(* CODESYS project PVCleaningRobot.project

Project tree, tasks and I/O mapping:
  Device : AC801-0221-U0R0, Shenzhen Inovance Technology Co., Ltd., version 3.5.11.50
      settings: PersistentStartAdddr = 0; PersistentStartEndAddr = 5242879; Mode = 0
    application Application
      libraries: Standard, * (System); CmpHCCom, 1.1.0.1 (Inovance); HC_CommBus, 1.3.12.0 (Inovance); CallCFunction, 1.7.2 (Inovance); CmpHCCom, 1.1.0.1 (Inovance); CmpEventMgr, 3.5.8.0 (System); ISysTypes2, 3.5.0.0 (System); CmpApp, 3.5.11.0 (System); IOBlockHandle, 1.3.0.0 (Inovance); HC_OmronUtils, 1.5.4.0 (Inovance); VisuDialogs, * (System); CmpHCTCPIP, 1.0.0.5 (Inovance); Util, 3.5.11.0 (System)
      task ETHERCAT_C (cyclic, interval 4000 µs, priority 0) calls ETHERCAT_C.EtherCAT_Task, 机械臂控制, 运动控制
      task 电池数据通讯 (cyclic, interval t#20ms, priority 16) calls 电池数据通讯
      task 业务逻辑 (cyclic, interval t#4ms, priority 1) calls DCH遥控控制, SLAM指令通讯, SLAM业务通讯
      task 伺服控制 (cyclic, interval t#5ms, priority 1) calls 底盘算法处理
      task 逻辑处理 (cyclic, interval t#20ms, priority 16) calls 报警处理
      program 机械臂控制 [ST]
      DifferentialMonitor
      Symbols
      trace Trace (task ETHERCAT_C): 机械臂控制.sMotionOutputs.dCmdPos[0], 机械臂控制.sMotionOutputs.dCmdPos[1], 机械臂控制.sMotionOutputs.dCmdPos[2], 机械臂控制.sMotionInputs.dFbPos[0], 机械臂控制.sMotionInputs.dFbPos[1], 机械臂控制.sMotionInputs.dFbPos[2], 机械臂控制.sMotionOutputs.dCmdSpace[0], 机械臂控制.sMotionOutputs.dCmdSpace[1], 机械臂控制.sMotionOutputs.dCmdSpace[2], 机械臂控制.sMotionInputs.dFbSpace[0], 机械臂控制.sMotionInputs.dFbPos[0], 机械臂控制.sMotionInputs.dFbPos[1], 机械臂控制.sMotionInputs.dFbPos[2], 机械臂控制.sMotionInputs.dFbPos[3], 机械臂控制.aiCcmdac[0], 机械臂控制.aiCcmdac[1], 机械臂控制.aiCcmdac[2]
      program 末端控制 [ST]: 上下卷扬控制, 传感器检测, 对中机构控制, 回零控制, 报警检测, 滚刷控制, ACT_test
      program 底盘算法处理 [ST]
      数据结构/
        data type 伺服参数结构体
        data type 底盘运行参数结构体
        data type 陀螺仪
        data type 机械臂参数结构体
        data type 系统状态
        data type 功能块状态
        data type PID控制参数
      函数/
        function block EventCallbackFunBLock [ST]: EventCallback, FB_Exit, FB_Init
        SLAM通讯/
          function block 上传信息处理 [ST]
          function block 校验功能块 [ST]
          function block 上传信息处理_1 [ST]
        运动控制/
          function block 伺服控制 [ST]
          function block 底盘平衡算法 [ST]
          function block 底盘控制运动 [ST]
          function block 清扫作业流程 [ST]
          function block 底盘控制运动_1 [ST]
          function block 低通滤波模块 [ST]
          function block 底盘控制运动_2 [ST]
          function block 超声波实时检测调整 [ST]
      全局变量/
        global variables 全局电池数据
        global variables 全局机械臂参数
        global variables 全局伺服参数
        global variables SLAM指令控制
        global variables 全局底盘参数
        global variables 业务流程
        global variables IO刷新数据
        global variables 末端控制参数
        global variables SLAM业务控制
        global variables 报警参数
      program 电池数据通讯 [ST]
      program SLAM指令通讯 [ST]: 系统状态上传, BMS数据上传, 温湿度数据上传, 单体电池电压数据上传, 单体电池温度数据上传, 行走电机状态上传, 悬挂电机状态上传, 轮速计数据上传, UPS数据上传, 超声波数据上传
      program 底盘控制 [ST]: 点动
      trace Trace_2 (task ETHERCAT_C): 末端控制.上卷扬滤波力矩, 末端控制.下卷扬滤波力矩, 末端控制.adFbForce[2]
      program 运动控制 [ST]
      trace Trace_1 (task ETHERCAT_C): 上卷扬运行位置保存, 下卷扬运行位置保存, DCH读遥控数据[0], test3
      program SLAM业务通讯 [ST]: 上装数据上传
      program DCH遥控控制 [ST]: DCH末端控制, DCH遥控数值刷新, DCH底盘控制, DCH机械臂控制
      trace Trace_3 (task ETHERCAT_C): 上侧滤波距离, 下侧滤波距离, 上侧距离, 下侧距离, 末端控制.PID_1.Y, 末端控制.PID_2.Y
      trace Trace_4 (task ETHERCAT_C): 右上轮.fActTorque, 右下轮.fActTorque, 左上轮.fActTorque, 左下轮.fActTorque, 左上轮.fActVelocity, 右上轮.fActVelocity, 左下轮.fActVelocity, 右下轮.fActVelocity, 右上轮.fSetTorque, 右下轮.fSetTorque, 左上轮.fSetTorque, 左下轮.fSetTorque, 左下轮.fSetVelocity, 右下轮.fSetVelocity, 左上轮.fSetVelocity, 右上轮.fSetVelocity, 左上轮.nAxisState, 右上轮.nAxisState, 右下轮.nAxisState, 左下轮.nAxisState, 左上轮.diActVelocity, 左上轮最大轮廓速度, 上卷扬伺服参数.运行位置, 下卷扬伺服参数.运行位置, 上下卷扬自动流程
      program 报警处理 [ST]
      trace Trace_5 (task ETHERCAT_C): 上卷扬运行位置保存, 上侧实际位置值暂存, 上卷扬伺服参数.运行位置, 上卷扬.fActPosition, 上侧距离, 左1滤波距离, 左2滤波距离, 下卷扬运行位置保存, 下侧实际位置值暂存, 下卷扬伺服参数.运行位置, 下卷扬.fActPosition, 下侧距离, 右1滤波距离, 右2滤波距离
    Network Configuration
      EtherCAT Config
    Resources List
    ConfigStorage
    HardWare Configuration
    Device Diagnosis
    SoftMotion General Axis Pool
    MODBUS_TCP : ModbusTCP本地从站, inovance, version 00.00.00.10
    HwConfiguratioinDevice : SystemConfig, Inovance, version 00.00.00.10
        settings: NetworkConfigArray.NetworkConfigArray.BusType = 10; NetworkConfigArray.NetworkConfigArray.RackSum = 1; NetworkConfigArray.NetworkConfigArray.HardwareConfigArray.HardwareConfigArray.RackNo = 1; EnableFun = 12
    ETHERCAT_C : EtherCAT Master SoftMotion, 3S - Smart Software Solutions GmbH, version 3.5.11.10
        settings:  = 0; Autoconfig = 0; NetworkName = 'enp3s0'; SelectNetworkByName = TRUE; DisableTaskGeneration = True
      InoSV630N_机械臂3轴 : SV630_1Axis_03715, Inovance, order no. InoSV630N, version Revision=16#00010000
          settings: Number of Outputs = 6; Number of Inputs = 10; Number of Infos about Outputs = 6; Number of Infos about Inputs = 10; Physical Address of the Slave = 1008; AutoIncr Address of the Slave = 4294967289; StationAlias = 0; Sync.Length = 18; Sync.Length = 32; FMMU.Global Start Address = 16#02000070; FMMU.Length = 18; FMMU.Physical Start Address = 16#1800; FMMU.Access = 16#02; FMMU.Global Start Address = 16#010000DE; FMMU.Length = 32; FMMU.Physical Start Address = 16#1C00; FMMU.Access = 16#01; FMMU.Global Start Address = 16#00080000; FMMU.StartBit = 6; FMMU.EndBit = 6; FMMU.Physical Start Address = 16#080D; FMMU.Access = 16#01; AutoUpdate = False; DC sync0 cycletime = 4000; DC sync1 cycletime = 4000; Number of SDO = 10; Homing method.Index = 16#6098; Homing method.Subindex = 16#00; Homing method.Value = 1; Homing method.Size = 8; Homing method.AbortIfError = FALSE; Homing method.JumpToLine = FALSE; Homing method.Line = 0; Homing method.CompleteAccess = FALSE; Actual Position Calculation Method.Index = 16#60E6; Actual Position Calculation Method.Subindex = 16#00; Actual Position Calculation Method.Value = 0; Actual Position Calculation Method.Size = 8; Actual Position Calculation Method.AbortIfError = FALSE; Actual Position Calculation Method.JumpToLine = FALSE;
            Actual Position Calculation Method.Line = 0; Actual Position Calculation Method.CompleteAccess = FALSE; Speed during search for switch.Index = 16#6099; Speed during search for switch.Subindex = 16#01; Speed during search for switch.Value = 436907; Speed during search for switch.Size = 32; Speed during search for switch.AbortIfError = FALSE; Speed during search for switch.JumpToLine = FALSE; Speed during search for switch.Line = 0; Speed during search for switch.CompleteAccess = FALSE; Homing acceleration.Index = 16#609A; Homing acceleration.Subindex = 16#00; Homing acceleration.Value = 43690666; Homing acceleration.Size = 32; Homing acceleration.AbortIfError = FALSE; Homing acceleration.JumpToLine = FALSE; Homing acceleration.Line = 0; Homing acceleration.CompleteAccess = FALSE; Speed during search for zero.Index = 16#6099; Speed during search for zero.Subindex = 16#02; Speed during search for zero.Value = 43691; Speed during search for zero.Size = 32; Speed during search for zero.AbortIfError = FALSE; Speed during search for zero.JumpToLine = FALSE; Speed during search for zero.Line = 0; Speed during search for zero.CompleteAccess = FALSE; Time of home searching.Index = 16#2005; Time of home searching.Subindex = 16#24; Time of home searching.Value = 50000; Time of home searching.Size = 16; Time of home searching.AbortIfError = FALSE; Time of home searching.JumpToLine = FALSE; Time of home searching.Line = 0; Time of home searching.CompleteAccess = FALSE; Positive torque limit value.Index = 16#60E0; Positive torque limit value.Subindex = 16#00; Positive torque limit value.Value = 3500; Positive torque limit value.Size = 16; Positive torque limit value.AbortIfError = FALSE; Positive torque limit value.JumpToLine = FALSE;
            Positive torque limit value.Line = 0; Positive torque limit value.CompleteAccess = FALSE; Negative torque limit value.Index = 16#60E1; Negative torque limit value.Subindex = 16#00; Negative torque limit value.Value = 3500; Negative torque limit value.Size = 16; Negative torque limit value.AbortIfError = FALSE; Negative torque limit value.JumpToLine = FALSE; Negative torque limit value.Line = 0; Negative torque limit value.CompleteAccess = FALSE; Max profile velocity.Index = 16#607F; Max profile velocity.Subindex = 16#00; Max profile velocity.Value = 26214400; Max profile velocity.Size = 32; Max profile velocity.AbortIfError = FALSE; Max profile velocity.JumpToLine = FALSE; Max profile velocity.Line = 0; Max profile velocity.CompleteAccess = FALSE; RxTxPdo.NumberofEntries = 6; RxTxPdo.Sm = 2; Controlword.Index = 16#6040; Controlword.SubIndex = 0; Controlword.Size = 16; Controlword.DependOnSlot = false; Controlword.DependOnSlotGroup = false; Target position.Index = 16#607A; Target position.SubIndex = 0; Target position.Size = 32; Target position.DependOnSlot = false; Target position.DependOnSlotGroup = false; Touch probe function.Index = 16#60B8; Touch probe function.SubIndex = 0; Touch probe function.Size = 16; Touch probe function.DependOnSlot = false; Touch probe function.DependOnSlotGroup = false; Physical outputs.Index = 16#60FE; Physical outputs.SubIndex = 1; Physical outputs.Size = 32; Physical outputs.DependOnSlot = false; Physical outputs.DependOnSlotGroup = false;
            Target velocity.Index = 16#60FF; Target velocity.SubIndex = 0; Target velocity.Size = 32; Target velocity.DependOnSlot = false; Target velocity.DependOnSlotGroup = false; Target torque.Index = 16#6071; Target torque.SubIndex = 0; Target torque.Size = 16; Target torque.DependOnSlot = false; Target torque.DependOnSlotGroup = false; RxTxPdo.Sm = -1; RxTxPdo.NumberofEntries = 10; RxTxPdo.Sm = 3; Error code.Index = 16#603F; Error code.SubIndex = 0; Error code.Size = 16; Error code.DependOnSlot = false; Error code.DependOnSlotGroup = false; Statusword.Index = 16#6041; Statusword.SubIndex = 0; Statusword.Size = 16; Statusword.DependOnSlot = false; Statusword.DependOnSlotGroup = false; Position actual value.Index = 16#6064; Position actual value.SubIndex = 0; Position actual value.Size = 32; Position actual value.DependOnSlot = false; Position actual value.DependOnSlotGroup = false; Torque actual value.Index = 16#6077; Torque actual value.SubIndex = 0; Torque actual value.Size = 16; Torque actual value.DependOnSlot = false; Torque actual value.DependOnSlotGroup = false; Following error actual value.Index = 16#60F4; Following error actual value.SubIndex = 0; Following error actual value.Size = 32; Following error actual value.DependOnSlot = false; Following error actual value.DependOnSlotGroup = false; Touch probe status.Index = 16#60B9; Touch probe status.SubIndex = 0;
            Touch probe status.Size = 16; Touch probe status.DependOnSlot = false; Touch probe status.DependOnSlotGroup = false; Touch probe pos1 pos value.Index = 16#60BA; Touch probe pos1 pos value.SubIndex = 0; Touch probe pos1 pos value.Size = 32; Touch probe pos1 pos value.DependOnSlot = false; Touch probe pos1 pos value.DependOnSlotGroup = false; Touch probe pos2 pos value.Index = 16#60BC; Touch probe pos2 pos value.SubIndex = 0; Touch probe pos2 pos value.Size = 32; Touch probe pos2 pos value.DependOnSlot = false; Touch probe pos2 pos value.DependOnSlotGroup = false; Digital inputs.Index = 16#60FD; Digital inputs.SubIndex = 0; Digital inputs.Size = 32; Digital inputs.DependOnSlot = false; Digital inputs.DependOnSlotGroup = false; Velocity actual value.Index = 16#606C; Velocity actual value.SubIndex = 0; Velocity actual value.Size = 32; Velocity actual value.DependOnSlot = false; Velocity actual value.DependOnSlotGroup = false; RxTxPdo.Sm = -1; Controlword.Name = 'Controlword'; Controlword.DataType = 'UINT'; Target position.Name = 'Target position'; Target position.DataType = 'DINT'; Touch probe function.Name = 'Touch probe function'; Touch probe function.DataType = 'UINT'; Physical outputs.Name = 'Physical outputs'; Physical outputs.DataType = 'UDINT'; Target velocity.Name = 'Target velocity'; Target velocity.DataType = 'DINT'; Target torque.Name = 'Target torque'; Target torque.DataType = 'INT'; Error code.Name = 'Error code'; Error code.DataType = 'UINT'; Statusword.Name = 'Statusword'; Statusword.DataType = 'UINT';
            Position actual value.Name = 'Position actual value'; Position actual value.DataType = 'DINT'; Torque actual value.Name = 'Torque actual value'; Torque actual value.DataType = 'INT'; Following error actual value.Name = 'Following error actual value'; Following error actual value.DataType = 'DINT'; Touch probe status.Name = 'Touch probe status'; Touch probe status.DataType = 'UINT'; Touch probe pos1 pos value.Name = 'Touch probe pos1 pos value'; Touch probe pos1 pos value.DataType = 'DINT'; Touch probe pos2 pos value.Name = 'Touch probe pos2 pos value'; Touch probe pos2 pos value.DataType = 'DINT'; Digital inputs.Name = 'Digital inputs'; Digital inputs.DataType = 'UDINT'; Velocity actual value.Name = 'Velocity actual value'; Velocity actual value.DataType = 'DINT'
          input  Application.机械臂控制.伺服错误码[2] : UINT  // Error code
          unmapped channels: Controlword, Target position, Touch probe function, Physical outputs, Target velocity, Target torque, Statusword, Position actual value, Torque actual value, Following error actual value, Touch probe status, Touch probe pos1 pos value, Touch probe pos2 pos value, Digital inputs, Velocity actual value
        机械臂3轴 : Axis, Inovance, order no. 0, version 1.0.0.0
            settings: wDriveID = 22; dwRatioTechUnitsDenom = 262144; fSWMaxVelocity = 1000; fSWMaxAcceleration = 10000; fSWMaxDeceleration = 10000; fSWMaxJerk = 100000; iEncoderType = 1; iAbsEncoderOption = 1; HomingMode = 10; ZeroSignal = 0; StartDirction = 1; EndDirection = 1; PosLimitMode = 0; NegLimitMode = 0; HomingVelocity = 10; HomingApproachVelocity = 2; HomingAcceleration = 100; HomingDeceleration = 100; HomingJerk = 0; HomeMaskDistance = 0; HomePositionOffset = 0; HomePushTime = 0; HomeCompensation = 0; HomeTimeout = 0; HomeCompensationVelocity = 1000; 4000 = 0; 4001 = 0; 4003 = true; 4004 = 3; 4005 = 0; 4006 = 1.666667; 4007 = 166.666666; 4008 = 0.166667; 4009 = 50000; 4010 = 3500; 4011 = 3500; 4012 = 100.000000; ScalingIncs = 16#40000; 6005 = 1; AdrOffset_8010 = 148;
              BitOffset_8010 = 0; BitLength_8010 = 16; Address_8010 = '%QW74'; Type_8010 = 'UINT'; AddressPointer_8010 = ADR(%QW74); AdrOffset_8020 = 152; BitOffset_8020 = 0; BitLength_8020 = 32; Address_8020 = '%QD38'; Type_8020 = 'DINT'; AddressPointer_8020 = ADR(%QD38); AdrOffset_8030 = 164; BitOffset_8030 = 0; BitLength_8030 = 32; Address_8030 = '%QD41'; Type_8030 = 'DINT'; AddressPointer_8030 = ADR(%QD41); AdrOffset_8040 = 168; BitOffset_8040 = 0; BitLength_8040 = 16; Address_8040 = '%QW84'; Type_8040 = 'INT'; AddressPointer_8040 = ADR(%QW84); AdrOffset_8050 = 4294967295; BitOffset_8050 = 0; BitLength_8050 = 0; Address_8050 = ''; Type_8050 = ''; AddressPointer_8050 = 0; AdrOffset_8060 = 156; BitOffset_8060 = 0; BitLength_8060 = 16; Address_8060 = '%QW78'; Type_8060 = 'UINT'; AddressPointer_8060 = ADR(%QW78); AdrOffset_8070 = 4294967295; BitOffset_8070 = 0; BitLength_8070 = 0; Address_8070 = ''; Type_8070 = '';
              AddressPointer_8070 = 0; AdrOffset_8080 = 4294967295; BitOffset_8080 = 0; BitLength_8080 = 0; Address_8080 = ''; Type_8080 = ''; AddressPointer_8080 = 0; AdrOffset_8090 = 160; BitOffset_8090 = 0; BitLength_8090 = 32; Address_8090 = '%QD40'; Type_8090 = 'UDINT'; AddressPointer_8090 = ADR(%QD40); AdrOffset_8100 = 4294967295; BitOffset_8100 = 0; BitLength_8100 = 0; Address_8100 = ''; Type_8100 = ''; AddressPointer_8100 = 0; AdrOffset_8510 = 250; BitOffset_8510 = 0; BitLength_8510 = 16; Address_8510 = '%IW125'; Type_8510 = 'UINT'; AddressPointer_8510 = ADR(%IW125); AdrOffset_8520 = 252; BitOffset_8520 = 0; BitLength_8520 = 32; Address_8520 = '%ID63'; Type_8520 = 'DINT'; AddressPointer_8520 = ADR(%ID63); AdrOffset_8530 = 280; BitOffset_8530 = 0; BitLength_8530 = 32; Address_8530 = '%ID70'; Type_8530 = 'DINT'; AddressPointer_8530 = ADR(%ID70); AdrOffset_8540 = 256; BitOffset_8540 = 0; BitLength_8540 = 16;
              Address_8540 = '%IW128'; Type_8540 = 'INT'; AddressPointer_8540 = ADR(%IW128); AdrOffset_8550 = 4294967295; BitOffset_8550 = 0; BitLength_8550 = 0; Address_8550 = ''; Type_8550 = ''; AddressPointer_8550 = 0; AdrOffset_8560 = 276; BitOffset_8560 = 0; BitLength_8560 = 32; Address_8560 = '%ID69'; Type_8560 = 'UDINT'; AddressPointer_8560 = ADR(%ID69); AdrOffset_8570 = 264; BitOffset_8570 = 0; BitLength_8570 = 16; Address_8570 = '%IW132'; Type_8570 = 'UINT'; AddressPointer_8570 = ADR(%IW132); AdrOffset_8580 = 268; BitOffset_8580 = 0; BitLength_8580 = 32; Address_8580 = '%ID67'; Type_8580 = 'DINT'; AddressPointer_8580 = ADR(%ID67); AdrOffset_8590 = 4294967295; BitOffset_8590 = 0; BitLength_8590 = 0; Address_8590 = ''; Type_8590 = ''; AddressPointer_8590 = 0; AdrOffset_8600 = 272; BitOffset_8600 = 0; BitLength_8600 = 32; Address_8600 = '%ID68'; Type_8600 = 'DINT'; AddressPointer_8600 = ADR(%ID68); AdrOffset_8600 = 4294967295;
              BitOffset_8600 = 0; BitLength_8600 = 0; Address_8610 = ''; Type_8610 = ''; AddressPointer_8610 = 0; AdrOffset_8620 = 0; BitOffset_8620 = 0; BitLength_8620 = 16; Address_8620 = '机械臂控制.伺服错误码[2]'; Type_8620 = 'UINT'; AddressPointer_8620 = ADR(机械臂控制.伺服错误码[2]); IsValid = True; IsHostHoming = False; PulseSelectIndex = 2
      InoSV630N_机械臂4轴 : SV630_1Axis_03715, Inovance, order no. InoSV630N, version Revision=16#00010000
          settings: Number of Outputs = 6; Number of Inputs = 10; Number of Infos about Outputs = 6; Number of Infos about Inputs = 10; Physical Address of the Slave = 1009; AutoIncr Address of the Slave = 4294967288; StationAlias = 0; Sync.Length = 18; Sync.Length = 32; FMMU.Global Start Address = 16#02000082; FMMU.Length = 18; FMMU.Physical Start Address = 16#1800; FMMU.Access = 16#02; FMMU.Global Start Address = 16#010000FE; FMMU.Length = 32; FMMU.Physical Start Address = 16#1C00; FMMU.Access = 16#01; FMMU.Global Start Address = 16#00080000; FMMU.StartBit = 7; FMMU.EndBit = 7; FMMU.Physical Start Address = 16#080D; FMMU.Access = 16#01; AutoUpdate = False; DC sync0 cycletime = 4000; DC sync1 cycletime = 4000; Number of SDO = 10; Homing method.Index = 16#6098; Homing method.Subindex = 16#00; Homing method.Value = 1; Homing method.Size = 8; Homing method.AbortIfError = FALSE; Homing method.JumpToLine = FALSE; Homing method.Line = 0; Homing method.CompleteAccess = FALSE; Actual Position Calculation Method.Index = 16#60E6; Actual Position Calculation Method.Subindex = 16#00; Actual Position Calculation Method.Value = 0; Actual Position Calculation Method.Size = 8; Actual Position Calculation Method.AbortIfError = FALSE; Actual Position Calculation Method.JumpToLine = FALSE;
            Actual Position Calculation Method.Line = 0; Actual Position Calculation Method.CompleteAccess = FALSE; Speed during search for switch.Index = 16#6099; Speed during search for switch.Subindex = 16#01; Speed during search for switch.Value = 436907; Speed during search for switch.Size = 32; Speed during search for switch.AbortIfError = FALSE; Speed during search for switch.JumpToLine = FALSE; Speed during search for switch.Line = 0; Speed during search for switch.CompleteAccess = FALSE; Homing acceleration.Index = 16#609A; Homing acceleration.Subindex = 16#00; Homing acceleration.Value = 43690666; Homing acceleration.Size = 32; Homing acceleration.AbortIfError = FALSE; Homing acceleration.JumpToLine = FALSE; Homing acceleration.Line = 0; Homing acceleration.CompleteAccess = FALSE; Speed during search for zero.Index = 16#6099; Speed during search for zero.Subindex = 16#02; Speed during search for zero.Value = 43691; Speed during search for zero.Size = 32; Speed during search for zero.AbortIfError = FALSE; Speed during search for zero.JumpToLine = FALSE; Speed during search for zero.Line = 0; Speed during search for zero.CompleteAccess = FALSE; Time of home searching.Index = 16#2005; Time of home searching.Subindex = 16#24; Time of home searching.Value = 50000; Time of home searching.Size = 16; Time of home searching.AbortIfError = FALSE; Time of home searching.JumpToLine = FALSE; Time of home searching.Line = 0; Time of home searching.CompleteAccess = FALSE; Positive torque limit value.Index = 16#60E0; Positive torque limit value.Subindex = 16#00; Positive torque limit value.Value = 3500; Positive torque limit value.Size = 16; Positive torque limit value.AbortIfError = FALSE; Positive torque limit value.JumpToLine = FALSE;
            Positive torque limit value.Line = 0; Positive torque limit value.CompleteAccess = FALSE; Negative torque limit value.Index = 16#60E1; Negative torque limit value.Subindex = 16#00; Negative torque limit value.Value = 3500; Negative torque limit value.Size = 16; Negative torque limit value.AbortIfError = FALSE; Negative torque limit value.JumpToLine = FALSE; Negative torque limit value.Line = 0; Negative torque limit value.CompleteAccess = FALSE; Max profile velocity.Index = 16#607F; Max profile velocity.Subindex = 16#00; Max profile velocity.Value = 26214400; Max profile velocity.Size = 32; Max profile velocity.AbortIfError = FALSE; Max profile velocity.JumpToLine = FALSE; Max profile velocity.Line = 0; Max profile velocity.CompleteAccess = FALSE; RxTxPdo.NumberofEntries = 6; RxTxPdo.Sm = 2; Controlword.Index = 16#6040; Controlword.SubIndex = 0; Controlword.Size = 16; Controlword.DependOnSlot = false; Controlword.DependOnSlotGroup = false; Target position.Index = 16#607A; Target position.SubIndex = 0; Target position.Size = 32; Target position.DependOnSlot = false; Target position.DependOnSlotGroup = false; Touch probe function.Index = 16#60B8; Touch probe function.SubIndex = 0; Touch probe function.Size = 16; Touch probe function.DependOnSlot = false; Touch probe function.DependOnSlotGroup = false; Physical outputs.Index = 16#60FE; Physical outputs.SubIndex = 1; Physical outputs.Size = 32; Physical outputs.DependOnSlot = false; Physical outputs.DependOnSlotGroup = false;
            Target velocity.Index = 16#60FF; Target velocity.SubIndex = 0; Target velocity.Size = 32; Target velocity.DependOnSlot = false; Target velocity.DependOnSlotGroup = false; Target torque.Index = 16#6071; Target torque.SubIndex = 0; Target torque.Size = 16; Target torque.DependOnSlot = false; Target torque.DependOnSlotGroup = false; RxTxPdo.Sm = -1; RxTxPdo.NumberofEntries = 10; RxTxPdo.Sm = 3; Error code.Index = 16#603F; Error code.SubIndex = 0; Error code.Size = 16; Error code.DependOnSlot = false; Error code.DependOnSlotGroup = false; Statusword.Index = 16#6041; Statusword.SubIndex = 0; Statusword.Size = 16; Statusword.DependOnSlot = false; Statusword.DependOnSlotGroup = false; Position actual value.Index = 16#6064; Position actual value.SubIndex = 0; Position actual value.Size = 32; Position actual value.DependOnSlot = false; Position actual value.DependOnSlotGroup = false; Torque actual value.Index = 16#6077; Torque actual value.SubIndex = 0; Torque actual value.Size = 16; Torque actual value.DependOnSlot = false; Torque actual value.DependOnSlotGroup = false; Following error actual value.Index = 16#60F4; Following error actual value.SubIndex = 0; Following error actual value.Size = 32; Following error actual value.DependOnSlot = false; Following error actual value.DependOnSlotGroup = false; Touch probe status.Index = 16#60B9; Touch probe status.SubIndex = 0;
            Touch probe status.Size = 16; Touch probe status.DependOnSlot = false; Touch probe status.DependOnSlotGroup = false; Touch probe pos1 pos value.Index = 16#60BA; Touch probe pos1 pos value.SubIndex = 0; Touch probe pos1 pos value.Size = 32; Touch probe pos1 pos value.DependOnSlot = false; Touch probe pos1 pos value.DependOnSlotGroup = false; Touch probe pos2 pos value.Index = 16#60BC; Touch probe pos2 pos value.SubIndex = 0; Touch probe pos2 pos value.Size = 32; Touch probe pos2 pos value.DependOnSlot = false; Touch probe pos2 pos value.DependOnSlotGroup = false; Digital inputs.Index = 16#60FD; Digital inputs.SubIndex = 0; Digital inputs.Size = 32; Digital inputs.DependOnSlot = false; Digital inputs.DependOnSlotGroup = false; Velocity actual value.Index = 16#606C; Velocity actual value.SubIndex = 0; Velocity actual value.Size = 32; Velocity actual value.DependOnSlot = false; Velocity actual value.DependOnSlotGroup = false; RxTxPdo.Sm = -1; Controlword.Name = 'Controlword'; Controlword.DataType = 'UINT'; Target position.Name = 'Target position'; Target position.DataType = 'DINT'; Touch probe function.Name = 'Touch probe function'; Touch probe function.DataType = 'UINT'; Physical outputs.Name = 'Physical outputs'; Physical outputs.DataType = 'UDINT'; Target velocity.Name = 'Target velocity'; Target velocity.DataType = 'DINT'; Target torque.Name = 'Target torque'; Target torque.DataType = 'INT'; Error code.Name = 'Error code'; Error code.DataType = 'UINT'; Statusword.Name = 'Statusword'; Statusword.DataType = 'UINT';
            Position actual value.Name = 'Position actual value'; Position actual value.DataType = 'DINT'; Torque actual value.Name = 'Torque actual value'; Torque actual value.DataType = 'INT'; Following error actual value.Name = 'Following error actual value'; Following error actual value.DataType = 'DINT'; Touch probe status.Name = 'Touch probe status'; Touch probe status.DataType = 'UINT'; Touch probe pos1 pos value.Name = 'Touch probe pos1 pos value'; Touch probe pos1 pos value.DataType = 'DINT'; Touch probe pos2 pos value.Name = 'Touch probe pos2 pos value'; Touch probe pos2 pos value.DataType = 'DINT'; Digital inputs.Name = 'Digital inputs'; Digital inputs.DataType = 'UDINT'; Velocity actual value.Name = 'Velocity actual value'; Velocity actual value.DataType = 'DINT'
          input  Application.机械臂控制.伺服错误码[3] : UINT  // Error code
          unmapped channels: Controlword, Target position, Touch probe function, Physical outputs, Target velocity, Target torque, Statusword, Position actual value, Torque actual value, Following error actual value, Touch probe status, Touch probe pos1 pos value, Touch probe pos2 pos value, Digital inputs, Velocity actual value
        机械臂4轴 : Axis, Inovance, order no. 0, version 1.0.0.0
            settings: wDriveID = 23; dwRatioTechUnitsDenom = 262144; fSWMaxVelocity = 1000; fSWMaxAcceleration = 10000; fSWMaxDeceleration = 10000; fSWMaxJerk = 100000; iEncoderType = 1; iAbsEncoderOption = 1; HomingMode = 10; ZeroSignal = 0; StartDirction = 1; EndDirection = 1; PosLimitMode = 0; NegLimitMode = 0; HomingVelocity = 10; HomingApproachVelocity = 2; HomingAcceleration = 100; HomingDeceleration = 100; HomingJerk = 0; HomeMaskDistance = 0; HomePositionOffset = 0; HomePushTime = 0; HomeCompensation = 0; HomeTimeout = 0; HomeCompensationVelocity = 1000; 4000 = 0; 4001 = 0; 4003 = true; 4004 = 3; 4005 = 0; 4006 = 1.666667; 4007 = 166.666666; 4008 = 0.166667; 4009 = 50000; 4010 = 3500; 4011 = 3500; 4012 = 100.000000; ScalingIncs = 16#40000; 6005 = 1; AdrOffset_8010 = 172;
              BitOffset_8010 = 0; BitLength_8010 = 16; Address_8010 = '%QW86'; Type_8010 = 'UINT'; AddressPointer_8010 = ADR(%QW86); AdrOffset_8020 = 176; BitOffset_8020 = 0; BitLength_8020 = 32; Address_8020 = '%QD44'; Type_8020 = 'DINT'; AddressPointer_8020 = ADR(%QD44); AdrOffset_8030 = 188; BitOffset_8030 = 0; BitLength_8030 = 32; Address_8030 = '%QD47'; Type_8030 = 'DINT'; AddressPointer_8030 = ADR(%QD47); AdrOffset_8040 = 192; BitOffset_8040 = 0; BitLength_8040 = 16; Address_8040 = '%QW96'; Type_8040 = 'INT'; AddressPointer_8040 = ADR(%QW96); AdrOffset_8050 = 4294967295; BitOffset_8050 = 0; BitLength_8050 = 0; Address_8050 = ''; Type_8050 = ''; AddressPointer_8050 = 0; AdrOffset_8060 = 180; BitOffset_8060 = 0; BitLength_8060 = 16; Address_8060 = '%QW90'; Type_8060 = 'UINT'; AddressPointer_8060 = ADR(%QW90); AdrOffset_8070 = 4294967295; BitOffset_8070 = 0; BitLength_8070 = 0; Address_8070 = ''; Type_8070 = '';
              AddressPointer_8070 = 0; AdrOffset_8080 = 4294967295; BitOffset_8080 = 0; BitLength_8080 = 0; Address_8080 = ''; Type_8080 = ''; AddressPointer_8080 = 0; AdrOffset_8090 = 184; BitOffset_8090 = 0; BitLength_8090 = 32; Address_8090 = '%QD46'; Type_8090 = 'UDINT'; AddressPointer_8090 = ADR(%QD46); AdrOffset_8100 = 4294967295; BitOffset_8100 = 0; BitLength_8100 = 0; Address_8100 = ''; Type_8100 = ''; AddressPointer_8100 = 0; AdrOffset_8510 = 286; BitOffset_8510 = 0; BitLength_8510 = 16; Address_8510 = '%IW143'; Type_8510 = 'UINT'; AddressPointer_8510 = ADR(%IW143); AdrOffset_8520 = 288; BitOffset_8520 = 0; BitLength_8520 = 32; Address_8520 = '%ID72'; Type_8520 = 'DINT'; AddressPointer_8520 = ADR(%ID72); AdrOffset_8530 = 316; BitOffset_8530 = 0; BitLength_8530 = 32; Address_8530 = '%ID79'; Type_8530 = 'DINT'; AddressPointer_8530 = ADR(%ID79); AdrOffset_8540 = 292; BitOffset_8540 = 0; BitLength_8540 = 16;
              Address_8540 = '%IW146'; Type_8540 = 'INT'; AddressPointer_8540 = ADR(%IW146); AdrOffset_8550 = 4294967295; BitOffset_8550 = 0; BitLength_8550 = 0; Address_8550 = ''; Type_8550 = ''; AddressPointer_8550 = 0; AdrOffset_8560 = 312; BitOffset_8560 = 0; BitLength_8560 = 32; Address_8560 = '%ID78'; Type_8560 = 'UDINT'; AddressPointer_8560 = ADR(%ID78); AdrOffset_8570 = 300; BitOffset_8570 = 0; BitLength_8570 = 16; Address_8570 = '%IW150'; Type_8570 = 'UINT'; AddressPointer_8570 = ADR(%IW150); AdrOffset_8580 = 304; BitOffset_8580 = 0; BitLength_8580 = 32; Address_8580 = '%ID76'; Type_8580 = 'DINT'; AddressPointer_8580 = ADR(%ID76); AdrOffset_8590 = 4294967295; BitOffset_8590 = 0; BitLength_8590 = 0; Address_8590 = ''; Type_8590 = ''; AddressPointer_8590 = 0; AdrOffset_8600 = 308; BitOffset_8600 = 0; BitLength_8600 = 32; Address_8600 = '%ID77'; Type_8600 = 'DINT'; AddressPointer_8600 = ADR(%ID77); AdrOffset_8600 = 4294967295;
              BitOffset_8600 = 0; BitLength_8600 = 0; Address_8610 = ''; Type_8610 = ''; AddressPointer_8610 = 0; AdrOffset_8620 = 0; BitOffset_8620 = 0; BitLength_8620 = 16; Address_8620 = '机械臂控制.伺服错误码[3]'; Type_8620 = 'UINT'; AddressPointer_8620 = ADR(机械臂控制.伺服错误码[3]); IsValid = True; IsHostHoming = False; PulseSelectIndex = 2
      InoSV630N_机械臂1轴 : SV630_1Axis_03715, Inovance, order no. InoSV630N, version Revision=16#00010000
          settings: Number of Outputs = 7; Number of Inputs = 10; Number of Infos about Outputs = 7; Number of Infos about Inputs = 10; EnableExpertSettings = True; Physical Address of the Slave = 1006; AutoIncr Address of the Slave = 4294967291; StationAlias = 0; Sync.Length = 19; Sync.Length = 32; FMMU.Global Start Address = 16#0200004B; FMMU.Length = 19; FMMU.Physical Start Address = 16#1800; FMMU.Access = 16#02; FMMU.Global Start Address = 16#0100009E; FMMU.Length = 32; FMMU.Physical Start Address = 16#1C00; FMMU.Access = 16#01; FMMU.Global Start Address = 16#00080000; FMMU.StartBit = 4; FMMU.EndBit = 4; FMMU.Physical Start Address = 16#080D; FMMU.Access = 16#01; AutoUpdate = False; DC sync0 cycletime = 4000; DC sync0 cycletime = 4000000; DC sync1 cycletime = 4000; DC sync1 cycletime = 4000000; Number of SDO = 10; Homing method.Index = 16#6098; Homing method.Subindex = 16#00; Homing method.Value = 1; Homing method.Size = 8; Homing method.AbortIfError = FALSE; Homing method.JumpToLine = FALSE; Homing method.Line = 0; Homing method.CompleteAccess = False; Actual Position Calculation Method.Index = 16#60E6; Actual Position Calculation Method.Subindex = 16#00; Actual Position Calculation Method.Value = 0;
            Actual Position Calculation Method.Size = 8; Actual Position Calculation Method.AbortIfError = FALSE; Actual Position Calculation Method.JumpToLine = FALSE; Actual Position Calculation Method.Line = 0; Actual Position Calculation Method.CompleteAccess = False; Speed during search for switch.Index = 16#6099; Speed during search for switch.Subindex = 16#01; Speed during search for switch.Value = 436907; Speed during search for switch.Size = 32; Speed during search for switch.AbortIfError = FALSE; Speed during search for switch.JumpToLine = FALSE; Speed during search for switch.Line = 0; Speed during search for switch.CompleteAccess = False; Homing acceleration.Index = 16#609A; Homing acceleration.Subindex = 16#00; Homing acceleration.Value = 43690666; Homing acceleration.Size = 32; Homing acceleration.AbortIfError = FALSE; Homing acceleration.JumpToLine = FALSE; Homing acceleration.Line = 0; Homing acceleration.CompleteAccess = False; Speed during search for zero.Index = 16#6099; Speed during search for zero.Subindex = 16#02; Speed during search for zero.Value = 43691; Speed during search for zero.Size = 32; Speed during search for zero.AbortIfError = FALSE; Speed during search for zero.JumpToLine = FALSE; Speed during search for zero.Line = 0; Speed during search for zero.CompleteAccess = False; Time of home searching.Index = 16#2005; Time of home searching.Subindex = 16#24; Time of home searching.Value = 50000; Time of home searching.Size = 16; Time of home searching.AbortIfError = FALSE; Time of home searching.JumpToLine = FALSE; Time of home searching.Line = 0; Time of home searching.CompleteAccess = False; Positive torque limit value.Index = 16#60E0; Positive torque limit value.Subindex = 16#00; Positive torque limit value.Value = 3500;
            Positive torque limit value.Size = 16; Positive torque limit value.AbortIfError = FALSE; Positive torque limit value.JumpToLine = FALSE; Positive torque limit value.Line = 0; Positive torque limit value.CompleteAccess = False; Negative torque limit value.Index = 16#60E1; Negative torque limit value.Subindex = 16#00; Negative torque limit value.Value = 3500; Negative torque limit value.Size = 16; Negative torque limit value.AbortIfError = FALSE; Negative torque limit value.JumpToLine = FALSE; Negative torque limit value.Line = 0; Negative torque limit value.CompleteAccess = False; Max profile velocity.Index = 16#607F; Max profile velocity.Subindex = 16#00; Max profile velocity.Value = 26214400; Max profile velocity.Size = 32; Max profile velocity.AbortIfError = FALSE; Max profile velocity.JumpToLine = FALSE; Max profile velocity.Line = 0; Max profile velocity.CompleteAccess = False; RxTxPdo.NumberofEntries = 7; RxTxPdo.Sm = 2; RxTxPdo.DependOnSlot = False; RxTxPdo.DependOnSlotGroup = False; RxTxPdo.OverwrittenByModule = False; Exclude = [16#1701,16#1702,16#1703,16#1704,16#1705]; Controlword.Index = 16#6040; Controlword.SubIndex = 0; Controlword.Size = 16; Controlword.Offset = 0; Controlword.DependOnSlot = False; Controlword.DependOnSlotGroup = False; Target position.Index = 16#607A; Target position.SubIndex = 0; Target position.Size = 32; Target position.Offset = 0; Target position.DependOnSlot = False; Target position.DependOnSlotGroup = False; Touch probe function.Index = 16#60B8;
            Touch probe function.SubIndex = 0; Touch probe function.Size = 16; Touch probe function.Offset = 0; Touch probe function.DependOnSlot = False; Touch probe function.DependOnSlotGroup = False; Physical outputs.Index = 16#60FE; Physical outputs.SubIndex = 1; Physical outputs.Size = 32; Physical outputs.Offset = 0; Physical outputs.DependOnSlot = False; Physical outputs.DependOnSlotGroup = False; Target velocity.Index = 16#60FF; Target velocity.SubIndex = 0; Target velocity.Size = 32; Target velocity.Offset = 0; Target velocity.DependOnSlot = False; Target velocity.DependOnSlotGroup = False; Modes of operation.Index = 16#6060; Modes of operation.SubIndex = 0; Modes of operation.Size = 8; Modes of operation.Offset = 0; Modes of operation.DependOnSlot = False; Modes of operation.DependOnSlotGroup = False; Target torque.Index = 16#6071; Target torque.SubIndex = 0; Target torque.Size = 16; Target torque.Offset = 0; Target torque.DependOnSlot = False; Target torque.DependOnSlotGroup = False; RxTxPdo.Sm = -1; RxTxPdo.NumberofEntries = 10; RxTxPdo.Sm = 3; Error code.Index = 16#603F; Error code.SubIndex = 0; Error code.Size = 16; Error code.DependOnSlot = false; Error code.DependOnSlotGroup = false; Statusword.Index = 16#6041; Statusword.SubIndex = 0; Statusword.Size = 16;
            Statusword.DependOnSlot = false; Statusword.DependOnSlotGroup = false; Position actual value.Index = 16#6064; Position actual value.SubIndex = 0; Position actual value.Size = 32; Position actual value.DependOnSlot = false; Position actual value.DependOnSlotGroup = false; Torque actual value.Index = 16#6077; Torque actual value.SubIndex = 0; Torque actual value.Size = 16; Torque actual value.DependOnSlot = false; Torque actual value.DependOnSlotGroup = false; Following error actual value.Index = 16#60F4; Following error actual value.SubIndex = 0; Following error actual value.Size = 32; Following error actual value.DependOnSlot = false; Following error actual value.DependOnSlotGroup = false; Touch probe status.Index = 16#60B9; Touch probe status.SubIndex = 0; Touch probe status.Size = 16; Touch probe status.DependOnSlot = false; Touch probe status.DependOnSlotGroup = false; Touch probe pos1 pos value.Index = 16#60BA; Touch probe pos1 pos value.SubIndex = 0; Touch probe pos1 pos value.Size = 32; Touch probe pos1 pos value.DependOnSlot = false; Touch probe pos1 pos value.DependOnSlotGroup = false; Touch probe pos2 pos value.Index = 16#60BC; Touch probe pos2 pos value.SubIndex = 0; Touch probe pos2 pos value.Size = 32; Touch probe pos2 pos value.DependOnSlot = false; Touch probe pos2 pos value.DependOnSlotGroup = false; Digital inputs.Index = 16#60FD; Digital inputs.SubIndex = 0; Digital inputs.Size = 32; Digital inputs.DependOnSlot = false; Digital inputs.DependOnSlotGroup = false; Velocity actual value.Index = 16#606C; Velocity actual value.SubIndex = 0; Velocity actual value.Size = 32;
            Velocity actual value.DependOnSlot = false; Velocity actual value.DependOnSlotGroup = false; RxTxPdo.Sm = -1; Controlword.Name = 'Controlword'; Controlword.DataType = 'UINT'; Controlword.Default = ''; Controlword.Comment = ''; Target position.Name = 'Target position'; Target position.DataType = 'DINT'; Target position.Default = ''; Target position.Comment = ''; Touch probe function.Name = 'Touch probe function'; Touch probe function.DataType = 'UINT'; Touch probe function.Default = ''; Touch probe function.Comment = ''; Physical outputs.Name = 'Physical outputs'; Physical outputs.DataType = 'UDINT'; Physical outputs.Default = ''; Physical outputs.Comment = ''; Target velocity.Name = 'Target velocity'; Target velocity.DataType = 'DINT'; Target velocity.Default = ''; Target velocity.Comment = ''; Modes of operation.Name = 'Modes of operation'; Modes of operation.DataType = 'SINT'; Modes of operation.Default = ''; Modes of operation.Comment = ''; Target torque.Name = 'Target torque'; Target torque.DataType = 'INT'; Target torque.Default = ''; Target torque.Comment = ''; Error code.Name = 'Error code'; Error code.DataType = 'UINT'; Statusword.Name = 'Statusword'; Statusword.DataType = 'UINT'; Position actual value.Name = 'Position actual value'; Position actual value.DataType = 'DINT'; Torque actual value.Name = 'Torque actual value'; Torque actual value.DataType = 'INT'; Following error actual value.Name = 'Following error actual value';
            Following error actual value.DataType = 'DINT'; Touch probe status.Name = 'Touch probe status'; Touch probe status.DataType = 'UINT'; Touch probe pos1 pos value.Name = 'Touch probe pos1 pos value'; Touch probe pos1 pos value.DataType = 'DINT'; Touch probe pos2 pos value.Name = 'Touch probe pos2 pos value'; Touch probe pos2 pos value.DataType = 'DINT'; Digital inputs.Name = 'Digital inputs'; Digital inputs.DataType = 'UDINT'; Velocity actual value.Name = 'Velocity actual value'; Velocity actual value.DataType = 'DINT'
          input  Application.机械臂控制.伺服错误码[0] : UINT  // Error code
          unmapped channels: Controlword, Target position, Touch probe function, Physical outputs, Target velocity, Modes of operation, Target torque, Statusword, Position actual value, Torque actual value, Following error actual value, Touch probe status, Touch probe pos1 pos value, Touch probe pos2 pos value, Digital inputs, Velocity actual value
        机械臂1轴 : Axis, Inovance, order no. 0, version 1.0.0.0
            settings: wDriveID = 20; dwRatioTechUnitsDenom = 262144; fSWMaxVelocity = 1000; fSWMaxAcceleration = 10000; fSWMaxDeceleration = 10000; fSWMaxJerk = 100000; iEncoderType = 1; iAbsEncoderOption = 1; HomingMode = 10; ZeroSignal = 0; StartDirction = 1; EndDirection = 1; PosLimitMode = 0; NegLimitMode = 0; HomingVelocity = 10; HomingApproachVelocity = 2; HomingAcceleration = 100; HomingDeceleration = 100; HomingJerk = 0; HomeMaskDistance = 0; HomePositionOffset = 0; HomePushTime = 0; HomeCompensation = 0; HomeTimeout = 0; HomeCompensationVelocity = 1000; 4000 = 0; 4001 = 0; 4003 = true; 4004 = 3; 4005 = 0; 4006 = 1.666667; 4007 = 166.666666; 4008 = 0.166667; 4009 = 50000; 4010 = 3500; 4011 = 3500; 4012 = 100.000000; ScalingIncs = 16#40000; 6005 = 1; AdrOffset_8010 = 100;
              BitOffset_8010 = 0; BitLength_8010 = 16; Address_8010 = '%QW50'; Type_8010 = 'UINT'; AddressPointer_8010 = ADR(%QW50); AdrOffset_8020 = 104; BitOffset_8020 = 0; BitLength_8020 = 32; Address_8020 = '%QD26'; Type_8020 = 'DINT'; AddressPointer_8020 = ADR(%QD26); AdrOffset_8030 = 116; BitOffset_8030 = 0; BitLength_8030 = 32; Address_8030 = '%QD29'; Type_8030 = 'DINT'; AddressPointer_8030 = ADR(%QD29); AdrOffset_8040 = 122; BitOffset_8040 = 0; BitLength_8040 = 16; Address_8040 = '%QW61'; Type_8040 = 'INT'; AddressPointer_8040 = ADR(%QW61); AdrOffset_8050 = 120; BitOffset_8050 = 0; BitLength_8050 = 8; Address_8050 = '%QB120'; Type_8050 = 'SINT'; AddressPointer_8050 = ADR(%QB120); AdrOffset_8060 = 108; BitOffset_8060 = 0; BitLength_8060 = 16; Address_8060 = '%QW54'; Type_8060 = 'UINT'; AddressPointer_8060 = ADR(%QW54); AdrOffset_8070 = 4294967295; BitOffset_8070 = 0; BitLength_8070 = 0; Address_8070 = ''; Type_8070 = '';
              AddressPointer_8070 = 0; AdrOffset_8080 = 4294967295; BitOffset_8080 = 0; BitLength_8080 = 0; Address_8080 = ''; Type_8080 = ''; AddressPointer_8080 = 0; AdrOffset_8090 = 112; BitOffset_8090 = 0; BitLength_8090 = 32; Address_8090 = '%QD28'; Type_8090 = 'UDINT'; AddressPointer_8090 = ADR(%QD28); AdrOffset_8100 = 4294967295; BitOffset_8100 = 0; BitLength_8100 = 0; Address_8100 = ''; Type_8100 = ''; AddressPointer_8100 = 0; AdrOffset_8510 = 178; BitOffset_8510 = 0; BitLength_8510 = 16; Address_8510 = '%IW89'; Type_8510 = 'UINT'; AddressPointer_8510 = ADR(%IW89); AdrOffset_8520 = 180; BitOffset_8520 = 0; BitLength_8520 = 32; Address_8520 = '%ID45'; Type_8520 = 'DINT'; AddressPointer_8520 = ADR(%ID45); AdrOffset_8530 = 208; BitOffset_8530 = 0; BitLength_8530 = 32; Address_8530 = '%ID52'; Type_8530 = 'DINT'; AddressPointer_8530 = ADR(%ID52); AdrOffset_8540 = 184; BitOffset_8540 = 0; BitLength_8540 = 16;
              Address_8540 = '%IW92'; Type_8540 = 'INT'; AddressPointer_8540 = ADR(%IW92); AdrOffset_8550 = 4294967295; BitOffset_8550 = 0; BitLength_8550 = 0; Address_8550 = ''; Type_8550 = ''; AddressPointer_8550 = 0; AdrOffset_8560 = 204; BitOffset_8560 = 0; BitLength_8560 = 32; Address_8560 = '%ID51'; Type_8560 = 'UDINT'; AddressPointer_8560 = ADR(%ID51); AdrOffset_8570 = 192; BitOffset_8570 = 0; BitLength_8570 = 16; Address_8570 = '%IW96'; Type_8570 = 'UINT'; AddressPointer_8570 = ADR(%IW96); AdrOffset_8580 = 196; BitOffset_8580 = 0; BitLength_8580 = 32; Address_8580 = '%ID49'; Type_8580 = 'DINT'; AddressPointer_8580 = ADR(%ID49); AdrOffset_8590 = 4294967295; BitOffset_8590 = 0; BitLength_8590 = 0; Address_8590 = ''; Type_8590 = ''; AddressPointer_8590 = 0; AdrOffset_8600 = 200; BitOffset_8600 = 0; BitLength_8600 = 32; Address_8600 = '%ID50'; Type_8600 = 'DINT'; AddressPointer_8600 = ADR(%ID50); AdrOffset_8600 = 4294967295;
              BitOffset_8600 = 0; BitLength_8600 = 0; Address_8610 = ''; Type_8610 = ''; AddressPointer_8610 = 0; AdrOffset_8620 = 0; BitOffset_8620 = 0; BitLength_8620 = 16; Address_8620 = '机械臂控制.伺服错误码[0]'; Type_8620 = 'UINT'; AddressPointer_8620 = ADR(机械臂控制.伺服错误码[0]); Automatic Mapping = True; IsValid = True; IsHostHoming = False; PulseSelectIndex = 2
      InoSV630N_机械臂2轴 : SV630_1Axis_03715, Inovance, order no. InoSV630N, version Revision=16#00010000
          settings: Number of Outputs = 6; Number of Inputs = 10; Number of Infos about Outputs = 6; Number of Infos about Inputs = 10; EnableExpertSettings = True; Physical Address of the Slave = 1007; AutoIncr Address of the Slave = 4294967290; StationAlias = 0; Sync.Length = 18; Sync.Length = 32; FMMU.Global Start Address = 16#0200005E; FMMU.Length = 18; FMMU.Physical Start Address = 16#1800; FMMU.Access = 16#02; FMMU.Global Start Address = 16#010000BE; FMMU.Length = 32; FMMU.Physical Start Address = 16#1C00; FMMU.Access = 16#01; FMMU.Global Start Address = 16#00080000; FMMU.StartBit = 5; FMMU.EndBit = 5; FMMU.Physical Start Address = 16#080D; FMMU.Access = 16#01; AutoUpdate = False; DC sync0 cycletime = 4000; DC sync0 cycletime = 4000000; DC sync1 cycletime = 4000; DC sync1 cycletime = 4000000; Number of SDO = 10; Homing method.Index = 16#6098; Homing method.Subindex = 16#00; Homing method.Value = 1; Homing method.Size = 8; Homing method.AbortIfError = FALSE; Homing method.JumpToLine = FALSE; Homing method.Line = 0; Homing method.CompleteAccess = FALSE; Actual Position Calculation Method.Index = 16#60E6; Actual Position Calculation Method.Subindex = 16#00; Actual Position Calculation Method.Value = 0;
            Actual Position Calculation Method.Size = 8; Actual Position Calculation Method.AbortIfError = FALSE; Actual Position Calculation Method.JumpToLine = FALSE; Actual Position Calculation Method.Line = 0; Actual Position Calculation Method.CompleteAccess = FALSE; Speed during search for switch.Index = 16#6099; Speed during search for switch.Subindex = 16#01; Speed during search for switch.Value = 436907; Speed during search for switch.Size = 32; Speed during search for switch.AbortIfError = FALSE; Speed during search for switch.JumpToLine = FALSE; Speed during search for switch.Line = 0; Speed during search for switch.CompleteAccess = FALSE; Homing acceleration.Index = 16#609A; Homing acceleration.Subindex = 16#00; Homing acceleration.Value = 43690666; Homing acceleration.Size = 32; Homing acceleration.AbortIfError = FALSE; Homing acceleration.JumpToLine = FALSE; Homing acceleration.Line = 0; Homing acceleration.CompleteAccess = FALSE; Speed during search for zero.Index = 16#6099; Speed during search for zero.Subindex = 16#02; Speed during search for zero.Value = 43691; Speed during search for zero.Size = 32; Speed during search for zero.AbortIfError = FALSE; Speed during search for zero.JumpToLine = FALSE; Speed during search for zero.Line = 0; Speed during search for zero.CompleteAccess = FALSE; Time of home searching.Index = 16#2005; Time of home searching.Subindex = 16#24; Time of home searching.Value = 50000; Time of home searching.Size = 16; Time of home searching.AbortIfError = FALSE; Time of home searching.JumpToLine = FALSE; Time of home searching.Line = 0; Time of home searching.CompleteAccess = FALSE; Positive torque limit value.Index = 16#60E0; Positive torque limit value.Subindex = 16#00; Positive torque limit value.Value = 3500;
            Positive torque limit value.Size = 16; Positive torque limit value.AbortIfError = FALSE; Positive torque limit value.JumpToLine = FALSE; Positive torque limit value.Line = 0; Positive torque limit value.CompleteAccess = FALSE; Negative torque limit value.Index = 16#60E1; Negative torque limit value.Subindex = 16#00; Negative torque limit value.Value = 3500; Negative torque limit value.Size = 16; Negative torque limit value.AbortIfError = FALSE; Negative torque limit value.JumpToLine = FALSE; Negative torque limit value.Line = 0; Negative torque limit value.CompleteAccess = FALSE; Max profile velocity.Index = 16#607F; Max profile velocity.Subindex = 16#00; Max profile velocity.Value = 26214400; Max profile velocity.Size = 32; Max profile velocity.AbortIfError = FALSE; Max profile velocity.JumpToLine = FALSE; Max profile velocity.Line = 0; Max profile velocity.CompleteAccess = FALSE; RxTxPdo.NumberofEntries = 6; RxTxPdo.Sm = 2; Controlword.Index = 16#6040; Controlword.SubIndex = 0; Controlword.Size = 16; Controlword.DependOnSlot = false; Controlword.DependOnSlotGroup = false; Target position.Index = 16#607A; Target position.SubIndex = 0; Target position.Size = 32; Target position.DependOnSlot = false; Target position.DependOnSlotGroup = false; Touch probe function.Index = 16#60B8; Touch probe function.SubIndex = 0; Touch probe function.Size = 16; Touch probe function.DependOnSlot = false; Touch probe function.DependOnSlotGroup = false; Physical outputs.Index = 16#60FE; Physical outputs.SubIndex = 1;
            Physical outputs.Size = 32; Physical outputs.DependOnSlot = false; Physical outputs.DependOnSlotGroup = false; Target velocity.Index = 16#60FF; Target velocity.SubIndex = 0; Target velocity.Size = 32; Target velocity.DependOnSlot = false; Target velocity.DependOnSlotGroup = false; Target torque.Index = 16#6071; Target torque.SubIndex = 0; Target torque.Size = 16; Target torque.DependOnSlot = false; Target torque.DependOnSlotGroup = false; RxTxPdo.Sm = -1; RxTxPdo.NumberofEntries = 10; RxTxPdo.Sm = 3; Error code.Index = 16#603F; Error code.SubIndex = 0; Error code.Size = 16; Error code.DependOnSlot = false; Error code.DependOnSlotGroup = false; Statusword.Index = 16#6041; Statusword.SubIndex = 0; Statusword.Size = 16; Statusword.DependOnSlot = false; Statusword.DependOnSlotGroup = false; Position actual value.Index = 16#6064; Position actual value.SubIndex = 0; Position actual value.Size = 32; Position actual value.DependOnSlot = false; Position actual value.DependOnSlotGroup = false; Torque actual value.Index = 16#6077; Torque actual value.SubIndex = 0; Torque actual value.Size = 16; Torque actual value.DependOnSlot = false; Torque actual value.DependOnSlotGroup = false; Following error actual value.Index = 16#60F4; Following error actual value.SubIndex = 0; Following error actual value.Size = 32; Following error actual value.DependOnSlot = false;
            Following error actual value.DependOnSlotGroup = false; Touch probe status.Index = 16#60B9; Touch probe status.SubIndex = 0; Touch probe status.Size = 16; Touch probe status.DependOnSlot = false; Touch probe status.DependOnSlotGroup = false; Touch probe pos1 pos value.Index = 16#60BA; Touch probe pos1 pos value.SubIndex = 0; Touch probe pos1 pos value.Size = 32; Touch probe pos1 pos value.DependOnSlot = false; Touch probe pos1 pos value.DependOnSlotGroup = false; Touch probe pos2 pos value.Index = 16#60BC; Touch probe pos2 pos value.SubIndex = 0; Touch probe pos2 pos value.Size = 32; Touch probe pos2 pos value.DependOnSlot = false; Touch probe pos2 pos value.DependOnSlotGroup = false; Digital inputs.Index = 16#60FD; Digital inputs.SubIndex = 0; Digital inputs.Size = 32; Digital inputs.DependOnSlot = false; Digital inputs.DependOnSlotGroup = false; Velocity actual value.Index = 16#606C; Velocity actual value.SubIndex = 0; Velocity actual value.Size = 32; Velocity actual value.DependOnSlot = false; Velocity actual value.DependOnSlotGroup = false; RxTxPdo.Sm = -1; Controlword.Name = 'Controlword'; Controlword.DataType = 'UINT'; Target position.Name = 'Target position'; Target position.DataType = 'DINT'; Touch probe function.Name = 'Touch probe function'; Touch probe function.DataType = 'UINT'; Physical outputs.Name = 'Physical outputs'; Physical outputs.DataType = 'UDINT'; Target velocity.Name = 'Target velocity'; Target velocity.DataType = 'DINT'; Target torque.Name = 'Target torque'; Target torque.DataType = 'INT'; Error code.Name = 'Error code';
            Error code.DataType = 'UINT'; Statusword.Name = 'Statusword'; Statusword.DataType = 'UINT'; Position actual value.Name = 'Position actual value'; Position actual value.DataType = 'DINT'; Torque actual value.Name = 'Torque actual value'; Torque actual value.DataType = 'INT'; Following error actual value.Name = 'Following error actual value'; Following error actual value.DataType = 'DINT'; Touch probe status.Name = 'Touch probe status'; Touch probe status.DataType = 'UINT'; Touch probe pos1 pos value.Name = 'Touch probe pos1 pos value'; Touch probe pos1 pos value.DataType = 'DINT'; Touch probe pos2 pos value.Name = 'Touch probe pos2 pos value'; Touch probe pos2 pos value.DataType = 'DINT'; Digital inputs.Name = 'Digital inputs'; Digital inputs.DataType = 'UDINT'; Velocity actual value.Name = 'Velocity actual value'; Velocity actual value.DataType = 'DINT'
          input  Application.机械臂控制.伺服错误码[1] : UINT  // Error code
          unmapped channels: Controlword, Target position, Touch probe function, Physical outputs, Target velocity, Target torque, Statusword, Position actual value, Torque actual value, Following error actual value, Touch probe status, Touch probe pos1 pos value, Touch probe pos2 pos value, Digital inputs, Velocity actual value
        机械臂2轴 : Axis, Inovance, order no. 0, version 1.0.0.0
            settings: wDriveID = 21; dwRatioTechUnitsDenom = 262144; fSWMaxVelocity = 1000; fSWMaxAcceleration = 10000; fSWMaxDeceleration = 10000; fSWMaxJerk = 100000; iEncoderType = 1; iAbsEncoderOption = 1; HomingMode = 10; ZeroSignal = 0; StartDirction = 1; EndDirection = 1; PosLimitMode = 0; NegLimitMode = 0; HomingVelocity = 10; HomingApproachVelocity = 2; HomingAcceleration = 100; HomingDeceleration = 100; HomingJerk = 0; HomeMaskDistance = 0; HomePositionOffset = 0; HomePushTime = 0; HomeCompensation = 0; HomeTimeout = 0; HomeCompensationVelocity = 1000; 4000 = 0; 4001 = 0; 4003 = true; 4004 = 3; 4005 = 0; 4006 = 1.666667; 4007 = 166.666666; 4008 = 0.166667; 4009 = 50000; 4010 = 3500; 4011 = 3500; 4012 = 100.000000; ScalingIncs = 16#40000; 6005 = 1; AdrOffset_8010 = 124;
              BitOffset_8010 = 0; BitLength_8010 = 16; Address_8010 = '%QW62'; Type_8010 = 'UINT'; AddressPointer_8010 = ADR(%QW62); AdrOffset_8020 = 128; BitOffset_8020 = 0; BitLength_8020 = 32; Address_8020 = '%QD32'; Type_8020 = 'DINT'; AddressPointer_8020 = ADR(%QD32); AdrOffset_8030 = 140; BitOffset_8030 = 0; BitLength_8030 = 32; Address_8030 = '%QD35'; Type_8030 = 'DINT'; AddressPointer_8030 = ADR(%QD35); AdrOffset_8040 = 144; BitOffset_8040 = 0; BitLength_8040 = 16; Address_8040 = '%QW72'; Type_8040 = 'INT'; AddressPointer_8040 = ADR(%QW72); AdrOffset_8050 = 4294967295; BitOffset_8050 = 0; BitLength_8050 = 0; Address_8050 = ''; Type_8050 = ''; AddressPointer_8050 = 0; AdrOffset_8060 = 132; BitOffset_8060 = 0; BitLength_8060 = 16; Address_8060 = '%QW66'; Type_8060 = 'UINT'; AddressPointer_8060 = ADR(%QW66); AdrOffset_8070 = 4294967295; BitOffset_8070 = 0; BitLength_8070 = 0; Address_8070 = ''; Type_8070 = '';
              AddressPointer_8070 = 0; AdrOffset_8080 = 4294967295; BitOffset_8080 = 0; BitLength_8080 = 0; Address_8080 = ''; Type_8080 = ''; AddressPointer_8080 = 0; AdrOffset_8090 = 136; BitOffset_8090 = 0; BitLength_8090 = 32; Address_8090 = '%QD34'; Type_8090 = 'UDINT'; AddressPointer_8090 = ADR(%QD34); AdrOffset_8100 = 4294967295; BitOffset_8100 = 0; BitLength_8100 = 0; Address_8100 = ''; Type_8100 = ''; AddressPointer_8100 = 0; AdrOffset_8510 = 214; BitOffset_8510 = 0; BitLength_8510 = 16; Address_8510 = '%IW107'; Type_8510 = 'UINT'; AddressPointer_8510 = ADR(%IW107); AdrOffset_8520 = 216; BitOffset_8520 = 0; BitLength_8520 = 32; Address_8520 = '%ID54'; Type_8520 = 'DINT'; AddressPointer_8520 = ADR(%ID54); AdrOffset_8530 = 244; BitOffset_8530 = 0; BitLength_8530 = 32; Address_8530 = '%ID61'; Type_8530 = 'DINT'; AddressPointer_8530 = ADR(%ID61); AdrOffset_8540 = 220; BitOffset_8540 = 0; BitLength_8540 = 16;
              Address_8540 = '%IW110'; Type_8540 = 'INT'; AddressPointer_8540 = ADR(%IW110); AdrOffset_8550 = 4294967295; BitOffset_8550 = 0; BitLength_8550 = 0; Address_8550 = ''; Type_8550 = ''; AddressPointer_8550 = 0; AdrOffset_8560 = 240; BitOffset_8560 = 0; BitLength_8560 = 32; Address_8560 = '%ID60'; Type_8560 = 'UDINT'; AddressPointer_8560 = ADR(%ID60); AdrOffset_8570 = 228; BitOffset_8570 = 0; BitLength_8570 = 16; Address_8570 = '%IW114'; Type_8570 = 'UINT'; AddressPointer_8570 = ADR(%IW114); AdrOffset_8580 = 232; BitOffset_8580 = 0; BitLength_8580 = 32; Address_8580 = '%ID58'; Type_8580 = 'DINT'; AddressPointer_8580 = ADR(%ID58); AdrOffset_8590 = 4294967295; BitOffset_8590 = 0; BitLength_8590 = 0; Address_8590 = ''; Type_8590 = ''; AddressPointer_8590 = 0; AdrOffset_8600 = 236; BitOffset_8600 = 0; BitLength_8600 = 32; Address_8600 = '%ID59'; Type_8600 = 'DINT'; AddressPointer_8600 = ADR(%ID59); AdrOffset_8600 = 4294967295;
              BitOffset_8600 = 0; BitLength_8600 = 0; Address_8610 = ''; Type_8610 = ''; AddressPointer_8610 = 0; AdrOffset_8620 = 0; BitOffset_8620 = 0; BitLength_8620 = 16; Address_8620 = '机械臂控制.伺服错误码[1]'; Type_8620 = 'UINT'; AddressPointer_8620 = ADR(机械臂控制.伺服错误码[1]); IsValid = True; IsHostHoming = False; PulseSelectIndex = 2
      InoSV630N_伸缩轴 : SV630_1Axis_03715, Inovance, order no. InoSV630N, version Revision=16#00010000
          settings: Number of Outputs = 6; Number of Inputs = 10; Number of Infos about Outputs = 6; Number of Infos about Inputs = 10; Physical Address of the Slave = 1001; StationAlias = 0; Sync.Length = 18; Sync.Length = 32; FMMU.Global Start Address = 16#02000000; FMMU.Length = 18; FMMU.Physical Start Address = 16#1800; FMMU.Access = 16#02; FMMU.Global Start Address = 16#01000000; FMMU.Length = 32; FMMU.Physical Start Address = 16#1C00; FMMU.Access = 16#01; FMMU.Global Start Address = 16#00080000; FMMU.Physical Start Address = 16#080D; FMMU.Access = 16#01; AutoUpdate = False; DC sync0 cycletime = 4000; DC sync1 cycletime = 4000; Number of SDO = 10; Homing method.Index = 16#6098; Homing method.Subindex = 16#00; Homing method.Value = 1; Homing method.Size = 8; Homing method.AbortIfError = FALSE; Homing method.JumpToLine = FALSE; Homing method.Line = 0; Homing method.CompleteAccess = FALSE; Actual Position Calculation Method.Index = 16#60E6; Actual Position Calculation Method.Subindex = 16#00; Actual Position Calculation Method.Value = 0; Actual Position Calculation Method.Size = 8; Actual Position Calculation Method.AbortIfError = FALSE; Actual Position Calculation Method.JumpToLine = FALSE; Actual Position Calculation Method.Line = 0; Actual Position Calculation Method.CompleteAccess = FALSE; Speed during search for switch.Index = 16#6099;
            Speed during search for switch.Subindex = 16#01; Speed during search for switch.Value = 87381; Speed during search for switch.Size = 32; Speed during search for switch.AbortIfError = FALSE; Speed during search for switch.JumpToLine = FALSE; Speed during search for switch.Line = 0; Speed during search for switch.CompleteAccess = FALSE; Homing acceleration.Index = 16#609A; Homing acceleration.Subindex = 16#00; Homing acceleration.Value = 8738133; Homing acceleration.Size = 32; Homing acceleration.AbortIfError = FALSE; Homing acceleration.JumpToLine = FALSE; Homing acceleration.Line = 0; Homing acceleration.CompleteAccess = FALSE; Speed during search for zero.Index = 16#6099; Speed during search for zero.Subindex = 16#02; Speed during search for zero.Value = 8738; Speed during search for zero.Size = 32; Speed during search for zero.AbortIfError = FALSE; Speed during search for zero.JumpToLine = FALSE; Speed during search for zero.Line = 0; Speed during search for zero.CompleteAccess = FALSE; Time of home searching.Index = 16#2005; Time of home searching.Subindex = 16#24; Time of home searching.Value = 50000; Time of home searching.Size = 16; Time of home searching.AbortIfError = FALSE; Time of home searching.JumpToLine = FALSE; Time of home searching.Line = 0; Time of home searching.CompleteAccess = FALSE; Positive torque limit value.Index = 16#60E0; Positive torque limit value.Subindex = 16#00; Positive torque limit value.Value = 3500; Positive torque limit value.Size = 16; Positive torque limit value.AbortIfError = FALSE; Positive torque limit value.JumpToLine = FALSE; Positive torque limit value.Line = 0; Positive torque limit value.CompleteAccess = FALSE; Negative torque limit value.Index = 16#60E1;
            Negative torque limit value.Subindex = 16#00; Negative torque limit value.Value = 3500; Negative torque limit value.Size = 16; Negative torque limit value.AbortIfError = FALSE; Negative torque limit value.JumpToLine = FALSE; Negative torque limit value.Line = 0; Negative torque limit value.CompleteAccess = FALSE; Max profile velocity.Index = 16#607F; Max profile velocity.Subindex = 16#00; Max profile velocity.Value = 5242880; Max profile velocity.Size = 32; Max profile velocity.AbortIfError = FALSE; Max profile velocity.JumpToLine = FALSE; Max profile velocity.Line = 0; Max profile velocity.CompleteAccess = FALSE; RxTxPdo.NumberofEntries = 6; RxTxPdo.Sm = 2; Controlword.Index = 16#6040; Controlword.SubIndex = 0; Controlword.Size = 16; Controlword.DependOnSlot = false; Controlword.DependOnSlotGroup = false; Target position.Index = 16#607A; Target position.SubIndex = 0; Target position.Size = 32; Target position.DependOnSlot = false; Target position.DependOnSlotGroup = false; Touch probe function.Index = 16#60B8; Touch probe function.SubIndex = 0; Touch probe function.Size = 16; Touch probe function.DependOnSlot = false; Touch probe function.DependOnSlotGroup = false; Physical outputs.Index = 16#60FE; Physical outputs.SubIndex = 1; Physical outputs.Size = 32; Physical outputs.DependOnSlot = false; Physical outputs.DependOnSlotGroup = false; Target velocity.Index = 16#60FF; Target velocity.SubIndex = 0; Target velocity.Size = 32;
            Target velocity.DependOnSlot = false; Target velocity.DependOnSlotGroup = false; Target torque.Index = 16#6071; Target torque.SubIndex = 0; Target torque.Size = 16; Target torque.DependOnSlot = false; Target torque.DependOnSlotGroup = false; RxTxPdo.Sm = -1; RxTxPdo.NumberofEntries = 10; RxTxPdo.Sm = 3; Error code.Index = 16#603F; Error code.SubIndex = 0; Error code.Size = 16; Error code.DependOnSlot = false; Error code.DependOnSlotGroup = false; Statusword.Index = 16#6041; Statusword.SubIndex = 0; Statusword.Size = 16; Statusword.DependOnSlot = false; Statusword.DependOnSlotGroup = false; Position actual value.Index = 16#6064; Position actual value.SubIndex = 0; Position actual value.Size = 32; Position actual value.DependOnSlot = false; Position actual value.DependOnSlotGroup = false; Torque actual value.Index = 16#6077; Torque actual value.SubIndex = 0; Torque actual value.Size = 16; Torque actual value.DependOnSlot = false; Torque actual value.DependOnSlotGroup = false; Following error actual value.Index = 16#60F4; Following error actual value.SubIndex = 0; Following error actual value.Size = 32; Following error actual value.DependOnSlot = false; Following error actual value.DependOnSlotGroup = false; Touch probe status.Index = 16#60B9; Touch probe status.SubIndex = 0; Touch probe status.Size = 16; Touch probe status.DependOnSlot = false; Touch probe status.DependOnSlotGroup = false;
            Touch probe pos1 pos value.Index = 16#60BA; Touch probe pos1 pos value.SubIndex = 0; Touch probe pos1 pos value.Size = 32; Touch probe pos1 pos value.DependOnSlot = false; Touch probe pos1 pos value.DependOnSlotGroup = false; Touch probe pos2 pos value.Index = 16#60BC; Touch probe pos2 pos value.SubIndex = 0; Touch probe pos2 pos value.Size = 32; Touch probe pos2 pos value.DependOnSlot = false; Touch probe pos2 pos value.DependOnSlotGroup = false; Digital inputs.Index = 16#60FD; Digital inputs.SubIndex = 0; Digital inputs.Size = 32; Digital inputs.DependOnSlot = false; Digital inputs.DependOnSlotGroup = false; Velocity actual value.Index = 16#606C; Velocity actual value.SubIndex = 0; Velocity actual value.Size = 32; Velocity actual value.DependOnSlot = false; Velocity actual value.DependOnSlotGroup = false; RxTxPdo.Sm = -1; Controlword.Name = 'Controlword'; Controlword.DataType = 'UINT'; Target position.Name = 'Target position'; Target position.DataType = 'DINT'; Touch probe function.Name = 'Touch probe function'; Touch probe function.DataType = 'UINT'; Physical outputs.Name = 'Physical outputs'; Physical outputs.DataType = 'UDINT'; Target velocity.Name = 'Target velocity'; Target velocity.DataType = 'DINT'; Target torque.Name = 'Target torque'; Target torque.DataType = 'INT'; Error code.Name = 'Error code'; Error code.DataType = 'UINT'; Statusword.Name = 'Statusword'; Statusword.DataType = 'UINT'; Position actual value.Name = 'Position actual value'; Position actual value.DataType = 'DINT'; Torque actual value.Name = 'Torque actual value';
            Torque actual value.DataType = 'INT'; Following error actual value.Name = 'Following error actual value'; Following error actual value.DataType = 'DINT'; Touch probe status.Name = 'Touch probe status'; Touch probe status.DataType = 'UINT'; Touch probe pos1 pos value.Name = 'Touch probe pos1 pos value'; Touch probe pos1 pos value.DataType = 'DINT'; Touch probe pos2 pos value.Name = 'Touch probe pos2 pos value'; Touch probe pos2 pos value.DataType = 'DINT'; Digital inputs.Name = 'Digital inputs'; Digital inputs.DataType = 'UDINT'; Velocity actual value.Name = 'Velocity actual value'; Velocity actual value.DataType = 'DINT'
          input  Application.末端控制.adFbForce[0] : INT  // Torque actual value
          unmapped channels: Controlword, Target position, Touch probe function, Physical outputs, Target velocity, Target torque, Error code, Statusword, Position actual value, Following error actual value, Touch probe status, Touch probe pos1 pos value, Touch probe pos2 pos value, Digital inputs, Velocity actual value
        伸缩轴 : Axis, Inovance, order no. 0, version 1.0.0.0
            settings: wDriveID = 16; dwRatioTechUnitsDenom = 262144; iRatioTechUnitsNum = 5; fSWMaxVelocity = 1000; fSWMaxAcceleration = 10000; fSWMaxDeceleration = 10000; fSWMaxJerk = 100000; iEncoderType = 1; iAbsEncoderOption = 1; HomingMode = 10; ZeroSignal = 0; StartDirction = 1; EndDirection = 1; PosLimitMode = 0; NegLimitMode = 0; HomingVelocity = 10; HomingApproachVelocity = 2; HomingAcceleration = 100; HomingDeceleration = 100; HomingJerk = 0; HomeMaskDistance = 0; HomePositionOffset = 0; HomePushTime = 0; HomeCompensation = 0; HomeTimeout = 0; HomeCompensationVelocity = 1000; 4000 = 0; 4001 = 0; 4003 = true; 4004 = 3; 4005 = 0; 4006 = 1.666667; 4007 = 166.666666; 4008 = 0.166667; 4009 = 50000; 4010 = 3500; 4011 = 3500; 4012 = 100.000000; ScalingIncs = 16#40000; 6005 = 5;
              AdrOffset_8010 = 0; BitOffset_8010 = 0; BitLength_8010 = 16; Address_8010 = '%QW0'; Type_8010 = 'UINT'; AddressPointer_8010 = ADR(%QW0); AdrOffset_8020 = 4; BitOffset_8020 = 0; BitLength_8020 = 32; Address_8020 = '%QD1'; Type_8020 = 'DINT'; AddressPointer_8020 = ADR(%QD1); AdrOffset_8030 = 16; BitOffset_8030 = 0; BitLength_8030 = 32; Address_8030 = '%QD4'; Type_8030 = 'DINT'; AddressPointer_8030 = ADR(%QD4); AdrOffset_8040 = 20; BitOffset_8040 = 0; BitLength_8040 = 16; Address_8040 = '%QW10'; Type_8040 = 'INT'; AddressPointer_8040 = ADR(%QW10); AdrOffset_8050 = 4294967295; BitOffset_8050 = 0; BitLength_8050 = 0; Address_8050 = ''; Type_8050 = ''; AddressPointer_8050 = 0; AdrOffset_8060 = 8; BitOffset_8060 = 0; BitLength_8060 = 16; Address_8060 = '%QW4'; Type_8060 = 'UINT'; AddressPointer_8060 = ADR(%QW4); AdrOffset_8070 = 4294967295; BitOffset_8070 = 0; BitLength_8070 = 0; Address_8070 = '';
              Type_8070 = ''; AddressPointer_8070 = 0; AdrOffset_8080 = 4294967295; BitOffset_8080 = 0; BitLength_8080 = 0; Address_8080 = ''; Type_8080 = ''; AddressPointer_8080 = 0; AdrOffset_8090 = 12; BitOffset_8090 = 0; BitLength_8090 = 32; Address_8090 = '%QD3'; Type_8090 = 'UDINT'; AddressPointer_8090 = ADR(%QD3); AdrOffset_8100 = 4294967295; BitOffset_8100 = 0; BitLength_8100 = 0; Address_8100 = ''; Type_8100 = ''; AddressPointer_8100 = 0; AdrOffset_8510 = 2; BitOffset_8510 = 0; BitLength_8510 = 16; Address_8510 = '%IW1'; Type_8510 = 'UINT'; AddressPointer_8510 = ADR(%IW1); AdrOffset_8520 = 4; BitOffset_8520 = 0; BitLength_8520 = 32; Address_8520 = '%ID1'; Type_8520 = 'DINT'; AddressPointer_8520 = ADR(%ID1); AdrOffset_8530 = 32; BitOffset_8530 = 0; BitLength_8530 = 32; Address_8530 = '%ID8'; Type_8530 = 'DINT'; AddressPointer_8530 = ADR(%ID8); AdrOffset_8540 = 0; BitOffset_8540 = 0;
              BitLength_8540 = 16; Address_8540 = '末端控制.adFbForce[0]'; Type_8540 = 'INT'; AddressPointer_8540 = ADR(末端控制.adFbForce[0]); AdrOffset_8550 = 4294967295; BitOffset_8550 = 0; BitLength_8550 = 0; Address_8550 = ''; Type_8550 = ''; AddressPointer_8550 = 0; AdrOffset_8560 = 28; BitOffset_8560 = 0; BitLength_8560 = 32; Address_8560 = '%ID7'; Type_8560 = 'UDINT'; AddressPointer_8560 = ADR(%ID7); AdrOffset_8570 = 16; BitOffset_8570 = 0; BitLength_8570 = 16; Address_8570 = '%IW8'; Type_8570 = 'UINT'; AddressPointer_8570 = ADR(%IW8); AdrOffset_8580 = 20; BitOffset_8580 = 0; BitLength_8580 = 32; Address_8580 = '%ID5'; Type_8580 = 'DINT'; AddressPointer_8580 = ADR(%ID5); AdrOffset_8590 = 4294967295; BitOffset_8590 = 0; BitLength_8590 = 0; Address_8590 = ''; Type_8590 = ''; AddressPointer_8590 = 0; AdrOffset_8600 = 24; BitOffset_8600 = 0; BitLength_8600 = 32; Address_8600 = '%ID6'; Type_8600 = 'DINT'; AddressPointer_8600 = ADR(%ID6);
              AdrOffset_8600 = 4294967295; BitOffset_8600 = 0; BitLength_8600 = 0; Address_8610 = ''; Type_8610 = ''; AddressPointer_8610 = 0; AdrOffset_8620 = 0; BitOffset_8620 = 0; BitLength_8620 = 16; Address_8620 = '%IW0'; Type_8620 = 'UINT'; AddressPointer_8620 = ADR(%IW0); IsValid = True; IsHostHoming = False; PulseSelectIndex = 2
      InoSV630N_上卷扬 : SV630_1Axis_03715, Inovance, order no. InoSV630N, version Revision=16#00010000
          settings: Number of Outputs = 6; Number of Inputs = 10; Number of Infos about Outputs = 6; Number of Infos about Inputs = 10; Physical Address of the Slave = 1002; AutoIncr Address of the Slave = 4294967295; StationAlias = 0; Sync.Length = 18; Sync.Length = 32; FMMU.Global Start Address = 16#02000012; FMMU.Length = 18; FMMU.Physical Start Address = 16#1800; FMMU.Access = 16#02; FMMU.Global Start Address = 16#01000020; FMMU.Length = 32; FMMU.Physical Start Address = 16#1C00; FMMU.Access = 16#01; FMMU.Global Start Address = 16#00080000; FMMU.StartBit = 1; FMMU.EndBit = 1; FMMU.Physical Start Address = 16#080D; FMMU.Access = 16#01; AutoUpdate = False; DC sync0 cycletime = 4000; DC sync1 cycletime = 4000; Number of SDO = 10; Homing method.Index = 16#6098; Homing method.Subindex = 16#00; Homing method.Value = 1; Homing method.Size = 8; Homing method.AbortIfError = FALSE; Homing method.JumpToLine = FALSE; Homing method.Line = 0; Homing method.CompleteAccess = FALSE; Actual Position Calculation Method.Index = 16#60E6; Actual Position Calculation Method.Subindex = 16#00; Actual Position Calculation Method.Value = 0; Actual Position Calculation Method.Size = 8; Actual Position Calculation Method.AbortIfError = FALSE; Actual Position Calculation Method.JumpToLine = FALSE;
            Actual Position Calculation Method.Line = 0; Actual Position Calculation Method.CompleteAccess = FALSE; Speed during search for switch.Index = 16#6099; Speed during search for switch.Subindex = 16#01; Speed during search for switch.Value = 43460; Speed during search for switch.Size = 32; Speed during search for switch.AbortIfError = FALSE; Speed during search for switch.JumpToLine = FALSE; Speed during search for switch.Line = 0; Speed during search for switch.CompleteAccess = FALSE; Homing acceleration.Index = 16#609A; Homing acceleration.Subindex = 16#00; Homing acceleration.Value = 4345995; Homing acceleration.Size = 32; Homing acceleration.AbortIfError = FALSE; Homing acceleration.JumpToLine = FALSE; Homing acceleration.Line = 0; Homing acceleration.CompleteAccess = FALSE; Speed during search for zero.Index = 16#6099; Speed during search for zero.Subindex = 16#02; Speed during search for zero.Value = 4346; Speed during search for zero.Size = 32; Speed during search for zero.AbortIfError = FALSE; Speed during search for zero.JumpToLine = FALSE; Speed during search for zero.Line = 0; Speed during search for zero.CompleteAccess = FALSE; Time of home searching.Index = 16#2005; Time of home searching.Subindex = 16#24; Time of home searching.Value = 50000; Time of home searching.Size = 16; Time of home searching.AbortIfError = FALSE; Time of home searching.JumpToLine = FALSE; Time of home searching.Line = 0; Time of home searching.CompleteAccess = FALSE; Positive torque limit value.Index = 16#60E0; Positive torque limit value.Subindex = 16#00; Positive torque limit value.Value = 3500; Positive torque limit value.Size = 16; Positive torque limit value.AbortIfError = FALSE; Positive torque limit value.JumpToLine = FALSE;
            Positive torque limit value.Line = 0; Positive torque limit value.CompleteAccess = FALSE; Negative torque limit value.Index = 16#60E1; Negative torque limit value.Subindex = 16#00; Negative torque limit value.Value = 3500; Negative torque limit value.Size = 16; Negative torque limit value.AbortIfError = FALSE; Negative torque limit value.JumpToLine = FALSE; Negative torque limit value.Line = 0; Negative torque limit value.CompleteAccess = FALSE; Max profile velocity.Index = 16#607F; Max profile velocity.Subindex = 16#00; Max profile velocity.Value = 2607597; Max profile velocity.Size = 32; Max profile velocity.AbortIfError = FALSE; Max profile velocity.JumpToLine = FALSE; Max profile velocity.Line = 0; Max profile velocity.CompleteAccess = FALSE; RxTxPdo.NumberofEntries = 6; RxTxPdo.Sm = 2; Controlword.Index = 16#6040; Controlword.SubIndex = 0; Controlword.Size = 16; Controlword.DependOnSlot = false; Controlword.DependOnSlotGroup = false; Target position.Index = 16#607A; Target position.SubIndex = 0; Target position.Size = 32; Target position.DependOnSlot = false; Target position.DependOnSlotGroup = false; Touch probe function.Index = 16#60B8; Touch probe function.SubIndex = 0; Touch probe function.Size = 16; Touch probe function.DependOnSlot = false; Touch probe function.DependOnSlotGroup = false; Physical outputs.Index = 16#60FE; Physical outputs.SubIndex = 1; Physical outputs.Size = 32; Physical outputs.DependOnSlot = false; Physical outputs.DependOnSlotGroup = false;
            Target velocity.Index = 16#60FF; Target velocity.SubIndex = 0; Target velocity.Size = 32; Target velocity.DependOnSlot = false; Target velocity.DependOnSlotGroup = false; Target torque.Index = 16#6071; Target torque.SubIndex = 0; Target torque.Size = 16; Target torque.DependOnSlot = false; Target torque.DependOnSlotGroup = false; RxTxPdo.Sm = -1; RxTxPdo.NumberofEntries = 10; RxTxPdo.Sm = 3; Error code.Index = 16#603F; Error code.SubIndex = 0; Error code.Size = 16; Error code.DependOnSlot = false; Error code.DependOnSlotGroup = false; Statusword.Index = 16#6041; Statusword.SubIndex = 0; Statusword.Size = 16; Statusword.DependOnSlot = false; Statusword.DependOnSlotGroup = false; Position actual value.Index = 16#6064; Position actual value.SubIndex = 0; Position actual value.Size = 32; Position actual value.DependOnSlot = false; Position actual value.DependOnSlotGroup = false; Torque actual value.Index = 16#6077; Torque actual value.SubIndex = 0; Torque actual value.Size = 16; Torque actual value.DependOnSlot = false; Torque actual value.DependOnSlotGroup = false; Following error actual value.Index = 16#60F4; Following error actual value.SubIndex = 0; Following error actual value.Size = 32; Following error actual value.DependOnSlot = false; Following error actual value.DependOnSlotGroup = false; Touch probe status.Index = 16#60B9; Touch probe status.SubIndex = 0;
            Touch probe status.Size = 16; Touch probe status.DependOnSlot = false; Touch probe status.DependOnSlotGroup = false; Touch probe pos1 pos value.Index = 16#60BA; Touch probe pos1 pos value.SubIndex = 0; Touch probe pos1 pos value.Size = 32; Touch probe pos1 pos value.DependOnSlot = false; Touch probe pos1 pos value.DependOnSlotGroup = false; Touch probe pos2 pos value.Index = 16#60BC; Touch probe pos2 pos value.SubIndex = 0; Touch probe pos2 pos value.Size = 32; Touch probe pos2 pos value.DependOnSlot = false; Touch probe pos2 pos value.DependOnSlotGroup = false; Digital inputs.Index = 16#60FD; Digital inputs.SubIndex = 0; Digital inputs.Size = 32; Digital inputs.DependOnSlot = false; Digital inputs.DependOnSlotGroup = false; Velocity actual value.Index = 16#606C; Velocity actual value.SubIndex = 0; Velocity actual value.Size = 32; Velocity actual value.DependOnSlot = false; Velocity actual value.DependOnSlotGroup = false; RxTxPdo.Sm = -1; Controlword.Name = 'Controlword'; Controlword.DataType = 'UINT'; Target position.Name = 'Target position'; Target position.DataType = 'DINT'; Touch probe function.Name = 'Touch probe function'; Touch probe function.DataType = 'UINT'; Physical outputs.Name = 'Physical outputs'; Physical outputs.DataType = 'UDINT'; Target velocity.Name = 'Target velocity'; Target velocity.DataType = 'DINT'; Target torque.Name = 'Target torque'; Target torque.DataType = 'INT'; Error code.Name = 'Error code'; Error code.DataType = 'UINT'; Statusword.Name = 'Statusword'; Statusword.DataType = 'UINT';
            Position actual value.Name = 'Position actual value'; Position actual value.DataType = 'DINT'; Torque actual value.Name = 'Torque actual value'; Torque actual value.DataType = 'INT'; Following error actual value.Name = 'Following error actual value'; Following error actual value.DataType = 'DINT'; Touch probe status.Name = 'Touch probe status'; Touch probe status.DataType = 'UINT'; Touch probe pos1 pos value.Name = 'Touch probe pos1 pos value'; Touch probe pos1 pos value.DataType = 'DINT'; Touch probe pos2 pos value.Name = 'Touch probe pos2 pos value'; Touch probe pos2 pos value.DataType = 'DINT'; Digital inputs.Name = 'Digital inputs'; Digital inputs.DataType = 'UDINT'; Velocity actual value.Name = 'Velocity actual value'; Velocity actual value.DataType = 'DINT'
          input  Application.末端控制.adFbForce[1] : INT  // Torque actual value
          unmapped channels: Controlword, Target position, Touch probe function, Physical outputs, Target velocity, Target torque, Error code, Statusword, Position actual value, Following error actual value, Touch probe status, Touch probe pos1 pos value, Touch probe pos2 pos value, Digital inputs, Velocity actual value
        上卷扬 : Axis, Inovance, order no. 0, version 1.0.0.0
            settings: wDriveID = 17; dwRatioTechUnitsDenom = 260759679; iRatioTechUnitsNum = 10000; fSWMaxVelocity = 1000; fSWMaxAcceleration = 10000; fSWMaxDeceleration = 10000; fSWMaxJerk = 100000; iEncoderType = 1; iAbsEncoderOption = 1; HomingMode = 10; ZeroSignal = 0; StartDirction = 1; EndDirection = 1; PosLimitMode = 0; NegLimitMode = 0; HomingVelocity = 10; HomingApproachVelocity = 2; HomingAcceleration = 100; HomingDeceleration = 100; HomingJerk = 0; HomeMaskDistance = 0; HomePositionOffset = 0; HomePushTime = 0; HomeCompensation = 0; HomeTimeout = 0; HomeCompensationVelocity = 1000; 4000 = 1; 4001 = 1; 4003 = true; 4004 = 3; 4005 = 0; 4006 = 1.666667; 4007 = 166.666666; 4008 = 0.166667; 4009 = 50000; 4010 = 3500; 4011 = 3500; 4012 = 100.000000; ScalingIncs = 16#40000; ScalingMotorTurns2 = 50;
              6005 = 502.6544; AdrOffset_8010 = 24; BitOffset_8010 = 0; BitLength_8010 = 16; Address_8010 = '%QW12'; Type_8010 = 'UINT'; AddressPointer_8010 = ADR(%QW12); AdrOffset_8020 = 28; BitOffset_8020 = 0; BitLength_8020 = 32; Address_8020 = '%QD7'; Type_8020 = 'DINT'; AddressPointer_8020 = ADR(%QD7); AdrOffset_8030 = 40; BitOffset_8030 = 0; BitLength_8030 = 32; Address_8030 = '%QD10'; Type_8030 = 'DINT'; AddressPointer_8030 = ADR(%QD10); AdrOffset_8040 = 44; BitOffset_8040 = 0; BitLength_8040 = 16; Address_8040 = '%QW22'; Type_8040 = 'INT'; AddressPointer_8040 = ADR(%QW22); AdrOffset_8050 = 4294967295; BitOffset_8050 = 0; BitLength_8050 = 0; Address_8050 = ''; Type_8050 = ''; AddressPointer_8050 = 0; AdrOffset_8060 = 32; BitOffset_8060 = 0; BitLength_8060 = 16; Address_8060 = '%QW16'; Type_8060 = 'UINT'; AddressPointer_8060 = ADR(%QW16); AdrOffset_8070 = 4294967295; BitOffset_8070 = 0; BitLength_8070 = 0;
              Address_8070 = ''; Type_8070 = ''; AddressPointer_8070 = 0; AdrOffset_8080 = 4294967295; BitOffset_8080 = 0; BitLength_8080 = 0; Address_8080 = ''; Type_8080 = ''; AddressPointer_8080 = 0; AdrOffset_8090 = 36; BitOffset_8090 = 0; BitLength_8090 = 32; Address_8090 = '%QD9'; Type_8090 = 'UDINT'; AddressPointer_8090 = ADR(%QD9); AdrOffset_8100 = 4294967295; BitOffset_8100 = 0; BitLength_8100 = 0; Address_8100 = ''; Type_8100 = ''; AddressPointer_8100 = 0; AdrOffset_8510 = 38; BitOffset_8510 = 0; BitLength_8510 = 16; Address_8510 = '%IW19'; Type_8510 = 'UINT'; AddressPointer_8510 = ADR(%IW19); AdrOffset_8520 = 40; BitOffset_8520 = 0; BitLength_8520 = 32; Address_8520 = '%ID10'; Type_8520 = 'DINT'; AddressPointer_8520 = ADR(%ID10); AdrOffset_8530 = 68; BitOffset_8530 = 0; BitLength_8530 = 32; Address_8530 = '%ID17'; Type_8530 = 'DINT'; AddressPointer_8530 = ADR(%ID17); AdrOffset_8540 = 0;
              BitOffset_8540 = 0; BitLength_8540 = 16; Address_8540 = '末端控制.adFbForce[1]'; Type_8540 = 'INT'; AddressPointer_8540 = ADR(末端控制.adFbForce[1]); AdrOffset_8550 = 4294967295; BitOffset_8550 = 0; BitLength_8550 = 0; Address_8550 = ''; Type_8550 = ''; AddressPointer_8550 = 0; AdrOffset_8560 = 64; BitOffset_8560 = 0; BitLength_8560 = 32; Address_8560 = '%ID16'; Type_8560 = 'UDINT'; AddressPointer_8560 = ADR(%ID16); AdrOffset_8570 = 52; BitOffset_8570 = 0; BitLength_8570 = 16; Address_8570 = '%IW26'; Type_8570 = 'UINT'; AddressPointer_8570 = ADR(%IW26); AdrOffset_8580 = 56; BitOffset_8580 = 0; BitLength_8580 = 32; Address_8580 = '%ID14'; Type_8580 = 'DINT'; AddressPointer_8580 = ADR(%ID14); AdrOffset_8590 = 4294967295; BitOffset_8590 = 0; BitLength_8590 = 0; Address_8590 = ''; Type_8590 = ''; AddressPointer_8590 = 0; AdrOffset_8600 = 60; BitOffset_8600 = 0; BitLength_8600 = 32; Address_8600 = '%ID15'; Type_8600 = 'DINT';
              AddressPointer_8600 = ADR(%ID15); AdrOffset_8600 = 4294967295; BitOffset_8600 = 0; BitLength_8600 = 0; Address_8610 = ''; Type_8610 = ''; AddressPointer_8610 = 0; AdrOffset_8620 = 36; BitOffset_8620 = 0; BitLength_8620 = 16; Address_8620 = '%IW18'; Type_8620 = 'UINT'; AddressPointer_8620 = ADR(%IW18); IsValid = True; IsHostHoming = False; PulseSelectIndex = 2
      InoSV630N_下卷扬 : SV630_1Axis_03715, Inovance, order no. InoSV630N, version Revision=16#00010000
          settings: Number of Outputs = 6; Number of Inputs = 10; Number of Infos about Outputs = 6; Number of Infos about Inputs = 10; Physical Address of the Slave = 1003; AutoIncr Address of the Slave = 4294967294; StationAlias = 0; Sync.Length = 18; Sync.Length = 32; FMMU.Global Start Address = 16#02000024; FMMU.Length = 18; FMMU.Physical Start Address = 16#1800; FMMU.Access = 16#02; FMMU.Global Start Address = 16#01000040; FMMU.Length = 32; FMMU.Physical Start Address = 16#1C00; FMMU.Access = 16#01; FMMU.Global Start Address = 16#00080000; FMMU.StartBit = 2; FMMU.EndBit = 2; FMMU.Physical Start Address = 16#080D; FMMU.Access = 16#01; AutoUpdate = False; DC sync0 cycletime = 4000; DC sync1 cycletime = 4000; Number of SDO = 10; Homing method.Index = 16#6098; Homing method.Subindex = 16#00; Homing method.Value = 1; Homing method.Size = 8; Homing method.AbortIfError = FALSE; Homing method.JumpToLine = FALSE; Homing method.Line = 0; Homing method.CompleteAccess = FALSE; Actual Position Calculation Method.Index = 16#60E6; Actual Position Calculation Method.Subindex = 16#00; Actual Position Calculation Method.Value = 0; Actual Position Calculation Method.Size = 8; Actual Position Calculation Method.AbortIfError = FALSE; Actual Position Calculation Method.JumpToLine = FALSE;
            Actual Position Calculation Method.Line = 0; Actual Position Calculation Method.CompleteAccess = FALSE; Speed during search for switch.Index = 16#6099; Speed during search for switch.Subindex = 16#01; Speed during search for switch.Value = 43460; Speed during search for switch.Size = 32; Speed during search for switch.AbortIfError = FALSE; Speed during search for switch.JumpToLine = FALSE; Speed during search for switch.Line = 0; Speed during search for switch.CompleteAccess = FALSE; Homing acceleration.Index = 16#609A; Homing acceleration.Subindex = 16#00; Homing acceleration.Value = 4345995; Homing acceleration.Size = 32; Homing acceleration.AbortIfError = FALSE; Homing acceleration.JumpToLine = FALSE; Homing acceleration.Line = 0; Homing acceleration.CompleteAccess = FALSE; Speed during search for zero.Index = 16#6099; Speed during search for zero.Subindex = 16#02; Speed during search for zero.Value = 4346; Speed during search for zero.Size = 32; Speed during search for zero.AbortIfError = FALSE; Speed during search for zero.JumpToLine = FALSE; Speed during search for zero.Line = 0; Speed during search for zero.CompleteAccess = FALSE; Time of home searching.Index = 16#2005; Time of home searching.Subindex = 16#24; Time of home searching.Value = 50000; Time of home searching.Size = 16; Time of home searching.AbortIfError = FALSE; Time of home searching.JumpToLine = FALSE; Time of home searching.Line = 0; Time of home searching.CompleteAccess = FALSE; Positive torque limit value.Index = 16#60E0; Positive torque limit value.Subindex = 16#00; Positive torque limit value.Value = 3500; Positive torque limit value.Size = 16; Positive torque limit value.AbortIfError = FALSE; Positive torque limit value.JumpToLine = FALSE;
            Positive torque limit value.Line = 0; Positive torque limit value.CompleteAccess = FALSE; Negative torque limit value.Index = 16#60E1; Negative torque limit value.Subindex = 16#00; Negative torque limit value.Value = 3500; Negative torque limit value.Size = 16; Negative torque limit value.AbortIfError = FALSE; Negative torque limit value.JumpToLine = FALSE; Negative torque limit value.Line = 0; Negative torque limit value.CompleteAccess = FALSE; Max profile velocity.Index = 16#607F; Max profile velocity.Subindex = 16#00; Max profile velocity.Value = 2607597; Max profile velocity.Size = 32; Max profile velocity.AbortIfError = FALSE; Max profile velocity.JumpToLine = FALSE; Max profile velocity.Line = 0; Max profile velocity.CompleteAccess = FALSE; RxTxPdo.NumberofEntries = 6; RxTxPdo.Sm = 2; Controlword.Index = 16#6040; Controlword.SubIndex = 0; Controlword.Size = 16; Controlword.DependOnSlot = false; Controlword.DependOnSlotGroup = false; Target position.Index = 16#607A; Target position.SubIndex = 0; Target position.Size = 32; Target position.DependOnSlot = false; Target position.DependOnSlotGroup = false; Touch probe function.Index = 16#60B8; Touch probe function.SubIndex = 0; Touch probe function.Size = 16; Touch probe function.DependOnSlot = false; Touch probe function.DependOnSlotGroup = false; Physical outputs.Index = 16#60FE; Physical outputs.SubIndex = 1; Physical outputs.Size = 32; Physical outputs.DependOnSlot = false; Physical outputs.DependOnSlotGroup = false;
            Target velocity.Index = 16#60FF; Target velocity.SubIndex = 0; Target velocity.Size = 32; Target velocity.DependOnSlot = false; Target velocity.DependOnSlotGroup = false; Target torque.Index = 16#6071; Target torque.SubIndex = 0; Target torque.Size = 16; Target torque.DependOnSlot = false; Target torque.DependOnSlotGroup = false; RxTxPdo.Sm = -1; RxTxPdo.NumberofEntries = 10; RxTxPdo.Sm = 3; Error code.Index = 16#603F; Error code.SubIndex = 0; Error code.Size = 16; Error code.DependOnSlot = false; Error code.DependOnSlotGroup = false; Statusword.Index = 16#6041; Statusword.SubIndex = 0; Statusword.Size = 16; Statusword.DependOnSlot = false; Statusword.DependOnSlotGroup = false; Position actual value.Index = 16#6064; Position actual value.SubIndex = 0; Position actual value.Size = 32; Position actual value.DependOnSlot = false; Position actual value.DependOnSlotGroup = false; Torque actual value.Index = 16#6077; Torque actual value.SubIndex = 0; Torque actual value.Size = 16; Torque actual value.DependOnSlot = false; Torque actual value.DependOnSlotGroup = false; Following error actual value.Index = 16#60F4; Following error actual value.SubIndex = 0; Following error actual value.Size = 32; Following error actual value.DependOnSlot = false; Following error actual value.DependOnSlotGroup = false; Touch probe status.Index = 16#60B9; Touch probe status.SubIndex = 0;
            Touch probe status.Size = 16; Touch probe status.DependOnSlot = false; Touch probe status.DependOnSlotGroup = false; Touch probe pos1 pos value.Index = 16#60BA; Touch probe pos1 pos value.SubIndex = 0; Touch probe pos1 pos value.Size = 32; Touch probe pos1 pos value.DependOnSlot = false; Touch probe pos1 pos value.DependOnSlotGroup = false; Touch probe pos2 pos value.Index = 16#60BC; Touch probe pos2 pos value.SubIndex = 0; Touch probe pos2 pos value.Size = 32; Touch probe pos2 pos value.DependOnSlot = false; Touch probe pos2 pos value.DependOnSlotGroup = false; Digital inputs.Index = 16#60FD; Digital inputs.SubIndex = 0; Digital inputs.Size = 32; Digital inputs.DependOnSlot = false; Digital inputs.DependOnSlotGroup = false; Velocity actual value.Index = 16#606C; Velocity actual value.SubIndex = 0; Velocity actual value.Size = 32; Velocity actual value.DependOnSlot = false; Velocity actual value.DependOnSlotGroup = false; RxTxPdo.Sm = -1; Controlword.Name = 'Controlword'; Controlword.DataType = 'UINT'; Target position.Name = 'Target position'; Target position.DataType = 'DINT'; Touch probe function.Name = 'Touch probe function'; Touch probe function.DataType = 'UINT'; Physical outputs.Name = 'Physical outputs'; Physical outputs.DataType = 'UDINT'; Target velocity.Name = 'Target velocity'; Target velocity.DataType = 'DINT'; Target torque.Name = 'Target torque'; Target torque.DataType = 'INT'; Error code.Name = 'Error code'; Error code.DataType = 'UINT'; Statusword.Name = 'Statusword'; Statusword.DataType = 'UINT';
            Position actual value.Name = 'Position actual value'; Position actual value.DataType = 'DINT'; Torque actual value.Name = 'Torque actual value'; Torque actual value.DataType = 'INT'; Following error actual value.Name = 'Following error actual value'; Following error actual value.DataType = 'DINT'; Touch probe status.Name = 'Touch probe status'; Touch probe status.DataType = 'UINT'; Touch probe pos1 pos value.Name = 'Touch probe pos1 pos value'; Touch probe pos1 pos value.DataType = 'DINT'; Touch probe pos2 pos value.Name = 'Touch probe pos2 pos value'; Touch probe pos2 pos value.DataType = 'DINT'; Digital inputs.Name = 'Digital inputs'; Digital inputs.DataType = 'UDINT'; Velocity actual value.Name = 'Velocity actual value'; Velocity actual value.DataType = 'DINT'
          input  Application.末端控制.adFbForce[2] : INT  // Torque actual value
          unmapped channels: Controlword, Target position, Touch probe function, Physical outputs, Target velocity, Target torque, Error code, Statusword, Position actual value, Following error actual value, Touch probe status, Touch probe pos1 pos value, Touch probe pos2 pos value, Digital inputs, Velocity actual value
        下卷扬 : Axis, Inovance, order no. 0, version 1.0.0.0
            settings: wDriveID = 18; dwRatioTechUnitsDenom = 260759679; iRatioTechUnitsNum = 10000; fSWMaxVelocity = 1000; fSWMaxAcceleration = 10000; fSWMaxDeceleration = 10000; fSWMaxJerk = 100000; iEncoderType = 1; iAbsEncoderOption = 1; HomingMode = 10; ZeroSignal = 0; StartDirction = 1; EndDirection = 1; PosLimitMode = 0; NegLimitMode = 0; HomingVelocity = 10; HomingApproachVelocity = 2; HomingAcceleration = 100; HomingDeceleration = 100; HomingJerk = 0; HomeMaskDistance = 0; HomePositionOffset = 0; HomePushTime = 0; HomeCompensation = 0; HomeTimeout = 0; HomeCompensationVelocity = 1000; 4000 = 1; 4001 = 1; 4003 = true; 4004 = 3; 4005 = 0; 4006 = 1.666667; 4007 = 166.666666; 4008 = 0.166667; 4009 = 50000; 4010 = 3500; 4011 = 3500; 4012 = 100.000000; ScalingIncs = 16#40000; ScalingMotorTurns2 = 50;
              6005 = 502.6544; AdrOffset_8010 = 48; BitOffset_8010 = 0; BitLength_8010 = 16; Address_8010 = '%QW24'; Type_8010 = 'UINT'; AddressPointer_8010 = ADR(%QW24); AdrOffset_8020 = 52; BitOffset_8020 = 0; BitLength_8020 = 32; Address_8020 = '%QD13'; Type_8020 = 'DINT'; AddressPointer_8020 = ADR(%QD13); AdrOffset_8030 = 64; BitOffset_8030 = 0; BitLength_8030 = 32; Address_8030 = '%QD16'; Type_8030 = 'DINT'; AddressPointer_8030 = ADR(%QD16); AdrOffset_8040 = 68; BitOffset_8040 = 0; BitLength_8040 = 16; Address_8040 = '%QW34'; Type_8040 = 'INT'; AddressPointer_8040 = ADR(%QW34); AdrOffset_8050 = 4294967295; BitOffset_8050 = 0; BitLength_8050 = 0; Address_8050 = ''; Type_8050 = ''; AddressPointer_8050 = 0; AdrOffset_8060 = 56; BitOffset_8060 = 0; BitLength_8060 = 16; Address_8060 = '%QW28'; Type_8060 = 'UINT'; AddressPointer_8060 = ADR(%QW28); AdrOffset_8070 = 4294967295; BitOffset_8070 = 0; BitLength_8070 = 0;
              Address_8070 = ''; Type_8070 = ''; AddressPointer_8070 = 0; AdrOffset_8080 = 4294967295; BitOffset_8080 = 0; BitLength_8080 = 0; Address_8080 = ''; Type_8080 = ''; AddressPointer_8080 = 0; AdrOffset_8090 = 60; BitOffset_8090 = 0; BitLength_8090 = 32; Address_8090 = '%QD15'; Type_8090 = 'UDINT'; AddressPointer_8090 = ADR(%QD15); AdrOffset_8100 = 4294967295; BitOffset_8100 = 0; BitLength_8100 = 0; Address_8100 = ''; Type_8100 = ''; AddressPointer_8100 = 0; AdrOffset_8510 = 74; BitOffset_8510 = 0; BitLength_8510 = 16; Address_8510 = '%IW37'; Type_8510 = 'UINT'; AddressPointer_8510 = ADR(%IW37); AdrOffset_8520 = 76; BitOffset_8520 = 0; BitLength_8520 = 32; Address_8520 = '%ID19'; Type_8520 = 'DINT'; AddressPointer_8520 = ADR(%ID19); AdrOffset_8530 = 104; BitOffset_8530 = 0; BitLength_8530 = 32; Address_8530 = '%ID26'; Type_8530 = 'DINT'; AddressPointer_8530 = ADR(%ID26); AdrOffset_8540 = 0;
              BitOffset_8540 = 0; BitLength_8540 = 16; Address_8540 = '末端控制.adFbForce[2]'; Type_8540 = 'INT'; AddressPointer_8540 = ADR(末端控制.adFbForce[2]); AdrOffset_8550 = 4294967295; BitOffset_8550 = 0; BitLength_8550 = 0; Address_8550 = ''; Type_8550 = ''; AddressPointer_8550 = 0; AdrOffset_8560 = 100; BitOffset_8560 = 0; BitLength_8560 = 32; Address_8560 = '%ID25'; Type_8560 = 'UDINT'; AddressPointer_8560 = ADR(%ID25); AdrOffset_8570 = 88; BitOffset_8570 = 0; BitLength_8570 = 16; Address_8570 = '%IW44'; Type_8570 = 'UINT'; AddressPointer_8570 = ADR(%IW44); AdrOffset_8580 = 92; BitOffset_8580 = 0; BitLength_8580 = 32; Address_8580 = '%ID23'; Type_8580 = 'DINT'; AddressPointer_8580 = ADR(%ID23); AdrOffset_8590 = 4294967295; BitOffset_8590 = 0; BitLength_8590 = 0; Address_8590 = ''; Type_8590 = ''; AddressPointer_8590 = 0; AdrOffset_8600 = 96; BitOffset_8600 = 0; BitLength_8600 = 32; Address_8600 = '%ID24'; Type_8600 = 'DINT';
              AddressPointer_8600 = ADR(%ID24); AdrOffset_8600 = 4294967295; BitOffset_8600 = 0; BitLength_8600 = 0; Address_8610 = ''; Type_8610 = ''; AddressPointer_8610 = 0; AdrOffset_8620 = 72; BitOffset_8620 = 0; BitLength_8620 = 16; Address_8620 = '%IW36'; Type_8620 = 'UINT'; AddressPointer_8620 = ADR(%IW36); IsValid = True; IsHostHoming = False; PulseSelectIndex = 2
      InoSV630N_滚刷 : SV630_1Axis_03715, Inovance, order no. InoSV630N, version Revision=16#00010000
          settings: Number of Outputs = 6; Number of Inputs = 10; Number of Infos about Outputs = 6; Number of Infos about Inputs = 10; Physical Address of the Slave = 1004; AutoIncr Address of the Slave = 4294967293; StationAlias = 0; Sync.Length = 18; Sync.Length = 32; FMMU.Global Start Address = 16#02000036; FMMU.Length = 18; FMMU.Physical Start Address = 16#1800; FMMU.Access = 16#02; FMMU.Global Start Address = 16#01000060; FMMU.Length = 32; FMMU.Physical Start Address = 16#1C00; FMMU.Access = 16#01; FMMU.Global Start Address = 16#00080000; FMMU.StartBit = 3; FMMU.EndBit = 3; FMMU.Physical Start Address = 16#080D; FMMU.Access = 16#01; AutoUpdate = False; DC sync0 cycletime = 4000; DC sync1 cycletime = 4000; Number of SDO = 10; Homing method.Index = 16#6098; Homing method.Subindex = 16#00; Homing method.Value = 1; Homing method.Size = 8; Homing method.AbortIfError = FALSE; Homing method.JumpToLine = FALSE; Homing method.Line = 0; Homing method.CompleteAccess = FALSE; Actual Position Calculation Method.Index = 16#60E6; Actual Position Calculation Method.Subindex = 16#00; Actual Position Calculation Method.Value = 0; Actual Position Calculation Method.Size = 8; Actual Position Calculation Method.AbortIfError = FALSE; Actual Position Calculation Method.JumpToLine = FALSE;
            Actual Position Calculation Method.Line = 0; Actual Position Calculation Method.CompleteAccess = FALSE; Speed during search for switch.Index = 16#6099; Speed during search for switch.Subindex = 16#01; Speed during search for switch.Value = 436907; Speed during search for switch.Size = 32; Speed during search for switch.AbortIfError = FALSE; Speed during search for switch.JumpToLine = FALSE; Speed during search for switch.Line = 0; Speed during search for switch.CompleteAccess = FALSE; Homing acceleration.Index = 16#609A; Homing acceleration.Subindex = 16#00; Homing acceleration.Value = 43690666; Homing acceleration.Size = 32; Homing acceleration.AbortIfError = FALSE; Homing acceleration.JumpToLine = FALSE; Homing acceleration.Line = 0; Homing acceleration.CompleteAccess = FALSE; Speed during search for zero.Index = 16#6099; Speed during search for zero.Subindex = 16#02; Speed during search for zero.Value = 43691; Speed during search for zero.Size = 32; Speed during search for zero.AbortIfError = FALSE; Speed during search for zero.JumpToLine = FALSE; Speed during search for zero.Line = 0; Speed during search for zero.CompleteAccess = FALSE; Time of home searching.Index = 16#2005; Time of home searching.Subindex = 16#24; Time of home searching.Value = 50000; Time of home searching.Size = 16; Time of home searching.AbortIfError = FALSE; Time of home searching.JumpToLine = FALSE; Time of home searching.Line = 0; Time of home searching.CompleteAccess = FALSE; Positive torque limit value.Index = 16#60E0; Positive torque limit value.Subindex = 16#00; Positive torque limit value.Value = 3500; Positive torque limit value.Size = 16; Positive torque limit value.AbortIfError = FALSE; Positive torque limit value.JumpToLine = FALSE;
            Positive torque limit value.Line = 0; Positive torque limit value.CompleteAccess = FALSE; Negative torque limit value.Index = 16#60E1; Negative torque limit value.Subindex = 16#00; Negative torque limit value.Value = 3500; Negative torque limit value.Size = 16; Negative torque limit value.AbortIfError = FALSE; Negative torque limit value.JumpToLine = FALSE; Negative torque limit value.Line = 0; Negative torque limit value.CompleteAccess = FALSE; Max profile velocity.Index = 16#607F; Max profile velocity.Subindex = 16#00; Max profile velocity.Value = 26214400; Max profile velocity.Size = 32; Max profile velocity.AbortIfError = FALSE; Max profile velocity.JumpToLine = FALSE; Max profile velocity.Line = 0; Max profile velocity.CompleteAccess = FALSE; RxTxPdo.NumberofEntries = 6; RxTxPdo.Sm = 2; Controlword.Index = 16#6040; Controlword.SubIndex = 0; Controlword.Size = 16; Controlword.DependOnSlot = false; Controlword.DependOnSlotGroup = false; Target position.Index = 16#607A; Target position.SubIndex = 0; Target position.Size = 32; Target position.DependOnSlot = false; Target position.DependOnSlotGroup = false; Touch probe function.Index = 16#60B8; Touch probe function.SubIndex = 0; Touch probe function.Size = 16; Touch probe function.DependOnSlot = false; Touch probe function.DependOnSlotGroup = false; Physical outputs.Index = 16#60FE; Physical outputs.SubIndex = 1; Physical outputs.Size = 32; Physical outputs.DependOnSlot = false; Physical outputs.DependOnSlotGroup = false;
            Target velocity.Index = 16#60FF; Target velocity.SubIndex = 0; Target velocity.Size = 32; Target velocity.DependOnSlot = false; Target velocity.DependOnSlotGroup = false; Target torque.Index = 16#6071; Target torque.SubIndex = 0; Target torque.Size = 16; Target torque.DependOnSlot = false; Target torque.DependOnSlotGroup = false; RxTxPdo.Sm = -1; RxTxPdo.NumberofEntries = 10; RxTxPdo.Sm = 3; Error code.Index = 16#603F; Error code.SubIndex = 0; Error code.Size = 16; Error code.DependOnSlot = false; Error code.DependOnSlotGroup = false; Statusword.Index = 16#6041; Statusword.SubIndex = 0; Statusword.Size = 16; Statusword.DependOnSlot = false; Statusword.DependOnSlotGroup = false; Position actual value.Index = 16#6064; Position actual value.SubIndex = 0; Position actual value.Size = 32; Position actual value.DependOnSlot = false; Position actual value.DependOnSlotGroup = false; Torque actual value.Index = 16#6077; Torque actual value.SubIndex = 0; Torque actual value.Size = 16; Torque actual value.DependOnSlot = false; Torque actual value.DependOnSlotGroup = false; Following error actual value.Index = 16#60F4; Following error actual value.SubIndex = 0; Following error actual value.Size = 32; Following error actual value.DependOnSlot = false; Following error actual value.DependOnSlotGroup = false; Touch probe status.Index = 16#60B9; Touch probe status.SubIndex = 0;
            Touch probe status.Size = 16; Touch probe status.DependOnSlot = false; Touch probe status.DependOnSlotGroup = false; Touch probe pos1 pos value.Index = 16#60BA; Touch probe pos1 pos value.SubIndex = 0; Touch probe pos1 pos value.Size = 32; Touch probe pos1 pos value.DependOnSlot = false; Touch probe pos1 pos value.DependOnSlotGroup = false; Touch probe pos2 pos value.Index = 16#60BC; Touch probe pos2 pos value.SubIndex = 0; Touch probe pos2 pos value.Size = 32; Touch probe pos2 pos value.DependOnSlot = false; Touch probe pos2 pos value.DependOnSlotGroup = false; Digital inputs.Index = 16#60FD; Digital inputs.SubIndex = 0; Digital inputs.Size = 32; Digital inputs.DependOnSlot = false; Digital inputs.DependOnSlotGroup = false; Velocity actual value.Index = 16#606C; Velocity actual value.SubIndex = 0; Velocity actual value.Size = 32; Velocity actual value.DependOnSlot = false; Velocity actual value.DependOnSlotGroup = false; RxTxPdo.Sm = -1; Controlword.Name = 'Controlword'; Controlword.DataType = 'UINT'; Target position.Name = 'Target position'; Target position.DataType = 'DINT'; Touch probe function.Name = 'Touch probe function'; Touch probe function.DataType = 'UINT'; Physical outputs.Name = 'Physical outputs'; Physical outputs.DataType = 'UDINT'; Target velocity.Name = 'Target velocity'; Target velocity.DataType = 'DINT'; Target torque.Name = 'Target torque'; Target torque.DataType = 'INT'; Error code.Name = 'Error code'; Error code.DataType = 'UINT'; Statusword.Name = 'Statusword'; Statusword.DataType = 'UINT';
            Position actual value.Name = 'Position actual value'; Position actual value.DataType = 'DINT'; Torque actual value.Name = 'Torque actual value'; Torque actual value.DataType = 'INT'; Following error actual value.Name = 'Following error actual value'; Following error actual value.DataType = 'DINT'; Touch probe status.Name = 'Touch probe status'; Touch probe status.DataType = 'UINT'; Touch probe pos1 pos value.Name = 'Touch probe pos1 pos value'; Touch probe pos1 pos value.DataType = 'DINT'; Touch probe pos2 pos value.Name = 'Touch probe pos2 pos value'; Touch probe pos2 pos value.DataType = 'DINT'; Digital inputs.Name = 'Digital inputs'; Digital inputs.DataType = 'UDINT'; Velocity actual value.Name = 'Velocity actual value'; Velocity actual value.DataType = 'DINT'
          input  Application.末端控制.adFbForce[3] : INT  // Torque actual value
          unmapped channels: Controlword, Target position, Touch probe function, Physical outputs, Target velocity, Target torque, Error code, Statusword, Position actual value, Following error actual value, Touch probe status, Touch probe pos1 pos value, Touch probe pos2 pos value, Digital inputs, Velocity actual value
        滚刷 : Axis, Inovance, order no. 0, version 1.0.0.0
            settings: wDriveID = 19; dwRatioTechUnitsDenom = 262144; fSWMaxVelocity = 1000; fSWMaxAcceleration = 10000; fSWMaxDeceleration = 10000; fSWMaxJerk = 100000; iEncoderType = 1; iAbsEncoderOption = 1; HomingMode = 10; ZeroSignal = 0; StartDirction = 1; EndDirection = 1; PosLimitMode = 0; NegLimitMode = 0; HomingVelocity = 10; HomingApproachVelocity = 2; HomingAcceleration = 100; HomingDeceleration = 100; HomingJerk = 0; HomeMaskDistance = 0; HomePositionOffset = 0; HomePushTime = 0; HomeCompensation = 0; HomeTimeout = 0; HomeCompensationVelocity = 1000; 4000 = 0; 4001 = 0; 4003 = true; 4004 = 3; 4005 = 0; 4006 = 1.666667; 4007 = 166.666666; 4008 = 0.166667; 4009 = 50000; 4010 = 3500; 4011 = 3500; 4012 = 100.000000; ScalingIncs = 16#40000; 6005 = 1; AdrOffset_8010 = 72;
              BitOffset_8010 = 0; BitLength_8010 = 16; Address_8010 = '%QW36'; Type_8010 = 'UINT'; AddressPointer_8010 = ADR(%QW36); AdrOffset_8020 = 76; BitOffset_8020 = 0; BitLength_8020 = 32; Address_8020 = '%QD19'; Type_8020 = 'DINT'; AddressPointer_8020 = ADR(%QD19); set velocity (diSetVelocity) = 1118; Object_8030 = 16#60FF:16#00; AdrOffset_8030 = 88; BitOffset_8030 = 0; BitLength_8030 = 32; Address_8030 = '%QD22'; Type_8030 = 'DINT'; AddressPointer_8030 = ADR(%QD22); set torque (wSetTorque) = 1168; Object_8040 = 16#6071:16#00; AdrOffset_8040 = 92; BitOffset_8040 = 0; BitLength_8040 = 16; Address_8040 = '%QW46'; Type_8040 = 'INT'; AddressPointer_8040 = ADR(%QW46); Modes of operation (OP) = 10096; Object_8050 = 16#6060:16#00; AdrOffset_8050 = 4294967295; BitOffset_8050 = 0; BitLength_8050 = 0; Address_8050 = ''; Type_8050 = ''; AddressPointer_8050 = 0; Touch Probe Function = 10184; Object_8060 = 16#60B8:16#00; AdrOffset_8060 = 80; BitOffset_8060 = 0; BitLength_8060 = 16;
              Address_8060 = '%QW40'; Type_8060 = 'UINT'; AddressPointer_8060 = ADR(%QW40); Add velocity value = 10177; Object_8070 = 16#60B1:16#00; AdrOffset_8070 = 4294967295; BitOffset_8070 = 0; BitLength_8070 = 0; Address_8070 = ''; Type_8070 = ''; AddressPointer_8070 = 0; Add torque value = 10178; Object_8080 = 16#60B2:16#00; AdrOffset_8080 = 4294967295; BitOffset_8080 = 0; BitLength_8080 = 0; Address_8080 = ''; Type_8080 = ''; AddressPointer_8080 = 0; Digital outputs (A637) = 10254; Object_8090 = 16#60FE:16#01; AdrOffset_8090 = 84; BitOffset_8090 = 0; BitLength_8090 = 32; Address_8090 = '%QD21'; Type_8090 = 'UDINT'; AddressPointer_8090 = ADR(%QD21); Max Profile Velocity = 2010; Object_8100 = 16#607F:16#00; AdrOffset_8100 = 4294967295; BitOffset_8100 = 0; BitLength_8100 = 0; Address_8100 = ''; Type_8100 = ''; AddressPointer_8100 = 0; AdrOffset_8510 = 110; BitOffset_8510 = 0; BitLength_8510 = 16; Address_8510 = '%IW55'; Type_8510 = 'UINT';
              AddressPointer_8510 = ADR(%IW55); AdrOffset_8520 = 112; BitOffset_8520 = 0; BitLength_8520 = 32; Address_8520 = '%ID28'; Type_8520 = 'DINT'; AddressPointer_8520 = ADR(%ID28); actual velocity (diActVelocity) = 1119; Object_8530 = 16#606C:16#00; AdrOffset_8530 = 140; BitOffset_8530 = 0; BitLength_8530 = 32; Address_8530 = '%ID35'; Type_8530 = 'DINT'; AddressPointer_8530 = ADR(%ID35); actual torque (wActTorque) = 1169; Object_8540 = 16#6077:16#00; AdrOffset_8540 = 0; BitOffset_8540 = 0; BitLength_8540 = 16; Address_8540 = '末端控制.adFbForce[3]'; Type_8540 = 'INT'; AddressPointer_8540 = ADR(末端控制.adFbForce[3]); Modes of operation display (OP) = 20097; Object_8550 = 16#6061:16#00; AdrOffset_8550 = 4294967295; BitOffset_8550 = 0; BitLength_8550 = 0; Address_8550 = ''; Type_8550 = ''; AddressPointer_8550 = 0; digital inputs (in.dwDigitalInputs) = 20253; Object_8560 = 16#60FD:16#00; AdrOffset_8560 = 136; BitOffset_8560 = 0; BitLength_8560 = 32; Address_8560 = '%ID34'; Type_8560 = 'UDINT'; AddressPointer_8560 = ADR(%ID34); Touch Probe Status = 20185;
              Object_8570 = 16#60B9:16#00; AdrOffset_8570 = 124; BitOffset_8570 = 0; BitLength_8570 = 16; Address_8570 = '%IW62'; Type_8570 = 'UINT'; AddressPointer_8570 = ADR(%IW62); Touch Probe 1 rising edge = 20186; Object_8580 = 16#60BA:16#00; AdrOffset_8580 = 128; BitOffset_8580 = 0; BitLength_8580 = 32; Address_8580 = '%ID32'; Type_8580 = 'DINT'; AddressPointer_8580 = ADR(%ID32); Touch Probe 1 falling edge = 20187; Object_8590 = 16#60BB:16#00; AdrOffset_8590 = 4294967295; BitOffset_8590 = 0; BitLength_8590 = 0; Address_8590 = ''; Type_8590 = ''; AddressPointer_8590 = 0; Touch Probe 2 rising edge = 20188; Object_8600 = 16#60BC:16#00; AdrOffset_8600 = 132; BitOffset_8600 = 0; BitLength_8600 = 32; Address_8600 = '%ID33'; Type_8600 = 'DINT'; AddressPointer_8600 = ADR(%ID33); Touch Probe 2 falling edge = 20189; Object_8600 = 16#60BD:16#00; AdrOffset_8600 = 4294967295; BitOffset_8600 = 0; BitLength_8600 = 0; Address_8610 = ''; Type_8610 = ''; AddressPointer_8610 = 0; Error Code(603F) = 2020;
              Object_8620 = 16#603F:16#00; AdrOffset_8620 = 108; BitOffset_8620 = 0; BitLength_8620 = 16; Address_8620 = '%IW54'; Type_8620 = 'UINT'; AddressPointer_8620 = ADR(%IW54); Automatic Mapping = True; IsValid = True; IsHostHoming = False; PulseSelectIndex = 2
      InoSV630N_左上轮 : SV630_1Axis_03715, Inovance, order no. InoSV630N, version Revision=16#00010000
          settings: Number of Outputs = 7; Number of Inputs = 10; Number of Infos about Outputs = 7; Number of Infos about Inputs = 10; EnableExpertSettings = True; Physical Address of the Slave = 1016; AutoIncr Address of the Slave = 4294967281; StationAlias = 0; Sync.Length = 19; Sync.Length = 32; FMMU.Global Start Address = 16#02000106; FMMU.Length = 19; FMMU.Physical Start Address = 16#1800; FMMU.Access = 16#02; FMMU.Global Start Address = 16#010001DE; FMMU.Length = 32; FMMU.Physical Start Address = 16#1C00; FMMU.Access = 16#01; FMMU.Global Start Address = 16#00080001; FMMU.StartBit = 6; FMMU.EndBit = 6; FMMU.Physical Start Address = 16#080D; FMMU.Access = 16#01; AutoUpdate = False; DC sync0 cycletime = 4000; DC sync0 cycletime = 4000000; DC sync1 cycletime = 4000; DC sync1 cycletime = 4000000; Number of SDO = 10; Homing method.Index = 16#6098; Homing method.Subindex = 16#00; Homing method.Value = 1; Homing method.Size = 8; Homing method.AbortIfError = FALSE; Homing method.JumpToLine = FALSE; Homing method.Line = 0; Homing method.CompleteAccess = FALSE; Actual Position Calculation Method.Index = 16#60E6; Actual Position Calculation Method.Subindex = 16#00; Actual Position Calculation Method.Value = 0;
            Actual Position Calculation Method.Size = 8; Actual Position Calculation Method.AbortIfError = FALSE; Actual Position Calculation Method.JumpToLine = FALSE; Actual Position Calculation Method.Line = 0; Actual Position Calculation Method.CompleteAccess = FALSE; Speed during search for switch.Index = 16#6099; Speed during search for switch.Subindex = 16#01; Speed during search for switch.Value = 11031; Speed during search for switch.Size = 32; Speed during search for switch.AbortIfError = FALSE; Speed during search for switch.JumpToLine = FALSE; Speed during search for switch.Line = 0; Speed during search for switch.CompleteAccess = FALSE; Homing acceleration.Index = 16#609A; Homing acceleration.Subindex = 16#00; Homing acceleration.Value = 1103102; Homing acceleration.Size = 32; Homing acceleration.AbortIfError = FALSE; Homing acceleration.JumpToLine = FALSE; Homing acceleration.Line = 0; Homing acceleration.CompleteAccess = FALSE; Speed during search for zero.Index = 16#6099; Speed during search for zero.Subindex = 16#02; Speed during search for zero.Value = 1103; Speed during search for zero.Size = 32; Speed during search for zero.AbortIfError = FALSE; Speed during search for zero.JumpToLine = FALSE; Speed during search for zero.Line = 0; Speed during search for zero.CompleteAccess = FALSE; Time of home searching.Index = 16#2005; Time of home searching.Subindex = 16#24; Time of home searching.Value = 50000; Time of home searching.Size = 16; Time of home searching.AbortIfError = FALSE; Time of home searching.JumpToLine = FALSE; Time of home searching.Line = 0; Time of home searching.CompleteAccess = FALSE; Positive torque limit value.Index = 16#60E0; Positive torque limit value.Subindex = 16#00; Positive torque limit value.Value = 3500;
            Positive torque limit value.Size = 16; Positive torque limit value.AbortIfError = FALSE; Positive torque limit value.JumpToLine = FALSE; Positive torque limit value.Line = 0; Positive torque limit value.CompleteAccess = FALSE; Negative torque limit value.Index = 16#60E1; Negative torque limit value.Subindex = 16#00; Negative torque limit value.Value = 3500; Negative torque limit value.Size = 16; Negative torque limit value.AbortIfError = FALSE; Negative torque limit value.JumpToLine = FALSE; Negative torque limit value.Line = 0; Negative torque limit value.CompleteAccess = FALSE; Max profile velocity.Index = 16#607F; Max profile velocity.Subindex = 16#00; Max profile velocity.Value = 661861; Max profile velocity.Size = 32; Max profile velocity.AbortIfError = FALSE; Max profile velocity.JumpToLine = FALSE; Max profile velocity.Line = 0; Max profile velocity.CompleteAccess = FALSE; RxTxPdo.NumberofEntries = 7; RxTxPdo.DependOnSlot = False; RxTxPdo.DependOnSlotGroup = False; RxTxPdo.OverwrittenByModule = False; Exclude = [16#1701,16#1702,16#1703,16#1704,16#1705]; Controlword.Index = 16#6040; Controlword.SubIndex = 0; Controlword.Size = 16; Controlword.Offset = 0; Controlword.DependOnSlot = False; Controlword.DependOnSlotGroup = False; Target position.Index = 16#607A; Target position.SubIndex = 0; Target position.Size = 32; Target position.Offset = 0; Target position.DependOnSlot = False; Target position.DependOnSlotGroup = False; Touch probe function.Index = 16#60B8; Touch probe function.SubIndex = 0;
            Touch probe function.Size = 16; Touch probe function.Offset = 0; Touch probe function.DependOnSlot = False; Touch probe function.DependOnSlotGroup = False; Physical outputs.Index = 16#60FE; Physical outputs.SubIndex = 1; Physical outputs.Size = 32; Physical outputs.Offset = 0; Physical outputs.DependOnSlot = False; Physical outputs.DependOnSlotGroup = False; Target velocity.Index = 16#60FF; Target velocity.SubIndex = 0; Target velocity.Size = 32; Target velocity.Offset = 0; Target velocity.DependOnSlot = False; Target velocity.DependOnSlotGroup = False; Modes of operation.Index = 16#6060; Modes of operation.SubIndex = 0; Modes of operation.Size = 8; Modes of operation.Offset = 0; Modes of operation.DependOnSlot = False; Modes of operation.DependOnSlotGroup = False; Target torque.Index = 16#6071; Target torque.SubIndex = 0; Target torque.Size = 16; Target torque.Offset = 0; Target torque.DependOnSlot = False; Target torque.DependOnSlotGroup = False; RxTxPdo.Sm = -1; RxTxPdo.Sm = 2; RxTxPdo.NumberofEntries = 10; RxTxPdo.Sm = 3; Error code.Index = 16#603F; Error code.SubIndex = 0; Error code.Size = 16; Error code.DependOnSlot = false; Error code.DependOnSlotGroup = false; Statusword.Index = 16#6041; Statusword.SubIndex = 0; Statusword.Size = 16;
            Statusword.DependOnSlot = false; Statusword.DependOnSlotGroup = false; Position actual value.Index = 16#6064; Position actual value.SubIndex = 0; Position actual value.Size = 32; Position actual value.DependOnSlot = false; Position actual value.DependOnSlotGroup = false; Torque actual value.Index = 16#6077; Torque actual value.SubIndex = 0; Torque actual value.Size = 16; Torque actual value.DependOnSlot = false; Torque actual value.DependOnSlotGroup = false; Following error actual value.Index = 16#60F4; Following error actual value.SubIndex = 0; Following error actual value.Size = 32; Following error actual value.DependOnSlot = false; Following error actual value.DependOnSlotGroup = false; Touch probe status.Index = 16#60B9; Touch probe status.SubIndex = 0; Touch probe status.Size = 16; Touch probe status.DependOnSlot = false; Touch probe status.DependOnSlotGroup = false; Touch probe pos1 pos value.Index = 16#60BA; Touch probe pos1 pos value.SubIndex = 0; Touch probe pos1 pos value.Size = 32; Touch probe pos1 pos value.DependOnSlot = false; Touch probe pos1 pos value.DependOnSlotGroup = false; Touch probe pos2 pos value.Index = 16#60BC; Touch probe pos2 pos value.SubIndex = 0; Touch probe pos2 pos value.Size = 32; Touch probe pos2 pos value.DependOnSlot = false; Touch probe pos2 pos value.DependOnSlotGroup = false; Digital inputs.Index = 16#60FD; Digital inputs.SubIndex = 0; Digital inputs.Size = 32; Digital inputs.DependOnSlot = false; Digital inputs.DependOnSlotGroup = false; Velocity actual value.Index = 16#606C; Velocity actual value.SubIndex = 0; Velocity actual value.Size = 32;
            Velocity actual value.DependOnSlot = false; Velocity actual value.DependOnSlotGroup = false; RxTxPdo.Sm = -1; Controlword.Name = 'Controlword'; Controlword.DataType = 'UINT'; Controlword.Default = ''; Controlword.Comment = ''; Target position.Name = 'Target position'; Target position.DataType = 'DINT'; Target position.Default = ''; Target position.Comment = ''; Touch probe function.Name = 'Touch probe function'; Touch probe function.DataType = 'UINT'; Touch probe function.Default = ''; Touch probe function.Comment = ''; Physical outputs.Name = 'Physical outputs'; Physical outputs.DataType = 'UDINT'; Physical outputs.Default = ''; Physical outputs.Comment = ''; Target velocity.Name = 'Target velocity'; Target velocity.DataType = 'DINT'; Target velocity.Default = ''; Target velocity.Comment = ''; Modes of operation.Name = 'Modes of operation'; Modes of operation.DataType = 'SINT'; Modes of operation.Default = ''; Modes of operation.Comment = ''; Target torque.Name = 'Target torque'; Target torque.DataType = 'INT'; Target torque.Default = ''; Target torque.Comment = ''; Error code.Name = 'Error code'; Error code.DataType = 'UINT'; Statusword.Name = 'Statusword'; Statusword.DataType = 'UINT'; Position actual value.Name = 'Position actual value'; Position actual value.DataType = 'DINT'; Torque actual value.Name = 'Torque actual value'; Torque actual value.DataType = 'INT'; Following error actual value.Name = 'Following error actual value';
            Following error actual value.DataType = 'DINT'; Touch probe status.Name = 'Touch probe status'; Touch probe status.DataType = 'UINT'; Touch probe pos1 pos value.Name = 'Touch probe pos1 pos value'; Touch probe pos1 pos value.DataType = 'DINT'; Touch probe pos2 pos value.Name = 'Touch probe pos2 pos value'; Touch probe pos2 pos value.DataType = 'DINT'; Digital inputs.Name = 'Digital inputs'; Digital inputs.DataType = 'UDINT'; Velocity actual value.Name = 'Velocity actual value'; Velocity actual value.DataType = 'DINT'
          output Application.左上轮最大轮廓速度 : UDINT  // Max profile velocity
          unmapped channels: Controlword, Target position, Target velocity, Target torque, Modes of operation, Touch probe function, Error code, Statusword, Position actual value, Torque actual value, Following error actual value, Touch probe status, Touch probe pos1 pos value, Touch probe pos2 pos value, Digital inputs, Velocity actual value
        左上轮 : Axis, Inovance, order no. 0, version 1.0.0.0
            settings: wDriveID = 8; dwRatioTechUnitsDenom = 2621440000; iRatioTechUnitsNum = 396071; fSWMaxVelocity = 1000; fSWMaxAcceleration = 10000; fSWMaxDeceleration = 10000; fSWMaxJerk = 100000; iEncoderType = 1; iAbsEncoderOption = 1; HomingMode = 10; ZeroSignal = 0; StartDirction = 1; EndDirection = 1; PosLimitMode = 0; NegLimitMode = 0; HomingVelocity = 10; HomingApproachVelocity = 2; HomingAcceleration = 100; HomingDeceleration = 100; HomingJerk = 0; HomeMaskDistance = 0; HomePositionOffset = 0; HomePushTime = 0; HomeCompensation = 0; HomeTimeout = 0; HomeCompensationVelocity = 1000; 4000 = 1; 4001 = 0; 4003 = true; 4004 = 3; 4005 = 0; 4006 = 1.666667; 4007 = 166.666666; 4008 = 0.166667; 4009 = 50000; 4010 = 3500; 4011 = 3500; 4012 = 100.000000; ScalingIncs = 16#40000; 6005 = 39.6071;
              AdrOffset_8010 = 340; BitOffset_8010 = 0; BitLength_8010 = 16; Address_8010 = '%QW170'; Type_8010 = 'UINT'; AddressPointer_8010 = ADR(%QW170); AdrOffset_8020 = 344; BitOffset_8020 = 0; BitLength_8020 = 32; Address_8020 = '%QD86'; Type_8020 = 'DINT'; AddressPointer_8020 = ADR(%QD86); AdrOffset_8030 = 348; BitOffset_8030 = 0; BitLength_8030 = 32; Address_8030 = '%QD87'; Type_8030 = 'DINT'; AddressPointer_8030 = ADR(%QD87); AdrOffset_8040 = 352; BitOffset_8040 = 0; BitLength_8040 = 16; Address_8040 = '%QW176'; Type_8040 = 'INT'; AddressPointer_8040 = ADR(%QW176); AdrOffset_8050 = 354; BitOffset_8050 = 0; BitLength_8050 = 8; Address_8050 = '%QB354'; Type_8050 = 'SINT'; AddressPointer_8050 = ADR(%QB354); AdrOffset_8060 = 356; BitOffset_8060 = 0; BitLength_8060 = 16; Address_8060 = '%QW178'; Type_8060 = 'UINT'; AddressPointer_8060 = ADR(%QW178); AdrOffset_8070 = 4294967295; BitOffset_8070 = 0; BitLength_8070 = 0; Address_8070 = '';
              Type_8070 = ''; AddressPointer_8070 = 0; AdrOffset_8080 = 4294967295; BitOffset_8080 = 0; BitLength_8080 = 0; Address_8080 = ''; Type_8080 = ''; AddressPointer_8080 = 0; AdrOffset_8090 = 4294967295; BitOffset_8090 = 0; BitLength_8090 = 0; Address_8090 = ''; Type_8090 = ''; AddressPointer_8090 = 0; AdrOffset_8100 = 0; BitOffset_8100 = 0; BitLength_8100 = 32; Address_8100 = '左上轮最大轮廓速度'; Type_8100 = 'UDINT'; AddressPointer_8100 = ADR(左上轮最大轮廓速度); AdrOffset_8510 = 538; BitOffset_8510 = 0; BitLength_8510 = 16; Address_8510 = '%IW269'; Type_8510 = 'UINT'; AddressPointer_8510 = ADR(%IW269); AdrOffset_8520 = 540; BitOffset_8520 = 0; BitLength_8520 = 32; Address_8520 = '%ID135'; Type_8520 = 'DINT'; AddressPointer_8520 = ADR(%ID135); AdrOffset_8530 = 568; BitOffset_8530 = 0; BitLength_8530 = 32; Address_8530 = '%ID142'; Type_8530 = 'DINT'; AddressPointer_8530 = ADR(%ID142); AdrOffset_8540 = 544; BitOffset_8540 = 0;
              BitLength_8540 = 16; Address_8540 = '%IW272'; Type_8540 = 'INT'; AddressPointer_8540 = ADR(%IW272); AdrOffset_8550 = 4294967295; BitOffset_8550 = 0; BitLength_8550 = 0; Address_8550 = ''; Type_8550 = ''; AddressPointer_8550 = 0; AdrOffset_8560 = 564; BitOffset_8560 = 0; BitLength_8560 = 32; Address_8560 = '%ID141'; Type_8560 = 'UDINT'; AddressPointer_8560 = ADR(%ID141); AdrOffset_8570 = 552; BitOffset_8570 = 0; BitLength_8570 = 16; Address_8570 = '%IW276'; Type_8570 = 'UINT'; AddressPointer_8570 = ADR(%IW276); AdrOffset_8580 = 556; BitOffset_8580 = 0; BitLength_8580 = 32; Address_8580 = '%ID139'; Type_8580 = 'DINT'; AddressPointer_8580 = ADR(%ID139); AdrOffset_8590 = 4294967295; BitOffset_8590 = 0; BitLength_8590 = 0; Address_8590 = ''; Type_8590 = ''; AddressPointer_8590 = 0; AdrOffset_8600 = 560; BitOffset_8600 = 0; BitLength_8600 = 32; Address_8600 = '%ID140'; Type_8600 = 'DINT'; AddressPointer_8600 = ADR(%ID140);
              AdrOffset_8600 = 4294967295; BitOffset_8600 = 0; BitLength_8600 = 0; Address_8610 = ''; Type_8610 = ''; AddressPointer_8610 = 0; AdrOffset_8620 = 536; BitOffset_8620 = 0; BitLength_8620 = 16; Address_8620 = '%IW268'; Type_8620 = 'UINT'; AddressPointer_8620 = ADR(%IW268); Automatic Mapping = True; IsValid = True; IsHostHoming = False; PulseSelectIndex = 2
      InoSV630N_左下轮 : SV630_1Axis_03715, Inovance, order no. InoSV630N, version Revision=16#00010000
          settings: Number of Outputs = 7; Number of Inputs = 10; Number of Infos about Outputs = 7; Number of Infos about Inputs = 10; EnableExpertSettings = True; Physical Address of the Slave = 1017; AutoIncr Address of the Slave = 4294967280; StationAlias = 0; Sync.Length = 19; Sync.Length = 32; FMMU.Global Start Address = 16#02000119; FMMU.Length = 19; FMMU.Physical Start Address = 16#1800; FMMU.Access = 16#02; FMMU.Global Start Address = 16#010001FE; FMMU.Length = 32; FMMU.Physical Start Address = 16#1C00; FMMU.Access = 16#01; FMMU.Global Start Address = 16#00080001; FMMU.StartBit = 7; FMMU.EndBit = 7; FMMU.Physical Start Address = 16#080D; FMMU.Access = 16#01; AutoUpdate = False; DC sync0 cycletime = 4000; DC sync0 cycletime = 4000000; DC sync1 cycletime = 4000; DC sync1 cycletime = 4000000; Number of SDO = 10; Homing method.Index = 16#6098; Homing method.Subindex = 16#00; Homing method.Value = 1; Homing method.Size = 8; Homing method.AbortIfError = FALSE; Homing method.JumpToLine = FALSE; Homing method.Line = 0; Homing method.CompleteAccess = FALSE; Actual Position Calculation Method.Index = 16#60E6; Actual Position Calculation Method.Subindex = 16#00; Actual Position Calculation Method.Value = 0;
            Actual Position Calculation Method.Size = 8; Actual Position Calculation Method.AbortIfError = FALSE; Actual Position Calculation Method.JumpToLine = FALSE; Actual Position Calculation Method.Line = 0; Actual Position Calculation Method.CompleteAccess = FALSE; Speed during search for switch.Index = 16#6099; Speed during search for switch.Subindex = 16#01; Speed during search for switch.Value = 11031; Speed during search for switch.Size = 32; Speed during search for switch.AbortIfError = FALSE; Speed during search for switch.JumpToLine = FALSE; Speed during search for switch.Line = 0; Speed during search for switch.CompleteAccess = FALSE; Homing acceleration.Index = 16#609A; Homing acceleration.Subindex = 16#00; Homing acceleration.Value = 1103102; Homing acceleration.Size = 32; Homing acceleration.AbortIfError = FALSE; Homing acceleration.JumpToLine = FALSE; Homing acceleration.Line = 0; Homing acceleration.CompleteAccess = FALSE; Speed during search for zero.Index = 16#6099; Speed during search for zero.Subindex = 16#02; Speed during search for zero.Value = 1103; Speed during search for zero.Size = 32; Speed during search for zero.AbortIfError = FALSE; Speed during search for zero.JumpToLine = FALSE; Speed during search for zero.Line = 0; Speed during search for zero.CompleteAccess = FALSE; Time of home searching.Index = 16#2005; Time of home searching.Subindex = 16#24; Time of home searching.Value = 50000; Time of home searching.Size = 16; Time of home searching.AbortIfError = FALSE; Time of home searching.JumpToLine = FALSE; Time of home searching.Line = 0; Time of home searching.CompleteAccess = FALSE; Positive torque limit value.Index = 16#60E0; Positive torque limit value.Subindex = 16#00; Positive torque limit value.Value = 3500;
            Positive torque limit value.Size = 16; Positive torque limit value.AbortIfError = FALSE; Positive torque limit value.JumpToLine = FALSE; Positive torque limit value.Line = 0; Positive torque limit value.CompleteAccess = FALSE; Negative torque limit value.Index = 16#60E1; Negative torque limit value.Subindex = 16#00; Negative torque limit value.Value = 3500; Negative torque limit value.Size = 16; Negative torque limit value.AbortIfError = FALSE; Negative torque limit value.JumpToLine = FALSE; Negative torque limit value.Line = 0; Negative torque limit value.CompleteAccess = FALSE; Max profile velocity.Index = 16#607F; Max profile velocity.Subindex = 16#00; Max profile velocity.Value = 661861; Max profile velocity.Size = 32; Max profile velocity.AbortIfError = FALSE; Max profile velocity.JumpToLine = FALSE; Max profile velocity.Line = 0; Max profile velocity.CompleteAccess = FALSE; RxTxPdo.NumberofEntries = 7; RxTxPdo.DependOnSlot = False; RxTxPdo.DependOnSlotGroup = False; RxTxPdo.OverwrittenByModule = False; Exclude = [16#1701,16#1702,16#1703,16#1704,16#1705]; Controlword.Index = 16#6040; Controlword.SubIndex = 0; Controlword.Size = 16; Controlword.Offset = 0; Controlword.DependOnSlot = False; Controlword.DependOnSlotGroup = False; Target position.Index = 16#607A; Target position.SubIndex = 0; Target position.Size = 32; Target position.Offset = 0; Target position.DependOnSlot = False; Target position.DependOnSlotGroup = False; Touch probe function.Index = 16#60B8; Touch probe function.SubIndex = 0;
            Touch probe function.Size = 16; Touch probe function.Offset = 0; Touch probe function.DependOnSlot = False; Touch probe function.DependOnSlotGroup = False; Physical outputs.Index = 16#60FE; Physical outputs.SubIndex = 1; Physical outputs.Size = 32; Physical outputs.Offset = 0; Physical outputs.DependOnSlot = False; Physical outputs.DependOnSlotGroup = False; Target velocity.Index = 16#60FF; Target velocity.SubIndex = 0; Target velocity.Size = 32; Target velocity.Offset = 0; Target velocity.DependOnSlot = False; Target velocity.DependOnSlotGroup = False; Modes of operation.Index = 16#6060; Modes of operation.SubIndex = 0; Modes of operation.Size = 8; Modes of operation.Offset = 0; Modes of operation.DependOnSlot = False; Modes of operation.DependOnSlotGroup = False; Target torque.Index = 16#6071; Target torque.SubIndex = 0; Target torque.Size = 16; Target torque.Offset = 0; Target torque.DependOnSlot = False; Target torque.DependOnSlotGroup = False; RxTxPdo.Sm = -1; RxTxPdo.Sm = 2; RxTxPdo.NumberofEntries = 10; RxTxPdo.Sm = 3; Error code.Index = 16#603F; Error code.SubIndex = 0; Error code.Size = 16; Error code.DependOnSlot = false; Error code.DependOnSlotGroup = false; Statusword.Index = 16#6041; Statusword.SubIndex = 0; Statusword.Size = 16;
            Statusword.DependOnSlot = false; Statusword.DependOnSlotGroup = false; Position actual value.Index = 16#6064; Position actual value.SubIndex = 0; Position actual value.Size = 32; Position actual value.DependOnSlot = false; Position actual value.DependOnSlotGroup = false; Torque actual value.Index = 16#6077; Torque actual value.SubIndex = 0; Torque actual value.Size = 16; Torque actual value.DependOnSlot = false; Torque actual value.DependOnSlotGroup = false; Following error actual value.Index = 16#60F4; Following error actual value.SubIndex = 0; Following error actual value.Size = 32; Following error actual value.DependOnSlot = false; Following error actual value.DependOnSlotGroup = false; Touch probe status.Index = 16#60B9; Touch probe status.SubIndex = 0; Touch probe status.Size = 16; Touch probe status.DependOnSlot = false; Touch probe status.DependOnSlotGroup = false; Touch probe pos1 pos value.Index = 16#60BA; Touch probe pos1 pos value.SubIndex = 0; Touch probe pos1 pos value.Size = 32; Touch probe pos1 pos value.DependOnSlot = false; Touch probe pos1 pos value.DependOnSlotGroup = false; Touch probe pos2 pos value.Index = 16#60BC; Touch probe pos2 pos value.SubIndex = 0; Touch probe pos2 pos value.Size = 32; Touch probe pos2 pos value.DependOnSlot = false; Touch probe pos2 pos value.DependOnSlotGroup = false; Digital inputs.Index = 16#60FD; Digital inputs.SubIndex = 0; Digital inputs.Size = 32; Digital inputs.DependOnSlot = false; Digital inputs.DependOnSlotGroup = false; Velocity actual value.Index = 16#606C; Velocity actual value.SubIndex = 0; Velocity actual value.Size = 32;
            Velocity actual value.DependOnSlot = false; Velocity actual value.DependOnSlotGroup = false; RxTxPdo.Sm = -1; Controlword.Name = 'Controlword'; Controlword.DataType = 'UINT'; Controlword.Default = ''; Controlword.Comment = ''; Target position.Name = 'Target position'; Target position.DataType = 'DINT'; Target position.Default = ''; Target position.Comment = ''; Touch probe function.Name = 'Touch probe function'; Touch probe function.DataType = 'UINT'; Touch probe function.Default = ''; Touch probe function.Comment = ''; Physical outputs.Name = 'Physical outputs'; Physical outputs.DataType = 'UDINT'; Physical outputs.Default = ''; Physical outputs.Comment = ''; Target velocity.Name = 'Target velocity'; Target velocity.DataType = 'DINT'; Target velocity.Default = ''; Target velocity.Comment = ''; Modes of operation.Name = 'Modes of operation'; Modes of operation.DataType = 'SINT'; Modes of operation.Default = ''; Modes of operation.Comment = ''; Target torque.Name = 'Target torque'; Target torque.DataType = 'INT'; Target torque.Default = ''; Target torque.Comment = ''; Error code.Name = 'Error code'; Error code.DataType = 'UINT'; Statusword.Name = 'Statusword'; Statusword.DataType = 'UINT'; Position actual value.Name = 'Position actual value'; Position actual value.DataType = 'DINT'; Torque actual value.Name = 'Torque actual value'; Torque actual value.DataType = 'INT'; Following error actual value.Name = 'Following error actual value';
            Following error actual value.DataType = 'DINT'; Touch probe status.Name = 'Touch probe status'; Touch probe status.DataType = 'UINT'; Touch probe pos1 pos value.Name = 'Touch probe pos1 pos value'; Touch probe pos1 pos value.DataType = 'DINT'; Touch probe pos2 pos value.Name = 'Touch probe pos2 pos value'; Touch probe pos2 pos value.DataType = 'DINT'; Digital inputs.Name = 'Digital inputs'; Digital inputs.DataType = 'UDINT'; Velocity actual value.Name = 'Velocity actual value'; Velocity actual value.DataType = 'DINT'
          unmapped channels: Controlword, Target position, Target velocity, Target torque, Modes of operation, Touch probe function, Max profile velocity, Error code, Statusword, Position actual value, Torque actual value, Following error actual value, Touch probe status, Touch probe pos1 pos value, Touch probe pos2 pos value, Digital inputs, Velocity actual value
        左下轮 : Axis, Inovance, order no. 0, version 1.0.0.0
            settings: wDriveID = 9; dwRatioTechUnitsDenom = 2621440000; iRatioTechUnitsNum = 396071; fSWMaxVelocity = 1000; fSWMaxAcceleration = 10000; fSWMaxDeceleration = 10000; fSWMaxJerk = 100000; iEncoderType = 1; iAbsEncoderOption = 1; HomingMode = 10; ZeroSignal = 0; StartDirction = 1; EndDirection = 1; PosLimitMode = 0; NegLimitMode = 0; HomingVelocity = 10; HomingApproachVelocity = 2; HomingAcceleration = 100; HomingDeceleration = 100; HomingJerk = 0; HomeMaskDistance = 0; HomePositionOffset = 0; HomePushTime = 0; HomeCompensation = 0; HomeTimeout = 0; HomeCompensationVelocity = 1000; 4000 = 1; 4001 = 0; 4003 = true; 4004 = 3; 4005 = 0; 4006 = 1.666667; 4007 = 166.666666; 4008 = 0.166667; 4009 = 50000; 4010 = 3500; 4011 = 3500; 4012 = 100.000000; ScalingIncs = 16#40000; 6005 = 39.6071;
              AdrOffset_8010 = 364; BitOffset_8010 = 0; BitLength_8010 = 16; Address_8010 = '%QW182'; Type_8010 = 'UINT'; AddressPointer_8010 = ADR(%QW182); AdrOffset_8020 = 368; BitOffset_8020 = 0; BitLength_8020 = 32; Address_8020 = '%QD92'; Type_8020 = 'DINT'; AddressPointer_8020 = ADR(%QD92); AdrOffset_8030 = 372; BitOffset_8030 = 0; BitLength_8030 = 32; Address_8030 = '%QD93'; Type_8030 = 'DINT'; AddressPointer_8030 = ADR(%QD93); AdrOffset_8040 = 376; BitOffset_8040 = 0; BitLength_8040 = 16; Address_8040 = '%QW188'; Type_8040 = 'INT'; AddressPointer_8040 = ADR(%QW188); AdrOffset_8050 = 378; BitOffset_8050 = 0; BitLength_8050 = 8; Address_8050 = '%QB378'; Type_8050 = 'SINT'; AddressPointer_8050 = ADR(%QB378); AdrOffset_8060 = 380; BitOffset_8060 = 0; BitLength_8060 = 16; Address_8060 = '%QW190'; Type_8060 = 'UINT'; AddressPointer_8060 = ADR(%QW190); AdrOffset_8070 = 4294967295; BitOffset_8070 = 0; BitLength_8070 = 0; Address_8070 = '';
              Type_8070 = ''; AddressPointer_8070 = 0; AdrOffset_8080 = 4294967295; BitOffset_8080 = 0; BitLength_8080 = 0; Address_8080 = ''; Type_8080 = ''; AddressPointer_8080 = 0; AdrOffset_8090 = 4294967295; BitOffset_8090 = 0; BitLength_8090 = 0; Address_8090 = ''; Type_8090 = ''; AddressPointer_8090 = 0; AdrOffset_8100 = 384; BitOffset_8100 = 0; BitLength_8100 = 32; Address_8100 = '%QD96'; Type_8100 = 'UDINT'; AddressPointer_8100 = ADR(%QD96); AdrOffset_8510 = 574; BitOffset_8510 = 0; BitLength_8510 = 16; Address_8510 = '%IW287'; Type_8510 = 'UINT'; AddressPointer_8510 = ADR(%IW287); AdrOffset_8520 = 576; BitOffset_8520 = 0; BitLength_8520 = 32; Address_8520 = '%ID144'; Type_8520 = 'DINT'; AddressPointer_8520 = ADR(%ID144); AdrOffset_8530 = 604; BitOffset_8530 = 0; BitLength_8530 = 32; Address_8530 = '%ID151'; Type_8530 = 'DINT'; AddressPointer_8530 = ADR(%ID151); AdrOffset_8540 = 580; BitOffset_8540 = 0;
              BitLength_8540 = 16; Address_8540 = '%IW290'; Type_8540 = 'INT'; AddressPointer_8540 = ADR(%IW290); AdrOffset_8550 = 4294967295; BitOffset_8550 = 0; BitLength_8550 = 0; Address_8550 = ''; Type_8550 = ''; AddressPointer_8550 = 0; AdrOffset_8560 = 600; BitOffset_8560 = 0; BitLength_8560 = 32; Address_8560 = '%ID150'; Type_8560 = 'UDINT'; AddressPointer_8560 = ADR(%ID150); AdrOffset_8570 = 588; BitOffset_8570 = 0; BitLength_8570 = 16; Address_8570 = '%IW294'; Type_8570 = 'UINT'; AddressPointer_8570 = ADR(%IW294); AdrOffset_8580 = 592; BitOffset_8580 = 0; BitLength_8580 = 32; Address_8580 = '%ID148'; Type_8580 = 'DINT'; AddressPointer_8580 = ADR(%ID148); AdrOffset_8590 = 4294967295; BitOffset_8590 = 0; BitLength_8590 = 0; Address_8590 = ''; Type_8590 = ''; AddressPointer_8590 = 0; AdrOffset_8600 = 596; BitOffset_8600 = 0; BitLength_8600 = 32; Address_8600 = '%ID149'; Type_8600 = 'DINT'; AddressPointer_8600 = ADR(%ID149);
              AdrOffset_8600 = 4294967295; BitOffset_8600 = 0; BitLength_8600 = 0; Address_8610 = ''; Type_8610 = ''; AddressPointer_8610 = 0; AdrOffset_8620 = 572; BitOffset_8620 = 0; BitLength_8620 = 16; Address_8620 = '%IW286'; Type_8620 = 'UINT'; AddressPointer_8620 = ADR(%IW286); Automatic Mapping = True; IsValid = True; IsHostHoming = False; PulseSelectIndex = 2
      InoSV630N_右上轮 : SV630_1Axis_03715, Inovance, order no. InoSV630N, version Revision=16#00010000
          settings: Number of Outputs = 7; Number of Inputs = 10; Number of Infos about Outputs = 7; Number of Infos about Inputs = 10; EnableExpertSettings = True; Physical Address of the Slave = 1014; AutoIncr Address of the Slave = 4294967283; StationAlias = 0; Sync.Length = 19; Sync.Length = 32; FMMU.Global Start Address = 16#020000E0; FMMU.Length = 19; FMMU.Physical Start Address = 16#1800; FMMU.Access = 16#02; FMMU.Global Start Address = 16#0100019E; FMMU.Length = 32; FMMU.Physical Start Address = 16#1C00; FMMU.Access = 16#01; FMMU.Global Start Address = 16#00080001; FMMU.StartBit = 4; FMMU.EndBit = 4; FMMU.Physical Start Address = 16#080D; FMMU.Access = 16#01; AutoUpdate = False; DC sync0 cycletime = 4000; DC sync0 cycletime = 4000000; DC sync1 cycletime = 4000; DC sync1 cycletime = 4000000; Number of SDO = 10; Homing method.Index = 16#6098; Homing method.Subindex = 16#00; Homing method.Value = 1; Homing method.Size = 8; Homing method.AbortIfError = FALSE; Homing method.JumpToLine = FALSE; Homing method.Line = 0; Homing method.CompleteAccess = FALSE; Actual Position Calculation Method.Index = 16#60E6; Actual Position Calculation Method.Subindex = 16#00; Actual Position Calculation Method.Value = 0;
            Actual Position Calculation Method.Size = 8; Actual Position Calculation Method.AbortIfError = FALSE; Actual Position Calculation Method.JumpToLine = FALSE; Actual Position Calculation Method.Line = 0; Actual Position Calculation Method.CompleteAccess = FALSE; Speed during search for switch.Index = 16#6099; Speed during search for switch.Subindex = 16#01; Speed during search for switch.Value = 11031; Speed during search for switch.Size = 32; Speed during search for switch.AbortIfError = FALSE; Speed during search for switch.JumpToLine = FALSE; Speed during search for switch.Line = 0; Speed during search for switch.CompleteAccess = FALSE; Homing acceleration.Index = 16#609A; Homing acceleration.Subindex = 16#00; Homing acceleration.Value = 1103102; Homing acceleration.Size = 32; Homing acceleration.AbortIfError = FALSE; Homing acceleration.JumpToLine = FALSE; Homing acceleration.Line = 0; Homing acceleration.CompleteAccess = FALSE; Speed during search for zero.Index = 16#6099; Speed during search for zero.Subindex = 16#02; Speed during search for zero.Value = 1103; Speed during search for zero.Size = 32; Speed during search for zero.AbortIfError = FALSE; Speed during search for zero.JumpToLine = FALSE; Speed during search for zero.Line = 0; Speed during search for zero.CompleteAccess = FALSE; Time of home searching.Index = 16#2005; Time of home searching.Subindex = 16#24; Time of home searching.Value = 50000; Time of home searching.Size = 16; Time of home searching.AbortIfError = FALSE; Time of home searching.JumpToLine = FALSE; Time of home searching.Line = 0; Time of home searching.CompleteAccess = FALSE; Positive torque limit value.Index = 16#60E0; Positive torque limit value.Subindex = 16#00; Positive torque limit value.Value = 3500;
            Positive torque limit value.Size = 16; Positive torque limit value.AbortIfError = FALSE; Positive torque limit value.JumpToLine = FALSE; Positive torque limit value.Line = 0; Positive torque limit value.CompleteAccess = FALSE; Negative torque limit value.Index = 16#60E1; Negative torque limit value.Subindex = 16#00; Negative torque limit value.Value = 3500; Negative torque limit value.Size = 16; Negative torque limit value.AbortIfError = FALSE; Negative torque limit value.JumpToLine = FALSE; Negative torque limit value.Line = 0; Negative torque limit value.CompleteAccess = FALSE; Max profile velocity.Index = 16#607F; Max profile velocity.Subindex = 16#00; Max profile velocity.Value = 661861; Max profile velocity.Size = 32; Max profile velocity.AbortIfError = FALSE; Max profile velocity.JumpToLine = FALSE; Max profile velocity.Line = 0; Max profile velocity.CompleteAccess = FALSE; RxTxPdo.NumberofEntries = 7; RxTxPdo.DependOnSlot = False; RxTxPdo.DependOnSlotGroup = False; RxTxPdo.OverwrittenByModule = False; Exclude = [16#1701,16#1702,16#1703,16#1704,16#1705]; Controlword.Index = 16#6040; Controlword.SubIndex = 0; Controlword.Size = 16; Controlword.Offset = 0; Controlword.DependOnSlot = False; Controlword.DependOnSlotGroup = False; Target position.Index = 16#607A; Target position.SubIndex = 0; Target position.Size = 32; Target position.Offset = 0; Target position.DependOnSlot = False; Target position.DependOnSlotGroup = False; Touch probe function.Index = 16#60B8; Touch probe function.SubIndex = 0;
            Touch probe function.Size = 16; Touch probe function.Offset = 0; Touch probe function.DependOnSlot = False; Touch probe function.DependOnSlotGroup = False; Physical outputs.Index = 16#60FE; Physical outputs.SubIndex = 1; Physical outputs.Size = 32; Physical outputs.Offset = 0; Physical outputs.DependOnSlot = False; Physical outputs.DependOnSlotGroup = False; Target velocity.Index = 16#60FF; Target velocity.SubIndex = 0; Target velocity.Size = 32; Target velocity.Offset = 0; Target velocity.DependOnSlot = False; Target velocity.DependOnSlotGroup = False; Modes of operation.Index = 16#6060; Modes of operation.SubIndex = 0; Modes of operation.Size = 8; Modes of operation.Offset = 0; Modes of operation.DependOnSlot = False; Modes of operation.DependOnSlotGroup = False; Target torque.Index = 16#6071; Target torque.SubIndex = 0; Target torque.Size = 16; Target torque.Offset = 0; Target torque.DependOnSlot = False; Target torque.DependOnSlotGroup = False; RxTxPdo.Sm = -1; RxTxPdo.Sm = 2; RxTxPdo.NumberofEntries = 10; RxTxPdo.Sm = 3; Error code.Index = 16#603F; Error code.SubIndex = 0; Error code.Size = 16; Error code.DependOnSlot = false; Error code.DependOnSlotGroup = false; Statusword.Index = 16#6041; Statusword.SubIndex = 0; Statusword.Size = 16;
            Statusword.DependOnSlot = false; Statusword.DependOnSlotGroup = false; Position actual value.Index = 16#6064; Position actual value.SubIndex = 0; Position actual value.Size = 32; Position actual value.DependOnSlot = false; Position actual value.DependOnSlotGroup = false; Torque actual value.Index = 16#6077; Torque actual value.SubIndex = 0; Torque actual value.Size = 16; Torque actual value.DependOnSlot = false; Torque actual value.DependOnSlotGroup = false; Following error actual value.Index = 16#60F4; Following error actual value.SubIndex = 0; Following error actual value.Size = 32; Following error actual value.DependOnSlot = false; Following error actual value.DependOnSlotGroup = false; Touch probe status.Index = 16#60B9; Touch probe status.SubIndex = 0; Touch probe status.Size = 16; Touch probe status.DependOnSlot = false; Touch probe status.DependOnSlotGroup = false; Touch probe pos1 pos value.Index = 16#60BA; Touch probe pos1 pos value.SubIndex = 0; Touch probe pos1 pos value.Size = 32; Touch probe pos1 pos value.DependOnSlot = false; Touch probe pos1 pos value.DependOnSlotGroup = false; Touch probe pos2 pos value.Index = 16#60BC; Touch probe pos2 pos value.SubIndex = 0; Touch probe pos2 pos value.Size = 32; Touch probe pos2 pos value.DependOnSlot = false; Touch probe pos2 pos value.DependOnSlotGroup = false; Digital inputs.Index = 16#60FD; Digital inputs.SubIndex = 0; Digital inputs.Size = 32; Digital inputs.DependOnSlot = false; Digital inputs.DependOnSlotGroup = false; Velocity actual value.Index = 16#606C; Velocity actual value.SubIndex = 0; Velocity actual value.Size = 32;
            Velocity actual value.DependOnSlot = false; Velocity actual value.DependOnSlotGroup = false; RxTxPdo.Sm = -1; Controlword.Name = 'Controlword'; Controlword.DataType = 'UINT'; Controlword.Default = ''; Controlword.Comment = ''; Target position.Name = 'Target position'; Target position.DataType = 'DINT'; Target position.Default = ''; Target position.Comment = ''; Touch probe function.Name = 'Touch probe function'; Touch probe function.DataType = 'UINT'; Touch probe function.Default = ''; Touch probe function.Comment = ''; Physical outputs.Name = 'Physical outputs'; Physical outputs.DataType = 'UDINT'; Physical outputs.Default = ''; Physical outputs.Comment = ''; Target velocity.Name = 'Target velocity'; Target velocity.DataType = 'DINT'; Target velocity.Default = ''; Target velocity.Comment = ''; Modes of operation.Name = 'Modes of operation'; Modes of operation.DataType = 'SINT'; Modes of operation.Default = ''; Modes of operation.Comment = ''; Target torque.Name = 'Target torque'; Target torque.DataType = 'INT'; Target torque.Default = ''; Target torque.Comment = ''; Error code.Name = 'Error code'; Error code.DataType = 'UINT'; Statusword.Name = 'Statusword'; Statusword.DataType = 'UINT'; Position actual value.Name = 'Position actual value'; Position actual value.DataType = 'DINT'; Torque actual value.Name = 'Torque actual value'; Torque actual value.DataType = 'INT'; Following error actual value.Name = 'Following error actual value';
            Following error actual value.DataType = 'DINT'; Touch probe status.Name = 'Touch probe status'; Touch probe status.DataType = 'UINT'; Touch probe pos1 pos value.Name = 'Touch probe pos1 pos value'; Touch probe pos1 pos value.DataType = 'DINT'; Touch probe pos2 pos value.Name = 'Touch probe pos2 pos value'; Touch probe pos2 pos value.DataType = 'DINT'; Digital inputs.Name = 'Digital inputs'; Digital inputs.DataType = 'UDINT'; Velocity actual value.Name = 'Velocity actual value'; Velocity actual value.DataType = 'DINT'
          output Application.右上轮最大轮廓速度 : UDINT  // Max profile velocity
          unmapped channels: Controlword, Target position, Target velocity, Target torque, Modes of operation, Touch probe function, Error code, Statusword, Position actual value, Torque actual value, Following error actual value, Touch probe status, Touch probe pos1 pos value, Touch probe pos2 pos value, Digital inputs, Velocity actual value
        右上轮 : Axis, Inovance, order no. 0, version 1.0.0.0
            settings: wDriveID = 26; dwRatioTechUnitsDenom = 2621440000; iRatioTechUnitsNum = 396071; fSWMaxVelocity = 1000; fSWMaxAcceleration = 10000; fSWMaxDeceleration = 10000; fSWMaxJerk = 100000; iEncoderType = 1; iAbsEncoderOption = 1; HomingMode = 10; ZeroSignal = 0; StartDirction = 1; EndDirection = 1; PosLimitMode = 0; NegLimitMode = 0; HomingVelocity = 10; HomingApproachVelocity = 2; HomingAcceleration = 100; HomingDeceleration = 100; HomingJerk = 0; HomeMaskDistance = 0; HomePositionOffset = 0; HomePushTime = 0; HomeCompensation = 0; HomeTimeout = 0; HomeCompensationVelocity = 1000; 4000 = 1; 4001 = 0; 4003 = true; 4004 = 3; 4005 = 0; 4006 = 1.666667; 4007 = 166.666666; 4008 = 0.166667; 4009 = 50000; 4010 = 3500; 4011 = 3500; 4012 = 100.000000; ScalingIncs = 16#40000; 6005 = 39.6071;
              AdrOffset_8010 = 292; BitOffset_8010 = 0; BitLength_8010 = 16; Address_8010 = '%QW146'; Type_8010 = 'UINT'; AddressPointer_8010 = ADR(%QW146); AdrOffset_8020 = 296; BitOffset_8020 = 0; BitLength_8020 = 32; Address_8020 = '%QD74'; Type_8020 = 'DINT'; AddressPointer_8020 = ADR(%QD74); AdrOffset_8030 = 300; BitOffset_8030 = 0; BitLength_8030 = 32; Address_8030 = '%QD75'; Type_8030 = 'DINT'; AddressPointer_8030 = ADR(%QD75); AdrOffset_8040 = 304; BitOffset_8040 = 0; BitLength_8040 = 16; Address_8040 = '%QW152'; Type_8040 = 'INT'; AddressPointer_8040 = ADR(%QW152); AdrOffset_8050 = 306; BitOffset_8050 = 0; BitLength_8050 = 8; Address_8050 = '%QB306'; Type_8050 = 'SINT'; AddressPointer_8050 = ADR(%QB306); AdrOffset_8060 = 308; BitOffset_8060 = 0; BitLength_8060 = 16; Address_8060 = '%QW154'; Type_8060 = 'UINT'; AddressPointer_8060 = ADR(%QW154); AdrOffset_8070 = 4294967295; BitOffset_8070 = 0; BitLength_8070 = 0; Address_8070 = '';
              Type_8070 = ''; AddressPointer_8070 = 0; AdrOffset_8080 = 4294967295; BitOffset_8080 = 0; BitLength_8080 = 0; Address_8080 = ''; Type_8080 = ''; AddressPointer_8080 = 0; AdrOffset_8090 = 4294967295; BitOffset_8090 = 0; BitLength_8090 = 0; Address_8090 = ''; Type_8090 = ''; AddressPointer_8090 = 0; AdrOffset_8100 = 0; BitOffset_8100 = 0; BitLength_8100 = 32; Address_8100 = '右上轮最大轮廓速度'; Type_8100 = 'UDINT'; AddressPointer_8100 = ADR(右上轮最大轮廓速度); AdrOffset_8510 = 466; BitOffset_8510 = 0; BitLength_8510 = 16; Address_8510 = '%IW233'; Type_8510 = 'UINT'; AddressPointer_8510 = ADR(%IW233); AdrOffset_8520 = 468; BitOffset_8520 = 0; BitLength_8520 = 32; Address_8520 = '%ID117'; Type_8520 = 'DINT'; AddressPointer_8520 = ADR(%ID117); AdrOffset_8530 = 496; BitOffset_8530 = 0; BitLength_8530 = 32; Address_8530 = '%ID124'; Type_8530 = 'DINT'; AddressPointer_8530 = ADR(%ID124); AdrOffset_8540 = 472; BitOffset_8540 = 0;
              BitLength_8540 = 16; Address_8540 = '%IW236'; Type_8540 = 'INT'; AddressPointer_8540 = ADR(%IW236); AdrOffset_8550 = 4294967295; BitOffset_8550 = 0; BitLength_8550 = 0; Address_8550 = ''; Type_8550 = ''; AddressPointer_8550 = 0; AdrOffset_8560 = 492; BitOffset_8560 = 0; BitLength_8560 = 32; Address_8560 = '%ID123'; Type_8560 = 'UDINT'; AddressPointer_8560 = ADR(%ID123); AdrOffset_8570 = 480; BitOffset_8570 = 0; BitLength_8570 = 16; Address_8570 = '%IW240'; Type_8570 = 'UINT'; AddressPointer_8570 = ADR(%IW240); AdrOffset_8580 = 484; BitOffset_8580 = 0; BitLength_8580 = 32; Address_8580 = '%ID121'; Type_8580 = 'DINT'; AddressPointer_8580 = ADR(%ID121); AdrOffset_8590 = 4294967295; BitOffset_8590 = 0; BitLength_8590 = 0; Address_8590 = ''; Type_8590 = ''; AddressPointer_8590 = 0; AdrOffset_8600 = 488; BitOffset_8600 = 0; BitLength_8600 = 32; Address_8600 = '%ID122'; Type_8600 = 'DINT'; AddressPointer_8600 = ADR(%ID122);
              AdrOffset_8600 = 4294967295; BitOffset_8600 = 0; BitLength_8600 = 0; Address_8610 = ''; Type_8610 = ''; AddressPointer_8610 = 0; AdrOffset_8620 = 464; BitOffset_8620 = 0; BitLength_8620 = 16; Address_8620 = '%IW232'; Type_8620 = 'UINT'; AddressPointer_8620 = ADR(%IW232); Automatic Mapping = True; IsValid = True; IsHostHoming = False; PulseSelectIndex = 2
      InoSV630N_右下轮 : SV630_1Axis_03715, Inovance, order no. InoSV630N, version Revision=16#00010000
          settings: Number of Outputs = 7; Number of Inputs = 10; Number of Infos about Outputs = 7; Number of Infos about Inputs = 10; EnableExpertSettings = True; Physical Address of the Slave = 1015; AutoIncr Address of the Slave = 4294967282; StationAlias = 0; Sync.Length = 19; Sync.Length = 32; FMMU.Global Start Address = 16#020000F3; FMMU.Length = 19; FMMU.Physical Start Address = 16#1800; FMMU.Access = 16#02; FMMU.Global Start Address = 16#010001BE; FMMU.Length = 32; FMMU.Physical Start Address = 16#1C00; FMMU.Access = 16#01; FMMU.Global Start Address = 16#00080001; FMMU.StartBit = 5; FMMU.EndBit = 5; FMMU.Physical Start Address = 16#080D; FMMU.Access = 16#01; AutoUpdate = False; DC sync0 cycletime = 4000; DC sync0 cycletime = 4000000; DC sync1 cycletime = 4000; DC sync1 cycletime = 4000000; Number of SDO = 10; Homing method.Index = 16#6098; Homing method.Subindex = 16#00; Homing method.Value = 1; Homing method.Size = 8; Homing method.AbortIfError = FALSE; Homing method.JumpToLine = FALSE; Homing method.Line = 0; Homing method.CompleteAccess = FALSE; Actual Position Calculation Method.Index = 16#60E6; Actual Position Calculation Method.Subindex = 16#00; Actual Position Calculation Method.Value = 0;
            Actual Position Calculation Method.Size = 8; Actual Position Calculation Method.AbortIfError = FALSE; Actual Position Calculation Method.JumpToLine = FALSE; Actual Position Calculation Method.Line = 0; Actual Position Calculation Method.CompleteAccess = FALSE; Speed during search for switch.Index = 16#6099; Speed during search for switch.Subindex = 16#01; Speed during search for switch.Value = 11031; Speed during search for switch.Size = 32; Speed during search for switch.AbortIfError = FALSE; Speed during search for switch.JumpToLine = FALSE; Speed during search for switch.Line = 0; Speed during search for switch.CompleteAccess = FALSE; Homing acceleration.Index = 16#609A; Homing acceleration.Subindex = 16#00; Homing acceleration.Value = 1103102; Homing acceleration.Size = 32; Homing acceleration.AbortIfError = FALSE; Homing acceleration.JumpToLine = FALSE; Homing acceleration.Line = 0; Homing acceleration.CompleteAccess = FALSE; Speed during search for zero.Index = 16#6099; Speed during search for zero.Subindex = 16#02; Speed during search for zero.Value = 1103; Speed during search for zero.Size = 32; Speed during search for zero.AbortIfError = FALSE; Speed during search for zero.JumpToLine = FALSE; Speed during search for zero.Line = 0; Speed during search for zero.CompleteAccess = FALSE; Time of home searching.Index = 16#2005; Time of home searching.Subindex = 16#24; Time of home searching.Value = 50000; Time of home searching.Size = 16; Time of home searching.AbortIfError = FALSE; Time of home searching.JumpToLine = FALSE; Time of home searching.Line = 0; Time of home searching.CompleteAccess = FALSE; Positive torque limit value.Index = 16#60E0; Positive torque limit value.Subindex = 16#00; Positive torque limit value.Value = 3500;
            Positive torque limit value.Size = 16; Positive torque limit value.AbortIfError = FALSE; Positive torque limit value.JumpToLine = FALSE; Positive torque limit value.Line = 0; Positive torque limit value.CompleteAccess = FALSE; Negative torque limit value.Index = 16#60E1; Negative torque limit value.Subindex = 16#00; Negative torque limit value.Value = 3500; Negative torque limit value.Size = 16; Negative torque limit value.AbortIfError = FALSE; Negative torque limit value.JumpToLine = FALSE; Negative torque limit value.Line = 0; Negative torque limit value.CompleteAccess = FALSE; Max profile velocity.Index = 16#607F; Max profile velocity.Subindex = 16#00; Max profile velocity.Value = 661861; Max profile velocity.Size = 32; Max profile velocity.AbortIfError = FALSE; Max profile velocity.JumpToLine = FALSE; Max profile velocity.Line = 0; Max profile velocity.CompleteAccess = FALSE; RxTxPdo.NumberofEntries = 7; RxTxPdo.DependOnSlot = False; RxTxPdo.DependOnSlotGroup = False; RxTxPdo.OverwrittenByModule = False; Exclude = [16#1701,16#1702,16#1703,16#1704,16#1705]; Controlword.Index = 16#6040; Controlword.SubIndex = 0; Controlword.Size = 16; Controlword.Offset = 0; Controlword.DependOnSlot = False; Controlword.DependOnSlotGroup = False; Target position.Index = 16#607A; Target position.SubIndex = 0; Target position.Size = 32; Target position.Offset = 0; Target position.DependOnSlot = False; Target position.DependOnSlotGroup = False; Touch probe function.Index = 16#60B8; Touch probe function.SubIndex = 0;
            Touch probe function.Size = 16; Touch probe function.Offset = 0; Touch probe function.DependOnSlot = False; Touch probe function.DependOnSlotGroup = False; Physical outputs.Index = 16#60FE; Physical outputs.SubIndex = 1; Physical outputs.Size = 32; Physical outputs.Offset = 0; Physical outputs.DependOnSlot = False; Physical outputs.DependOnSlotGroup = False; Target velocity.Index = 16#60FF; Target velocity.SubIndex = 0; Target velocity.Size = 32; Target velocity.Offset = 0; Target velocity.DependOnSlot = False; Target velocity.DependOnSlotGroup = False; Modes of operation.Index = 16#6060; Modes of operation.SubIndex = 0; Modes of operation.Size = 8; Modes of operation.Offset = 0; Modes of operation.DependOnSlot = False; Modes of operation.DependOnSlotGroup = False; Target torque.Index = 16#6071; Target torque.SubIndex = 0; Target torque.Size = 16; Target torque.Offset = 0; Target torque.DependOnSlot = False; Target torque.DependOnSlotGroup = False; RxTxPdo.Sm = -1; RxTxPdo.Sm = 2; RxTxPdo.NumberofEntries = 10; RxTxPdo.Sm = 3; Error code.Index = 16#603F; Error code.SubIndex = 0; Error code.Size = 16; Error code.DependOnSlot = false; Error code.DependOnSlotGroup = false; Statusword.Index = 16#6041; Statusword.SubIndex = 0; Statusword.Size = 16;
            Statusword.DependOnSlot = false; Statusword.DependOnSlotGroup = false; Position actual value.Index = 16#6064; Position actual value.SubIndex = 0; Position actual value.Size = 32; Position actual value.DependOnSlot = false; Position actual value.DependOnSlotGroup = false; Torque actual value.Index = 16#6077; Torque actual value.SubIndex = 0; Torque actual value.Size = 16; Torque actual value.DependOnSlot = false; Torque actual value.DependOnSlotGroup = false; Following error actual value.Index = 16#60F4; Following error actual value.SubIndex = 0; Following error actual value.Size = 32; Following error actual value.DependOnSlot = false; Following error actual value.DependOnSlotGroup = false; Touch probe status.Index = 16#60B9; Touch probe status.SubIndex = 0; Touch probe status.Size = 16; Touch probe status.DependOnSlot = false; Touch probe status.DependOnSlotGroup = false; Touch probe pos1 pos value.Index = 16#60BA; Touch probe pos1 pos value.SubIndex = 0; Touch probe pos1 pos value.Size = 32; Touch probe pos1 pos value.DependOnSlot = false; Touch probe pos1 pos value.DependOnSlotGroup = false; Touch probe pos2 pos value.Index = 16#60BC; Touch probe pos2 pos value.SubIndex = 0; Touch probe pos2 pos value.Size = 32; Touch probe pos2 pos value.DependOnSlot = false; Touch probe pos2 pos value.DependOnSlotGroup = false; Digital inputs.Index = 16#60FD; Digital inputs.SubIndex = 0; Digital inputs.Size = 32; Digital inputs.DependOnSlot = false; Digital inputs.DependOnSlotGroup = false; Velocity actual value.Index = 16#606C; Velocity actual value.SubIndex = 0; Velocity actual value.Size = 32;
            Velocity actual value.DependOnSlot = false; Velocity actual value.DependOnSlotGroup = false; RxTxPdo.Sm = -1; Controlword.Name = 'Controlword'; Controlword.DataType = 'UINT'; Controlword.Default = ''; Controlword.Comment = ''; Target position.Name = 'Target position'; Target position.DataType = 'DINT'; Target position.Default = ''; Target position.Comment = ''; Touch probe function.Name = 'Touch probe function'; Touch probe function.DataType = 'UINT'; Touch probe function.Default = ''; Touch probe function.Comment = ''; Physical outputs.Name = 'Physical outputs'; Physical outputs.DataType = 'UDINT'; Physical outputs.Default = ''; Physical outputs.Comment = ''; Target velocity.Name = 'Target velocity'; Target velocity.DataType = 'DINT'; Target velocity.Default = ''; Target velocity.Comment = ''; Modes of operation.Name = 'Modes of operation'; Modes of operation.DataType = 'SINT'; Modes of operation.Default = ''; Modes of operation.Comment = ''; Target torque.Name = 'Target torque'; Target torque.DataType = 'INT'; Target torque.Default = ''; Target torque.Comment = ''; Error code.Name = 'Error code'; Error code.DataType = 'UINT'; Statusword.Name = 'Statusword'; Statusword.DataType = 'UINT'; Position actual value.Name = 'Position actual value'; Position actual value.DataType = 'DINT'; Torque actual value.Name = 'Torque actual value'; Torque actual value.DataType = 'INT'; Following error actual value.Name = 'Following error actual value';
            Following error actual value.DataType = 'DINT'; Touch probe status.Name = 'Touch probe status'; Touch probe status.DataType = 'UINT'; Touch probe pos1 pos value.Name = 'Touch probe pos1 pos value'; Touch probe pos1 pos value.DataType = 'DINT'; Touch probe pos2 pos value.Name = 'Touch probe pos2 pos value'; Touch probe pos2 pos value.DataType = 'DINT'; Digital inputs.Name = 'Digital inputs'; Digital inputs.DataType = 'UDINT'; Velocity actual value.Name = 'Velocity actual value'; Velocity actual value.DataType = 'DINT'
          unmapped channels: Controlword, Target position, Target velocity, Target torque, Modes of operation, Touch probe function, Max profile velocity, Error code, Statusword, Position actual value, Torque actual value, Following error actual value, Touch probe status, Touch probe pos1 pos value, Touch probe pos2 pos value, Digital inputs, Velocity actual value
        右下轮 : Axis, Inovance, order no. 0, version 1.0.0.0
            settings: wDriveID = 27; dwRatioTechUnitsDenom = 2621440000; iRatioTechUnitsNum = 396071; fSWMaxVelocity = 1000; fSWMaxAcceleration = 10000; fSWMaxDeceleration = 10000; fSWMaxJerk = 100000; iEncoderType = 1; iAbsEncoderOption = 1; HomingMode = 10; ZeroSignal = 0; StartDirction = 1; EndDirection = 1; PosLimitMode = 0; NegLimitMode = 0; HomingVelocity = 10; HomingApproachVelocity = 2; HomingAcceleration = 100; HomingDeceleration = 100; HomingJerk = 0; HomeMaskDistance = 0; HomePositionOffset = 0; HomePushTime = 0; HomeCompensation = 0; HomeTimeout = 0; HomeCompensationVelocity = 1000; 4000 = 1; 4001 = 0; 4003 = true; 4004 = 3; 4005 = 0; 4006 = 1.666667; 4007 = 166.666666; 4008 = 0.166667; 4009 = 50000; 4010 = 3500; 4011 = 3500; 4012 = 100.000000; ScalingIncs = 16#40000; 6005 = 39.6071;
              AdrOffset_8010 = 316; BitOffset_8010 = 0; BitLength_8010 = 16; Address_8010 = '%QW158'; Type_8010 = 'UINT'; AddressPointer_8010 = ADR(%QW158); AdrOffset_8020 = 320; BitOffset_8020 = 0; BitLength_8020 = 32; Address_8020 = '%QD80'; Type_8020 = 'DINT'; AddressPointer_8020 = ADR(%QD80); AdrOffset_8030 = 324; BitOffset_8030 = 0; BitLength_8030 = 32; Address_8030 = '%QD81'; Type_8030 = 'DINT'; AddressPointer_8030 = ADR(%QD81); AdrOffset_8040 = 328; BitOffset_8040 = 0; BitLength_8040 = 16; Address_8040 = '%QW164'; Type_8040 = 'INT'; AddressPointer_8040 = ADR(%QW164); AdrOffset_8050 = 330; BitOffset_8050 = 0; BitLength_8050 = 8; Address_8050 = '%QB330'; Type_8050 = 'SINT'; AddressPointer_8050 = ADR(%QB330); AdrOffset_8060 = 332; BitOffset_8060 = 0; BitLength_8060 = 16; Address_8060 = '%QW166'; Type_8060 = 'UINT'; AddressPointer_8060 = ADR(%QW166); AdrOffset_8070 = 4294967295; BitOffset_8070 = 0; BitLength_8070 = 0; Address_8070 = '';
              Type_8070 = ''; AddressPointer_8070 = 0; AdrOffset_8080 = 4294967295; BitOffset_8080 = 0; BitLength_8080 = 0; Address_8080 = ''; Type_8080 = ''; AddressPointer_8080 = 0; AdrOffset_8090 = 4294967295; BitOffset_8090 = 0; BitLength_8090 = 0; Address_8090 = ''; Type_8090 = ''; AddressPointer_8090 = 0; AdrOffset_8100 = 336; BitOffset_8100 = 0; BitLength_8100 = 32; Address_8100 = '%QD84'; Type_8100 = 'UDINT'; AddressPointer_8100 = ADR(%QD84); AdrOffset_8510 = 502; BitOffset_8510 = 0; BitLength_8510 = 16; Address_8510 = '%IW251'; Type_8510 = 'UINT'; AddressPointer_8510 = ADR(%IW251); AdrOffset_8520 = 504; BitOffset_8520 = 0; BitLength_8520 = 32; Address_8520 = '%ID126'; Type_8520 = 'DINT'; AddressPointer_8520 = ADR(%ID126); AdrOffset_8530 = 532; BitOffset_8530 = 0; BitLength_8530 = 32; Address_8530 = '%ID133'; Type_8530 = 'DINT'; AddressPointer_8530 = ADR(%ID133); AdrOffset_8540 = 508; BitOffset_8540 = 0;
              BitLength_8540 = 16; Address_8540 = '%IW254'; Type_8540 = 'INT'; AddressPointer_8540 = ADR(%IW254); AdrOffset_8550 = 4294967295; BitOffset_8550 = 0; BitLength_8550 = 0; Address_8550 = ''; Type_8550 = ''; AddressPointer_8550 = 0; AdrOffset_8560 = 528; BitOffset_8560 = 0; BitLength_8560 = 32; Address_8560 = '%ID132'; Type_8560 = 'UDINT'; AddressPointer_8560 = ADR(%ID132); AdrOffset_8570 = 516; BitOffset_8570 = 0; BitLength_8570 = 16; Address_8570 = '%IW258'; Type_8570 = 'UINT'; AddressPointer_8570 = ADR(%IW258); AdrOffset_8580 = 520; BitOffset_8580 = 0; BitLength_8580 = 32; Address_8580 = '%ID130'; Type_8580 = 'DINT'; AddressPointer_8580 = ADR(%ID130); AdrOffset_8590 = 4294967295; BitOffset_8590 = 0; BitLength_8590 = 0; Address_8590 = ''; Type_8590 = ''; AddressPointer_8590 = 0; AdrOffset_8600 = 524; BitOffset_8600 = 0; BitLength_8600 = 32; Address_8600 = '%ID131'; Type_8600 = 'DINT'; AddressPointer_8600 = ADR(%ID131);
              AdrOffset_8600 = 4294967295; BitOffset_8600 = 0; BitLength_8600 = 0; Address_8610 = ''; Type_8610 = ''; AddressPointer_8610 = 0; AdrOffset_8620 = 500; BitOffset_8620 = 0; BitLength_8620 = 16; Address_8620 = '%IW250'; Type_8620 = 'UINT'; AddressPointer_8620 = ADR(%IW250); Automatic Mapping = True; IsValid = True; IsHostHoming = False; PulseSelectIndex = 2
      InoSV630N_左上气缸 : SV630_1Axis_03715, Inovance, order no. InoSV630N, version Revision=16#00010000
          settings: Number of Outputs = 7; Number of Inputs = 10; Number of Infos about Outputs = 7; Number of Infos about Inputs = 10; EnableExpertSettings = True; Physical Address of the Slave = 1012; AutoIncr Address of the Slave = 4294967285; StationAlias = 0; Sync.Length = 19; Sync.Length = 32; FMMU.Global Start Address = 16#020000BA; FMMU.Length = 19; FMMU.Physical Start Address = 16#1800; FMMU.Access = 16#02; FMMU.Global Start Address = 16#0100015E; FMMU.Length = 32; FMMU.Physical Start Address = 16#1C00; FMMU.Access = 16#01; FMMU.Global Start Address = 16#00080001; FMMU.StartBit = 2; FMMU.EndBit = 2; FMMU.Physical Start Address = 16#080D; FMMU.Access = 16#01; AutoUpdate = False; DC sync0 cycletime = 4000; DC sync0 cycletime = 4000000; DC sync1 cycletime = 4000; DC sync1 cycletime = 4000000; Number of SDO = 10; Homing method.Index = 16#6098; Homing method.Subindex = 16#00; Homing method.Value = 35; Homing method.Size = 8; Homing method.AbortIfError = FALSE; Homing method.JumpToLine = FALSE; Homing method.Line = 0; Homing method.CompleteAccess = FALSE; Actual Position Calculation Method.Index = 16#60E6; Actual Position Calculation Method.Subindex = 16#00; Actual Position Calculation Method.Value = 0;
            Actual Position Calculation Method.Size = 8; Actual Position Calculation Method.AbortIfError = FALSE; Actual Position Calculation Method.JumpToLine = FALSE; Actual Position Calculation Method.Line = 0; Actual Position Calculation Method.CompleteAccess = FALSE; Speed during search for switch.Index = 16#6099; Speed during search for switch.Subindex = 16#01; Speed during search for switch.Value = 87381; Speed during search for switch.Size = 32; Speed during search for switch.AbortIfError = FALSE; Speed during search for switch.JumpToLine = FALSE; Speed during search for switch.Line = 0; Speed during search for switch.CompleteAccess = FALSE; Homing acceleration.Index = 16#609A; Homing acceleration.Subindex = 16#00; Homing acceleration.Value = 8738133; Homing acceleration.Size = 32; Homing acceleration.AbortIfError = FALSE; Homing acceleration.JumpToLine = FALSE; Homing acceleration.Line = 0; Homing acceleration.CompleteAccess = FALSE; Speed during search for zero.Index = 16#6099; Speed during search for zero.Subindex = 16#02; Speed during search for zero.Value = 8738; Speed during search for zero.Size = 32; Speed during search for zero.AbortIfError = FALSE; Speed during search for zero.JumpToLine = FALSE; Speed during search for zero.Line = 0; Speed during search for zero.CompleteAccess = FALSE; Time of home searching.Index = 16#2005; Time of home searching.Subindex = 16#24; Time of home searching.Value = 50000; Time of home searching.Size = 16; Time of home searching.AbortIfError = FALSE; Time of home searching.JumpToLine = FALSE; Time of home searching.Line = 0; Time of home searching.CompleteAccess = FALSE; Positive torque limit value.Index = 16#60E0; Positive torque limit value.Subindex = 16#00; Positive torque limit value.Value = 3500;
            Positive torque limit value.Size = 16; Positive torque limit value.AbortIfError = FALSE; Positive torque limit value.JumpToLine = FALSE; Positive torque limit value.Line = 0; Positive torque limit value.CompleteAccess = FALSE; Negative torque limit value.Index = 16#60E1; Negative torque limit value.Subindex = 16#00; Negative torque limit value.Value = 3500; Negative torque limit value.Size = 16; Negative torque limit value.AbortIfError = FALSE; Negative torque limit value.JumpToLine = FALSE; Negative torque limit value.Line = 0; Negative torque limit value.CompleteAccess = FALSE; Max profile velocity.Index = 16#607F; Max profile velocity.Subindex = 16#00; Max profile velocity.Value = 5242880; Max profile velocity.Size = 32; Max profile velocity.AbortIfError = FALSE; Max profile velocity.JumpToLine = FALSE; Max profile velocity.Line = 0; Max profile velocity.CompleteAccess = FALSE; RxTxPdo.NumberofEntries = 7; RxTxPdo.Sm = 2; RxTxPdo.DependOnSlot = False; RxTxPdo.DependOnSlotGroup = False; RxTxPdo.OverwrittenByModule = False; Exclude = [16#1701,16#1702,16#1703,16#1704,16#1705]; Controlword.Index = 16#6040; Controlword.SubIndex = 0; Controlword.Size = 16; Controlword.Offset = 0; Controlword.DependOnSlot = False; Controlword.DependOnSlotGroup = False; Target position.Index = 16#607A; Target position.SubIndex = 0; Target position.Size = 32; Target position.Offset = 0; Target position.DependOnSlot = False; Target position.DependOnSlotGroup = False; Touch probe function.Index = 16#60B8;
            Touch probe function.SubIndex = 0; Touch probe function.Size = 16; Touch probe function.Offset = 0; Touch probe function.DependOnSlot = False; Touch probe function.DependOnSlotGroup = False; Physical outputs.Index = 16#60FE; Physical outputs.SubIndex = 1; Physical outputs.Size = 32; Physical outputs.Offset = 0; Physical outputs.DependOnSlot = False; Physical outputs.DependOnSlotGroup = False; Target velocity.Index = 16#60FF; Target velocity.SubIndex = 0; Target velocity.Size = 32; Target velocity.Offset = 0; Target velocity.DependOnSlot = False; Target velocity.DependOnSlotGroup = False; Modes of operation.Index = 16#6060; Modes of operation.SubIndex = 0; Modes of operation.Size = 8; Modes of operation.Offset = 0; Modes of operation.DependOnSlot = False; Modes of operation.DependOnSlotGroup = False; Target torque.Index = 16#6071; Target torque.SubIndex = 0; Target torque.Size = 16; Target torque.Offset = 0; Target torque.DependOnSlot = False; Target torque.DependOnSlotGroup = False; RxTxPdo.Sm = -1; RxTxPdo.NumberofEntries = 10; RxTxPdo.Sm = 3; Error code.Index = 16#603F; Error code.SubIndex = 0; Error code.Size = 16; Error code.DependOnSlot = false; Error code.DependOnSlotGroup = false; Statusword.Index = 16#6041; Statusword.SubIndex = 0; Statusword.Size = 16;
            Statusword.DependOnSlot = false; Statusword.DependOnSlotGroup = false; Position actual value.Index = 16#6064; Position actual value.SubIndex = 0; Position actual value.Size = 32; Position actual value.DependOnSlot = false; Position actual value.DependOnSlotGroup = false; Torque actual value.Index = 16#6077; Torque actual value.SubIndex = 0; Torque actual value.Size = 16; Torque actual value.DependOnSlot = false; Torque actual value.DependOnSlotGroup = false; Following error actual value.Index = 16#60F4; Following error actual value.SubIndex = 0; Following error actual value.Size = 32; Following error actual value.DependOnSlot = false; Following error actual value.DependOnSlotGroup = false; Touch probe status.Index = 16#60B9; Touch probe status.SubIndex = 0; Touch probe status.Size = 16; Touch probe status.DependOnSlot = false; Touch probe status.DependOnSlotGroup = false; Touch probe pos1 pos value.Index = 16#60BA; Touch probe pos1 pos value.SubIndex = 0; Touch probe pos1 pos value.Size = 32; Touch probe pos1 pos value.DependOnSlot = false; Touch probe pos1 pos value.DependOnSlotGroup = false; Touch probe pos2 pos value.Index = 16#60BC; Touch probe pos2 pos value.SubIndex = 0; Touch probe pos2 pos value.Size = 32; Touch probe pos2 pos value.DependOnSlot = false; Touch probe pos2 pos value.DependOnSlotGroup = false; Digital inputs.Index = 16#60FD; Digital inputs.SubIndex = 0; Digital inputs.Size = 32; Digital inputs.DependOnSlot = false; Digital inputs.DependOnSlotGroup = false; Velocity actual value.Index = 16#606C; Velocity actual value.SubIndex = 0; Velocity actual value.Size = 32;
            Velocity actual value.DependOnSlot = false; Velocity actual value.DependOnSlotGroup = false; RxTxPdo.Sm = -1; Controlword.Name = 'Controlword'; Controlword.DataType = 'UINT'; Controlword.Default = ''; Controlword.Comment = ''; Target position.Name = 'Target position'; Target position.DataType = 'DINT'; Target position.Default = ''; Target position.Comment = ''; Touch probe function.Name = 'Touch probe function'; Touch probe function.DataType = 'UINT'; Touch probe function.Default = ''; Touch probe function.Comment = ''; Physical outputs.Name = 'Physical outputs'; Physical outputs.DataType = 'UDINT'; Physical outputs.Default = ''; Physical outputs.Comment = ''; Target velocity.Name = 'Target velocity'; Target velocity.DataType = 'DINT'; Target velocity.Default = ''; Target velocity.Comment = ''; Modes of operation.Name = 'Modes of operation'; Modes of operation.DataType = 'SINT'; Modes of operation.Default = ''; Modes of operation.Comment = ''; Target torque.Name = 'Target torque'; Target torque.DataType = 'INT'; Target torque.Default = ''; Target torque.Comment = ''; Error code.Name = 'Error code'; Error code.DataType = 'UINT'; Statusword.Name = 'Statusword'; Statusword.DataType = 'UINT'; Position actual value.Name = 'Position actual value'; Position actual value.DataType = 'DINT'; Torque actual value.Name = 'Torque actual value'; Torque actual value.DataType = 'INT'; Following error actual value.Name = 'Following error actual value';
            Following error actual value.DataType = 'DINT'; Touch probe status.Name = 'Touch probe status'; Touch probe status.DataType = 'UINT'; Touch probe pos1 pos value.Name = 'Touch probe pos1 pos value'; Touch probe pos1 pos value.DataType = 'DINT'; Touch probe pos2 pos value.Name = 'Touch probe pos2 pos value'; Touch probe pos2 pos value.DataType = 'DINT'; Digital inputs.Name = 'Digital inputs'; Digital inputs.DataType = 'UDINT'; Velocity actual value.Name = 'Velocity actual value'; Velocity actual value.DataType = 'DINT'
          unmapped channels: Controlword, Target position, Touch probe function, Physical outputs, Target velocity, Modes of operation, Target torque, Error code, Statusword, Position actual value, Torque actual value, Following error actual value, Touch probe status, Touch probe pos1 pos value, Touch probe pos2 pos value, Digital inputs, Velocity actual value
        左上气缸 : Axis, Inovance, order no. 0, version 1.0.0.0
            settings: wDriveID = 12; dwRatioTechUnitsDenom = 262144; iRatioTechUnitsNum = 5; fSWMaxVelocity = 1000; fSWMaxAcceleration = 10000; fSWMaxDeceleration = 10000; fSWMaxJerk = 100000; iEncoderType = 1; iAbsEncoderOption = 1; HomingMode = 10; ZeroSignal = 0; StartDirction = 1; EndDirection = 1; PosLimitMode = 0; NegLimitMode = 0; HomingVelocity = 10; HomingApproachVelocity = 2; HomingAcceleration = 100; HomingDeceleration = 100; HomingJerk = 0; HomeMaskDistance = 0; HomePositionOffset = 0; HomePushTime = 0; HomeCompensation = 0; HomeTimeout = 0; HomeCompensationVelocity = 1000; 4000 = 1; 4001 = 1; 4003 = true; 4004 = 33; 4005 = 0; 4006 = 1.666667; 4007 = 166.666666; 4008 = 0.166667; 4009 = 50000; 4010 = 3500; 4011 = 3500; 4012 = 100.000000; ScalingIncs = 16#40000; ScalingMotorTurns2 = 2;
              6005 = 10; AdrOffset_8010 = 244; BitOffset_8010 = 0; BitLength_8010 = 16; Address_8010 = '%QW122'; Type_8010 = 'UINT'; AddressPointer_8010 = ADR(%QW122); AdrOffset_8020 = 248; BitOffset_8020 = 0; BitLength_8020 = 32; Address_8020 = '%QD62'; Type_8020 = 'DINT'; AddressPointer_8020 = ADR(%QD62); AdrOffset_8030 = 260; BitOffset_8030 = 0; BitLength_8030 = 32; Address_8030 = '%QD65'; Type_8030 = 'DINT'; AddressPointer_8030 = ADR(%QD65); AdrOffset_8040 = 266; BitOffset_8040 = 0; BitLength_8040 = 16; Address_8040 = '%QW133'; Type_8040 = 'INT'; AddressPointer_8040 = ADR(%QW133); AdrOffset_8050 = 264; BitOffset_8050 = 0; BitLength_8050 = 8; Address_8050 = '%QB264'; Type_8050 = 'SINT'; AddressPointer_8050 = ADR(%QB264); AdrOffset_8060 = 252; BitOffset_8060 = 0; BitLength_8060 = 16; Address_8060 = '%QW126'; Type_8060 = 'UINT'; AddressPointer_8060 = ADR(%QW126); AdrOffset_8070 = 4294967295; BitOffset_8070 = 0; BitLength_8070 = 0;
              Address_8070 = ''; Type_8070 = ''; AddressPointer_8070 = 0; AdrOffset_8080 = 4294967295; BitOffset_8080 = 0; BitLength_8080 = 0; Address_8080 = ''; Type_8080 = ''; AddressPointer_8080 = 0; AdrOffset_8090 = 256; BitOffset_8090 = 0; BitLength_8090 = 32; Address_8090 = '%QD64'; Type_8090 = 'UDINT'; AddressPointer_8090 = ADR(%QD64); AdrOffset_8100 = 4294967295; BitOffset_8100 = 0; BitLength_8100 = 0; Address_8100 = ''; Type_8100 = ''; AddressPointer_8100 = 0; AdrOffset_8510 = 394; BitOffset_8510 = 0; BitLength_8510 = 16; Address_8510 = '%IW197'; Type_8510 = 'UINT'; AddressPointer_8510 = ADR(%IW197); AdrOffset_8520 = 396; BitOffset_8520 = 0; BitLength_8520 = 32; Address_8520 = '%ID99'; Type_8520 = 'DINT'; AddressPointer_8520 = ADR(%ID99); AdrOffset_8530 = 424; BitOffset_8530 = 0; BitLength_8530 = 32; Address_8530 = '%ID106'; Type_8530 = 'DINT'; AddressPointer_8530 = ADR(%ID106); AdrOffset_8540 = 400;
              BitOffset_8540 = 0; BitLength_8540 = 16; Address_8540 = '%IW200'; Type_8540 = 'INT'; AddressPointer_8540 = ADR(%IW200); AdrOffset_8550 = 4294967295; BitOffset_8550 = 0; BitLength_8550 = 0; Address_8550 = ''; Type_8550 = ''; AddressPointer_8550 = 0; AdrOffset_8560 = 420; BitOffset_8560 = 0; BitLength_8560 = 32; Address_8560 = '%ID105'; Type_8560 = 'UDINT'; AddressPointer_8560 = ADR(%ID105); AdrOffset_8570 = 408; BitOffset_8570 = 0; BitLength_8570 = 16; Address_8570 = '%IW204'; Type_8570 = 'UINT'; AddressPointer_8570 = ADR(%IW204); AdrOffset_8580 = 412; BitOffset_8580 = 0; BitLength_8580 = 32; Address_8580 = '%ID103'; Type_8580 = 'DINT'; AddressPointer_8580 = ADR(%ID103); AdrOffset_8590 = 4294967295; BitOffset_8590 = 0; BitLength_8590 = 0; Address_8590 = ''; Type_8590 = ''; AddressPointer_8590 = 0; AdrOffset_8600 = 416; BitOffset_8600 = 0; BitLength_8600 = 32; Address_8600 = '%ID104'; Type_8600 = 'DINT';
              AddressPointer_8600 = ADR(%ID104); AdrOffset_8600 = 4294967295; BitOffset_8600 = 0; BitLength_8600 = 0; Address_8610 = ''; Type_8610 = ''; AddressPointer_8610 = 0; AdrOffset_8620 = 392; BitOffset_8620 = 0; BitLength_8620 = 16; Address_8620 = '%IW196'; Type_8620 = 'UINT'; AddressPointer_8620 = ADR(%IW196); Automatic Mapping = True; IsValid = True; IsHostHoming = False; PulseSelectIndex = 2
      InoSV630N_左下气缸 : SV630_1Axis_03715, Inovance, order no. InoSV630N, version Revision=16#00010000
          settings: Number of Outputs = 7; Number of Inputs = 10; Number of Infos about Outputs = 7; Number of Infos about Inputs = 10; EnableExpertSettings = True; Physical Address of the Slave = 1013; AutoIncr Address of the Slave = 4294967284; StationAlias = 0; Sync.Length = 19; Sync.Length = 32; FMMU.Global Start Address = 16#020000CD; FMMU.Length = 19; FMMU.Physical Start Address = 16#1800; FMMU.Access = 16#02; FMMU.Global Start Address = 16#0100017E; FMMU.Length = 32; FMMU.Physical Start Address = 16#1C00; FMMU.Access = 16#01; FMMU.Global Start Address = 16#00080001; FMMU.StartBit = 3; FMMU.EndBit = 3; FMMU.Physical Start Address = 16#080D; FMMU.Access = 16#01; AutoUpdate = False; DC sync0 cycletime = 4000; DC sync0 cycletime = 4000000; DC sync1 cycletime = 4000; DC sync1 cycletime = 4000000; Number of SDO = 10; Homing method.Index = 16#6098; Homing method.Subindex = 16#00; Homing method.Value = 35; Homing method.Size = 8; Homing method.AbortIfError = FALSE; Homing method.JumpToLine = FALSE; Homing method.Line = 0; Homing method.CompleteAccess = FALSE; Actual Position Calculation Method.Index = 16#60E6; Actual Position Calculation Method.Subindex = 16#00; Actual Position Calculation Method.Value = 0;
            Actual Position Calculation Method.Size = 8; Actual Position Calculation Method.AbortIfError = FALSE; Actual Position Calculation Method.JumpToLine = FALSE; Actual Position Calculation Method.Line = 0; Actual Position Calculation Method.CompleteAccess = FALSE; Speed during search for switch.Index = 16#6099; Speed during search for switch.Subindex = 16#01; Speed during search for switch.Value = 87381; Speed during search for switch.Size = 32; Speed during search for switch.AbortIfError = FALSE; Speed during search for switch.JumpToLine = FALSE; Speed during search for switch.Line = 0; Speed during search for switch.CompleteAccess = FALSE; Homing acceleration.Index = 16#609A; Homing acceleration.Subindex = 16#00; Homing acceleration.Value = 8738133; Homing acceleration.Size = 32; Homing acceleration.AbortIfError = FALSE; Homing acceleration.JumpToLine = FALSE; Homing acceleration.Line = 0; Homing acceleration.CompleteAccess = FALSE; Speed during search for zero.Index = 16#6099; Speed during search for zero.Subindex = 16#02; Speed during search for zero.Value = 8738; Speed during search for zero.Size = 32; Speed during search for zero.AbortIfError = FALSE; Speed during search for zero.JumpToLine = FALSE; Speed during search for zero.Line = 0; Speed during search for zero.CompleteAccess = FALSE; Time of home searching.Index = 16#2005; Time of home searching.Subindex = 16#24; Time of home searching.Value = 50000; Time of home searching.Size = 16; Time of home searching.AbortIfError = FALSE; Time of home searching.JumpToLine = FALSE; Time of home searching.Line = 0; Time of home searching.CompleteAccess = FALSE; Positive torque limit value.Index = 16#60E0; Positive torque limit value.Subindex = 16#00; Positive torque limit value.Value = 3500;
            Positive torque limit value.Size = 16; Positive torque limit value.AbortIfError = FALSE; Positive torque limit value.JumpToLine = FALSE; Positive torque limit value.Line = 0; Positive torque limit value.CompleteAccess = FALSE; Negative torque limit value.Index = 16#60E1; Negative torque limit value.Subindex = 16#00; Negative torque limit value.Value = 3500; Negative torque limit value.Size = 16; Negative torque limit value.AbortIfError = FALSE; Negative torque limit value.JumpToLine = FALSE; Negative torque limit value.Line = 0; Negative torque limit value.CompleteAccess = FALSE; Max profile velocity.Index = 16#607F; Max profile velocity.Subindex = 16#00; Max profile velocity.Value = 5242880; Max profile velocity.Size = 32; Max profile velocity.AbortIfError = FALSE; Max profile velocity.JumpToLine = FALSE; Max profile velocity.Line = 0; Max profile velocity.CompleteAccess = FALSE; RxTxPdo.NumberofEntries = 7; RxTxPdo.Sm = 2; RxTxPdo.DependOnSlot = False; RxTxPdo.DependOnSlotGroup = False; RxTxPdo.OverwrittenByModule = False; Exclude = [16#1701,16#1702,16#1703,16#1704,16#1705]; Controlword.Index = 16#6040; Controlword.SubIndex = 0; Controlword.Size = 16; Controlword.Offset = 0; Controlword.DependOnSlot = False; Controlword.DependOnSlotGroup = False; Target position.Index = 16#607A; Target position.SubIndex = 0; Target position.Size = 32; Target position.Offset = 0; Target position.DependOnSlot = False; Target position.DependOnSlotGroup = False; Touch probe function.Index = 16#60B8;
            Touch probe function.SubIndex = 0; Touch probe function.Size = 16; Touch probe function.Offset = 0; Touch probe function.DependOnSlot = False; Touch probe function.DependOnSlotGroup = False; Physical outputs.Index = 16#60FE; Physical outputs.SubIndex = 1; Physical outputs.Size = 32; Physical outputs.Offset = 0; Physical outputs.DependOnSlot = False; Physical outputs.DependOnSlotGroup = False; Target velocity.Index = 16#60FF; Target velocity.SubIndex = 0; Target velocity.Size = 32; Target velocity.Offset = 0; Target velocity.DependOnSlot = False; Target velocity.DependOnSlotGroup = False; Modes of operation.Index = 16#6060; Modes of operation.SubIndex = 0; Modes of operation.Size = 8; Modes of operation.Offset = 0; Modes of operation.DependOnSlot = False; Modes of operation.DependOnSlotGroup = False; Target torque.Index = 16#6071; Target torque.SubIndex = 0; Target torque.Size = 16; Target torque.Offset = 0; Target torque.DependOnSlot = False; Target torque.DependOnSlotGroup = False; RxTxPdo.Sm = -1; RxTxPdo.NumberofEntries = 10; RxTxPdo.Sm = 3; Error code.Index = 16#603F; Error code.SubIndex = 0; Error code.Size = 16; Error code.DependOnSlot = false; Error code.DependOnSlotGroup = false; Statusword.Index = 16#6041; Statusword.SubIndex = 0; Statusword.Size = 16;
            Statusword.DependOnSlot = false; Statusword.DependOnSlotGroup = false; Position actual value.Index = 16#6064; Position actual value.SubIndex = 0; Position actual value.Size = 32; Position actual value.DependOnSlot = false; Position actual value.DependOnSlotGroup = false; Torque actual value.Index = 16#6077; Torque actual value.SubIndex = 0; Torque actual value.Size = 16; Torque actual value.DependOnSlot = false; Torque actual value.DependOnSlotGroup = false; Following error actual value.Index = 16#60F4; Following error actual value.SubIndex = 0; Following error actual value.Size = 32; Following error actual value.DependOnSlot = false; Following error actual value.DependOnSlotGroup = false; Touch probe status.Index = 16#60B9; Touch probe status.SubIndex = 0; Touch probe status.Size = 16; Touch probe status.DependOnSlot = false; Touch probe status.DependOnSlotGroup = false; Touch probe pos1 pos value.Index = 16#60BA; Touch probe pos1 pos value.SubIndex = 0; Touch probe pos1 pos value.Size = 32; Touch probe pos1 pos value.DependOnSlot = false; Touch probe pos1 pos value.DependOnSlotGroup = false; Touch probe pos2 pos value.Index = 16#60BC; Touch probe pos2 pos value.SubIndex = 0; Touch probe pos2 pos value.Size = 32; Touch probe pos2 pos value.DependOnSlot = false; Touch probe pos2 pos value.DependOnSlotGroup = false; Digital inputs.Index = 16#60FD; Digital inputs.SubIndex = 0; Digital inputs.Size = 32; Digital inputs.DependOnSlot = false; Digital inputs.DependOnSlotGroup = false; Velocity actual value.Index = 16#606C; Velocity actual value.SubIndex = 0; Velocity actual value.Size = 32;
            Velocity actual value.DependOnSlot = false; Velocity actual value.DependOnSlotGroup = false; RxTxPdo.Sm = -1; Controlword.Name = 'Controlword'; Controlword.DataType = 'UINT'; Controlword.Default = ''; Controlword.Comment = ''; Target position.Name = 'Target position'; Target position.DataType = 'DINT'; Target position.Default = ''; Target position.Comment = ''; Touch probe function.Name = 'Touch probe function'; Touch probe function.DataType = 'UINT'; Touch probe function.Default = ''; Touch probe function.Comment = ''; Physical outputs.Name = 'Physical outputs'; Physical outputs.DataType = 'UDINT'; Physical outputs.Default = ''; Physical outputs.Comment = ''; Target velocity.Name = 'Target velocity'; Target velocity.DataType = 'DINT'; Target velocity.Default = ''; Target velocity.Comment = ''; Modes of operation.Name = 'Modes of operation'; Modes of operation.DataType = 'SINT'; Modes of operation.Default = ''; Modes of operation.Comment = ''; Target torque.Name = 'Target torque'; Target torque.DataType = 'INT'; Target torque.Default = ''; Target torque.Comment = ''; Error code.Name = 'Error code'; Error code.DataType = 'UINT'; Statusword.Name = 'Statusword'; Statusword.DataType = 'UINT'; Position actual value.Name = 'Position actual value'; Position actual value.DataType = 'DINT'; Torque actual value.Name = 'Torque actual value'; Torque actual value.DataType = 'INT'; Following error actual value.Name = 'Following error actual value';
            Following error actual value.DataType = 'DINT'; Touch probe status.Name = 'Touch probe status'; Touch probe status.DataType = 'UINT'; Touch probe pos1 pos value.Name = 'Touch probe pos1 pos value'; Touch probe pos1 pos value.DataType = 'DINT'; Touch probe pos2 pos value.Name = 'Touch probe pos2 pos value'; Touch probe pos2 pos value.DataType = 'DINT'; Digital inputs.Name = 'Digital inputs'; Digital inputs.DataType = 'UDINT'; Velocity actual value.Name = 'Velocity actual value'; Velocity actual value.DataType = 'DINT'
          unmapped channels: Controlword, Target position, Touch probe function, Physical outputs, Target velocity, Modes of operation, Target torque, Error code, Statusword, Position actual value, Torque actual value, Following error actual value, Touch probe status, Touch probe pos1 pos value, Touch probe pos2 pos value, Digital inputs, Velocity actual value
        左下气缸 : Axis, Inovance, order no. 0, version 1.0.0.0
            settings: wDriveID = 13; dwRatioTechUnitsDenom = 262144; iRatioTechUnitsNum = 5; fSWMaxVelocity = 1000; fSWMaxAcceleration = 10000; fSWMaxDeceleration = 10000; fSWMaxJerk = 100000; iEncoderType = 1; iAbsEncoderOption = 1; HomingMode = 10; ZeroSignal = 0; StartDirction = 1; EndDirection = 1; PosLimitMode = 0; NegLimitMode = 0; HomingVelocity = 10; HomingApproachVelocity = 2; HomingAcceleration = 100; HomingDeceleration = 100; HomingJerk = 0; HomeMaskDistance = 0; HomePositionOffset = 0; HomePushTime = 0; HomeCompensation = 0; HomeTimeout = 0; HomeCompensationVelocity = 1000; 4000 = 1; 4001 = 1; 4003 = true; 4004 = 33; 4005 = 0; 4006 = 1.666667; 4007 = 166.666666; 4008 = 0.166667; 4009 = 50000; 4010 = 3500; 4011 = 3500; 4012 = 100.000000; ScalingIncs = 16#40000; ScalingMotorTurns2 = 2;
              6005 = 10; AdrOffset_8010 = 268; BitOffset_8010 = 0; BitLength_8010 = 16; Address_8010 = '%QW134'; Type_8010 = 'UINT'; AddressPointer_8010 = ADR(%QW134); AdrOffset_8020 = 272; BitOffset_8020 = 0; BitLength_8020 = 32; Address_8020 = '%QD68'; Type_8020 = 'DINT'; AddressPointer_8020 = ADR(%QD68); AdrOffset_8030 = 284; BitOffset_8030 = 0; BitLength_8030 = 32; Address_8030 = '%QD71'; Type_8030 = 'DINT'; AddressPointer_8030 = ADR(%QD71); AdrOffset_8040 = 290; BitOffset_8040 = 0; BitLength_8040 = 16; Address_8040 = '%QW145'; Type_8040 = 'INT'; AddressPointer_8040 = ADR(%QW145); AdrOffset_8050 = 288; BitOffset_8050 = 0; BitLength_8050 = 8; Address_8050 = '%QB288'; Type_8050 = 'SINT'; AddressPointer_8050 = ADR(%QB288); AdrOffset_8060 = 276; BitOffset_8060 = 0; BitLength_8060 = 16; Address_8060 = '%QW138'; Type_8060 = 'UINT'; AddressPointer_8060 = ADR(%QW138); AdrOffset_8070 = 4294967295; BitOffset_8070 = 0; BitLength_8070 = 0;
              Address_8070 = ''; Type_8070 = ''; AddressPointer_8070 = 0; AdrOffset_8080 = 4294967295; BitOffset_8080 = 0; BitLength_8080 = 0; Address_8080 = ''; Type_8080 = ''; AddressPointer_8080 = 0; AdrOffset_8090 = 280; BitOffset_8090 = 0; BitLength_8090 = 32; Address_8090 = '%QD70'; Type_8090 = 'UDINT'; AddressPointer_8090 = ADR(%QD70); AdrOffset_8100 = 4294967295; BitOffset_8100 = 0; BitLength_8100 = 0; Address_8100 = ''; Type_8100 = ''; AddressPointer_8100 = 0; AdrOffset_8510 = 430; BitOffset_8510 = 0; BitLength_8510 = 16; Address_8510 = '%IW215'; Type_8510 = 'UINT'; AddressPointer_8510 = ADR(%IW215); AdrOffset_8520 = 432; BitOffset_8520 = 0; BitLength_8520 = 32; Address_8520 = '%ID108'; Type_8520 = 'DINT'; AddressPointer_8520 = ADR(%ID108); AdrOffset_8530 = 460; BitOffset_8530 = 0; BitLength_8530 = 32; Address_8530 = '%ID115'; Type_8530 = 'DINT'; AddressPointer_8530 = ADR(%ID115); AdrOffset_8540 = 436;
              BitOffset_8540 = 0; BitLength_8540 = 16; Address_8540 = '%IW218'; Type_8540 = 'INT'; AddressPointer_8540 = ADR(%IW218); AdrOffset_8550 = 4294967295; BitOffset_8550 = 0; BitLength_8550 = 0; Address_8550 = ''; Type_8550 = ''; AddressPointer_8550 = 0; AdrOffset_8560 = 456; BitOffset_8560 = 0; BitLength_8560 = 32; Address_8560 = '%ID114'; Type_8560 = 'UDINT'; AddressPointer_8560 = ADR(%ID114); AdrOffset_8570 = 444; BitOffset_8570 = 0; BitLength_8570 = 16; Address_8570 = '%IW222'; Type_8570 = 'UINT'; AddressPointer_8570 = ADR(%IW222); AdrOffset_8580 = 448; BitOffset_8580 = 0; BitLength_8580 = 32; Address_8580 = '%ID112'; Type_8580 = 'DINT'; AddressPointer_8580 = ADR(%ID112); AdrOffset_8590 = 4294967295; BitOffset_8590 = 0; BitLength_8590 = 0; Address_8590 = ''; Type_8590 = ''; AddressPointer_8590 = 0; AdrOffset_8600 = 452; BitOffset_8600 = 0; BitLength_8600 = 32; Address_8600 = '%ID113'; Type_8600 = 'DINT';
              AddressPointer_8600 = ADR(%ID113); AdrOffset_8600 = 4294967295; BitOffset_8600 = 0; BitLength_8600 = 0; Address_8610 = ''; Type_8610 = ''; AddressPointer_8610 = 0; AdrOffset_8620 = 428; BitOffset_8620 = 0; BitLength_8620 = 16; Address_8620 = '%IW214'; Type_8620 = 'UINT'; AddressPointer_8620 = ADR(%IW214); Automatic Mapping = True; IsValid = True; IsHostHoming = False; PulseSelectIndex = 2
      InoSV630N_右上气缸 : SV630_1Axis_03715, Inovance, order no. InoSV630N, version Revision=16#00010000
          settings: Number of Outputs = 7; Number of Inputs = 10; Number of Infos about Outputs = 7; Number of Infos about Inputs = 10; EnableExpertSettings = True; Physical Address of the Slave = 1010; AutoIncr Address of the Slave = 4294967287; StationAlias = 0; Sync.Length = 19; Sync.Length = 32; FMMU.Global Start Address = 16#02000094; FMMU.Length = 19; FMMU.Physical Start Address = 16#1800; FMMU.Access = 16#02; FMMU.Global Start Address = 16#0100011E; FMMU.Length = 32; FMMU.Physical Start Address = 16#1C00; FMMU.Access = 16#01; FMMU.Global Start Address = 16#00080001; FMMU.Physical Start Address = 16#080D; FMMU.Access = 16#01; AutoUpdate = False; DC sync0 cycletime = 4000; DC sync0 cycletime = 4000000; DC sync1 cycletime = 4000; DC sync1 cycletime = 4000000; Number of SDO = 10; Homing method.Index = 16#6098; Homing method.Subindex = 16#00; Homing method.Value = 35; Homing method.Size = 8; Homing method.AbortIfError = FALSE; Homing method.JumpToLine = FALSE; Homing method.Line = 0; Homing method.CompleteAccess = FALSE; Actual Position Calculation Method.Index = 16#60E6; Actual Position Calculation Method.Subindex = 16#00; Actual Position Calculation Method.Value = 0; Actual Position Calculation Method.Size = 8; Actual Position Calculation Method.AbortIfError = FALSE;
            Actual Position Calculation Method.JumpToLine = FALSE; Actual Position Calculation Method.Line = 0; Actual Position Calculation Method.CompleteAccess = FALSE; Speed during search for switch.Index = 16#6099; Speed during search for switch.Subindex = 16#01; Speed during search for switch.Value = 87381; Speed during search for switch.Size = 32; Speed during search for switch.AbortIfError = FALSE; Speed during search for switch.JumpToLine = FALSE; Speed during search for switch.Line = 0; Speed during search for switch.CompleteAccess = FALSE; Homing acceleration.Index = 16#609A; Homing acceleration.Subindex = 16#00; Homing acceleration.Value = 8738133; Homing acceleration.Size = 32; Homing acceleration.AbortIfError = FALSE; Homing acceleration.JumpToLine = FALSE; Homing acceleration.Line = 0; Homing acceleration.CompleteAccess = FALSE; Speed during search for zero.Index = 16#6099; Speed during search for zero.Subindex = 16#02; Speed during search for zero.Value = 8738; Speed during search for zero.Size = 32; Speed during search for zero.AbortIfError = FALSE; Speed during search for zero.JumpToLine = FALSE; Speed during search for zero.Line = 0; Speed during search for zero.CompleteAccess = FALSE; Time of home searching.Index = 16#2005; Time of home searching.Subindex = 16#24; Time of home searching.Value = 50000; Time of home searching.Size = 16; Time of home searching.AbortIfError = FALSE; Time of home searching.JumpToLine = FALSE; Time of home searching.Line = 0; Time of home searching.CompleteAccess = FALSE; Positive torque limit value.Index = 16#60E0; Positive torque limit value.Subindex = 16#00; Positive torque limit value.Value = 3500; Positive torque limit value.Size = 16; Positive torque limit value.AbortIfError = FALSE;
            Positive torque limit value.JumpToLine = FALSE; Positive torque limit value.Line = 0; Positive torque limit value.CompleteAccess = FALSE; Negative torque limit value.Index = 16#60E1; Negative torque limit value.Subindex = 16#00; Negative torque limit value.Value = 3500; Negative torque limit value.Size = 16; Negative torque limit value.AbortIfError = FALSE; Negative torque limit value.JumpToLine = FALSE; Negative torque limit value.Line = 0; Negative torque limit value.CompleteAccess = FALSE; Max profile velocity.Index = 16#607F; Max profile velocity.Subindex = 16#00; Max profile velocity.Value = 5242880; Max profile velocity.Size = 32; Max profile velocity.AbortIfError = FALSE; Max profile velocity.JumpToLine = FALSE; Max profile velocity.Line = 0; Max profile velocity.CompleteAccess = FALSE; RxTxPdo.NumberofEntries = 7; RxTxPdo.Sm = 2; RxTxPdo.DependOnSlot = False; RxTxPdo.DependOnSlotGroup = False; RxTxPdo.OverwrittenByModule = False; Exclude = [16#1701,16#1702,16#1703,16#1704,16#1705]; Controlword.Index = 16#6040; Controlword.SubIndex = 0; Controlword.Size = 16; Controlword.Offset = 0; Controlword.DependOnSlot = False; Controlword.DependOnSlotGroup = False; Target position.Index = 16#607A; Target position.SubIndex = 0; Target position.Size = 32; Target position.Offset = 0; Target position.DependOnSlot = False; Target position.DependOnSlotGroup = False; Touch probe function.Index = 16#60B8; Touch probe function.SubIndex = 0; Touch probe function.Size = 16;
            Touch probe function.Offset = 0; Touch probe function.DependOnSlot = False; Touch probe function.DependOnSlotGroup = False; Physical outputs.Index = 16#60FE; Physical outputs.SubIndex = 1; Physical outputs.Size = 32; Physical outputs.Offset = 0; Physical outputs.DependOnSlot = False; Physical outputs.DependOnSlotGroup = False; Target velocity.Index = 16#60FF; Target velocity.SubIndex = 0; Target velocity.Size = 32; Target velocity.Offset = 0; Target velocity.DependOnSlot = False; Target velocity.DependOnSlotGroup = False; Modes of operation.Index = 16#6060; Modes of operation.SubIndex = 0; Modes of operation.Size = 8; Modes of operation.Offset = 0; Modes of operation.DependOnSlot = False; Modes of operation.DependOnSlotGroup = False; Target torque.Index = 16#6071; Target torque.SubIndex = 0; Target torque.Size = 16; Target torque.Offset = 0; Target torque.DependOnSlot = False; Target torque.DependOnSlotGroup = False; RxTxPdo.Sm = -1; RxTxPdo.NumberofEntries = 10; RxTxPdo.Sm = 3; Error code.Index = 16#603F; Error code.SubIndex = 0; Error code.Size = 16; Error code.DependOnSlot = false; Error code.DependOnSlotGroup = false; Statusword.Index = 16#6041; Statusword.SubIndex = 0; Statusword.Size = 16; Statusword.DependOnSlot = false; Statusword.DependOnSlotGroup = false;
            Position actual value.Index = 16#6064; Position actual value.SubIndex = 0; Position actual value.Size = 32; Position actual value.DependOnSlot = false; Position actual value.DependOnSlotGroup = false; Torque actual value.Index = 16#6077; Torque actual value.SubIndex = 0; Torque actual value.Size = 16; Torque actual value.DependOnSlot = false; Torque actual value.DependOnSlotGroup = false; Following error actual value.Index = 16#60F4; Following error actual value.SubIndex = 0; Following error actual value.Size = 32; Following error actual value.DependOnSlot = false; Following error actual value.DependOnSlotGroup = false; Touch probe status.Index = 16#60B9; Touch probe status.SubIndex = 0; Touch probe status.Size = 16; Touch probe status.DependOnSlot = false; Touch probe status.DependOnSlotGroup = false; Touch probe pos1 pos value.Index = 16#60BA; Touch probe pos1 pos value.SubIndex = 0; Touch probe pos1 pos value.Size = 32; Touch probe pos1 pos value.DependOnSlot = false; Touch probe pos1 pos value.DependOnSlotGroup = false; Touch probe pos2 pos value.Index = 16#60BC; Touch probe pos2 pos value.SubIndex = 0; Touch probe pos2 pos value.Size = 32; Touch probe pos2 pos value.DependOnSlot = false; Touch probe pos2 pos value.DependOnSlotGroup = false; Digital inputs.Index = 16#60FD; Digital inputs.SubIndex = 0; Digital inputs.Size = 32; Digital inputs.DependOnSlot = false; Digital inputs.DependOnSlotGroup = false; Velocity actual value.Index = 16#606C; Velocity actual value.SubIndex = 0; Velocity actual value.Size = 32; Velocity actual value.DependOnSlot = false; Velocity actual value.DependOnSlotGroup = false;
            RxTxPdo.Sm = -1; Controlword.Name = 'Controlword'; Controlword.DataType = 'UINT'; Controlword.Default = ''; Controlword.Comment = ''; Target position.Name = 'Target position'; Target position.DataType = 'DINT'; Target position.Default = ''; Target position.Comment = ''; Touch probe function.Name = 'Touch probe function'; Touch probe function.DataType = 'UINT'; Touch probe function.Default = ''; Touch probe function.Comment = ''; Physical outputs.Name = 'Physical outputs'; Physical outputs.DataType = 'UDINT'; Physical outputs.Default = ''; Physical outputs.Comment = ''; Target velocity.Name = 'Target velocity'; Target velocity.DataType = 'DINT'; Target velocity.Default = ''; Target velocity.Comment = ''; Modes of operation.Name = 'Modes of operation'; Modes of operation.DataType = 'SINT'; Modes of operation.Default = ''; Modes of operation.Comment = ''; Target torque.Name = 'Target torque'; Target torque.DataType = 'INT'; Target torque.Default = ''; Target torque.Comment = ''; Error code.Name = 'Error code'; Error code.DataType = 'UINT'; Statusword.Name = 'Statusword'; Statusword.DataType = 'UINT'; Position actual value.Name = 'Position actual value'; Position actual value.DataType = 'DINT'; Torque actual value.Name = 'Torque actual value'; Torque actual value.DataType = 'INT'; Following error actual value.Name = 'Following error actual value'; Following error actual value.DataType = 'DINT'; Touch probe status.Name = 'Touch probe status';
            Touch probe status.DataType = 'UINT'; Touch probe pos1 pos value.Name = 'Touch probe pos1 pos value'; Touch probe pos1 pos value.DataType = 'DINT'; Touch probe pos2 pos value.Name = 'Touch probe pos2 pos value'; Touch probe pos2 pos value.DataType = 'DINT'; Digital inputs.Name = 'Digital inputs'; Digital inputs.DataType = 'UDINT'; Velocity actual value.Name = 'Velocity actual value'; Velocity actual value.DataType = 'DINT'
          unmapped channels: Controlword, Target position, Touch probe function, Physical outputs, Target velocity, Modes of operation, Target torque, Error code, Statusword, Position actual value, Torque actual value, Following error actual value, Touch probe status, Touch probe pos1 pos value, Touch probe pos2 pos value, Digital inputs, Velocity actual value
        右上气缸 : Axis, Inovance, order no. 0, version 1.0.0.0
            settings: wDriveID = 24; dwRatioTechUnitsDenom = 262144; iRatioTechUnitsNum = 5; fSWMaxVelocity = 1000; fSWMaxAcceleration = 10000; fSWMaxDeceleration = 10000; fSWMaxJerk = 100000; iEncoderType = 1; iAbsEncoderOption = 1; HomingMode = 10; ZeroSignal = 0; StartDirction = 1; EndDirection = 1; PosLimitMode = 0; NegLimitMode = 0; HomingVelocity = 10; HomingApproachVelocity = 2; HomingAcceleration = 100; HomingDeceleration = 100; HomingJerk = 0; HomeMaskDistance = 0; HomePositionOffset = 0; HomePushTime = 0; HomeCompensation = 0; HomeTimeout = 0; HomeCompensationVelocity = 1000; 4000 = 1; 4001 = 1; 4003 = true; 4004 = 33; 4005 = 0; 4006 = 1.666667; 4007 = 166.666666; 4008 = 0.166667; 4009 = 50000; 4010 = 3500; 4011 = 3500; 4012 = 100.000000; ScalingIncs = 16#40000; ScalingMotorTurns2 = 2;
              6005 = 10; AdrOffset_8010 = 196; BitOffset_8010 = 0; BitLength_8010 = 16; Address_8010 = '%QW98'; Type_8010 = 'UINT'; AddressPointer_8010 = ADR(%QW98); AdrOffset_8020 = 200; BitOffset_8020 = 0; BitLength_8020 = 32; Address_8020 = '%QD50'; Type_8020 = 'DINT'; AddressPointer_8020 = ADR(%QD50); AdrOffset_8030 = 212; BitOffset_8030 = 0; BitLength_8030 = 32; Address_8030 = '%QD53'; Type_8030 = 'DINT'; AddressPointer_8030 = ADR(%QD53); AdrOffset_8040 = 218; BitOffset_8040 = 0; BitLength_8040 = 16; Address_8040 = '%QW109'; Type_8040 = 'INT'; AddressPointer_8040 = ADR(%QW109); AdrOffset_8050 = 216; BitOffset_8050 = 0; BitLength_8050 = 8; Address_8050 = '%QB216'; Type_8050 = 'SINT'; AddressPointer_8050 = ADR(%QB216); AdrOffset_8060 = 204; BitOffset_8060 = 0; BitLength_8060 = 16; Address_8060 = '%QW102'; Type_8060 = 'UINT'; AddressPointer_8060 = ADR(%QW102); AdrOffset_8070 = 4294967295; BitOffset_8070 = 0; BitLength_8070 = 0;
              Address_8070 = ''; Type_8070 = ''; AddressPointer_8070 = 0; AdrOffset_8080 = 4294967295; BitOffset_8080 = 0; BitLength_8080 = 0; Address_8080 = ''; Type_8080 = ''; AddressPointer_8080 = 0; AdrOffset_8090 = 208; BitOffset_8090 = 0; BitLength_8090 = 32; Address_8090 = '%QD52'; Type_8090 = 'UDINT'; AddressPointer_8090 = ADR(%QD52); AdrOffset_8100 = 4294967295; BitOffset_8100 = 0; BitLength_8100 = 0; Address_8100 = ''; Type_8100 = ''; AddressPointer_8100 = 0; AdrOffset_8510 = 322; BitOffset_8510 = 0; BitLength_8510 = 16; Address_8510 = '%IW161'; Type_8510 = 'UINT'; AddressPointer_8510 = ADR(%IW161); AdrOffset_8520 = 324; BitOffset_8520 = 0; BitLength_8520 = 32; Address_8520 = '%ID81'; Type_8520 = 'DINT'; AddressPointer_8520 = ADR(%ID81); AdrOffset_8530 = 352; BitOffset_8530 = 0; BitLength_8530 = 32; Address_8530 = '%ID88'; Type_8530 = 'DINT'; AddressPointer_8530 = ADR(%ID88); AdrOffset_8540 = 328;
              BitOffset_8540 = 0; BitLength_8540 = 16; Address_8540 = '%IW164'; Type_8540 = 'INT'; AddressPointer_8540 = ADR(%IW164); AdrOffset_8550 = 4294967295; BitOffset_8550 = 0; BitLength_8550 = 0; Address_8550 = ''; Type_8550 = ''; AddressPointer_8550 = 0; AdrOffset_8560 = 348; BitOffset_8560 = 0; BitLength_8560 = 32; Address_8560 = '%ID87'; Type_8560 = 'UDINT'; AddressPointer_8560 = ADR(%ID87); AdrOffset_8570 = 336; BitOffset_8570 = 0; BitLength_8570 = 16; Address_8570 = '%IW168'; Type_8570 = 'UINT'; AddressPointer_8570 = ADR(%IW168); AdrOffset_8580 = 340; BitOffset_8580 = 0; BitLength_8580 = 32; Address_8580 = '%ID85'; Type_8580 = 'DINT'; AddressPointer_8580 = ADR(%ID85); AdrOffset_8590 = 4294967295; BitOffset_8590 = 0; BitLength_8590 = 0; Address_8590 = ''; Type_8590 = ''; AddressPointer_8590 = 0; AdrOffset_8600 = 344; BitOffset_8600 = 0; BitLength_8600 = 32; Address_8600 = '%ID86'; Type_8600 = 'DINT';
              AddressPointer_8600 = ADR(%ID86); AdrOffset_8600 = 4294967295; BitOffset_8600 = 0; BitLength_8600 = 0; Address_8610 = ''; Type_8610 = ''; AddressPointer_8610 = 0; AdrOffset_8620 = 320; BitOffset_8620 = 0; BitLength_8620 = 16; Address_8620 = '%IW160'; Type_8620 = 'UINT'; AddressPointer_8620 = ADR(%IW160); Automatic Mapping = True; IsValid = True; IsHostHoming = False; PulseSelectIndex = 2
      InoSV630N_右下气缸 : SV630_1Axis_03715, Inovance, order no. InoSV630N, version Revision=16#00010000
          settings: Number of Outputs = 7; Number of Inputs = 10; Number of Infos about Outputs = 7; Number of Infos about Inputs = 10; EnableExpertSettings = True; Physical Address of the Slave = 1011; AutoIncr Address of the Slave = 4294967286; StationAlias = 0; Sync.Length = 19; Sync.Length = 32; FMMU.Global Start Address = 16#020000A7; FMMU.Length = 19; FMMU.Physical Start Address = 16#1800; FMMU.Access = 16#02; FMMU.Global Start Address = 16#0100013E; FMMU.Length = 32; FMMU.Physical Start Address = 16#1C00; FMMU.Access = 16#01; FMMU.Global Start Address = 16#00080001; FMMU.StartBit = 1; FMMU.EndBit = 1; FMMU.Physical Start Address = 16#080D; FMMU.Access = 16#01; AutoUpdate = False; DC sync0 cycletime = 4000; DC sync0 cycletime = 4000000; DC sync1 cycletime = 4000; DC sync1 cycletime = 4000000; Number of SDO = 10; Homing method.Index = 16#6098; Homing method.Subindex = 16#00; Homing method.Value = 35; Homing method.Size = 8; Homing method.AbortIfError = FALSE; Homing method.JumpToLine = FALSE; Homing method.Line = 0; Homing method.CompleteAccess = FALSE; Actual Position Calculation Method.Index = 16#60E6; Actual Position Calculation Method.Subindex = 16#00; Actual Position Calculation Method.Value = 0;
            Actual Position Calculation Method.Size = 8; Actual Position Calculation Method.AbortIfError = FALSE; Actual Position Calculation Method.JumpToLine = FALSE; Actual Position Calculation Method.Line = 0; Actual Position Calculation Method.CompleteAccess = FALSE; Speed during search for switch.Index = 16#6099; Speed during search for switch.Subindex = 16#01; Speed during search for switch.Value = 87381; Speed during search for switch.Size = 32; Speed during search for switch.AbortIfError = FALSE; Speed during search for switch.JumpToLine = FALSE; Speed during search for switch.Line = 0; Speed during search for switch.CompleteAccess = FALSE; Homing acceleration.Index = 16#609A; Homing acceleration.Subindex = 16#00; Homing acceleration.Value = 8738133; Homing acceleration.Size = 32; Homing acceleration.AbortIfError = FALSE; Homing acceleration.JumpToLine = FALSE; Homing acceleration.Line = 0; Homing acceleration.CompleteAccess = FALSE; Speed during search for zero.Index = 16#6099; Speed during search for zero.Subindex = 16#02; Speed during search for zero.Value = 8738; Speed during search for zero.Size = 32; Speed during search for zero.AbortIfError = FALSE; Speed during search for zero.JumpToLine = FALSE; Speed during search for zero.Line = 0; Speed during search for zero.CompleteAccess = FALSE; Time of home searching.Index = 16#2005; Time of home searching.Subindex = 16#24; Time of home searching.Value = 50000; Time of home searching.Size = 16; Time of home searching.AbortIfError = FALSE; Time of home searching.JumpToLine = FALSE; Time of home searching.Line = 0; Time of home searching.CompleteAccess = FALSE; Positive torque limit value.Index = 16#60E0; Positive torque limit value.Subindex = 16#00; Positive torque limit value.Value = 3500;
            Positive torque limit value.Size = 16; Positive torque limit value.AbortIfError = FALSE; Positive torque limit value.JumpToLine = FALSE; Positive torque limit value.Line = 0; Positive torque limit value.CompleteAccess = FALSE; Negative torque limit value.Index = 16#60E1; Negative torque limit value.Subindex = 16#00; Negative torque limit value.Value = 3500; Negative torque limit value.Size = 16; Negative torque limit value.AbortIfError = FALSE; Negative torque limit value.JumpToLine = FALSE; Negative torque limit value.Line = 0; Negative torque limit value.CompleteAccess = FALSE; Max profile velocity.Index = 16#607F; Max profile velocity.Subindex = 16#00; Max profile velocity.Value = 5242880; Max profile velocity.Size = 32; Max profile velocity.AbortIfError = FALSE; Max profile velocity.JumpToLine = FALSE; Max profile velocity.Line = 0; Max profile velocity.CompleteAccess = FALSE; RxTxPdo.NumberofEntries = 7; RxTxPdo.Sm = 2; RxTxPdo.DependOnSlot = False; RxTxPdo.DependOnSlotGroup = False; RxTxPdo.OverwrittenByModule = False; Exclude = [16#1701,16#1702,16#1703,16#1704,16#1705]; Controlword.Index = 16#6040; Controlword.SubIndex = 0; Controlword.Size = 16; Controlword.Offset = 0; Controlword.DependOnSlot = False; Controlword.DependOnSlotGroup = False; Target position.Index = 16#607A; Target position.SubIndex = 0; Target position.Size = 32; Target position.Offset = 0; Target position.DependOnSlot = False; Target position.DependOnSlotGroup = False; Touch probe function.Index = 16#60B8;
            Touch probe function.SubIndex = 0; Touch probe function.Size = 16; Touch probe function.Offset = 0; Touch probe function.DependOnSlot = False; Touch probe function.DependOnSlotGroup = False; Physical outputs.Index = 16#60FE; Physical outputs.SubIndex = 1; Physical outputs.Size = 32; Physical outputs.Offset = 0; Physical outputs.DependOnSlot = False; Physical outputs.DependOnSlotGroup = False; Target velocity.Index = 16#60FF; Target velocity.SubIndex = 0; Target velocity.Size = 32; Target velocity.Offset = 0; Target velocity.DependOnSlot = False; Target velocity.DependOnSlotGroup = False; Modes of operation.Index = 16#6060; Modes of operation.SubIndex = 0; Modes of operation.Size = 8; Modes of operation.Offset = 0; Modes of operation.DependOnSlot = False; Modes of operation.DependOnSlotGroup = False; Target torque.Index = 16#6071; Target torque.SubIndex = 0; Target torque.Size = 16; Target torque.Offset = 0; Target torque.DependOnSlot = False; Target torque.DependOnSlotGroup = False; RxTxPdo.Sm = -1; RxTxPdo.NumberofEntries = 10; RxTxPdo.Sm = 3; Error code.Index = 16#603F; Error code.SubIndex = 0; Error code.Size = 16; Error code.DependOnSlot = false; Error code.DependOnSlotGroup = false; Statusword.Index = 16#6041; Statusword.SubIndex = 0; Statusword.Size = 16;
            Statusword.DependOnSlot = false; Statusword.DependOnSlotGroup = false; Position actual value.Index = 16#6064; Position actual value.SubIndex = 0; Position actual value.Size = 32; Position actual value.DependOnSlot = false; Position actual value.DependOnSlotGroup = false; Torque actual value.Index = 16#6077; Torque actual value.SubIndex = 0; Torque actual value.Size = 16; Torque actual value.DependOnSlot = false; Torque actual value.DependOnSlotGroup = false; Following error actual value.Index = 16#60F4; Following error actual value.SubIndex = 0; Following error actual value.Size = 32; Following error actual value.DependOnSlot = false; Following error actual value.DependOnSlotGroup = false; Touch probe status.Index = 16#60B9; Touch probe status.SubIndex = 0; Touch probe status.Size = 16; Touch probe status.DependOnSlot = false; Touch probe status.DependOnSlotGroup = false; Touch probe pos1 pos value.Index = 16#60BA; Touch probe pos1 pos value.SubIndex = 0; Touch probe pos1 pos value.Size = 32; Touch probe pos1 pos value.DependOnSlot = false; Touch probe pos1 pos value.DependOnSlotGroup = false; Touch probe pos2 pos value.Index = 16#60BC; Touch probe pos2 pos value.SubIndex = 0; Touch probe pos2 pos value.Size = 32; Touch probe pos2 pos value.DependOnSlot = false; Touch probe pos2 pos value.DependOnSlotGroup = false; Digital inputs.Index = 16#60FD; Digital inputs.SubIndex = 0; Digital inputs.Size = 32; Digital inputs.DependOnSlot = false; Digital inputs.DependOnSlotGroup = false; Velocity actual value.Index = 16#606C; Velocity actual value.SubIndex = 0; Velocity actual value.Size = 32;
            Velocity actual value.DependOnSlot = false; Velocity actual value.DependOnSlotGroup = false; RxTxPdo.Sm = -1; Controlword.Name = 'Controlword'; Controlword.DataType = 'UINT'; Controlword.Default = ''; Controlword.Comment = ''; Target position.Name = 'Target position'; Target position.DataType = 'DINT'; Target position.Default = ''; Target position.Comment = ''; Touch probe function.Name = 'Touch probe function'; Touch probe function.DataType = 'UINT'; Touch probe function.Default = ''; Touch probe function.Comment = ''; Physical outputs.Name = 'Physical outputs'; Physical outputs.DataType = 'UDINT'; Physical outputs.Default = ''; Physical outputs.Comment = ''; Target velocity.Name = 'Target velocity'; Target velocity.DataType = 'DINT'; Target velocity.Default = ''; Target velocity.Comment = ''; Modes of operation.Name = 'Modes of operation'; Modes of operation.DataType = 'SINT'; Modes of operation.Default = ''; Modes of operation.Comment = ''; Target torque.Name = 'Target torque'; Target torque.DataType = 'INT'; Target torque.Default = ''; Target torque.Comment = ''; Error code.Name = 'Error code'; Error code.DataType = 'UINT'; Statusword.Name = 'Statusword'; Statusword.DataType = 'UINT'; Position actual value.Name = 'Position actual value'; Position actual value.DataType = 'DINT'; Torque actual value.Name = 'Torque actual value'; Torque actual value.DataType = 'INT'; Following error actual value.Name = 'Following error actual value';
            Following error actual value.DataType = 'DINT'; Touch probe status.Name = 'Touch probe status'; Touch probe status.DataType = 'UINT'; Touch probe pos1 pos value.Name = 'Touch probe pos1 pos value'; Touch probe pos1 pos value.DataType = 'DINT'; Touch probe pos2 pos value.Name = 'Touch probe pos2 pos value'; Touch probe pos2 pos value.DataType = 'DINT'; Digital inputs.Name = 'Digital inputs'; Digital inputs.DataType = 'UDINT'; Velocity actual value.Name = 'Velocity actual value'; Velocity actual value.DataType = 'DINT'
          unmapped channels: Controlword, Target position, Touch probe function, Physical outputs, Target velocity, Modes of operation, Target torque, Error code, Statusword, Position actual value, Torque actual value, Following error actual value, Touch probe status, Touch probe pos1 pos value, Touch probe pos2 pos value, Digital inputs, Velocity actual value
        右下气缸 : Axis, Inovance, order no. 0, version 1.0.0.0
            settings: wDriveID = 25; dwRatioTechUnitsDenom = 262144; iRatioTechUnitsNum = 5; fSWMaxVelocity = 1000; fSWMaxAcceleration = 10000; fSWMaxDeceleration = 10000; fSWMaxJerk = 100000; iEncoderType = 1; iAbsEncoderOption = 1; HomingMode = 10; ZeroSignal = 0; StartDirction = 1; EndDirection = 1; PosLimitMode = 0; NegLimitMode = 0; HomingVelocity = 10; HomingApproachVelocity = 2; HomingAcceleration = 100; HomingDeceleration = 100; HomingJerk = 0; HomeMaskDistance = 0; HomePositionOffset = 0; HomePushTime = 0; HomeCompensation = 0; HomeTimeout = 0; HomeCompensationVelocity = 1000; 4000 = 1; 4001 = 1; 4003 = true; 4004 = 33; 4005 = 0; 4006 = 1.666667; 4007 = 166.666666; 4008 = 0.166667; 4009 = 50000; 4010 = 3500; 4011 = 3500; 4012 = 100.000000; ScalingIncs = 16#40000; ScalingMotorTurns2 = 2;
              6005 = 10; AdrOffset_8010 = 220; BitOffset_8010 = 0; BitLength_8010 = 16; Address_8010 = '%QW110'; Type_8010 = 'UINT'; AddressPointer_8010 = ADR(%QW110); AdrOffset_8020 = 224; BitOffset_8020 = 0; BitLength_8020 = 32; Address_8020 = '%QD56'; Type_8020 = 'DINT'; AddressPointer_8020 = ADR(%QD56); AdrOffset_8030 = 236; BitOffset_8030 = 0; BitLength_8030 = 32; Address_8030 = '%QD59'; Type_8030 = 'DINT'; AddressPointer_8030 = ADR(%QD59); AdrOffset_8040 = 242; BitOffset_8040 = 0; BitLength_8040 = 16; Address_8040 = '%QW121'; Type_8040 = 'INT'; AddressPointer_8040 = ADR(%QW121); AdrOffset_8050 = 240; BitOffset_8050 = 0; BitLength_8050 = 8; Address_8050 = '%QB240'; Type_8050 = 'SINT'; AddressPointer_8050 = ADR(%QB240); AdrOffset_8060 = 228; BitOffset_8060 = 0; BitLength_8060 = 16; Address_8060 = '%QW114'; Type_8060 = 'UINT'; AddressPointer_8060 = ADR(%QW114); AdrOffset_8070 = 4294967295; BitOffset_8070 = 0; BitLength_8070 = 0;
              Address_8070 = ''; Type_8070 = ''; AddressPointer_8070 = 0; AdrOffset_8080 = 4294967295; BitOffset_8080 = 0; BitLength_8080 = 0; Address_8080 = ''; Type_8080 = ''; AddressPointer_8080 = 0; AdrOffset_8090 = 232; BitOffset_8090 = 0; BitLength_8090 = 32; Address_8090 = '%QD58'; Type_8090 = 'UDINT'; AddressPointer_8090 = ADR(%QD58); AdrOffset_8100 = 4294967295; BitOffset_8100 = 0; BitLength_8100 = 0; Address_8100 = ''; Type_8100 = ''; AddressPointer_8100 = 0; AdrOffset_8510 = 358; BitOffset_8510 = 0; BitLength_8510 = 16; Address_8510 = '%IW179'; Type_8510 = 'UINT'; AddressPointer_8510 = ADR(%IW179); AdrOffset_8520 = 360; BitOffset_8520 = 0; BitLength_8520 = 32; Address_8520 = '%ID90'; Type_8520 = 'DINT'; AddressPointer_8520 = ADR(%ID90); AdrOffset_8530 = 388; BitOffset_8530 = 0; BitLength_8530 = 32; Address_8530 = '%ID97'; Type_8530 = 'DINT'; AddressPointer_8530 = ADR(%ID97); AdrOffset_8540 = 364;
              BitOffset_8540 = 0; BitLength_8540 = 16; Address_8540 = '%IW182'; Type_8540 = 'INT'; AddressPointer_8540 = ADR(%IW182); AdrOffset_8550 = 4294967295; BitOffset_8550 = 0; BitLength_8550 = 0; Address_8550 = ''; Type_8550 = ''; AddressPointer_8550 = 0; AdrOffset_8560 = 384; BitOffset_8560 = 0; BitLength_8560 = 32; Address_8560 = '%ID96'; Type_8560 = 'UDINT'; AddressPointer_8560 = ADR(%ID96); AdrOffset_8570 = 372; BitOffset_8570 = 0; BitLength_8570 = 16; Address_8570 = '%IW186'; Type_8570 = 'UINT'; AddressPointer_8570 = ADR(%IW186); AdrOffset_8580 = 376; BitOffset_8580 = 0; BitLength_8580 = 32; Address_8580 = '%ID94'; Type_8580 = 'DINT'; AddressPointer_8580 = ADR(%ID94); AdrOffset_8590 = 4294967295; BitOffset_8590 = 0; BitLength_8590 = 0; Address_8590 = ''; Type_8590 = ''; AddressPointer_8590 = 0; AdrOffset_8600 = 380; BitOffset_8600 = 0; BitLength_8600 = 32; Address_8600 = '%ID95'; Type_8600 = 'DINT';
              AddressPointer_8600 = ADR(%ID95); AdrOffset_8600 = 4294967295; BitOffset_8600 = 0; BitLength_8600 = 0; Address_8610 = ''; Type_8610 = ''; AddressPointer_8610 = 0; AdrOffset_8620 = 356; BitOffset_8620 = 0; BitLength_8620 = 16; Address_8620 = '%IW178'; Type_8620 = 'UINT'; AddressPointer_8620 = ADR(%IW178); Automatic Mapping = True; IsValid = True; IsHostHoming = False; PulseSelectIndex = 2
      GL20_RTU_ECT : GL20-RTU-ECT_1.3.21.0, Inovance, order no. GL20-RTU-ECT, version Revision=16#01006000
          settings:  = 'de05f461-72c4-4d66-9ca2-fa428033ce23';  = 'de05f461-72c4-4d66-9ca2-fa428033ce23';  = 'de05f461-72c4-4d66-9ca2-fa428033ce23';  = 'd1c8065f-f08a-471f-8c7e-6f9e70c1fa64';  = 'f6588388-f26e-434d-9296-0c048c46a018';  = 'f6588388-f26e-434d-9296-0c048c46a018';  = 'f6588388-f26e-434d-9296-0c048c46a018';  = 'd1c8065f-f08a-471f-8c7e-6f9e70c1fa64'; Number of Outputs = 17; Number of Inputs = 21; IOModuleSize = 3; IOModuleName = "GL20_1600END,GL20_0008ER,GL20_2S485"; IOModuleGuid = f6588388-f26e-434d-9296-0c048c46a018,de05f461-72c4-4d66-9ca2-fa428033ce23,d1c8065f-f08a-471f-8c7e-6f9e70c1fa64; Number of Infos about Outputs = 17; Number of Infos about Inputs = 21; Physical Address of the Slave = 1018; AutoIncr Address of the Slave = 4294967279; Sync.Length = 63; Sync.Length = 74; FMMU.Global Start Address = 16#0200012C; FMMU.Length = 63; FMMU.Physical Start Address = 16#1800; FMMU.Access = 16#02; FMMU.Global Start Address = 16#0100021E; FMMU.Length = 74; FMMU.Physical Start Address = 16#1C00; FMMU.Access = 16#01; Number of RxPDOs of the Slave = 5; Number of TxPDOs of the Slave = 6; AutoUpdate = False; DC sync0 cycletime = 4000; DC sync1 cycletime = 4000; Number of SDO = 28; DI module CH0 filter time.Index = 16#8000; DI module CH0 filter time.Subindex = 16#01; DI module CH0 filter time.Value = 4; DI module CH0 filter time.Size = 16; DI module CH0 filter time.AbortIfError = FALSE; DI module CH0 filter time.JumpToLine = FALSE; DI module CH0 filter time.Line = 0;
            DI module CH0 filter time.CompleteAccess = False; DI module CH1 filter time.Index = 16#8000; DI module CH1 filter time.Subindex = 16#02; DI module CH1 filter time.Value = 4; DI module CH1 filter time.Size = 16; DI module CH1 filter time.AbortIfError = FALSE; DI module CH1 filter time.JumpToLine = FALSE; DI module CH1 filter time.Line = 0; DI module CH1 filter time.CompleteAccess = False; DO module CH0 stopmode after EtherCAT lost link.Index = 16#8040; DO module CH0 stopmode after EtherCAT lost link.Subindex = 16#01; DO module CH0 stopmode after EtherCAT lost link.Value = 255; DO module CH0 stopmode after EtherCAT lost link.Size = 8; DO module CH0 stopmode after EtherCAT lost link.AbortIfError = FALSE; DO module CH0 stopmode after EtherCAT lost link.JumpToLine = FALSE; DO module CH0 stopmode after EtherCAT lost link.Line = 0; DO module CH0 stopmode after EtherCAT lost link.CompleteAccess = False; DO module CH0 stopvalue after EtherCAT lost link.Index = 16#8041; DO module CH0 stopvalue after EtherCAT lost link.Subindex = 16#01; DO module CH0 stopvalue after EtherCAT lost link.Value = 0; DO module CH0 stopvalue after EtherCAT lost link.Size = 8; DO module CH0 stopvalue after EtherCAT lost link.AbortIfError = FALSE; DO module CH0 stopvalue after EtherCAT lost link.JumpToLine = FALSE; DO module CH0 stopvalue after EtherCAT lost link.Line = 0; DO module CH0 stopvalue after EtherCAT lost link.CompleteAccess = False; 2S485-0 enable and settings.Index = 16#8080; 2S485-0 enable and settings.Subindex = 16#01; 2S485-0 enable and settings.Value = 132; 2S485-0 enable and settings.Size = 16; 2S485-0 enable and settings.AbortIfError = FALSE; 2S485-0 enable and settings.JumpToLine = FALSE; 2S485-0 enable and settings.Line = 0; 2S485-0 enable and settings.CompleteAccess = False; 2S485-0 message_interval.Index = 16#8080; 2S485-0 message_interval.Subindex = 16#02; 2S485-0 message_interval.Value = 35; 2S485-0 message_interval.Size = 16; 2S485-0 message_interval.AbortIfError = FALSE; 2S485-0 message_interval.JumpToLine = FALSE; 2S485-0 message_interval.Line = 0;
            2S485-0 message_interval.CompleteAccess = False; 2S485-0 Number_terminals.Index = 16#8080; 2S485-0 Number_terminals.Subindex = 16#03; 2S485-0 Number_terminals.Value = 31; 2S485-0 Number_terminals.Size = 16; 2S485-0 Number_terminals.AbortIfError = FALSE; 2S485-0 Number_terminals.JumpToLine = FALSE; 2S485-0 Number_terminals.Line = 0; 2S485-0 Number_terminals.CompleteAccess = False; 2S485-0 datapacket_size.Index = 16#8080; 2S485-0 datapacket_size.Subindex = 16#04; 2S485-0 datapacket_size.Value = 20; 2S485-0 datapacket_size.Size = 16; 2S485-0 datapacket_size.AbortIfError = FALSE; 2S485-0 datapacket_size.JumpToLine = FALSE; 2S485-0 datapacket_size.Line = 0; 2S485-0 datapacket_size.CompleteAccess = False; 2S485-0 TX_buffersize.Index = 16#8080; 2S485-0 TX_buffersize.Subindex = 16#05; 2S485-0 TX_buffersize.Value = 1536; 2S485-0 TX_buffersize.Size = 16; 2S485-0 TX_buffersize.AbortIfError = FALSE; 2S485-0 TX_buffersize.JumpToLine = FALSE; 2S485-0 TX_buffersize.Line = 0; 2S485-0 TX_buffersize.CompleteAccess = False; 2S485-0 RX_buffersize.Index = 16#8080; 2S485-0 RX_buffersize.Subindex = 16#06; 2S485-0 RX_buffersize.Value = 1536; 2S485-0 RX_buffersize.Size = 16; 2S485-0 RX_buffersize.AbortIfError = FALSE; 2S485-0 RX_buffersize.JumpToLine = FALSE; 2S485-0 RX_buffersize.Line = 0; 2S485-0 RX_buffersize.CompleteAccess = False; 2S485-1 enable and settings.Index = 16#8080; 2S485-1 enable and settings.Subindex = 16#07; 2S485-1 enable and settings.Value = 644; 2S485-1 enable and settings.Size = 16; 2S485-1 enable and settings.AbortIfError = FALSE; 2S485-1 enable and settings.JumpToLine = FALSE; 2S485-1 enable and settings.Line = 0;
            2S485-1 enable and settings.CompleteAccess = False; 2S485-1 message_interval.Index = 16#8080; 2S485-1 message_interval.Subindex = 16#08; 2S485-1 message_interval.Value = 35; 2S485-1 message_interval.Size = 16; 2S485-1 message_interval.AbortIfError = FALSE; 2S485-1 message_interval.JumpToLine = FALSE; 2S485-1 message_interval.Line = 0; 2S485-1 message_interval.CompleteAccess = False; 2S485-1 Number_terminals.Index = 16#8080; 2S485-1 Number_terminals.Subindex = 16#09; 2S485-1 Number_terminals.Value = 31; 2S485-1 Number_terminals.Size = 16; 2S485-1 Number_terminals.AbortIfError = FALSE; 2S485-1 Number_terminals.JumpToLine = FALSE; 2S485-1 Number_terminals.Line = 0; 2S485-1 Number_terminals.CompleteAccess = False; 2S485-1 datapacket_size.Index = 16#8080; 2S485-1 datapacket_size.Subindex = 16#0A; 2S485-1 datapacket_size.Value = 20; 2S485-1 datapacket_size.Size = 16; 2S485-1 datapacket_size.AbortIfError = FALSE; 2S485-1 datapacket_size.JumpToLine = FALSE; 2S485-1 datapacket_size.Line = 0; 2S485-1 datapacket_size.CompleteAccess = False; 2S485-1 TX_buffersize.Index = 16#8080; 2S485-1 TX_buffersize.Subindex = 16#0B; 2S485-1 TX_buffersize.Value = 1536; 2S485-1 TX_buffersize.Size = 16; 2S485-1 TX_buffersize.AbortIfError = FALSE; 2S485-1 TX_buffersize.JumpToLine = FALSE; 2S485-1 TX_buffersize.Line = 0; 2S485-1 TX_buffersize.CompleteAccess = False; 2S485-1 RX_buffersize.Index = 16#8080; 2S485-1 RX_buffersize.Subindex = 16#0C; 2S485-1 RX_buffersize.Value = 1536; 2S485-1 RX_buffersize.Size = 16; 2S485-1 RX_buffersize.AbortIfError = FALSE; 2S485-1 RX_buffersize.JumpToLine = FALSE; 2S485-1 RX_buffersize.Line = 0;
            2S485-1 RX_buffersize.CompleteAccess = False; module bar_code_H.Index = 16#8080; module bar_code_H.Subindex = 16#0D; module bar_code_H.Value = 512; module bar_code_H.Size = 16; module bar_code_H.AbortIfError = FALSE; module bar_code_H.JumpToLine = FALSE; module bar_code_H.Line = 0; module bar_code_H.CompleteAccess = False; module bar_code_L.Index = 16#8080; module bar_code_L.Subindex = 16#0E; module bar_code_L.Value = 512; module bar_code_L.Size = 16; module bar_code_L.AbortIfError = FALSE; module bar_code_L.JumpToLine = FALSE; module bar_code_L.Line = 0; module bar_code_L.CompleteAccess = False; Reserved parameters.Index = 16#8080; Reserved parameters.Subindex = 16#0F; Reserved parameters.Value = 512; Reserved parameters.Size = 16; Reserved parameters.AbortIfError = FALSE; Reserved parameters.JumpToLine = FALSE; Reserved parameters.Line = 0; Reserved parameters.CompleteAccess = False; clear slot cfg 0xf030 entries.Index = 16#F030; clear slot cfg 0xf030 entries.Subindex = 16#00; clear slot cfg 0xf030 entries.Value = 0; clear slot cfg 0xf030 entries.Size = 8; clear slot cfg 0xf030 entries.AbortIfError = FALSE; clear slot cfg 0xf030 entries.JumpToLine = FALSE; clear slot cfg 0xf030 entries.Line = 0; clear slot cfg 0xf030 entries.CompleteAccess = False; download slot cfg 0xf030 entry.Index = 16#F030; download slot cfg 0xf030 entry.Subindex = 16#01; download slot cfg 0xf030 entry.Value = 284430352; download slot cfg 0xf030 entry.Size = 32; download slot cfg 0xf030 entry.AbortIfError = FALSE; download slot cfg 0xf030 entry.JumpToLine = FALSE; download slot cfg 0xf030 entry.Line = 0;
            download slot cfg 0xf030 entry.CompleteAccess = False; download slot cfg 0xf030 entry.Index = 16#F030; download slot cfg 0xf030 entry.Subindex = 16#02; download slot cfg 0xf030 entry.Value = 284430371; download slot cfg 0xf030 entry.Size = 32; download slot cfg 0xf030 entry.AbortIfError = FALSE; download slot cfg 0xf030 entry.JumpToLine = FALSE; download slot cfg 0xf030 entry.Line = 0; download slot cfg 0xf030 entry.CompleteAccess = False; download slot cfg 0xf030 entry.Index = 16#F030; download slot cfg 0xf030 entry.Subindex = 16#03; download slot cfg 0xf030 entry.Value = 284430481; download slot cfg 0xf030 entry.Size = 32; download slot cfg 0xf030 entry.AbortIfError = FALSE; download slot cfg 0xf030 entry.JumpToLine = FALSE; download slot cfg 0xf030 entry.Line = 0; download slot cfg 0xf030 entry.CompleteAccess = False; download slot cfg 0xf030 entry count.Index = 16#F030; download slot cfg 0xf030 entry count.Subindex = 16#00; download slot cfg 0xf030 entry count.Value = 3; download slot cfg 0xf030 entry count.Size = 8; download slot cfg 0xf030 entry count.AbortIfError = FALSE; download slot cfg 0xf030 entry count.JumpToLine = FALSE; download slot cfg 0xf030 entry count.Line = 0; download slot cfg 0xf030 entry count.CompleteAccess = False; RxTxPdo.NumberofExcludes = 0; RxTxPdo.NumberofEntries = 1; RxTxPdo.Index = 16#17A0; RxTxPdo.Fixed = True; RxTxPdo.Mandatory = False; RxTxPdo.Virtual = False; RxTxPdo.Sm = 2; RxTxPdo.Su = 2; RxTxPdo.Name = 'Device RPDO Mapping parameter'; RxTxPdo.DependOnSlot = False; RxTxPdo.DependOnSlotGroup = False; RxTxPdo.OverwrittenByModule = False; Device control.Index = 16#FB00; Device control.SubIndex = 0; Device control.Size = 16;
            Device control.Offset = 0; Device control.DependOnSlot = False; Device control.DependOnSlotGroup = False; RxTxPdo.NumberofExcludes = 2; RxTxPdo.NumberofEntries = 1; RxTxPdo.Index = 16#1609; RxTxPdo.Fixed = True; RxTxPdo.Mandatory = False; RxTxPdo.Virtual = False; RxTxPdo.Sm = 2; RxTxPdo.Su = 0; RxTxPdo.Name = '0008ER Output-8bit maping'; RxTxPdo.DependOnSlot = True; RxTxPdo.DependOnSlotGroup = False; RxTxPdo.OverwrittenByModule = True; Exclude = [16#1608,16#160A]; GL20_0008ER Digital output CH0-8bit.Index = 16#7041; GL20_0008ER Digital output CH0-8bit.SubIndex = 1; GL20_0008ER Digital output CH0-8bit.Size = 8; GL20_0008ER Digital output CH0-8bit.Offset = 0; GL20_0008ER Digital output CH0-8bit.DependOnSlot = True; GL20_0008ER Digital output CH0-8bit.DependOnSlotGroup = False; RxTxPdo.NumberofExcludes = 2; RxTxPdo.NumberofEntries = 1; RxTxPdo.Index = 16#160A; RxTxPdo.Fixed = True; RxTxPdo.Mandatory = False; RxTxPdo.Virtual = False; RxTxPdo.Sm = -1; RxTxPdo.Su = 0; RxTxPdo.Name = '0008ER Output-16bit maping'; RxTxPdo.DependOnSlot = True; RxTxPdo.DependOnSlotGroup = False; RxTxPdo.OverwrittenByModule = True; Exclude = [16#1608,16#1609]; GL20_0008ER Digital output CH0-16bit.Index = 16#7042; GL20_0008ER Digital output CH0-16bit.SubIndex = 1; GL20_0008ER Digital output CH0-16bit.Size = 16; GL20_0008ER Digital output CH0-16bit.Offset = 0; GL20_0008ER Digital output CH0-16bit.DependOnSlot = True;
            GL20_0008ER Digital output CH0-16bit.DependOnSlotGroup = False; RxTxPdo.NumberofExcludes = 2; RxTxPdo.NumberofEntries = 8; RxTxPdo.Index = 16#1608; RxTxPdo.Fixed = True; RxTxPdo.Mandatory = False; RxTxPdo.Virtual = False; RxTxPdo.Sm = -1; RxTxPdo.Su = 0; RxTxPdo.Name = '0008ER Output-bit maping'; RxTxPdo.DependOnSlot = True; RxTxPdo.DependOnSlotGroup = False; RxTxPdo.OverwrittenByModule = True; Exclude = [16#1609,16#160A]; GL20_0008ER Digital output bit0.Index = 16#7040; GL20_0008ER Digital output bit0.SubIndex = 1; GL20_0008ER Digital output bit0.Size = 1; GL20_0008ER Digital output bit0.Offset = 0; GL20_0008ER Digital output bit0.DependOnSlot = True; GL20_0008ER Digital output bit0.DependOnSlotGroup = False; GL20_0008ER Digital output bit1.Index = 16#7040; GL20_0008ER Digital output bit1.SubIndex = 2; GL20_0008ER Digital output bit1.Size = 1; GL20_0008ER Digital output bit1.Offset = 0; GL20_0008ER Digital output bit1.DependOnSlot = True; GL20_0008ER Digital output bit1.DependOnSlotGroup = False; GL20_0008ER Digital output bit2.Index = 16#7040; GL20_0008ER Digital output bit2.SubIndex = 3; GL20_0008ER Digital output bit2.Size = 1; GL20_0008ER Digital output bit2.Offset = 0; GL20_0008ER Digital output bit2.DependOnSlot = True; GL20_0008ER Digital output bit2.DependOnSlotGroup = False; GL20_0008ER Digital output bit3.Index = 16#7040; GL20_0008ER Digital output bit3.SubIndex = 4; GL20_0008ER Digital output bit3.Size = 1; GL20_0008ER Digital output bit3.Offset = 0; GL20_0008ER Digital output bit3.DependOnSlot = True; GL20_0008ER Digital output bit3.DependOnSlotGroup = False; GL20_0008ER Digital output bit4.Index = 16#7040; GL20_0008ER Digital output bit4.SubIndex = 5;
            GL20_0008ER Digital output bit4.Size = 1; GL20_0008ER Digital output bit4.Offset = 0; GL20_0008ER Digital output bit4.DependOnSlot = True; GL20_0008ER Digital output bit4.DependOnSlotGroup = False; GL20_0008ER Digital output bit5.Index = 16#7040; GL20_0008ER Digital output bit5.SubIndex = 6; GL20_0008ER Digital output bit5.Size = 1; GL20_0008ER Digital output bit5.Offset = 0; GL20_0008ER Digital output bit5.DependOnSlot = True; GL20_0008ER Digital output bit5.DependOnSlotGroup = False; GL20_0008ER Digital output bit6.Index = 16#7040; GL20_0008ER Digital output bit6.SubIndex = 7; GL20_0008ER Digital output bit6.Size = 1; GL20_0008ER Digital output bit6.Offset = 0; GL20_0008ER Digital output bit6.DependOnSlot = True; GL20_0008ER Digital output bit6.DependOnSlotGroup = False; GL20_0008ER Digital output bit7.Index = 16#7040; GL20_0008ER Digital output bit7.SubIndex = 8; GL20_0008ER Digital output bit7.Size = 1; GL20_0008ER Digital output bit7.Offset = 0; GL20_0008ER Digital output bit7.DependOnSlot = True; GL20_0008ER Digital output bit7.DependOnSlotGroup = False; RxTxPdo.NumberofExcludes = 0; RxTxPdo.NumberofEntries = 15; RxTxPdo.Index = 16#1613; RxTxPdo.Fixed = True; RxTxPdo.Mandatory = True; RxTxPdo.Virtual = False; RxTxPdo.Sm = 2; RxTxPdo.Su = 0; RxTxPdo.Name = 'RS485 Output maping'; RxTxPdo.DependOnSlot = True; RxTxPdo.DependOnSlotGroup = False; RxTxPdo.OverwrittenByModule = True; GL20_2S485 RS485-0 TXCOUNTER and length.Index = 16#7080; GL20_2S485 RS485-0 TXCOUNTER and length.SubIndex = 1; GL20_2S485 RS485-0 TXCOUNTER and length.Size = 32; GL20_2S485 RS485-0 TXCOUNTER and length.Offset = 0; GL20_2S485 RS485-0 TXCOUNTER and length.DependOnSlot = True; GL20_2S485 RS485-0 TXCOUNTER and length.DependOnSlotGroup = False;
            GL20_2S485 RS485-0 TX_DATA1.Index = 16#7080; GL20_2S485 RS485-0 TX_DATA1.SubIndex = 2; GL20_2S485 RS485-0 TX_DATA1.Size = 32; GL20_2S485 RS485-0 TX_DATA1.Offset = 0; GL20_2S485 RS485-0 TX_DATA1.DependOnSlot = True; GL20_2S485 RS485-0 TX_DATA1.DependOnSlotGroup = False; GL20_2S485 RS485-0 TX_DATA2.Index = 16#7080; GL20_2S485 RS485-0 TX_DATA2.SubIndex = 3; GL20_2S485 RS485-0 TX_DATA2.Size = 32; GL20_2S485 RS485-0 TX_DATA2.Offset = 0; GL20_2S485 RS485-0 TX_DATA2.DependOnSlot = True; GL20_2S485 RS485-0 TX_DATA2.DependOnSlotGroup = False; GL20_2S485 RS485-0 TX_DATA3.Index = 16#7080; GL20_2S485 RS485-0 TX_DATA3.SubIndex = 4; GL20_2S485 RS485-0 TX_DATA3.Size = 32; GL20_2S485 RS485-0 TX_DATA3.Offset = 0; GL20_2S485 RS485-0 TX_DATA3.DependOnSlot = True; GL20_2S485 RS485-0 TX_DATA3.DependOnSlotGroup = False; GL20_2S485 RS485-0 TX_DATA4.Index = 16#7080; GL20_2S485 RS485-0 TX_DATA4.SubIndex = 5; GL20_2S485 RS485-0 TX_DATA4.Size = 32; GL20_2S485 RS485-0 TX_DATA4.Offset = 0; GL20_2S485 RS485-0 TX_DATA4.DependOnSlot = True; GL20_2S485 RS485-0 TX_DATA4.DependOnSlotGroup = False; GL20_2S485 RS485-0 TX_DATA5.Index = 16#7080; GL20_2S485 RS485-0 TX_DATA5.SubIndex = 6; GL20_2S485 RS485-0 TX_DATA5.Size = 32; GL20_2S485 RS485-0 TX_DATA5.Offset = 0; GL20_2S485 RS485-0 TX_DATA5.DependOnSlot = True; GL20_2S485 RS485-0 TX_DATA5.DependOnSlotGroup = False; GL20_2S485 RS485-0 TX_DATA6.Index = 16#7080; GL20_2S485 RS485-0 TX_DATA6.SubIndex = 7; GL20_2S485 RS485-0 TX_DATA6.Size = 32; GL20_2S485 RS485-0 TX_DATA6.Offset = 0; GL20_2S485 RS485-0 TX_DATA6.DependOnSlot = True; GL20_2S485 RS485-0 TX_DATA6.DependOnSlotGroup = False; GL20_2S485 RS485-1 TXCOUNTER and length.Index = 16#7080; GL20_2S485 RS485-1 TXCOUNTER and length.SubIndex = 8; GL20_2S485 RS485-1 TXCOUNTER and length.Size = 32; GL20_2S485 RS485-1 TXCOUNTER and length.Offset = 0;
            GL20_2S485 RS485-1 TXCOUNTER and length.DependOnSlot = True; GL20_2S485 RS485-1 TXCOUNTER and length.DependOnSlotGroup = False; GL20_2S485 RS485-1 TX_DATA1.Index = 16#7080; GL20_2S485 RS485-1 TX_DATA1.SubIndex = 9; GL20_2S485 RS485-1 TX_DATA1.Size = 32; GL20_2S485 RS485-1 TX_DATA1.Offset = 0; GL20_2S485 RS485-1 TX_DATA1.DependOnSlot = True; GL20_2S485 RS485-1 TX_DATA1.DependOnSlotGroup = False; GL20_2S485 RS485-1 TX_DATA2.Index = 16#7080; GL20_2S485 RS485-1 TX_DATA2.SubIndex = 10; GL20_2S485 RS485-1 TX_DATA2.Size = 32; GL20_2S485 RS485-1 TX_DATA2.Offset = 0; GL20_2S485 RS485-1 TX_DATA2.DependOnSlot = True; GL20_2S485 RS485-1 TX_DATA2.DependOnSlotGroup = False; GL20_2S485 RS485-1 TX_DATA3.Index = 16#7080; GL20_2S485 RS485-1 TX_DATA3.SubIndex = 11; GL20_2S485 RS485-1 TX_DATA3.Size = 32; GL20_2S485 RS485-1 TX_DATA3.Offset = 0; GL20_2S485 RS485-1 TX_DATA3.DependOnSlot = True; GL20_2S485 RS485-1 TX_DATA3.DependOnSlotGroup = False; GL20_2S485 RS485-1 TX_DATA4.Index = 16#7080; GL20_2S485 RS485-1 TX_DATA4.SubIndex = 12; GL20_2S485 RS485-1 TX_DATA4.Size = 32; GL20_2S485 RS485-1 TX_DATA4.Offset = 0; GL20_2S485 RS485-1 TX_DATA4.DependOnSlot = True; GL20_2S485 RS485-1 TX_DATA4.DependOnSlotGroup = False; GL20_2S485 RS485-1 TX_DATA5.Index = 16#7080; GL20_2S485 RS485-1 TX_DATA5.SubIndex = 13; GL20_2S485 RS485-1 TX_DATA5.Size = 32; GL20_2S485 RS485-1 TX_DATA5.Offset = 0; GL20_2S485 RS485-1 TX_DATA5.DependOnSlot = True; GL20_2S485 RS485-1 TX_DATA5.DependOnSlotGroup = False; GL20_2S485 RS485-1 TX_DATA6.Index = 16#7080; GL20_2S485 RS485-1 TX_DATA6.SubIndex = 14; GL20_2S485 RS485-1 TX_DATA6.Size = 32; GL20_2S485 RS485-1 TX_DATA6.Offset = 0; GL20_2S485 RS485-1 TX_DATA6.DependOnSlot = True; GL20_2S485 RS485-1 TX_DATA6.DependOnSlotGroup = False; GL20_2S485 TX_status.Index = 16#7080; GL20_2S485 TX_status.SubIndex = 15;
            GL20_2S485 TX_status.Size = 32; GL20_2S485 TX_status.Offset = 0; GL20_2S485 TX_status.DependOnSlot = True; GL20_2S485 TX_status.DependOnSlotGroup = False; RxTxPdo.NumberofExcludes = 0; RxTxPdo.NumberofEntries = 2; RxTxPdo.Index = 16#1BA0; RxTxPdo.Fixed = True; RxTxPdo.Mandatory = False; RxTxPdo.Virtual = False; RxTxPdo.Sm = 3; RxTxPdo.Su = 3; RxTxPdo.Name = 'Device TPDO Mapping parameter'; RxTxPdo.DependOnSlot = False; RxTxPdo.DependOnSlotGroup = False; RxTxPdo.OverwrittenByModule = False; LBus status.Index = 16#F100; LBus status.SubIndex = 1; LBus status.Size = 16; LBus status.Offset = 0; LBus status.DependOnSlot = False; LBus status.DependOnSlotGroup = False; Fault ID.Index = 16#F100; Fault ID.SubIndex = 2; Fault ID.Size = 16; Fault ID.Offset = 0; Fault ID.DependOnSlot = False; Fault ID.DependOnSlotGroup = False; RxTxPdo.NumberofExcludes = 0; RxTxPdo.NumberofEntries = 2; RxTxPdo.Index = 16#1BA1; RxTxPdo.Fixed = True; RxTxPdo.Mandatory = False; RxTxPdo.Virtual = False; RxTxPdo.Sm = 3; RxTxPdo.Su = 3; RxTxPdo.Name = 'ErrorSolt TPDO Mapping parameter'; RxTxPdo.DependOnSlot = False; RxTxPdo.DependOnSlotGroup = False; RxTxPdo.OverwrittenByModule = False;
            ErrorSolt1.Index = 16#F110; ErrorSolt1.SubIndex = 1; ErrorSolt1.Size = 32; ErrorSolt1.Offset = 0; ErrorSolt1.DependOnSlot = False; ErrorSolt1.DependOnSlotGroup = False; ErrorSolt2.Index = 16#F110; ErrorSolt2.SubIndex = 2; ErrorSolt2.Size = 32; ErrorSolt2.Offset = 0; ErrorSolt2.DependOnSlot = False; ErrorSolt2.DependOnSlotGroup = False; RxTxPdo.NumberofExcludes = 2; RxTxPdo.NumberofEntries = 2; RxTxPdo.Index = 16#1A01; RxTxPdo.Fixed = True; RxTxPdo.Mandatory = False; RxTxPdo.Virtual = False; RxTxPdo.Sm = 3; RxTxPdo.Su = 0; RxTxPdo.Name = '1600END input-8bit maping'; RxTxPdo.DependOnSlot = True; RxTxPdo.DependOnSlotGroup = False; RxTxPdo.OverwrittenByModule = True; Exclude = [16#1A00,16#1A02]; GL20_1600END Digital input CH0-8bit.Index = 16#6001; GL20_1600END Digital input CH0-8bit.SubIndex = 1; GL20_1600END Digital input CH0-8bit.Size = 8; GL20_1600END Digital input CH0-8bit.Offset = 0; GL20_1600END Digital input CH0-8bit.DependOnSlot = True; GL20_1600END Digital input CH0-8bit.DependOnSlotGroup = False; GL20_1600END Digital input CH1-8bit.Index = 16#6001; GL20_1600END Digital input CH1-8bit.SubIndex = 2; GL20_1600END Digital input CH1-8bit.Size = 8; GL20_1600END Digital input CH1-8bit.Offset = 0; GL20_1600END Digital input CH1-8bit.DependOnSlot = True; GL20_1600END Digital input CH1-8bit.DependOnSlotGroup = False; RxTxPdo.NumberofExcludes = 2; RxTxPdo.NumberofEntries = 1; RxTxPdo.Index = 16#1A02;
            RxTxPdo.Fixed = True; RxTxPdo.Mandatory = False; RxTxPdo.Virtual = False; RxTxPdo.Sm = -1; RxTxPdo.Su = 0; RxTxPdo.Name = '1600END input-16bit maping'; RxTxPdo.DependOnSlot = True; RxTxPdo.DependOnSlotGroup = False; RxTxPdo.OverwrittenByModule = True; Exclude = [16#1A00,16#1A01]; GL20_1600END Digital input CH0-16bit.Index = 16#6002; GL20_1600END Digital input CH0-16bit.SubIndex = 1; GL20_1600END Digital input CH0-16bit.Size = 16; GL20_1600END Digital input CH0-16bit.Offset = 0; GL20_1600END Digital input CH0-16bit.DependOnSlot = True; GL20_1600END Digital input CH0-16bit.DependOnSlotGroup = False; RxTxPdo.NumberofExcludes = 2; RxTxPdo.NumberofEntries = 16; RxTxPdo.Index = 16#1A00; RxTxPdo.Fixed = True; RxTxPdo.Mandatory = False; RxTxPdo.Virtual = False; RxTxPdo.Sm = -1; RxTxPdo.Su = 0; RxTxPdo.Name = '1600END input-bit maping'; RxTxPdo.DependOnSlot = True; RxTxPdo.DependOnSlotGroup = False; RxTxPdo.OverwrittenByModule = True; Exclude = [16#1A01,16#1A02]; GL20_1600END Digital input bit0.Index = 16#6000; GL20_1600END Digital input bit0.SubIndex = 1; GL20_1600END Digital input bit0.Size = 1; GL20_1600END Digital input bit0.Offset = 0; GL20_1600END Digital input bit0.DependOnSlot = True; GL20_1600END Digital input bit0.DependOnSlotGroup = False; GL20_1600END Digital input bit1.Index = 16#6000; GL20_1600END Digital input bit1.SubIndex = 2; GL20_1600END Digital input bit1.Size = 1; GL20_1600END Digital input bit1.Offset = 0; GL20_1600END Digital input bit1.DependOnSlot = True;
            GL20_1600END Digital input bit1.DependOnSlotGroup = False; GL20_1600END Digital input bit2.Index = 16#6000; GL20_1600END Digital input bit2.SubIndex = 3; GL20_1600END Digital input bit2.Size = 1; GL20_1600END Digital input bit2.Offset = 0; GL20_1600END Digital input bit2.DependOnSlot = True; GL20_1600END Digital input bit2.DependOnSlotGroup = False; GL20_1600END Digital input bit3.Index = 16#6000; GL20_1600END Digital input bit3.SubIndex = 4; GL20_1600END Digital input bit3.Size = 1; GL20_1600END Digital input bit3.Offset = 0; GL20_1600END Digital input bit3.DependOnSlot = True; GL20_1600END Digital input bit3.DependOnSlotGroup = False; GL20_1600END Digital input bit4.Index = 16#6000; GL20_1600END Digital input bit4.SubIndex = 5; GL20_1600END Digital input bit4.Size = 1; GL20_1600END Digital input bit4.Offset = 0; GL20_1600END Digital input bit4.DependOnSlot = True; GL20_1600END Digital input bit4.DependOnSlotGroup = False; GL20_1600END Digital input bit5.Index = 16#6000; GL20_1600END Digital input bit5.SubIndex = 6; GL20_1600END Digital input bit5.Size = 1; GL20_1600END Digital input bit5.Offset = 0; GL20_1600END Digital input bit5.DependOnSlot = True; GL20_1600END Digital input bit5.DependOnSlotGroup = False; GL20_1600END Digital input bit6.Index = 16#6000; GL20_1600END Digital input bit6.SubIndex = 7; GL20_1600END Digital input bit6.Size = 1; GL20_1600END Digital input bit6.Offset = 0; GL20_1600END Digital input bit6.DependOnSlot = True; GL20_1600END Digital input bit6.DependOnSlotGroup = False; GL20_1600END Digital input bit7.Index = 16#6000; GL20_1600END Digital input bit7.SubIndex = 8; GL20_1600END Digital input bit7.Size = 1; GL20_1600END Digital input bit7.Offset = 0; GL20_1600END Digital input bit7.DependOnSlot = True; GL20_1600END Digital input bit7.DependOnSlotGroup = False; GL20_1600END Digital input bit8.Index = 16#6000; GL20_1600END Digital input bit8.SubIndex = 9; GL20_1600END Digital input bit8.Size = 1;
            GL20_1600END Digital input bit8.Offset = 0; GL20_1600END Digital input bit8.DependOnSlot = True; GL20_1600END Digital input bit8.DependOnSlotGroup = False; GL20_1600END Digital input bit9.Index = 16#6000; GL20_1600END Digital input bit9.SubIndex = 10; GL20_1600END Digital input bit9.Size = 1; GL20_1600END Digital input bit9.Offset = 0; GL20_1600END Digital input bit9.DependOnSlot = True; GL20_1600END Digital input bit9.DependOnSlotGroup = False; GL20_1600END Digital input bit10.Index = 16#6000; GL20_1600END Digital input bit10.SubIndex = 11; GL20_1600END Digital input bit10.Size = 1; GL20_1600END Digital input bit10.Offset = 0; GL20_1600END Digital input bit10.DependOnSlot = True; GL20_1600END Digital input bit10.DependOnSlotGroup = False; GL20_1600END Digital input bit11.Index = 16#6000; GL20_1600END Digital input bit11.SubIndex = 12; GL20_1600END Digital input bit11.Size = 1; GL20_1600END Digital input bit11.Offset = 0; GL20_1600END Digital input bit11.DependOnSlot = True; GL20_1600END Digital input bit11.DependOnSlotGroup = False; GL20_1600END Digital input bit12.Index = 16#6000; GL20_1600END Digital input bit12.SubIndex = 13; GL20_1600END Digital input bit12.Size = 1; GL20_1600END Digital input bit12.Offset = 0; GL20_1600END Digital input bit12.DependOnSlot = True; GL20_1600END Digital input bit12.DependOnSlotGroup = False; GL20_1600END Digital input bit13.Index = 16#6000; GL20_1600END Digital input bit13.SubIndex = 14; GL20_1600END Digital input bit13.Size = 1; GL20_1600END Digital input bit13.Offset = 0; GL20_1600END Digital input bit13.DependOnSlot = True; GL20_1600END Digital input bit13.DependOnSlotGroup = False; GL20_1600END Digital input bit14.Index = 16#6000; GL20_1600END Digital input bit14.SubIndex = 15; GL20_1600END Digital input bit14.Size = 1; GL20_1600END Digital input bit14.Offset = 0; GL20_1600END Digital input bit14.DependOnSlot = True; GL20_1600END Digital input bit14.DependOnSlotGroup = False; GL20_1600END Digital input bit15.Index = 16#6000;
            GL20_1600END Digital input bit15.SubIndex = 16; GL20_1600END Digital input bit15.Size = 1; GL20_1600END Digital input bit15.Offset = 0; GL20_1600END Digital input bit15.DependOnSlot = True; GL20_1600END Digital input bit15.DependOnSlotGroup = False; RxTxPdo.NumberofExcludes = 0; RxTxPdo.NumberofEntries = 15; RxTxPdo.Index = 16#1A13; RxTxPdo.Fixed = True; RxTxPdo.Mandatory = True; RxTxPdo.Virtual = False; RxTxPdo.Sm = 3; RxTxPdo.Su = 0; RxTxPdo.Name = 'RS485 Input maping'; RxTxPdo.DependOnSlot = True; RxTxPdo.DependOnSlotGroup = False; RxTxPdo.OverwrittenByModule = True; GL20_2S485 RS485-0 RXCOUNTER and length.Index = 16#6080; GL20_2S485 RS485-0 RXCOUNTER and length.SubIndex = 1; GL20_2S485 RS485-0 RXCOUNTER and length.Size = 32; GL20_2S485 RS485-0 RXCOUNTER and length.Offset = 0; GL20_2S485 RS485-0 RXCOUNTER and length.DependOnSlot = True; GL20_2S485 RS485-0 RXCOUNTER and length.DependOnSlotGroup = False; GL20_2S485 RS485-0 RX_DATA1.Index = 16#6080; GL20_2S485 RS485-0 RX_DATA1.SubIndex = 2; GL20_2S485 RS485-0 RX_DATA1.Size = 32; GL20_2S485 RS485-0 RX_DATA1.Offset = 0; GL20_2S485 RS485-0 RX_DATA1.DependOnSlot = True; GL20_2S485 RS485-0 RX_DATA1.DependOnSlotGroup = False; GL20_2S485 RS485-0 RX_DATA2.Index = 16#6080; GL20_2S485 RS485-0 RX_DATA2.SubIndex = 3; GL20_2S485 RS485-0 RX_DATA2.Size = 32; GL20_2S485 RS485-0 RX_DATA2.Offset = 0; GL20_2S485 RS485-0 RX_DATA2.DependOnSlot = True; GL20_2S485 RS485-0 RX_DATA2.DependOnSlotGroup = False; GL20_2S485 RS485-0 RX_DATA3.Index = 16#6080; GL20_2S485 RS485-0 RX_DATA3.SubIndex = 4; GL20_2S485 RS485-0 RX_DATA3.Size = 32; GL20_2S485 RS485-0 RX_DATA3.Offset = 0; GL20_2S485 RS485-0 RX_DATA3.DependOnSlot = True;
            GL20_2S485 RS485-0 RX_DATA3.DependOnSlotGroup = False; GL20_2S485 RS485-0 RX_DATA4.Index = 16#6080; GL20_2S485 RS485-0 RX_DATA4.SubIndex = 5; GL20_2S485 RS485-0 RX_DATA4.Size = 32; GL20_2S485 RS485-0 RX_DATA4.Offset = 0; GL20_2S485 RS485-0 RX_DATA4.DependOnSlot = True; GL20_2S485 RS485-0 RX_DATA4.DependOnSlotGroup = False; GL20_2S485 RS485-0 RX_DATA5.Index = 16#6080; GL20_2S485 RS485-0 RX_DATA5.SubIndex = 6; GL20_2S485 RS485-0 RX_DATA5.Size = 32; GL20_2S485 RS485-0 RX_DATA5.Offset = 0; GL20_2S485 RS485-0 RX_DATA5.DependOnSlot = True; GL20_2S485 RS485-0 RX_DATA5.DependOnSlotGroup = False; GL20_2S485 RS485-0 RX_DATA6.Index = 16#6080; GL20_2S485 RS485-0 RX_DATA6.SubIndex = 7; GL20_2S485 RS485-0 RX_DATA6.Size = 32; GL20_2S485 RS485-0 RX_DATA6.Offset = 0; GL20_2S485 RS485-0 RX_DATA6.DependOnSlot = True; GL20_2S485 RS485-0 RX_DATA6.DependOnSlotGroup = False; GL20_2S485 RS485-1 RXCOUNTER and length.Index = 16#6080; GL20_2S485 RS485-1 RXCOUNTER and length.SubIndex = 8; GL20_2S485 RS485-1 RXCOUNTER and length.Size = 32; GL20_2S485 RS485-1 RXCOUNTER and length.Offset = 0; GL20_2S485 RS485-1 RXCOUNTER and length.DependOnSlot = True; GL20_2S485 RS485-1 RXCOUNTER and length.DependOnSlotGroup = False; GL20_2S485 RS485-1 RX_DATA1.Index = 16#6080; GL20_2S485 RS485-1 RX_DATA1.SubIndex = 9; GL20_2S485 RS485-1 RX_DATA1.Size = 32; GL20_2S485 RS485-1 RX_DATA1.Offset = 0; GL20_2S485 RS485-1 RX_DATA1.DependOnSlot = True; GL20_2S485 RS485-1 RX_DATA1.DependOnSlotGroup = False; GL20_2S485 RS485-1 RX_DATA2.Index = 16#6080; GL20_2S485 RS485-1 RX_DATA2.SubIndex = 10; GL20_2S485 RS485-1 RX_DATA2.Size = 32; GL20_2S485 RS485-1 RX_DATA2.Offset = 0; GL20_2S485 RS485-1 RX_DATA2.DependOnSlot = True; GL20_2S485 RS485-1 RX_DATA2.DependOnSlotGroup = False; GL20_2S485 RS485-1 RX_DATA3.Index = 16#6080; GL20_2S485 RS485-1 RX_DATA3.SubIndex = 11; GL20_2S485 RS485-1 RX_DATA3.Size = 32;
            GL20_2S485 RS485-1 RX_DATA3.Offset = 0; GL20_2S485 RS485-1 RX_DATA3.DependOnSlot = True; GL20_2S485 RS485-1 RX_DATA3.DependOnSlotGroup = False; GL20_2S485 RS485-1 RX_DATA4.Index = 16#6080; GL20_2S485 RS485-1 RX_DATA4.SubIndex = 12; GL20_2S485 RS485-1 RX_DATA4.Size = 32; GL20_2S485 RS485-1 RX_DATA4.Offset = 0; GL20_2S485 RS485-1 RX_DATA4.DependOnSlot = True; GL20_2S485 RS485-1 RX_DATA4.DependOnSlotGroup = False; GL20_2S485 RS485-1 RX_DATA5.Index = 16#6080; GL20_2S485 RS485-1 RX_DATA5.SubIndex = 13; GL20_2S485 RS485-1 RX_DATA5.Size = 32; GL20_2S485 RS485-1 RX_DATA5.Offset = 0; GL20_2S485 RS485-1 RX_DATA5.DependOnSlot = True; GL20_2S485 RS485-1 RX_DATA5.DependOnSlotGroup = False; GL20_2S485 RS485-1 RX_DATA6.Index = 16#6080; GL20_2S485 RS485-1 RX_DATA6.SubIndex = 14; GL20_2S485 RS485-1 RX_DATA6.Size = 32; GL20_2S485 RS485-1 RX_DATA6.Offset = 0; GL20_2S485 RS485-1 RX_DATA6.DependOnSlot = True; GL20_2S485 RS485-1 RX_DATA6.DependOnSlotGroup = False; GL20_2S485 RX_status.Index = 16#6080; GL20_2S485 RX_status.SubIndex = 15; GL20_2S485 RX_status.Size = 32; GL20_2S485 RX_status.Offset = 0; GL20_2S485 RX_status.DependOnSlot = True; GL20_2S485 RX_status.DependOnSlotGroup = False; Device control.Name = 'Device control'; Device control.DataType = 'UINT'; Device control.Default = ''; Device control.Comment = ''; GL20_0008ER Digital output CH0-8bit.Name = 'GL20_0008ER Digital output CH0-8bit'; GL20_0008ER Digital output CH0-8bit.DataType = 'USINT'; GL20_0008ER Digital output CH0-8bit.Default = ''; GL20_0008ER Digital output CH0-8bit.Comment = ''; GL20_0008ER Digital output CH0-16bit.Name = 'GL20_0008ER Digital output CH0-16bit'; GL20_0008ER Digital output CH0-16bit.DataType = 'UINT'; GL20_0008ER Digital output CH0-16bit.Default = ''; GL20_0008ER Digital output CH0-16bit.Comment = ''; GL20_0008ER Digital output bit0.Name = 'GL20_0008ER Digital output bit0';
            GL20_0008ER Digital output bit0.DataType = 'BOOL'; GL20_0008ER Digital output bit0.Default = ''; GL20_0008ER Digital output bit0.Comment = ''; GL20_0008ER Digital output bit1.Name = 'GL20_0008ER Digital output bit1'; GL20_0008ER Digital output bit1.DataType = 'BOOL'; GL20_0008ER Digital output bit1.Default = ''; GL20_0008ER Digital output bit1.Comment = ''; GL20_0008ER Digital output bit2.Name = 'GL20_0008ER Digital output bit2'; GL20_0008ER Digital output bit2.DataType = 'BOOL'; GL20_0008ER Digital output bit2.Default = ''; GL20_0008ER Digital output bit2.Comment = ''; GL20_0008ER Digital output bit3.Name = 'GL20_0008ER Digital output bit3'; GL20_0008ER Digital output bit3.DataType = 'BOOL'; GL20_0008ER Digital output bit3.Default = ''; GL20_0008ER Digital output bit3.Comment = ''; GL20_0008ER Digital output bit4.Name = 'GL20_0008ER Digital output bit4'; GL20_0008ER Digital output bit4.DataType = 'BOOL'; GL20_0008ER Digital output bit4.Default = ''; GL20_0008ER Digital output bit4.Comment = ''; GL20_0008ER Digital output bit5.Name = 'GL20_0008ER Digital output bit5'; GL20_0008ER Digital output bit5.DataType = 'BOOL'; GL20_0008ER Digital output bit5.Default = ''; GL20_0008ER Digital output bit5.Comment = ''; GL20_0008ER Digital output bit6.Name = 'GL20_0008ER Digital output bit6'; GL20_0008ER Digital output bit6.DataType = 'BOOL'; GL20_0008ER Digital output bit6.Default = ''; GL20_0008ER Digital output bit6.Comment = ''; GL20_0008ER Digital output bit7.Name = 'GL20_0008ER Digital output bit7'; GL20_0008ER Digital output bit7.DataType = 'BOOL'; GL20_0008ER Digital output bit7.Default = ''; GL20_0008ER Digital output bit7.Comment = ''; GL20_2S485 RS485-0 TXCOUNTER and length.Name = 'GL20_2S485 RS485-0 TXCOUNTER and length'; GL20_2S485 RS485-0 TXCOUNTER and length.DataType = 'UDINT'; GL20_2S485 RS485-0 TXCOUNTER and length.Default = ''; GL20_2S485 RS485-0 TXCOUNTER and length.Comment = ''; GL20_2S485 RS485-0 TX_DATA1.Name = 'GL20_2S485 RS485-0 TX_DATA1'; GL20_2S485 RS485-0 TX_DATA1.DataType = 'UDINT'; GL20_2S485 RS485-0 TX_DATA1.Default = ''; GL20_2S485 RS485-0 TX_DATA1.Comment = ''; GL20_2S485 RS485-0 TX_DATA2.Name = 'GL20_2S485 RS485-0 TX_DATA2';
            GL20_2S485 RS485-0 TX_DATA2.DataType = 'UDINT'; GL20_2S485 RS485-0 TX_DATA2.Default = ''; GL20_2S485 RS485-0 TX_DATA2.Comment = ''; GL20_2S485 RS485-0 TX_DATA3.Name = 'GL20_2S485 RS485-0 TX_DATA3'; GL20_2S485 RS485-0 TX_DATA3.DataType = 'UDINT'; GL20_2S485 RS485-0 TX_DATA3.Default = ''; GL20_2S485 RS485-0 TX_DATA3.Comment = ''; GL20_2S485 RS485-0 TX_DATA4.Name = 'GL20_2S485 RS485-0 TX_DATA4'; GL20_2S485 RS485-0 TX_DATA4.DataType = 'UDINT'; GL20_2S485 RS485-0 TX_DATA4.Default = ''; GL20_2S485 RS485-0 TX_DATA4.Comment = ''; GL20_2S485 RS485-0 TX_DATA5.Name = 'GL20_2S485 RS485-0 TX_DATA5'; GL20_2S485 RS485-0 TX_DATA5.DataType = 'UDINT'; GL20_2S485 RS485-0 TX_DATA5.Default = ''; GL20_2S485 RS485-0 TX_DATA5.Comment = ''; GL20_2S485 RS485-0 TX_DATA6.Name = 'GL20_2S485 RS485-0 TX_DATA6'; GL20_2S485 RS485-0 TX_DATA6.DataType = 'UDINT'; GL20_2S485 RS485-0 TX_DATA6.Default = ''; GL20_2S485 RS485-0 TX_DATA6.Comment = ''; GL20_2S485 RS485-1 TXCOUNTER and length.Name = 'GL20_2S485 RS485-1 TXCOUNTER and length'; GL20_2S485 RS485-1 TXCOUNTER and length.DataType = 'UDINT'; GL20_2S485 RS485-1 TXCOUNTER and length.Default = ''; GL20_2S485 RS485-1 TXCOUNTER and length.Comment = ''; GL20_2S485 RS485-1 TX_DATA1.Name = 'GL20_2S485 RS485-1 TX_DATA1'; GL20_2S485 RS485-1 TX_DATA1.DataType = 'UDINT'; GL20_2S485 RS485-1 TX_DATA1.Default = ''; GL20_2S485 RS485-1 TX_DATA1.Comment = ''; GL20_2S485 RS485-1 TX_DATA2.Name = 'GL20_2S485 RS485-1 TX_DATA2'; GL20_2S485 RS485-1 TX_DATA2.DataType = 'UDINT'; GL20_2S485 RS485-1 TX_DATA2.Default = ''; GL20_2S485 RS485-1 TX_DATA2.Comment = ''; GL20_2S485 RS485-1 TX_DATA3.Name = 'GL20_2S485 RS485-1 TX_DATA3'; GL20_2S485 RS485-1 TX_DATA3.DataType = 'UDINT'; GL20_2S485 RS485-1 TX_DATA3.Default = ''; GL20_2S485 RS485-1 TX_DATA3.Comment = ''; GL20_2S485 RS485-1 TX_DATA4.Name = 'GL20_2S485 RS485-1 TX_DATA4'; GL20_2S485 RS485-1 TX_DATA4.DataType = 'UDINT'; GL20_2S485 RS485-1 TX_DATA4.Default = ''; GL20_2S485 RS485-1 TX_DATA4.Comment = ''; GL20_2S485 RS485-1 TX_DATA5.Name = 'GL20_2S485 RS485-1 TX_DATA5';
            GL20_2S485 RS485-1 TX_DATA5.DataType = 'UDINT'; GL20_2S485 RS485-1 TX_DATA5.Default = ''; GL20_2S485 RS485-1 TX_DATA5.Comment = ''; GL20_2S485 RS485-1 TX_DATA6.Name = 'GL20_2S485 RS485-1 TX_DATA6'; GL20_2S485 RS485-1 TX_DATA6.DataType = 'UDINT'; GL20_2S485 RS485-1 TX_DATA6.Default = ''; GL20_2S485 RS485-1 TX_DATA6.Comment = ''; GL20_2S485 TX_status.Name = 'GL20_2S485 TX_status'; GL20_2S485 TX_status.DataType = 'UDINT'; GL20_2S485 TX_status.Default = ''; GL20_2S485 TX_status.Comment = ''; LBus status.Name = 'LBus status'; LBus status.DataType = 'UINT'; LBus status.Default = ''; LBus status.Comment = ''; Fault ID.Name = 'Fault ID'; Fault ID.DataType = 'UINT'; Fault ID.Default = ''; Fault ID.Comment = ''; ErrorSolt1.Name = 'ErrorSolt1'; ErrorSolt1.DataType = 'UDINT'; ErrorSolt1.Default = ''; ErrorSolt1.Comment = ''; ErrorSolt2.Name = 'ErrorSolt2'; ErrorSolt2.DataType = 'UDINT'; ErrorSolt2.Default = ''; ErrorSolt2.Comment = ''; GL20_1600END Digital input CH0-8bit.Name = 'GL20_1600END Digital input CH0-8bit'; GL20_1600END Digital input CH0-8bit.DataType = 'USINT'; GL20_1600END Digital input CH0-8bit.Default = ''; GL20_1600END Digital input CH0-8bit.Comment = ''; GL20_1600END Digital input CH1-8bit.Name = 'GL20_1600END Digital input CH1-8bit'; GL20_1600END Digital input CH1-8bit.DataType = 'USINT'; GL20_1600END Digital input CH1-8bit.Default = ''; GL20_1600END Digital input CH1-8bit.Comment = ''; GL20_1600END Digital input CH0-16bit.Name = 'GL20_1600END Digital input CH0-16bit'; GL20_1600END Digital input CH0-16bit.DataType = 'UINT'; GL20_1600END Digital input CH0-16bit.Default = ''; GL20_1600END Digital input CH0-16bit.Comment = ''; GL20_1600END Digital input bit0.Name = 'GL20_1600END Digital input bit0';
            GL20_1600END Digital input bit0.DataType = 'BOOL'; GL20_1600END Digital input bit0.Default = ''; GL20_1600END Digital input bit0.Comment = ''; GL20_1600END Digital input bit1.Name = 'GL20_1600END Digital input bit1'; GL20_1600END Digital input bit1.DataType = 'BOOL'; GL20_1600END Digital input bit1.Default = ''; GL20_1600END Digital input bit1.Comment = ''; GL20_1600END Digital input bit2.Name = 'GL20_1600END Digital input bit2'; GL20_1600END Digital input bit2.DataType = 'BOOL'; GL20_1600END Digital input bit2.Default = ''; GL20_1600END Digital input bit2.Comment = ''; GL20_1600END Digital input bit3.Name = 'GL20_1600END Digital input bit3'; GL20_1600END Digital input bit3.DataType = 'BOOL'; GL20_1600END Digital input bit3.Default = ''; GL20_1600END Digital input bit3.Comment = ''; GL20_1600END Digital input bit4.Name = 'GL20_1600END Digital input bit4'; GL20_1600END Digital input bit4.DataType = 'BOOL'; GL20_1600END Digital input bit4.Default = ''; GL20_1600END Digital input bit4.Comment = ''; GL20_1600END Digital input bit5.Name = 'GL20_1600END Digital input bit5'; GL20_1600END Digital input bit5.DataType = 'BOOL'; GL20_1600END Digital input bit5.Default = ''; GL20_1600END Digital input bit5.Comment = ''; GL20_1600END Digital input bit6.Name = 'GL20_1600END Digital input bit6'; GL20_1600END Digital input bit6.DataType = 'BOOL'; GL20_1600END Digital input bit6.Default = ''; GL20_1600END Digital input bit6.Comment = ''; GL20_1600END Digital input bit7.Name = 'GL20_1600END Digital input bit7'; GL20_1600END Digital input bit7.DataType = 'BOOL'; GL20_1600END Digital input bit7.Default = ''; GL20_1600END Digital input bit7.Comment = ''; GL20_1600END Digital input bit8.Name = 'GL20_1600END Digital input bit8'; GL20_1600END Digital input bit8.DataType = 'BOOL'; GL20_1600END Digital input bit8.Default = ''; GL20_1600END Digital input bit8.Comment = ''; GL20_1600END Digital input bit9.Name = 'GL20_1600END Digital input bit9'; GL20_1600END Digital input bit9.DataType = 'BOOL'; GL20_1600END Digital input bit9.Default = ''; GL20_1600END Digital input bit9.Comment = ''; GL20_1600END Digital input bit10.Name = 'GL20_1600END Digital input bit10';
            GL20_1600END Digital input bit10.DataType = 'BOOL'; GL20_1600END Digital input bit10.Default = ''; GL20_1600END Digital input bit10.Comment = ''; GL20_1600END Digital input bit11.Name = 'GL20_1600END Digital input bit11'; GL20_1600END Digital input bit11.DataType = 'BOOL'; GL20_1600END Digital input bit11.Default = ''; GL20_1600END Digital input bit11.Comment = ''; GL20_1600END Digital input bit12.Name = 'GL20_1600END Digital input bit12'; GL20_1600END Digital input bit12.DataType = 'BOOL'; GL20_1600END Digital input bit12.Default = ''; GL20_1600END Digital input bit12.Comment = ''; GL20_1600END Digital input bit13.Name = 'GL20_1600END Digital input bit13'; GL20_1600END Digital input bit13.DataType = 'BOOL'; GL20_1600END Digital input bit13.Default = ''; GL20_1600END Digital input bit13.Comment = ''; GL20_1600END Digital input bit14.Name = 'GL20_1600END Digital input bit14'; GL20_1600END Digital input bit14.DataType = 'BOOL'; GL20_1600END Digital input bit14.Default = ''; GL20_1600END Digital input bit14.Comment = ''; GL20_1600END Digital input bit15.Name = 'GL20_1600END Digital input bit15'; GL20_1600END Digital input bit15.DataType = 'BOOL'; GL20_1600END Digital input bit15.Default = ''; GL20_1600END Digital input bit15.Comment = ''; GL20_2S485 RS485-0 RXCOUNTER and length.Name = 'GL20_2S485 RS485-0 RXCOUNTER and length'; GL20_2S485 RS485-0 RXCOUNTER and length.DataType = 'UDINT'; GL20_2S485 RS485-0 RXCOUNTER and length.Default = ''; GL20_2S485 RS485-0 RXCOUNTER and length.Comment = ''; GL20_2S485 RS485-0 RX_DATA1.Name = 'GL20_2S485 RS485-0 RX_DATA1'; GL20_2S485 RS485-0 RX_DATA1.DataType = 'UDINT'; GL20_2S485 RS485-0 RX_DATA1.Default = ''; GL20_2S485 RS485-0 RX_DATA1.Comment = ''; GL20_2S485 RS485-0 RX_DATA2.Name = 'GL20_2S485 RS485-0 RX_DATA2'; GL20_2S485 RS485-0 RX_DATA2.DataType = 'UDINT'; GL20_2S485 RS485-0 RX_DATA2.Default = ''; GL20_2S485 RS485-0 RX_DATA2.Comment = ''; GL20_2S485 RS485-0 RX_DATA3.Name = 'GL20_2S485 RS485-0 RX_DATA3'; GL20_2S485 RS485-0 RX_DATA3.DataType = 'UDINT'; GL20_2S485 RS485-0 RX_DATA3.Default = ''; GL20_2S485 RS485-0 RX_DATA3.Comment = ''; GL20_2S485 RS485-0 RX_DATA4.Name = 'GL20_2S485 RS485-0 RX_DATA4';
            GL20_2S485 RS485-0 RX_DATA4.DataType = 'UDINT'; GL20_2S485 RS485-0 RX_DATA4.Default = ''; GL20_2S485 RS485-0 RX_DATA4.Comment = ''; GL20_2S485 RS485-0 RX_DATA5.Name = 'GL20_2S485 RS485-0 RX_DATA5'; GL20_2S485 RS485-0 RX_DATA5.DataType = 'UDINT'; GL20_2S485 RS485-0 RX_DATA5.Default = ''; GL20_2S485 RS485-0 RX_DATA5.Comment = ''; GL20_2S485 RS485-0 RX_DATA6.Name = 'GL20_2S485 RS485-0 RX_DATA6'; GL20_2S485 RS485-0 RX_DATA6.DataType = 'UDINT'; GL20_2S485 RS485-0 RX_DATA6.Default = ''; GL20_2S485 RS485-0 RX_DATA6.Comment = ''; GL20_2S485 RS485-1 RXCOUNTER and length.Name = 'GL20_2S485 RS485-1 RXCOUNTER and length'; GL20_2S485 RS485-1 RXCOUNTER and length.DataType = 'UDINT'; GL20_2S485 RS485-1 RXCOUNTER and length.Default = ''; GL20_2S485 RS485-1 RXCOUNTER and length.Comment = ''; GL20_2S485 RS485-1 RX_DATA1.Name = 'GL20_2S485 RS485-1 RX_DATA1'; GL20_2S485 RS485-1 RX_DATA1.DataType = 'UDINT'; GL20_2S485 RS485-1 RX_DATA1.Default = ''; GL20_2S485 RS485-1 RX_DATA1.Comment = ''; GL20_2S485 RS485-1 RX_DATA2.Name = 'GL20_2S485 RS485-1 RX_DATA2'; GL20_2S485 RS485-1 RX_DATA2.DataType = 'UDINT'; GL20_2S485 RS485-1 RX_DATA2.Default = ''; GL20_2S485 RS485-1 RX_DATA2.Comment = ''; GL20_2S485 RS485-1 RX_DATA3.Name = 'GL20_2S485 RS485-1 RX_DATA3'; GL20_2S485 RS485-1 RX_DATA3.DataType = 'UDINT'; GL20_2S485 RS485-1 RX_DATA3.Default = ''; GL20_2S485 RS485-1 RX_DATA3.Comment = ''; GL20_2S485 RS485-1 RX_DATA4.Name = 'GL20_2S485 RS485-1 RX_DATA4'; GL20_2S485 RS485-1 RX_DATA4.DataType = 'UDINT'; GL20_2S485 RS485-1 RX_DATA4.Default = ''; GL20_2S485 RS485-1 RX_DATA4.Comment = ''; GL20_2S485 RS485-1 RX_DATA5.Name = 'GL20_2S485 RS485-1 RX_DATA5'; GL20_2S485 RS485-1 RX_DATA5.DataType = 'UDINT'; GL20_2S485 RS485-1 RX_DATA5.Default = ''; GL20_2S485 RS485-1 RX_DATA5.Comment = ''; GL20_2S485 RS485-1 RX_DATA6.Name = 'GL20_2S485 RS485-1 RX_DATA6'; GL20_2S485 RS485-1 RX_DATA6.DataType = 'UDINT'; GL20_2S485 RS485-1 RX_DATA6.Default = ''; GL20_2S485 RS485-1 RX_DATA6.Comment = ''; GL20_2S485 RX_status.Name = 'GL20_2S485 RX_status';
            GL20_2S485 RX_status.DataType = 'UDINT'; GL20_2S485 RX_status.Default = ''; GL20_2S485 RX_status.Comment = ''
          output Application.DCH遥控控制.发动机开关 : BOOL  // GL20_0008ER Digital output CH0-8bit.Bit0
          output Application.DCH遥控控制.发动机启动 : BOOL  // GL20_0008ER Digital output CH0-8bit.Bit1
          input  Application.报警代码3 : USINT  // GL20_1600END Digital input CH0-8bit
          input  Application.报警代码4 : USINT  // GL20_1600END Digital input CH1-8bit
          unmapped channels: Device control, GL20_0008ER Digital output CH0-8bit, GL20_2S485 RS485-0 TXCOUNTER and length, GL20_2S485 RS485-0 TX_DATA1, GL20_2S485 RS485-0 TX_DATA2, GL20_2S485 RS485-0 TX_DATA3, GL20_2S485 RS485-0 TX_DATA4, GL20_2S485 RS485-0 TX_DATA5, GL20_2S485 RS485-0 TX_DATA6, GL20_2S485 RS485-1 TXCOUNTER and length, GL20_2S485 RS485-1 TX_DATA1, GL20_2S485 RS485-1 TX_DATA2, GL20_2S485 RS485-1 TX_DATA3, GL20_2S485 RS485-1 TX_DATA4, GL20_2S485 RS485-1 TX_DATA5, GL20_2S485 RS485-1 TX_DATA6, GL20_2S485 TX_status, LBus status, Fault ID, ErrorSolt1, ErrorSolt2, GL20_2S485 RS485-0 RXCOUNTER and length, GL20_2S485 RS485-0 RX_DATA1, GL20_2S485 RS485-0 RX_DATA2, GL20_2S485 RS485-0 RX_DATA3, GL20_2S485 RS485-0 RX_DATA4, GL20_2S485 RS485-0 RX_DATA5, GL20_2S485 RS485-0 RX_DATA6, GL20_2S485 RS485-1 RXCOUNTER and length, GL20_2S485 RS485-1 RX_DATA1, GL20_2S485 RS485-1 RX_DATA2, GL20_2S485 RS485-1 RX_DATA3, GL20_2S485 RS485-1 RX_DATA4, GL20_2S485 RS485-1 RX_DATA5, GL20_2S485 RS485-1 RX_DATA6, GL20_2S485 RX_status
        GL20_1600END : GL20(GL20S)-1600END(16 channels DI module), Inovance, order no. GL20(GL20S)-1600END, version 0
        GL20_0008ER : GL20(GL20S)-0008ER(8 channels DO module), Inovance, order no. GL20(GL20S)-0008ER, version 0
        GL20_2S485 : GL20-2S485(2 channels RS485 converter), Inovance, order no. GL20-2S485, version 0
            settings: 2S485-1 enable and settings.Value = 644
      GL20_RTU_ECT_1 : GL20-RTU-ECT_1.3.21.0, Inovance, order no. GL20-RTU-ECT, version Revision=16#01006000
          settings: Number of Outputs = 2; Number of Inputs = 14; IOModuleSize = 4; IOModuleName = "GL20_4AD,GL20_4AD_1,GL20_1600END_1,GL20_0008ER_1"; Number of Infos about Outputs = 2; Number of Infos about Inputs = 14; Physical Address of the Slave = 1005; AutoIncr Address of the Slave = 4294967292; Sync.Length = 3; Sync.Length = 30; FMMU.Global Start Address = 16#02000048; FMMU.Length = 3; FMMU.Physical Start Address = 16#1800; FMMU.Access = 16#02; FMMU.Global Start Address = 16#01000080; FMMU.Length = 30; FMMU.Physical Start Address = 16#1C00; FMMU.Access = 16#01; Number of RxPDOs of the Slave = 4; Number of TxPDOs of the Slave = 7; AutoUpdate = False; DC sync0 cycletime = 4000; DC sync1 cycletime = 4000; Number of SDO = 38; 4AD module CH0 transform mode.Index = 16#8000; 4AD module CH0 transform mode.Subindex = 16#01; 4AD module CH0 transform mode.Value = 135; 4AD module CH0 transform mode.Size = 8; 4AD module CH0 transform mode.AbortIfError = FALSE; 4AD module CH0 transform mode.JumpToLine = FALSE; 4AD module CH0 transform mode.Line = 0; 4AD module CH0 transform mode.CompleteAccess = False; 4AD module CH1 transform mode.Index = 16#8000; 4AD module CH1 transform mode.Subindex = 16#02; 4AD module CH1 transform mode.Value = 135; 4AD module CH1 transform mode.Size = 8; 4AD module CH1 transform mode.AbortIfError = FALSE; 4AD module CH1 transform mode.JumpToLine = FALSE; 4AD module CH1 transform mode.Line = 0; 4AD module CH1 transform mode.CompleteAccess = False;
            4AD module CH2 transform mode.Index = 16#8000; 4AD module CH2 transform mode.Subindex = 16#03; 4AD module CH2 transform mode.Value = 135; 4AD module CH2 transform mode.Size = 8; 4AD module CH2 transform mode.AbortIfError = FALSE; 4AD module CH2 transform mode.JumpToLine = FALSE; 4AD module CH2 transform mode.Line = 0; 4AD module CH2 transform mode.CompleteAccess = False; 4AD module CH3 transform mode.Index = 16#8000; 4AD module CH3 transform mode.Subindex = 16#04; 4AD module CH3 transform mode.Value = 135; 4AD module CH3 transform mode.Size = 8; 4AD module CH3 transform mode.AbortIfError = FALSE; 4AD module CH3 transform mode.JumpToLine = FALSE; 4AD module CH3 transform mode.Line = 0; 4AD module CH3 transform mode.CompleteAccess = False; 4AD module CH0 Filter.Index = 16#8001; 4AD module CH0 Filter.Subindex = 16#01; 4AD module CH0 Filter.Value = 8; 4AD module CH0 Filter.Size = 8; 4AD module CH0 Filter.AbortIfError = FALSE; 4AD module CH0 Filter.JumpToLine = FALSE; 4AD module CH0 Filter.Line = 0; 4AD module CH0 Filter.CompleteAccess = False; 4AD module CH1 Filter.Index = 16#8001; 4AD module CH1 Filter.Subindex = 16#02; 4AD module CH1 Filter.Value = 8; 4AD module CH1 Filter.Size = 8; 4AD module CH1 Filter.AbortIfError = FALSE; 4AD module CH1 Filter.JumpToLine = FALSE; 4AD module CH1 Filter.Line = 0; 4AD module CH1 Filter.CompleteAccess = False; 4AD module CH2 Filter.Index = 16#8001; 4AD module CH2 Filter.Subindex = 16#03; 4AD module CH2 Filter.Value = 8; 4AD module CH2 Filter.Size = 8; 4AD module CH2 Filter.AbortIfError = FALSE; 4AD module CH2 Filter.JumpToLine = FALSE; 4AD module CH2 Filter.Line = 0; 4AD module CH2 Filter.CompleteAccess = False;
            4AD module CH3 Filter.Index = 16#8001; 4AD module CH3 Filter.Subindex = 16#04; 4AD module CH3 Filter.Value = 8; 4AD module CH3 Filter.Size = 8; 4AD module CH3 Filter.AbortIfError = FALSE; 4AD module CH3 Filter.JumpToLine = FALSE; 4AD module CH3 Filter.Line = 0; 4AD module CH3 Filter.CompleteAccess = False; 4AD module CH0 Detect.Index = 16#8002; 4AD module CH0 Detect.Subindex = 16#01; 4AD module CH0 Detect.Value = 0; 4AD module CH0 Detect.Size = 8; 4AD module CH0 Detect.AbortIfError = FALSE; 4AD module CH0 Detect.JumpToLine = FALSE; 4AD module CH0 Detect.Line = 0; 4AD module CH0 Detect.CompleteAccess = False; 4AD module CH1 Detect.Index = 16#8002; 4AD module CH1 Detect.Subindex = 16#02; 4AD module CH1 Detect.Value = 0; 4AD module CH1 Detect.Size = 8; 4AD module CH1 Detect.AbortIfError = FALSE; 4AD module CH1 Detect.JumpToLine = FALSE; 4AD module CH1 Detect.Line = 0; 4AD module CH1 Detect.CompleteAccess = False; 4AD module CH2 Detect.Index = 16#8002; 4AD module CH2 Detect.Subindex = 16#03; 4AD module CH2 Detect.Value = 0; 4AD module CH2 Detect.Size = 8; 4AD module CH2 Detect.AbortIfError = FALSE; 4AD module CH2 Detect.JumpToLine = FALSE; 4AD module CH2 Detect.Line = 0; 4AD module CH2 Detect.CompleteAccess = False; 4AD module CH3 Detect.Index = 16#8002; 4AD module CH3 Detect.Subindex = 16#04; 4AD module CH3 Detect.Value = 0; 4AD module CH3 Detect.Size = 8; 4AD module CH3 Detect.AbortIfError = FALSE; 4AD module CH3 Detect.JumpToLine = FALSE; 4AD module CH3 Detect.Line = 0; 4AD module CH3 Detect.CompleteAccess = False;
            4AD module CH0 transform mode.Index = 16#8040; 4AD module CH0 transform mode.Subindex = 16#01; 4AD module CH0 transform mode.Value = 135; 4AD module CH0 transform mode.Size = 8; 4AD module CH0 transform mode.AbortIfError = FALSE; 4AD module CH0 transform mode.JumpToLine = FALSE; 4AD module CH0 transform mode.Line = 0; 4AD module CH0 transform mode.CompleteAccess = False; 4AD module CH1 transform mode.Index = 16#8040; 4AD module CH1 transform mode.Subindex = 16#02; 4AD module CH1 transform mode.Value = 135; 4AD module CH1 transform mode.Size = 8; 4AD module CH1 transform mode.AbortIfError = FALSE; 4AD module CH1 transform mode.JumpToLine = FALSE; 4AD module CH1 transform mode.Line = 0; 4AD module CH1 transform mode.CompleteAccess = False; 4AD module CH2 transform mode.Index = 16#8040; 4AD module CH2 transform mode.Subindex = 16#03; 4AD module CH2 transform mode.Value = 135; 4AD module CH2 transform mode.Size = 8; 4AD module CH2 transform mode.AbortIfError = FALSE; 4AD module CH2 transform mode.JumpToLine = FALSE; 4AD module CH2 transform mode.Line = 0; 4AD module CH2 transform mode.CompleteAccess = False; 4AD module CH3 transform mode.Index = 16#8040; 4AD module CH3 transform mode.Subindex = 16#04; 4AD module CH3 transform mode.Value = 135; 4AD module CH3 transform mode.Size = 8; 4AD module CH3 transform mode.AbortIfError = FALSE; 4AD module CH3 transform mode.JumpToLine = FALSE; 4AD module CH3 transform mode.Line = 0; 4AD module CH3 transform mode.CompleteAccess = False; 4AD module CH0 Filter.Index = 16#8041; 4AD module CH0 Filter.Subindex = 16#01; 4AD module CH0 Filter.Value = 8; 4AD module CH0 Filter.Size = 8; 4AD module CH0 Filter.AbortIfError = FALSE; 4AD module CH0 Filter.JumpToLine = FALSE; 4AD module CH0 Filter.Line = 0; 4AD module CH0 Filter.CompleteAccess = False;
            4AD module CH1 Filter.Index = 16#8041; 4AD module CH1 Filter.Subindex = 16#02; 4AD module CH1 Filter.Value = 8; 4AD module CH1 Filter.Size = 8; 4AD module CH1 Filter.AbortIfError = FALSE; 4AD module CH1 Filter.JumpToLine = FALSE; 4AD module CH1 Filter.Line = 0; 4AD module CH1 Filter.CompleteAccess = False; 4AD module CH2 Filter.Index = 16#8041; 4AD module CH2 Filter.Subindex = 16#03; 4AD module CH2 Filter.Value = 8; 4AD module CH2 Filter.Size = 8; 4AD module CH2 Filter.AbortIfError = FALSE; 4AD module CH2 Filter.JumpToLine = FALSE; 4AD module CH2 Filter.Line = 0; 4AD module CH2 Filter.CompleteAccess = False; 4AD module CH3 Filter.Index = 16#8041; 4AD module CH3 Filter.Subindex = 16#04; 4AD module CH3 Filter.Value = 8; 4AD module CH3 Filter.Size = 8; 4AD module CH3 Filter.AbortIfError = FALSE; 4AD module CH3 Filter.JumpToLine = FALSE; 4AD module CH3 Filter.Line = 0; 4AD module CH3 Filter.CompleteAccess = False; 4AD module CH0 Detect.Index = 16#8042; 4AD module CH0 Detect.Subindex = 16#01; 4AD module CH0 Detect.Value = 0; 4AD module CH0 Detect.Size = 8; 4AD module CH0 Detect.AbortIfError = FALSE; 4AD module CH0 Detect.JumpToLine = FALSE; 4AD module CH0 Detect.Line = 0; 4AD module CH0 Detect.CompleteAccess = False; 4AD module CH1 Detect.Index = 16#8042; 4AD module CH1 Detect.Subindex = 16#02; 4AD module CH1 Detect.Value = 0; 4AD module CH1 Detect.Size = 8; 4AD module CH1 Detect.AbortIfError = FALSE; 4AD module CH1 Detect.JumpToLine = FALSE; 4AD module CH1 Detect.Line = 0; 4AD module CH1 Detect.CompleteAccess = False;
            4AD module CH2 Detect.Index = 16#8042; 4AD module CH2 Detect.Subindex = 16#03; 4AD module CH2 Detect.Value = 0; 4AD module CH2 Detect.Size = 8; 4AD module CH2 Detect.AbortIfError = FALSE; 4AD module CH2 Detect.JumpToLine = FALSE; 4AD module CH2 Detect.Line = 0; 4AD module CH2 Detect.CompleteAccess = False; 4AD module CH3 Detect.Index = 16#8042; 4AD module CH3 Detect.Subindex = 16#04; 4AD module CH3 Detect.Value = 0; 4AD module CH3 Detect.Size = 8; 4AD module CH3 Detect.AbortIfError = FALSE; 4AD module CH3 Detect.JumpToLine = FALSE; 4AD module CH3 Detect.Line = 0; 4AD module CH3 Detect.CompleteAccess = False; DI module CH0 filter time.Index = 16#8080; DI module CH0 filter time.Subindex = 16#01; DI module CH0 filter time.Value = 4; DI module CH0 filter time.Size = 16; DI module CH0 filter time.AbortIfError = FALSE; DI module CH0 filter time.JumpToLine = FALSE; DI module CH0 filter time.Line = 0; DI module CH0 filter time.CompleteAccess = False; DI module CH1 filter time.Index = 16#8080; DI module CH1 filter time.Subindex = 16#02; DI module CH1 filter time.Value = 4; DI module CH1 filter time.Size = 16; DI module CH1 filter time.AbortIfError = FALSE; DI module CH1 filter time.JumpToLine = FALSE; DI module CH1 filter time.Line = 0; DI module CH1 filter time.CompleteAccess = False; DO module CH0 stopmode after EtherCAT lost link.Index = 16#80C0; DO module CH0 stopmode after EtherCAT lost link.Subindex = 16#01; DO module CH0 stopmode after EtherCAT lost link.Value = 255; DO module CH0 stopmode after EtherCAT lost link.Size = 8; DO module CH0 stopmode after EtherCAT lost link.AbortIfError = FALSE; DO module CH0 stopmode after EtherCAT lost link.JumpToLine = FALSE; DO module CH0 stopmode after EtherCAT lost link.Line = 0; DO module CH0 stopmode after EtherCAT lost link.CompleteAccess = False;
            DO module CH0 stopvalue after EtherCAT lost link.Index = 16#80C1; DO module CH0 stopvalue after EtherCAT lost link.Subindex = 16#01; DO module CH0 stopvalue after EtherCAT lost link.Value = 0; DO module CH0 stopvalue after EtherCAT lost link.Size = 8; DO module CH0 stopvalue after EtherCAT lost link.AbortIfError = FALSE; DO module CH0 stopvalue after EtherCAT lost link.JumpToLine = FALSE; DO module CH0 stopvalue after EtherCAT lost link.Line = 0; DO module CH0 stopvalue after EtherCAT lost link.CompleteAccess = False; clear slot cfg 0xf030 entries.Index = 16#F030; clear slot cfg 0xf030 entries.Subindex = 16#00; clear slot cfg 0xf030 entries.Value = 0; clear slot cfg 0xf030 entries.Size = 8; clear slot cfg 0xf030 entries.AbortIfError = FALSE; clear slot cfg 0xf030 entries.JumpToLine = FALSE; clear slot cfg 0xf030 entries.Line = 0; clear slot cfg 0xf030 entries.CompleteAccess = False; download slot cfg 0xf030 entry.Index = 16#F030; download slot cfg 0xf030 entry.Subindex = 16#01; download slot cfg 0xf030 entry.Value = 284430384; download slot cfg 0xf030 entry.Size = 32; download slot cfg 0xf030 entry.AbortIfError = FALSE; download slot cfg 0xf030 entry.JumpToLine = FALSE; download slot cfg 0xf030 entry.Line = 0; download slot cfg 0xf030 entry.CompleteAccess = False; download slot cfg 0xf030 entry.Index = 16#F030; download slot cfg 0xf030 entry.Subindex = 16#02; download slot cfg 0xf030 entry.Value = 284430384; download slot cfg 0xf030 entry.Size = 32; download slot cfg 0xf030 entry.AbortIfError = FALSE; download slot cfg 0xf030 entry.JumpToLine = FALSE; download slot cfg 0xf030 entry.Line = 0; download slot cfg 0xf030 entry.CompleteAccess = False; download slot cfg 0xf030 entry.Index = 16#F030; download slot cfg 0xf030 entry.Subindex = 16#03; download slot cfg 0xf030 entry.Value = 284430352; download slot cfg 0xf030 entry.Size = 32; download slot cfg 0xf030 entry.AbortIfError = FALSE; download slot cfg 0xf030 entry.JumpToLine = FALSE; download slot cfg 0xf030 entry.Line = 0; download slot cfg 0xf030 entry.CompleteAccess = False;
            download slot cfg 0xf030 entry.Index = 16#F030; download slot cfg 0xf030 entry.Subindex = 16#04; download slot cfg 0xf030 entry.Value = 284430371; download slot cfg 0xf030 entry.Size = 32; download slot cfg 0xf030 entry.AbortIfError = FALSE; download slot cfg 0xf030 entry.JumpToLine = FALSE; download slot cfg 0xf030 entry.Line = 0; download slot cfg 0xf030 entry.CompleteAccess = False; download slot cfg 0xf030 entry count.Index = 16#F030; download slot cfg 0xf030 entry count.Subindex = 16#00; download slot cfg 0xf030 entry count.Value = 4; download slot cfg 0xf030 entry count.Size = 8; download slot cfg 0xf030 entry count.AbortIfError = FALSE; download slot cfg 0xf030 entry count.JumpToLine = FALSE; download slot cfg 0xf030 entry count.Line = 0; download slot cfg 0xf030 entry count.CompleteAccess = False; RxTxPdo.NumberofExcludes = 0; RxTxPdo.NumberofEntries = 1; RxTxPdo.Index = 16#17A0; RxTxPdo.Fixed = True; RxTxPdo.Mandatory = False; RxTxPdo.Virtual = False; RxTxPdo.Sm = 2; RxTxPdo.Su = 2; RxTxPdo.Name = 'Device RPDO Mapping parameter'; RxTxPdo.DependOnSlot = False; RxTxPdo.DependOnSlotGroup = False; RxTxPdo.OverwrittenByModule = False; Device control.Index = 16#FB00; Device control.SubIndex = 0; Device control.Size = 16; Device control.Offset = 0; Device control.DependOnSlot = False; Device control.DependOnSlotGroup = False; RxTxPdo.NumberofExcludes = 2; RxTxPdo.NumberofEntries = 1; RxTxPdo.Index = 16#1619; RxTxPdo.Fixed = True; RxTxPdo.Mandatory = False; RxTxPdo.Virtual = False;
            RxTxPdo.Sm = 2; RxTxPdo.Su = 0; RxTxPdo.Name = '0008ER Output-8bit maping'; RxTxPdo.DependOnSlot = True; RxTxPdo.DependOnSlotGroup = False; RxTxPdo.OverwrittenByModule = True; Exclude = [16#1618,16#161A]; GL20_0008ER_1 Digital output CH0-8bit.Index = 16#70C1; GL20_0008ER_1 Digital output CH0-8bit.SubIndex = 1; GL20_0008ER_1 Digital output CH0-8bit.Size = 8; GL20_0008ER_1 Digital output CH0-8bit.Offset = 0; GL20_0008ER_1 Digital output CH0-8bit.DependOnSlot = True; GL20_0008ER_1 Digital output CH0-8bit.DependOnSlotGroup = False; RxTxPdo.NumberofExcludes = 2; RxTxPdo.NumberofEntries = 1; RxTxPdo.Index = 16#161A; RxTxPdo.Fixed = True; RxTxPdo.Mandatory = False; RxTxPdo.Virtual = False; RxTxPdo.Sm = -1; RxTxPdo.Su = 0; RxTxPdo.Name = '0008ER Output-16bit maping'; RxTxPdo.DependOnSlot = True; RxTxPdo.DependOnSlotGroup = False; RxTxPdo.OverwrittenByModule = True; Exclude = [16#1618,16#1619]; GL20_0008ER_1 Digital output CH0-16bit.Index = 16#70C2; GL20_0008ER_1 Digital output CH0-16bit.SubIndex = 1; GL20_0008ER_1 Digital output CH0-16bit.Size = 16; GL20_0008ER_1 Digital output CH0-16bit.Offset = 0; GL20_0008ER_1 Digital output CH0-16bit.DependOnSlot = True; GL20_0008ER_1 Digital output CH0-16bit.DependOnSlotGroup = False; RxTxPdo.NumberofExcludes = 2; RxTxPdo.NumberofEntries = 8; RxTxPdo.Index = 16#1618; RxTxPdo.Fixed = True; RxTxPdo.Mandatory = False; RxTxPdo.Virtual = False; RxTxPdo.Sm = -1; RxTxPdo.Su = 0;
            RxTxPdo.Name = '0008ER Output-bit maping'; RxTxPdo.DependOnSlot = True; RxTxPdo.DependOnSlotGroup = False; RxTxPdo.OverwrittenByModule = True; Exclude = [16#1619,16#161A]; GL20_0008ER_1 Digital output bit0.Index = 16#70C0; GL20_0008ER_1 Digital output bit0.SubIndex = 1; GL20_0008ER_1 Digital output bit0.Size = 1; GL20_0008ER_1 Digital output bit0.Offset = 0; GL20_0008ER_1 Digital output bit0.DependOnSlot = True; GL20_0008ER_1 Digital output bit0.DependOnSlotGroup = False; GL20_0008ER_1 Digital output bit1.Index = 16#70C0; GL20_0008ER_1 Digital output bit1.SubIndex = 2; GL20_0008ER_1 Digital output bit1.Size = 1; GL20_0008ER_1 Digital output bit1.Offset = 0; GL20_0008ER_1 Digital output bit1.DependOnSlot = True; GL20_0008ER_1 Digital output bit1.DependOnSlotGroup = False; GL20_0008ER_1 Digital output bit2.Index = 16#70C0; GL20_0008ER_1 Digital output bit2.SubIndex = 3; GL20_0008ER_1 Digital output bit2.Size = 1; GL20_0008ER_1 Digital output bit2.Offset = 0; GL20_0008ER_1 Digital output bit2.DependOnSlot = True; GL20_0008ER_1 Digital output bit2.DependOnSlotGroup = False; GL20_0008ER_1 Digital output bit3.Index = 16#70C0; GL20_0008ER_1 Digital output bit3.SubIndex = 4; GL20_0008ER_1 Digital output bit3.Size = 1; GL20_0008ER_1 Digital output bit3.Offset = 0; GL20_0008ER_1 Digital output bit3.DependOnSlot = True; GL20_0008ER_1 Digital output bit3.DependOnSlotGroup = False; GL20_0008ER_1 Digital output bit4.Index = 16#70C0; GL20_0008ER_1 Digital output bit4.SubIndex = 5; GL20_0008ER_1 Digital output bit4.Size = 1; GL20_0008ER_1 Digital output bit4.Offset = 0; GL20_0008ER_1 Digital output bit4.DependOnSlot = True; GL20_0008ER_1 Digital output bit4.DependOnSlotGroup = False; GL20_0008ER_1 Digital output bit5.Index = 16#70C0; GL20_0008ER_1 Digital output bit5.SubIndex = 6; GL20_0008ER_1 Digital output bit5.Size = 1; GL20_0008ER_1 Digital output bit5.Offset = 0; GL20_0008ER_1 Digital output bit5.DependOnSlot = True;
            GL20_0008ER_1 Digital output bit5.DependOnSlotGroup = False; GL20_0008ER_1 Digital output bit6.Index = 16#70C0; GL20_0008ER_1 Digital output bit6.SubIndex = 7; GL20_0008ER_1 Digital output bit6.Size = 1; GL20_0008ER_1 Digital output bit6.Offset = 0; GL20_0008ER_1 Digital output bit6.DependOnSlot = True; GL20_0008ER_1 Digital output bit6.DependOnSlotGroup = False; GL20_0008ER_1 Digital output bit7.Index = 16#70C0; GL20_0008ER_1 Digital output bit7.SubIndex = 8; GL20_0008ER_1 Digital output bit7.Size = 1; GL20_0008ER_1 Digital output bit7.Offset = 0; GL20_0008ER_1 Digital output bit7.DependOnSlot = True; GL20_0008ER_1 Digital output bit7.DependOnSlotGroup = False; RxTxPdo.NumberofExcludes = 0; RxTxPdo.NumberofEntries = 2; RxTxPdo.Index = 16#1BA0; RxTxPdo.Fixed = True; RxTxPdo.Mandatory = False; RxTxPdo.Virtual = False; RxTxPdo.Sm = 3; RxTxPdo.Su = 3; RxTxPdo.Name = 'Device TPDO Mapping parameter'; RxTxPdo.DependOnSlot = False; RxTxPdo.DependOnSlotGroup = False; RxTxPdo.OverwrittenByModule = False; LBus status.Index = 16#F100; LBus status.SubIndex = 1; LBus status.Size = 16; LBus status.Offset = 0; LBus status.DependOnSlot = False; LBus status.DependOnSlotGroup = False; Fault ID.Index = 16#F100; Fault ID.SubIndex = 2; Fault ID.Size = 16; Fault ID.Offset = 0; Fault ID.DependOnSlot = False; Fault ID.DependOnSlotGroup = False; RxTxPdo.NumberofExcludes = 0; RxTxPdo.NumberofEntries = 2; RxTxPdo.Index = 16#1BA1;
            RxTxPdo.Fixed = True; RxTxPdo.Mandatory = False; RxTxPdo.Virtual = False; RxTxPdo.Sm = 3; RxTxPdo.Su = 3; RxTxPdo.Name = 'ErrorSolt TPDO Mapping parameter'; RxTxPdo.DependOnSlot = False; RxTxPdo.DependOnSlotGroup = False; RxTxPdo.OverwrittenByModule = False; ErrorSolt1.Index = 16#F110; ErrorSolt1.SubIndex = 1; ErrorSolt1.Size = 32; ErrorSolt1.Offset = 0; ErrorSolt1.DependOnSlot = False; ErrorSolt1.DependOnSlotGroup = False; ErrorSolt2.Index = 16#F110; ErrorSolt2.SubIndex = 2; ErrorSolt2.Size = 32; ErrorSolt2.Offset = 0; ErrorSolt2.DependOnSlot = False; ErrorSolt2.DependOnSlotGroup = False; RxTxPdo.NumberofExcludes = 0; RxTxPdo.NumberofEntries = 4; RxTxPdo.Index = 16#1A02; RxTxPdo.Fixed = True; RxTxPdo.Mandatory = True; RxTxPdo.Virtual = False; RxTxPdo.Sm = 3; RxTxPdo.Su = 0; RxTxPdo.Name = '4AD Input maping'; RxTxPdo.DependOnSlot = True; RxTxPdo.DependOnSlotGroup = False; RxTxPdo.OverwrittenByModule = True; GL20_4AD AD CH0.Index = 16#6000; GL20_4AD AD CH0.SubIndex = 1; GL20_4AD AD CH0.Size = 16; GL20_4AD AD CH0.Offset = 0; GL20_4AD AD CH0.DependOnSlot = True; GL20_4AD AD CH0.DependOnSlotGroup = False; GL20_4AD AD CH1.Index = 16#6000;
            GL20_4AD AD CH1.SubIndex = 2; GL20_4AD AD CH1.Size = 16; GL20_4AD AD CH1.Offset = 0; GL20_4AD AD CH1.DependOnSlot = True; GL20_4AD AD CH1.DependOnSlotGroup = False; GL20_4AD AD CH2.Index = 16#6000; GL20_4AD AD CH2.SubIndex = 3; GL20_4AD AD CH2.Size = 16; GL20_4AD AD CH2.Offset = 0; GL20_4AD AD CH2.DependOnSlot = True; GL20_4AD AD CH2.DependOnSlotGroup = False; GL20_4AD AD CH3.Index = 16#6000; GL20_4AD AD CH3.SubIndex = 4; GL20_4AD AD CH3.Size = 16; GL20_4AD AD CH3.Offset = 0; GL20_4AD AD CH3.DependOnSlot = True; GL20_4AD AD CH3.DependOnSlotGroup = False; RxTxPdo.NumberofExcludes = 0; RxTxPdo.NumberofEntries = 4; RxTxPdo.Index = 16#1A0A; RxTxPdo.Fixed = True; RxTxPdo.Mandatory = True; RxTxPdo.Virtual = False; RxTxPdo.Sm = 3; RxTxPdo.Su = 0; RxTxPdo.Name = '4AD Input maping'; RxTxPdo.DependOnSlot = True; RxTxPdo.DependOnSlotGroup = False; RxTxPdo.OverwrittenByModule = True; GL20_4AD_1 AD CH0.Index = 16#6040; GL20_4AD_1 AD CH0.SubIndex = 1; GL20_4AD_1 AD CH0.Size = 16; GL20_4AD_1 AD CH0.Offset = 0; GL20_4AD_1 AD CH0.DependOnSlot = True; GL20_4AD_1 AD CH0.DependOnSlotGroup = False; GL20_4AD_1 AD CH1.Index = 16#6040; GL20_4AD_1 AD CH1.SubIndex = 2; GL20_4AD_1 AD CH1.Size = 16; GL20_4AD_1 AD CH1.Offset = 0; GL20_4AD_1 AD CH1.DependOnSlot = True;
            GL20_4AD_1 AD CH1.DependOnSlotGroup = False; GL20_4AD_1 AD CH2.Index = 16#6040; GL20_4AD_1 AD CH2.SubIndex = 3; GL20_4AD_1 AD CH2.Size = 16; GL20_4AD_1 AD CH2.Offset = 0; GL20_4AD_1 AD CH2.DependOnSlot = True; GL20_4AD_1 AD CH2.DependOnSlotGroup = False; GL20_4AD_1 AD CH3.Index = 16#6040; GL20_4AD_1 AD CH3.SubIndex = 4; GL20_4AD_1 AD CH3.Size = 16; GL20_4AD_1 AD CH3.Offset = 0; GL20_4AD_1 AD CH3.DependOnSlot = True; GL20_4AD_1 AD CH3.DependOnSlotGroup = False; RxTxPdo.NumberofExcludes = 2; RxTxPdo.NumberofEntries = 2; RxTxPdo.Index = 16#1A11; RxTxPdo.Fixed = True; RxTxPdo.Mandatory = False; RxTxPdo.Virtual = False; RxTxPdo.Sm = 3; RxTxPdo.Su = 0; RxTxPdo.Name = '1600END input-8bit maping'; RxTxPdo.DependOnSlot = True; RxTxPdo.DependOnSlotGroup = False; RxTxPdo.OverwrittenByModule = True; Exclude = [16#1A10,16#1A12]; GL20_1600END_1 Digital input CH0-8bit.Index = 16#6081; GL20_1600END_1 Digital input CH0-8bit.SubIndex = 1; GL20_1600END_1 Digital input CH0-8bit.Size = 8; GL20_1600END_1 Digital input CH0-8bit.Offset = 0; GL20_1600END_1 Digital input CH0-8bit.DependOnSlot = True; GL20_1600END_1 Digital input CH0-8bit.DependOnSlotGroup = False; GL20_1600END_1 Digital input CH1-8bit.Index = 16#6081; GL20_1600END_1 Digital input CH1-8bit.SubIndex = 2; GL20_1600END_1 Digital input CH1-8bit.Size = 8; GL20_1600END_1 Digital input CH1-8bit.Offset = 0; GL20_1600END_1 Digital input CH1-8bit.DependOnSlot = True; GL20_1600END_1 Digital input CH1-8bit.DependOnSlotGroup = False; RxTxPdo.NumberofExcludes = 2; RxTxPdo.NumberofEntries = 1;
            RxTxPdo.Index = 16#1A12; RxTxPdo.Fixed = True; RxTxPdo.Mandatory = False; RxTxPdo.Virtual = False; RxTxPdo.Sm = -1; RxTxPdo.Su = 0; RxTxPdo.Name = '1600END input-16bit maping'; RxTxPdo.DependOnSlot = True; RxTxPdo.DependOnSlotGroup = False; RxTxPdo.OverwrittenByModule = True; Exclude = [16#1A10,16#1A11]; GL20_1600END_1 Digital input CH0-16bit.Index = 16#6082; GL20_1600END_1 Digital input CH0-16bit.SubIndex = 1; GL20_1600END_1 Digital input CH0-16bit.Size = 16; GL20_1600END_1 Digital input CH0-16bit.Offset = 0; GL20_1600END_1 Digital input CH0-16bit.DependOnSlot = True; GL20_1600END_1 Digital input CH0-16bit.DependOnSlotGroup = False; RxTxPdo.NumberofExcludes = 2; RxTxPdo.NumberofEntries = 16; RxTxPdo.Index = 16#1A10; RxTxPdo.Fixed = True; RxTxPdo.Mandatory = False; RxTxPdo.Virtual = False; RxTxPdo.Sm = -1; RxTxPdo.Su = 0; RxTxPdo.Name = '1600END input-bit maping'; RxTxPdo.DependOnSlot = True; RxTxPdo.DependOnSlotGroup = False; RxTxPdo.OverwrittenByModule = True; Exclude = [16#1A11,16#1A12]; GL20_1600END_1 Digital input bit0.Index = 16#6080; GL20_1600END_1 Digital input bit0.SubIndex = 1; GL20_1600END_1 Digital input bit0.Size = 1; GL20_1600END_1 Digital input bit0.Offset = 0; GL20_1600END_1 Digital input bit0.DependOnSlot = True; GL20_1600END_1 Digital input bit0.DependOnSlotGroup = False; GL20_1600END_1 Digital input bit1.Index = 16#6080; GL20_1600END_1 Digital input bit1.SubIndex = 2; GL20_1600END_1 Digital input bit1.Size = 1; GL20_1600END_1 Digital input bit1.Offset = 0;
            GL20_1600END_1 Digital input bit1.DependOnSlot = True; GL20_1600END_1 Digital input bit1.DependOnSlotGroup = False; GL20_1600END_1 Digital input bit2.Index = 16#6080; GL20_1600END_1 Digital input bit2.SubIndex = 3; GL20_1600END_1 Digital input bit2.Size = 1; GL20_1600END_1 Digital input bit2.Offset = 0; GL20_1600END_1 Digital input bit2.DependOnSlot = True; GL20_1600END_1 Digital input bit2.DependOnSlotGroup = False; GL20_1600END_1 Digital input bit3.Index = 16#6080; GL20_1600END_1 Digital input bit3.SubIndex = 4; GL20_1600END_1 Digital input bit3.Size = 1; GL20_1600END_1 Digital input bit3.Offset = 0; GL20_1600END_1 Digital input bit3.DependOnSlot = True; GL20_1600END_1 Digital input bit3.DependOnSlotGroup = False; GL20_1600END_1 Digital input bit4.Index = 16#6080; GL20_1600END_1 Digital input bit4.SubIndex = 5; GL20_1600END_1 Digital input bit4.Size = 1; GL20_1600END_1 Digital input bit4.Offset = 0; GL20_1600END_1 Digital input bit4.DependOnSlot = True; GL20_1600END_1 Digital input bit4.DependOnSlotGroup = False; GL20_1600END_1 Digital input bit5.Index = 16#6080; GL20_1600END_1 Digital input bit5.SubIndex = 6; GL20_1600END_1 Digital input bit5.Size = 1; GL20_1600END_1 Digital input bit5.Offset = 0; GL20_1600END_1 Digital input bit5.DependOnSlot = True; GL20_1600END_1 Digital input bit5.DependOnSlotGroup = False; GL20_1600END_1 Digital input bit6.Index = 16#6080; GL20_1600END_1 Digital input bit6.SubIndex = 7; GL20_1600END_1 Digital input bit6.Size = 1; GL20_1600END_1 Digital input bit6.Offset = 0; GL20_1600END_1 Digital input bit6.DependOnSlot = True; GL20_1600END_1 Digital input bit6.DependOnSlotGroup = False; GL20_1600END_1 Digital input bit7.Index = 16#6080; GL20_1600END_1 Digital input bit7.SubIndex = 8; GL20_1600END_1 Digital input bit7.Size = 1; GL20_1600END_1 Digital input bit7.Offset = 0; GL20_1600END_1 Digital input bit7.DependOnSlot = True; GL20_1600END_1 Digital input bit7.DependOnSlotGroup = False; GL20_1600END_1 Digital input bit8.Index = 16#6080; GL20_1600END_1 Digital input bit8.SubIndex = 9;
            GL20_1600END_1 Digital input bit8.Size = 1; GL20_1600END_1 Digital input bit8.Offset = 0; GL20_1600END_1 Digital input bit8.DependOnSlot = True; GL20_1600END_1 Digital input bit8.DependOnSlotGroup = False; GL20_1600END_1 Digital input bit9.Index = 16#6080; GL20_1600END_1 Digital input bit9.SubIndex = 10; GL20_1600END_1 Digital input bit9.Size = 1; GL20_1600END_1 Digital input bit9.Offset = 0; GL20_1600END_1 Digital input bit9.DependOnSlot = True; GL20_1600END_1 Digital input bit9.DependOnSlotGroup = False; GL20_1600END_1 Digital input bit10.Index = 16#6080; GL20_1600END_1 Digital input bit10.SubIndex = 11; GL20_1600END_1 Digital input bit10.Size = 1; GL20_1600END_1 Digital input bit10.Offset = 0; GL20_1600END_1 Digital input bit10.DependOnSlot = True; GL20_1600END_1 Digital input bit10.DependOnSlotGroup = False; GL20_1600END_1 Digital input bit11.Index = 16#6080; GL20_1600END_1 Digital input bit11.SubIndex = 12; GL20_1600END_1 Digital input bit11.Size = 1; GL20_1600END_1 Digital input bit11.Offset = 0; GL20_1600END_1 Digital input bit11.DependOnSlot = True; GL20_1600END_1 Digital input bit11.DependOnSlotGroup = False; GL20_1600END_1 Digital input bit12.Index = 16#6080; GL20_1600END_1 Digital input bit12.SubIndex = 13; GL20_1600END_1 Digital input bit12.Size = 1; GL20_1600END_1 Digital input bit12.Offset = 0; GL20_1600END_1 Digital input bit12.DependOnSlot = True; GL20_1600END_1 Digital input bit12.DependOnSlotGroup = False; GL20_1600END_1 Digital input bit13.Index = 16#6080; GL20_1600END_1 Digital input bit13.SubIndex = 14; GL20_1600END_1 Digital input bit13.Size = 1; GL20_1600END_1 Digital input bit13.Offset = 0; GL20_1600END_1 Digital input bit13.DependOnSlot = True; GL20_1600END_1 Digital input bit13.DependOnSlotGroup = False; GL20_1600END_1 Digital input bit14.Index = 16#6080; GL20_1600END_1 Digital input bit14.SubIndex = 15; GL20_1600END_1 Digital input bit14.Size = 1; GL20_1600END_1 Digital input bit14.Offset = 0; GL20_1600END_1 Digital input bit14.DependOnSlot = True; GL20_1600END_1 Digital input bit14.DependOnSlotGroup = False;
            GL20_1600END_1 Digital input bit15.Index = 16#6080; GL20_1600END_1 Digital input bit15.SubIndex = 16; GL20_1600END_1 Digital input bit15.Size = 1; GL20_1600END_1 Digital input bit15.Offset = 0; GL20_1600END_1 Digital input bit15.DependOnSlot = True; GL20_1600END_1 Digital input bit15.DependOnSlotGroup = False; Device control.Name = 'Device control'; Device control.DataType = 'UINT'; Device control.Default = ''; Device control.Comment = ''; GL20_0008ER_1 Digital output CH0-8bit.Name = 'GL20_0008ER_1 Digital output CH0-8bit'; GL20_0008ER_1 Digital output CH0-8bit.DataType = 'USINT'; GL20_0008ER_1 Digital output CH0-8bit.Default = ''; GL20_0008ER_1 Digital output CH0-8bit.Comment = ''; GL20_0008ER_1 Digital output CH0-16bit.Name = 'GL20_0008ER_1 Digital output CH0-16bit'; GL20_0008ER_1 Digital output CH0-16bit.DataType = 'UINT'; GL20_0008ER_1 Digital output CH0-16bit.Default = ''; GL20_0008ER_1 Digital output CH0-16bit.Comment = ''; GL20_0008ER_1 Digital output bit0.Name = 'GL20_0008ER_1 Digital output bit0'; GL20_0008ER_1 Digital output bit0.DataType = 'BOOL'; GL20_0008ER_1 Digital output bit0.Default = ''; GL20_0008ER_1 Digital output bit0.Comment = ''; GL20_0008ER_1 Digital output bit1.Name = 'GL20_0008ER_1 Digital output bit1'; GL20_0008ER_1 Digital output bit1.DataType = 'BOOL'; GL20_0008ER_1 Digital output bit1.Default = ''; GL20_0008ER_1 Digital output bit1.Comment = ''; GL20_0008ER_1 Digital output bit2.Name = 'GL20_0008ER_1 Digital output bit2'; GL20_0008ER_1 Digital output bit2.DataType = 'BOOL'; GL20_0008ER_1 Digital output bit2.Default = ''; GL20_0008ER_1 Digital output bit2.Comment = ''; GL20_0008ER_1 Digital output bit3.Name = 'GL20_0008ER_1 Digital output bit3'; GL20_0008ER_1 Digital output bit3.DataType = 'BOOL'; GL20_0008ER_1 Digital output bit3.Default = ''; GL20_0008ER_1 Digital output bit3.Comment = ''; GL20_0008ER_1 Digital output bit4.Name = 'GL20_0008ER_1 Digital output bit4'; GL20_0008ER_1 Digital output bit4.DataType = 'BOOL'; GL20_0008ER_1 Digital output bit4.Default = ''; GL20_0008ER_1 Digital output bit4.Comment = ''; GL20_0008ER_1 Digital output bit5.Name = 'GL20_0008ER_1 Digital output bit5'; GL20_0008ER_1 Digital output bit5.DataType = 'BOOL';
            GL20_0008ER_1 Digital output bit5.Default = ''; GL20_0008ER_1 Digital output bit5.Comment = ''; GL20_0008ER_1 Digital output bit6.Name = 'GL20_0008ER_1 Digital output bit6'; GL20_0008ER_1 Digital output bit6.DataType = 'BOOL'; GL20_0008ER_1 Digital output bit6.Default = ''; GL20_0008ER_1 Digital output bit6.Comment = ''; GL20_0008ER_1 Digital output bit7.Name = 'GL20_0008ER_1 Digital output bit7'; GL20_0008ER_1 Digital output bit7.DataType = 'BOOL'; GL20_0008ER_1 Digital output bit7.Default = ''; GL20_0008ER_1 Digital output bit7.Comment = ''; LBus status.Name = 'LBus status'; LBus status.DataType = 'UINT'; LBus status.Default = ''; LBus status.Comment = ''; Fault ID.Name = 'Fault ID'; Fault ID.DataType = 'UINT'; Fault ID.Default = ''; Fault ID.Comment = ''; ErrorSolt1.Name = 'ErrorSolt1'; ErrorSolt1.DataType = 'UDINT'; ErrorSolt1.Default = ''; ErrorSolt1.Comment = ''; ErrorSolt2.Name = 'ErrorSolt2'; ErrorSolt2.DataType = 'UDINT'; ErrorSolt2.Default = ''; ErrorSolt2.Comment = ''; GL20_4AD AD CH0.Name = 'GL20_4AD AD CH0'; GL20_4AD AD CH0.DataType = 'INT'; GL20_4AD AD CH0.Default = ''; GL20_4AD AD CH0.Comment = ''; GL20_4AD AD CH1.Name = 'GL20_4AD AD CH1'; GL20_4AD AD CH1.DataType = 'INT'; GL20_4AD AD CH1.Default = ''; GL20_4AD AD CH1.Comment = ''; GL20_4AD AD CH2.Name = 'GL20_4AD AD CH2'; GL20_4AD AD CH2.DataType = 'INT'; GL20_4AD AD CH2.Default = ''; GL20_4AD AD CH2.Comment = ''; GL20_4AD AD CH3.Name = 'GL20_4AD AD CH3'; GL20_4AD AD CH3.DataType = 'INT';
            GL20_4AD AD CH3.Default = ''; GL20_4AD AD CH3.Comment = ''; GL20_4AD_1 AD CH0.Name = 'GL20_4AD_1 AD CH0'; GL20_4AD_1 AD CH0.DataType = 'INT'; GL20_4AD_1 AD CH0.Default = ''; GL20_4AD_1 AD CH0.Comment = ''; GL20_4AD_1 AD CH1.Name = 'GL20_4AD_1 AD CH1'; GL20_4AD_1 AD CH1.DataType = 'INT'; GL20_4AD_1 AD CH1.Default = ''; GL20_4AD_1 AD CH1.Comment = ''; GL20_4AD_1 AD CH2.Name = 'GL20_4AD_1 AD CH2'; GL20_4AD_1 AD CH2.DataType = 'INT'; GL20_4AD_1 AD CH2.Default = ''; GL20_4AD_1 AD CH2.Comment = ''; GL20_4AD_1 AD CH3.Name = 'GL20_4AD_1 AD CH3'; GL20_4AD_1 AD CH3.DataType = 'INT'; GL20_4AD_1 AD CH3.Default = ''; GL20_4AD_1 AD CH3.Comment = ''; GL20_1600END_1 Digital input CH0-8bit.Name = 'GL20_1600END_1 Digital input CH0-8bit'; GL20_1600END_1 Digital input CH0-8bit.DataType = 'USINT'; GL20_1600END_1 Digital input CH0-8bit.Default = ''; GL20_1600END_1 Digital input CH0-8bit.Comment = ''; GL20_1600END_1 Digital input CH1-8bit.Name = 'GL20_1600END_1 Digital input CH1-8bit'; GL20_1600END_1 Digital input CH1-8bit.DataType = 'USINT'; GL20_1600END_1 Digital input CH1-8bit.Default = ''; GL20_1600END_1 Digital input CH1-8bit.Comment = ''; GL20_1600END_1 Digital input CH0-16bit.Name = 'GL20_1600END_1 Digital input CH0-16bit'; GL20_1600END_1 Digital input CH0-16bit.DataType = 'UINT'; GL20_1600END_1 Digital input CH0-16bit.Default = ''; GL20_1600END_1 Digital input CH0-16bit.Comment = ''; GL20_1600END_1 Digital input bit0.Name = 'GL20_1600END_1 Digital input bit0'; GL20_1600END_1 Digital input bit0.DataType = 'BOOL'; GL20_1600END_1 Digital input bit0.Default = ''; GL20_1600END_1 Digital input bit0.Comment = ''; GL20_1600END_1 Digital input bit1.Name = 'GL20_1600END_1 Digital input bit1'; GL20_1600END_1 Digital input bit1.DataType = 'BOOL'; GL20_1600END_1 Digital input bit1.Default = ''; GL20_1600END_1 Digital input bit1.Comment = ''; GL20_1600END_1 Digital input bit2.Name = 'GL20_1600END_1 Digital input bit2'; GL20_1600END_1 Digital input bit2.DataType = 'BOOL';
            GL20_1600END_1 Digital input bit2.Default = ''; GL20_1600END_1 Digital input bit2.Comment = ''; GL20_1600END_1 Digital input bit3.Name = 'GL20_1600END_1 Digital input bit3'; GL20_1600END_1 Digital input bit3.DataType = 'BOOL'; GL20_1600END_1 Digital input bit3.Default = ''; GL20_1600END_1 Digital input bit3.Comment = ''; GL20_1600END_1 Digital input bit4.Name = 'GL20_1600END_1 Digital input bit4'; GL20_1600END_1 Digital input bit4.DataType = 'BOOL'; GL20_1600END_1 Digital input bit4.Default = ''; GL20_1600END_1 Digital input bit4.Comment = ''; GL20_1600END_1 Digital input bit5.Name = 'GL20_1600END_1 Digital input bit5'; GL20_1600END_1 Digital input bit5.DataType = 'BOOL'; GL20_1600END_1 Digital input bit5.Default = ''; GL20_1600END_1 Digital input bit5.Comment = ''; GL20_1600END_1 Digital input bit6.Name = 'GL20_1600END_1 Digital input bit6'; GL20_1600END_1 Digital input bit6.DataType = 'BOOL'; GL20_1600END_1 Digital input bit6.Default = ''; GL20_1600END_1 Digital input bit6.Comment = ''; GL20_1600END_1 Digital input bit7.Name = 'GL20_1600END_1 Digital input bit7'; GL20_1600END_1 Digital input bit7.DataType = 'BOOL'; GL20_1600END_1 Digital input bit7.Default = ''; GL20_1600END_1 Digital input bit7.Comment = ''; GL20_1600END_1 Digital input bit8.Name = 'GL20_1600END_1 Digital input bit8'; GL20_1600END_1 Digital input bit8.DataType = 'BOOL'; GL20_1600END_1 Digital input bit8.Default = ''; GL20_1600END_1 Digital input bit8.Comment = ''; GL20_1600END_1 Digital input bit9.Name = 'GL20_1600END_1 Digital input bit9'; GL20_1600END_1 Digital input bit9.DataType = 'BOOL'; GL20_1600END_1 Digital input bit9.Default = ''; GL20_1600END_1 Digital input bit9.Comment = ''; GL20_1600END_1 Digital input bit10.Name = 'GL20_1600END_1 Digital input bit10'; GL20_1600END_1 Digital input bit10.DataType = 'BOOL'; GL20_1600END_1 Digital input bit10.Default = ''; GL20_1600END_1 Digital input bit10.Comment = ''; GL20_1600END_1 Digital input bit11.Name = 'GL20_1600END_1 Digital input bit11'; GL20_1600END_1 Digital input bit11.DataType = 'BOOL'; GL20_1600END_1 Digital input bit11.Default = ''; GL20_1600END_1 Digital input bit11.Comment = ''; GL20_1600END_1 Digital input bit12.Name = 'GL20_1600END_1 Digital input bit12'; GL20_1600END_1 Digital input bit12.DataType = 'BOOL';
            GL20_1600END_1 Digital input bit12.Default = ''; GL20_1600END_1 Digital input bit12.Comment = ''; GL20_1600END_1 Digital input bit13.Name = 'GL20_1600END_1 Digital input bit13'; GL20_1600END_1 Digital input bit13.DataType = 'BOOL'; GL20_1600END_1 Digital input bit13.Default = ''; GL20_1600END_1 Digital input bit13.Comment = ''; GL20_1600END_1 Digital input bit14.Name = 'GL20_1600END_1 Digital input bit14'; GL20_1600END_1 Digital input bit14.DataType = 'BOOL'; GL20_1600END_1 Digital input bit14.Default = ''; GL20_1600END_1 Digital input bit14.Comment = ''; GL20_1600END_1 Digital input bit15.Name = 'GL20_1600END_1 Digital input bit15'; GL20_1600END_1 Digital input bit15.DataType = 'BOOL'; GL20_1600END_1 Digital input bit15.Default = ''; GL20_1600END_1 Digital input bit15.Comment = ''
          output Application.绿灯 : BOOL  // GL20_0008ER_1 Digital output CH0-8bit.Bit0
          output Application.黄灯 : BOOL  // GL20_0008ER_1 Digital output CH0-8bit.Bit2
          output Application.蜂鸣器 : BOOL  // GL20_0008ER_1 Digital output CH0-8bit.Bit4
          input  Application.i_模拟量4 : INT  // GL20_4AD AD CH0
          input  Application.i_模拟量2 : INT  // GL20_4AD AD CH1
          input  Application.i_模拟量8 : INT  // GL20_4AD AD CH2
          input  Application.i_模拟量5 : INT  // GL20_4AD AD CH3
          input  Application.i_模拟量1 : INT  // GL20_4AD_1 AD CH0
          input  Application.i_模拟量3 : INT  // GL20_4AD_1 AD CH1
          input  Application.i_模拟量6 : INT  // GL20_4AD_1 AD CH2
          input  Application.i_模拟量7 : INT  // GL20_4AD_1 AD CH3
          input  Application.报警代码1 : USINT  // GL20_1600END_1 Digital input CH0-8bit
          input  Application.报警代码2 : USINT  // GL20_1600END_1 Digital input CH1-8bit
          unmapped channels: Device control, GL20_0008ER_1 Digital output CH0-8bit, LBus status, Fault ID, ErrorSolt1, ErrorSolt2
        GL20_4AD : GL20-4AD(4 channels AD Module), Inovance, order no. GL20-4AD, version 0
            settings: 4AD module CH0 transform mode.Value = 135; 4AD module CH1 transform mode.Value = 135; 4AD module CH2 transform mode.Value = 135; 4AD module CH3 transform mode.Value = 135
        GL20_4AD_1 : GL20-4AD(4 channels AD Module), Inovance, order no. GL20-4AD, version 0
            settings: 4AD module CH0 transform mode.Value = 135; 4AD module CH1 transform mode.Value = 135; 4AD module CH2 transform mode.Value = 135; 4AD module CH3 transform mode.Value = 135
        GL20_1600END_1 : GL20(GL20S)-1600END(16 channels DI module), Inovance, order no. GL20(GL20S)-1600END, version 0
        GL20_0008ER_1 : GL20(GL20S)-0008ER(8 channels DO module), Inovance, order no. GL20(GL20S)-0008ER, version 0
    MODBUS_COM1 : Modbus主站, inovance, version 00.00.00.10
        settings: Vendor.parameterset.Bit0 = True; Vendor.parameterset.Bit1 = False; Vendor.parameterset.Bit2 = True; Vendor.parameterset.Bit3 = False; Vendor.parameterset.Bit6 = False; Vendor.parameterset.Bit7 = False; Vendor.baudset = 9; modbus master com port.SlaveNum = 1; modbus master com port.FrameDelay = 10;  = 1; IsVirtual = False
      底盘陀螺仪通讯 : Modbus Slave, Inovance, version 00.00.00.10
          settings: UseDec = False; modbus slave com port.ChannelNum = 5; modbus slave com port.SlaveAddr = 2; modbus slave com port.ModbusComSet = 1; modbus slave com port.EnableSlaveVariable = 2002; channel.PremeterSet.Bit3 = TRUE; channel.CycleTimes = 40; channel.ReadRegOffSet = 61; channel.ReadRegLeg = 6; channel.WriteRegOffSet = 0; channel.IOChannel = 0; channel.ResendCount = 1; channel.ChannelName = '读角度'; channel.ChannelNote = ''; channel.PremeterSet.Bit2 = TRUE; channel.PremeterSet.Bit4 = TRUE; channel.CycleTimes = 65535; channel.ReadRegOffSet = 0; channel.WriteRegOffSet = 105; channel.ResendCount = 1; channel.ChannelName = '解锁'; channel.ChannelNote = ''; channel.PremeterSet.Bit2 = TRUE; channel.PremeterSet.Bit4 = TRUE; channel.CycleTimes = 65535; channel.ReadRegOffSet = 0; channel.IOChannel = 2; channel.ResendCount = 1; channel.ChannelName = '校准模式'; channel.ChannelNote = ''; channel.PremeterSet.Bit2 = TRUE; channel.PremeterSet.Bit4 = TRUE; channel.CycleTimes = 65535; channel.ReadRegOffSet = 0; channel.WriteRegOffSet = 0; channel.IOChannel = 4; channel.ResendCount = 1; channel.ChannelName = '保存'; channel.ChannelNote = ''; channel.PremeterSet.Bit3 = TRUE;
            channel.CycleTimes = 40; channel.ReadRegOffSet = 55; channel.ReadRegLeg = 3; channel.WriteRegOffSet = 0; channel.IOChannel = 3; channel.ResendCount = 1; channel.ChannelName = '读角速度'; channel.ChannelNote = ''
          input  Application.底盘陀螺仪.orign_arry :  ARRAY[0..5] OF WORD  // 读角度
          input  Application.底盘陀螺仪.orign_arry_speed :  ARRAY[0..2] OF WORD  // 读角速度
          unmapped channels: 解锁, 校准模式, 保存
    COM : 虚拟Modbus主站, inovance, version 00.00.00.20
        settings: Vendor.parameterset.Bit0 = False; Vendor.parameterset.Bit1 = False; Vendor.parameterset.Bit2 = True; Vendor.parameterset.Bit3 = False; Vendor.parameterset.Bit6 = False; Vendor.parameterset.Bit7 = False; Vendor.res = 16; modbus master com port.SlaveNum = 1; modbus master com port.FrameDelay = 20; RxCount = 7; Index0 = 16#7080; SubIndex0 = 1; Address0 = ADR(%QD98); Index3 = 16#7080; SubIndex3 = 2; Address3 = ADR(%QD99); Index6 = 16#7080; SubIndex6 = 3; Address6 = ADR(%QD100); Index9 = 16#7080; SubIndex9 = 4; Address9 = ADR(%QD101); Index12 = 16#7080; SubIndex12 = 5; Address12 = ADR(%QD102); Index15 = 16#7080; SubIndex15 = 6; Address15 = ADR(%QD103); Index18 = 16#7080; SubIndex18 = 7; Address18 = ADR(%QD104); TxCount = 7; Index0 = 16#6080; SubIndex0 = 1; Address0 = ADR(%ID156); Index3 = 16#6080; SubIndex3 = 2; Address3 = ADR(%ID157); Index6 = 16#6080; SubIndex6 = 3;
          Address6 = ADR(%ID158); Index9 = 16#6080; SubIndex9 = 4; Address9 = ADR(%ID159); Index12 = 16#6080; SubIndex12 = 5; Address12 = ADR(%ID160); Index15 = 16#6080; SubIndex15 = 6; Address15 = ADR(%ID161); Index18 = 16#6080; SubIndex18 = 7; Address18 = ADR(%ID162); OtherData = 2; Index0 = 16#6080; SubIndex0 = 15; Address0 = ADR(%ID170); Index3 = 16#7080; SubIndex3 = 15; Address3 = ADR(%QD112); VirtualProtocol = 1; DeviceTaskName = 'ETHERCAT_C'; IsVirtual = True; VirtualInterface = 0; VirtualDevice = 'd1c8065f-f08a-471f-8c7e-6f9e70c1fa64'
      modbus_protocol : Modbus Slave, Inovance, version 00.00.00.10
          settings: UseDec = False; modbus slave com port.ChannelNum = 10; modbus slave com port.ModbusComSet = 1; modbus slave com port.EnableSlaveVariable = 2001; channel.PremeterSet.Bit3 = TRUE; channel.CycleTimes = 200; channel.ReadRegOffSet = 45056; channel.ReadRegLeg = 28; channel.WriteRegOffSet = 0; channel.IOChannel = 0; channel.ResendCount = 1; channel.ChannelName = 'BMS数据'; channel.ChannelNote = ''; channel.PremeterSet.Bit3 = TRUE; channel.CycleTimes = 200; channel.ReadRegOffSet = 4352; channel.ReadRegLeg = 30; channel.WriteRegOffSet = 0; channel.ResendCount = 1; channel.ChannelName = '电池反馈数据组1'; channel.ChannelNote = ''; channel.PremeterSet.Bit3 = TRUE; channel.ReadRegOffSet = 4416; channel.ReadRegLeg = 30; channel.WriteRegOffSet = 0; channel.IOChannel = 2; channel.ResendCount = 1; channel.ChannelName = '电池反馈数据组2'; channel.ChannelNote = ''; channel.PremeterSet.Bit3 = TRUE; channel.ReadRegOffSet = 4480; channel.ReadRegLeg = 30; channel.WriteRegOffSet = 0; channel.IOChannel = 3; channel.ResendCount = 1; channel.ChannelName = '电池反馈数据组3'; channel.ChannelNote = ''; channel.PremeterSet.Bit3 = TRUE; channel.CycleTimes = 200; channel.ReadRegOffSet = 4544;
            channel.ReadRegLeg = 30; channel.WriteRegOffSet = 0; channel.IOChannel = 4; channel.ResendCount = 1; channel.ChannelName = '电池反馈数据组4'; channel.ChannelNote = ''; channel.PremeterSet.Bit3 = TRUE; channel.CycleTimes = 200; channel.ReadRegOffSet = 16640; channel.ReadRegLeg = 10; channel.WriteRegOffSet = 0; channel.IOChannel = 5; channel.ResendCount = 1; channel.ChannelName = '电池温度组1'; channel.ChannelNote = ''; channel.PremeterSet.Bit3 = TRUE; channel.ReadRegOffSet = 16706; channel.ReadRegLeg = 10; channel.WriteRegOffSet = 0; channel.IOChannel = 6; channel.ResendCount = 1; channel.ChannelName = '电池温度组2'; channel.ChannelNote = ''; channel.PremeterSet.Bit3 = TRUE; channel.CycleTimes = 200; channel.ReadRegOffSet = 16772; channel.ReadRegLeg = 10; channel.WriteRegOffSet = 0; channel.IOChannel = 7; channel.ResendCount = 1; channel.ChannelName = '电池温度组3'; channel.ChannelNote = ''; channel.PremeterSet.Bit3 = TRUE; channel.CycleTimes = 200; channel.ReadRegOffSet = 16838; channel.ReadRegLeg = 10; channel.WriteRegOffSet = 0; channel.IOChannel = 8; channel.ResendCount = 1; channel.ChannelName = '电池温度组4';
            channel.ChannelNote = ''; channel.PremeterSet.Bit3 = TRUE; channel.CycleTimes = 200; channel.ReadRegOffSet = 40960; channel.ReadRegLeg = 27; channel.WriteRegOffSet = 0; channel.IOChannel = 9; channel.ResendCount = 1; channel.ChannelName = 'UPS反馈数据'; channel.ChannelNote = ''
          input  Application.BMS映射数据 :  ARRAY[0..27] OF WORD  // BMS数据
          input  Application.电池映射电压组1 :  ARRAY[0..29] OF WORD  // 电池反馈数据组1
          input  Application.电池映射电压组2 :  ARRAY[0..29] OF WORD  // 电池反馈数据组2
          input  Application.电池映射电压组3 :  ARRAY[0..29] OF WORD  // 电池反馈数据组3
          input  Application.电池映射电压组4 :  ARRAY[0..29] OF WORD  // 电池反馈数据组4
          input  Application.电池映射温度组1 :  ARRAY[0..9] OF WORD  // 电池温度组1
          input  Application.电池映射温度组2 :  ARRAY[0..9] OF WORD  // 电池温度组2
          input  Application.电池映射温度组3 :  ARRAY[0..9] OF WORD  // 电池温度组3
          input  Application.电池映射温度组4 :  ARRAY[0..9] OF WORD  // 电池温度组4
          input  Application.UPS映射数据 :  ARRAY[0..26] OF WORD  // UPS反馈数据
    MODBUS_TCP_1 : ModbusTCP主站, inovance, version 00.00.00.10
        settings: ModbusTcpMaster.AckDelay = 2;  = 0
      modbusTcp : ModbusTCP Slave, Inovance, version 00.00.00.10
          settings: UseDec = False; ModbusTcpSlave.ChannelNum = 2; ModbusTcpSlave.SlaveAddr = 3; ModbusTcpSlave.Port = 5502; ModbusTcpSlave.EnableSlaveVariable = 3001; ModbusTcpSlave.IpAddr = 201894080; channel.PremeterSet.Bit2 = TRUE; channel.PremeterSet.Bit3 = TRUE; channel.CycleTimes = 200; channel.ReadRegOffSet = 0; channel.ReadRegLeg = 8; channel.WriteRegOffSet = 0; channel.IOChannel = 0; channel.ResendCount = 3; channel.ChannelName = '读取遥控数据'; channel.ChannelNote = ''; channel.PremeterSet.Bit2 = TRUE; channel.PremeterSet.Bit3 = TRUE; channel.PremeterSet.Bit4 = TRUE; channel.CycleTimes = 200; channel.ReadRegOffSet = 0; channel.WriteRegOffSet = 0; channel.WriteRegLeg = 5; channel.ResendCount = 3; channel.ChannelName = '写入数据'; channel.ChannelNote = ''
          input  Application.DCH读遥控数据 :  ARRAY[0..7] OF WORD  // 读取遥控数据
          output Application.DCH写遥控数据 :  ARRAY[0..4] OF WORD  // 写入数据
  libraries: VisuSymbols, 3.5.10.0 (System)
  text list GlobalTextList
  data type MYIOBLOCK
  data type MOTION_INPUTS
  data type MOTION_OUTPUTS
  data type MOTION_EXTRADATA
*)

// MYIOBLOCK
{attribute 'pack_mode' := '1'}
TYPE MYIOBLOCK :
STRUCT
	ptr      : POINTER TO BYTE;           // inputs or outputs, and this ptr must be the first one
	len      : UINT;                      // size of the inputs or outpus
	name     : STRING(125);               // inputs or outputs name
END_STRUCT
END_TYPE

// MOTION_INPUTS
{attribute 'pack_mode' := '1'}
TYPE MOTION_INPUTS :
STRUCT
	iStatus   : INT;
	iServoErr : INT;
	dFbPos 	  : ARRAY[0..8] OF LREAL;
	dFbVel 	  : ARRAY[0..8] OF LREAL;
	dFbAcc 	  : ARRAY[0..8] OF LREAL;
	dFbSpace  : ARRAY[0..8] OF LREAL;
END_STRUCT
END_TYPE

// MOTION_OUTPUTS
{attribute 'pack_mode' := '1'}
TYPE MOTION_OUTPUTS :
STRUCT
	iRobStatus : INT;	//0-错误 1-等待 2-运行中 3-完成 4-停止完成
	iErrorNum  : INT;
	dCmdPos  : ARRAY[0..8] OF LREAL;
	dCmdVel  : ARRAY[0..8] OF LREAL;
	dCmdAcc  : ARRAY[0..8] OF LREAL;
	dCmdSpace  : ARRAY[0..8] OF LREAL;
END_STRUCT
END_TYPE

// MOTION_EXTRADATA
{attribute 'pack_mode' := '1'}
TYPE MOTION_EXTRADATA :
STRUCT
	iPlanMode : INT;	// 0-手动, 1-自动
	bIsJoint  : BOOL;
	iAxisNum  : INT;
	bDir      : BOOL;
	lRatio	  : LREAL;
	dPos	  : ARRAY[0..8] OF LREAL;
END_STRUCT
END_TYPE

// Device/Application/数据结构/伺服参数结构体
TYPE 伺服参数结构体 :
STRUCT
	//输入
	运行模式		: INT := 0;	//0-无运行, 1-点动运行, 2-运动到点, 3-相对运动
	使能			: BOOL := FALSE;
	运行方向		: BOOL := FALSE;
	运行速度		: LREAL := 2;
	运行位置		: LREAL;
	运行位置1		: LREAL;
	运行力矩		: LREAL;
	结束运行速度    : LREAL;
	// 运行控制速度
	运行控制速度: LREAL;
	运行控制速度1: LREAL;
	运行控制方向: INT;
	
	控制模式:SMC_CONTROLLER_MODE;
	//控制模式切换完成:BOOL;
	// 设定力矩
	设定力矩: LREAL;
	设定力矩1: LREAL;
	
	停止控制    : BOOL := FALSE;
	//停止完成    : BOOL := FALSE;
	
	轴复位        : BOOL := FALSE;
	轴初始化    : BOOL := FALSE;
	//输出
	指令位置		: LREAL;
	指令力矩		: LREAL;
	指令速度		: LREAL;
	反馈位置		: LREAL;
	反馈力矩		: LREAL;
	反馈速度		: LREAL;
	反馈电流		: LREAL;
	零点位置		: LREAL;
	反馈状态        : LREAL;
	
	点动运行中	: BOOL;
	//运动到点完成			: BOOL ;
	//运动到点完成1			: BOOL ;
	//相对运动到点完成			: BOOL ;
	//连续运动到点完成			: BOOL ;
	
	//复位完成:BOOL;
	//轴初始化完成:BOOL;
	
	使能状态:功能块状态;
	ETHERCAT复位状态: 功能块状态;
	复位状态:功能块状态;
	点动状态:功能块状态;
	回零状态:功能块状态;
	绝对增量定位状态: 功能块状态;
	绝对定位状态:功能块状态;
	绝对定位状态1:功能块状态;
	相对定位状态:功能块状态;
	速度运动状态:功能块状态;
	速度运动状态1:功能块状态;
	力矩运动状态:功能块状态;
	修改模式运动状态: 功能块状态;
	软限位设置: 功能块状态;
	停止状态:功能块状态;
	暂停状态:功能块状态;
	初始化状态:功能块状态;
	控制模式切换状态:功能块状态;
END_STRUCT
END_TYPE

// Device/Application/数据结构/底盘运行参数结构体
TYPE 底盘运行参数结构体 :
STRUCT
	底盘运行倍率		: LREAL := 0.5;
	底盘运行速度		: LREAL := 500;
	底盘运动方向		: INT := 0; //0-无运动, 1-前进, 2-后退, 3-左转, 4-右转
END_STRUCT
END_TYPE

// Device/Application/数据结构/陀螺仪
TYPE 陀螺仪 :
STRUCT
	// 站号
	站号 : BYTE;
	
	// X
	X : REAL;
	// Y
	Y : REAL;
	// Z
	Z : REAL;
	
	// orign_arry
	orign_arry : ARRAY[0..5] OF WORD;
	// unlock
	unlock : WORD := 16#B588;
	// save
	save : WORD := 0;
	// XY_RESET
	XY_RESET : WORD := 16#08;
	// Z_RESET
	Z_RESET : WORD := 16#04;
	// 校准模式
	校准模式 : WORD;
	
	// 角度复位触发
	角度复位触发 : BOOL;
	// Z轴复位触发
	Z轴复位触发  : BOOL;
	
	
	// orign_arry_speed
	orign_arry_speed: ARRAY[1..3] OF WORD;
	// 角速度X
	角速度X: REAL;
	// 角速度Y
	角速度Y: REAL;
	// 角速度Z
	角速度Z: REAL;
END_STRUCT
END_TYPE

// Device/Application/数据结构/机械臂参数结构体
{attribute 'pack_mode' := '1'}
TYPE 机械臂参数结构体 :
STRUCT
	规划模式 		: INT;	// 0-无规划, 1-手动运行, 2-自动运行, 3-手动停止, 4-运动到点, 5-自动停止
	是否关节运动  : BOOL;
	轴号  		: INT;
	方向      	: BOOL;
	倍率	  		: LREAL;
	运行点位		: ARRAY[0..8] OF LREAL;
END_STRUCT
END_TYPE

// Device/Application/数据结构/系统状态
TYPE 系统状态 :
STRUCT
	// 自动状态
	自动状态: BOOL := FALSE;
	// 手动状态
	手动状态: BOOL := FALSE;
	// 运行状态
	运行状态: BOOL := FALSE;
	// 报警状态
	报警状态: BOOL := FALSE;
	// 急停状态
	急停状态: BOOL := FALSE;
	// 停止信号
	停止信号: BOOL := FALSE;
	// 停止完成
	停止完成: ARRAY[1..30] OF BOOL;
	// 启动异常
	启动异常: ARRAY[1..30] OF BOOL;
	// 暂停状态
	暂停状态: BOOL := FALSE;
	END_STRUCT
END_TYPE

// Device/Application/数据结构/功能块状态
TYPE 功能块状态 :
STRUCT
	// DONE
	DONE: BOOL := FALSE;
	// BUSY
	BUSY: BOOL := FALSE;
	// Error
	Error: BOOL := FALSE;
	// ErrorID
	ErrorID:WORD:= 16#00;
	// CommandAborted
	CommandAborted: BOOL := FALSE;
	
	
	
END_STRUCT
END_TYPE

// Device/Application/数据结构/PID控制参数
TYPE PID控制参数 :
STRUCT
	// 比例
	KP: REAL := 30;
	// 积分
	TN: REAL := 0.5;
	// 微分
	TV: REAL := 1;
	// 输出最小值
	输出最小值: REAL := -500;
	// 输出最大值
	输出最大值: REAL := 500;
	// 允许偏差
	允许偏差: REAL := 20;
END_STRUCT
END_TYPE

// Device/Application/全局变量/全局电池数据
VAR_GLOBAL
	电量报警	: BOOL := FALSE;
	电量状态	: INT := 0; //0-低电量 1-正常电量 2-满电量
	系统状态 : INT := 0;
	电池状态 : INT := 0;
	一级保护状态 : DWORD := 0;
	二级保护状态 : DWORD := 0;
	三级保护状态 : DWORD := 0;
	故障状态 : DWORD := 0;
	采集电压 : LREAL := 0.0;
	负载电压 : LREAL := 0.0;
	上桥累计电压 : LREAL := 0.0;
	下桥累计电压 : LREAL := 0.0;
	上桥电流 : LREAL := 0.0;
	下桥电流 : LREAL := 0.0;
	上桥SOC : LREAL := 0.0;
	下桥SOC : LREAL := 0.0;
	上桥SOH : LREAL := 0.0;
	下桥SOH : LREAL := 0.0;
	上桥电池剩余容量 : LREAL := 0.0;
	下桥电池剩余容量 : LREAL := 0.0;
	上桥系统功率 : LREAL := 0.0;
	下桥系统功率 : LREAL := 0.0;
	
	UPS警告项1 : WORD := 0;
	UPS警告项2 : WORD := 0;
	UPS警告项3 : WORD := 0;
	UPS警告项4 : WORD := 0;
	UPS警告项5 : WORD := 0;
	R输入电压 : LREAL := 0.0;
	S输入电压 : LREAL := 0.0;
	T输入电压 : LREAL := 0.0;
	R输出电压 : LREAL := 0.0;
	S输出电压 : LREAL := 0.0;
	T输出电压 : LREAL := 0.0;
	输出频率 : LREAL := 0.0;
	R输出电流 : LREAL := 0.0;
	S输出电流 : LREAL := 0.0;
	T输出电流 : LREAL := 0.0;
	R输出负载百分比 : LREAL := 0.0;
	S输出负载百分比 : LREAL := 0.0;
	T输出负载百分比 : LREAL := 0.0;
	总输出负载百分比 : LREAL := 0.0;
	UPS状态 : WORD := 0;
	散热器温度1 : LREAL := 0.0;
	散热器温度2 : LREAL := 0.0;
	机柜温度 : LREAL := 0.0;
	UPS模式 : WORD := 0;
	UPS故障信息 : WORD := 0;			
	当前功率 : LREAL := 0.0;

	电池反馈电压组1 : ARRAY [0..29] OF LREAL;
	电池反馈电压组2 : ARRAY [0..29] OF LREAL;
	电池反馈电压组3 : ARRAY [0..29] OF LREAL;
	电池反馈电压组4 : ARRAY [0..29] OF LREAL;
	电池反馈温度组1 : ARRAY [0..9] OF LREAL;
	电池反馈温度组2 : ARRAY [0..9] OF LREAL;
	电池反馈温度组3 : ARRAY [0..9] OF LREAL;
	电池反馈温度组4 : ARRAY [0..9] OF LREAL;
	
	BMS映射数据 : ARRAY [0..27] OF WORD; // 16位数组
	UPS映射数据 : ARRAY [0..26] OF WORD; // 0x3030为正常状态
	电池映射电压组1 : ARRAY [0..29] OF WORD;
	电池映射电压组2 : ARRAY [0..29] OF WORD;
	电池映射电压组3 : ARRAY [0..29] OF WORD;
	电池映射电压组4 : ARRAY [0..29] OF WORD;
	电池映射温度组1 : ARRAY [0..9] OF WORD;
	电池映射温度组2 : ARRAY [0..9] OF WORD;
	电池映射温度组3 : ARRAY [0..9] OF WORD;
	电池映射温度组4 : ARRAY [0..9] OF WORD;
END_VAR

// Device/Application/全局变量/全局机械臂参数
VAR_GLOBAL
	sMotionInputs   : MOTION_INPUTS;
	sMotionOutputs  : MOTION_OUTPUTS;
	机械臂使能		: BOOL := FALSE;
	机械臂运行启动	: BOOL := FALSE;
	机械臂运行参数	: 机械臂参数结构体;
END_VAR

// Device/Application/全局变量/全局伺服参数
VAR_GLOBAL
	伸缩轴伺服参数    	: 伺服参数结构体;
	上卷扬伺服参数    	: 伺服参数结构体;
	下卷扬伺服参数    	: 伺服参数结构体;
	滚刷伺服参数    		: 伺服参数结构体;
	
	左上气缸伺服参数    	: 伺服参数结构体;
	左下气缸伺服参数    	: 伺服参数结构体;
	右上气缸伺服参数    	: 伺服参数结构体;
	右下气缸伺服参数    	: 伺服参数结构体;
	
	左上轮伺服参数    	: 伺服参数结构体;
	左下轮伺服参数    	: 伺服参数结构体;
	右上轮伺服参数    	: 伺服参数结构体;
	右下轮伺服参数    	: 伺服参数结构体;
END_VAR

// Device/Application/全局变量/SLAM指令控制
VAR_GLOBAL
	SLAM急停: BOOL;
	Vx: INT;
	Vy: INT;
	Wz: INT;
	SLAM速度有效: BOOL;
	SLAM控制方式: BOOL;	//0-导航有效, 1-手动有效
	上传序列号: WORD := 0;
	待发送缓存数组: ARRAY[0..2048] OF BYTE;
	待发送缓存数组长度: WORD;
	SLAM左轮速度: LREAL;
	SLAM右轮速度: LREAL;
	SLAM连接状态: BOOL;
	SLAM通讯复位: BOOL;
	自动重连: BOOL := 1;
END_VAR

// Device/Application/全局变量/全局底盘参数
VAR_GLOBAL
	底盘使能			: BOOL := FALSE;
	末端使能			: BOOL := FALSE;
	手动底盘联动		: BOOL := TRUE;
	底盘运行参数		: 底盘运行参数结构体;
	底盘陀螺仪		: 陀螺仪;
	底盘运行模式:INT;
	底盘自动运行:BOOL;
    底盘算法运行:BOOL;
	启动底盘自动运行:BOOL;
	启动底盘手动运行:BOOL;
	左上气缸控制,左下气缸控制,右上气缸控制,右下气缸控制:底盘控制运动;
	左上轮速度控制,左下轮速度控制,右上轮速度控制,右下轮速度控制:底盘控制运动_1;
	左上轮力矩控制,右上轮力矩控制,左下轮力矩控制,右下轮力矩控制:底盘控制运动_2;
	上卷扬实时控制,下卷扬实时控制,伸缩装置实时控制:超声波实时检测调整;
	
	底盘气缸运行速度:LREAL:=2;
	// 左轮初始力矩
	左轮初始力矩: LREAL := 80;
	// 右轮初始力矩
	右轮初始力矩: LREAL := 80;
	// 左轮正转力矩补偿
	左轮正转力矩补偿: LREAL := 0;
	// 左轮反转力矩补偿
	左轮反转力矩补偿: LREAL := 0;
	// 右轮正转力矩补偿
	右轮正转力矩补偿: LREAL := 0;
	// 右轮反转力矩补偿
	右轮反转力矩补偿: LREAL := 0;
	左上轮最大轮廓速度: UDINT;
	右上轮最大轮廓速度: UDINT;
	左下轮最大轮廓速度: UDINT;
	右下轮最大轮廓速度: UDINT;
	// 速度控制误差
	速度控制误差: REAL := 0.05;
	
	手动左轮速度:LREAL;
	手动右轮速度:LREAL;
END_VAR

// Device/Application/全局变量/业务流程
VAR_GLOBAL
	控制方式				: INT := 0;			//0-手动控制, 1-自动控制
	光伏板离底盘中心距离	: LREAL := 300.0; 	//单位：mm
	光伏板离地高度			: LREAL := 1000.0; 	//单位：mm
	光伏板角度				: LREAL := 30.0; 	//单位：度
	光伏板方向				: LREAL := -1.0; 	//-1-左, 1-右
	清扫作业开始			: BOOL;
END_VAR

// Device/Application/全局变量/IO刷新数据
VAR_GLOBAL
	边沿检测1: REAL;
	边沿检测2: REAL;
	边沿检测3: REAL;
	边沿检测4: REAL;
	超声波检测左1: REAL;
	超声波检测左2: REAL;
	超声波检测右1: REAL;
	超声波检测右2: REAL;
	平衡器1: REAL;
	平衡器2: REAL;
	卷扬机1: REAL;
	卷扬机2: REAL;
	上下卷扬距离工作面距离: REAL:=220;
	上下卷扬距离工作面距离1: REAL:=	210;
	补偿值1: REAL:=3;
    补偿值2: REAL:=0;
	上侧距离: LREAL;
	下侧距离: LREAL;
	上侧实际位置值暂存: LREAL;
	下侧实际位置值暂存: LREAL;
	上侧滤波距离: LREAL;
	下侧滤波距离: LREAL;
	左1滤波距离: LREAL;
	左2滤波距离: LREAL;
	右1滤波距离: LREAL;
	右2滤波距离: LREAL;
	上下侧距离差值: LREAL;
	上下卷扬滤波系数:LREAL:=0.1;
	滤波幅值: LREAL:=20;
	误差限制值: LREAL:=100;
	
	//模拟量
	i_模拟量1 :INT;
	i_模拟量2 :INT;
	i_模拟量3 :INT;
	i_模拟量4 :INT;
	
	i_模拟量5 :INT;
	i_模拟量6 :INT;
	i_模拟量7 :INT;
	i_模拟量8 :INT;
	
	DCH读遥控数据	: ARRAY [0..7] OF WORD;
	DCH写遥控数据	: ARRAY [0..4] OF WORD;
END_VAR

// Device/Application/全局变量/末端控制参数
VAR_GLOBAL
	启动滚刷自动运行:BOOL;
	滚刷正转:BOOL;
	滚刷反转:BOOL;
	上下卷扬自动流程:INT;
	上下卷扬检测数据有误:BOOL;
	上卷扬到达清扫面:BOOL;
	下卷扬到达清扫面:BOOL;
	上下卷扬工作完成:BOOL;
	对中机构自动流程:INT;
	启动上下扬自动运行:BOOL;
	启动对中机构自动运行:BOOL;
	对中工作完成:BOOL;
	回零自动流程:INT;
	启动回零自动运行:BOOL;
	回零工作完成:BOOL;
	上卷扬回零完成:BOOL;
	下卷扬回零完成:BOOL;
	伸缩架回零完成:BOOL;
	上卷扬零点位置:LREAL;
	下卷扬零点位置:LREAL;
	伸缩架零点位置:LREAL;
	上装自动运行:BOOL;
	上装自动流程:INT;
	上测超声波低通滤波模块,下测超声波低通滤波模块,上测力矩低通滤波模块,下测力矩低通滤波模块:低通滤波模块;
	左1超声波低通滤波模块,左2超声波低通滤波模块,右1超声波低通滤波模块,右2超声波低通滤波模块:低通滤波模块;
	//上下卷扬异常:BOOL;
	上侧距离保存:LREAL;
	下侧距离保存:LREAL;
	// 卷扬1PID
	卷扬1PID: PID控制参数;
	// 卷扬2PID
	卷扬2PID: PID控制参数;
	上卷扬速度控制,下卷扬速度控制:底盘控制运动_1;
	力矩kp设置值:LREAL:=0.005;
	力矩kp设置值1:LREAL:=0.005;
	上卷扬力矩偏差值:LREAL:=0;
	下卷扬力矩偏差值:LREAL:=0;
	kp设置值:LREAL:=0.05;
	ki设置值:LREAL:=0.01;
	上卷扬力矩偏差保存:LREAL;
	下卷扬力矩偏差保存:LREAL;
	上卷扬运行位置保存:LREAL;
	下卷扬运行位置保存:LREAL;
END_VAR

// Device/Application/全局变量/SLAM业务控制
VAR_GLOBAL
	业务通讯待发送缓存数组: ARRAY[0..2048] OF BYTE;
	业务通讯待发送缓存数组长度: WORD;
	业务通讯连接状态: BOOL;
	业务通讯复位: BOOL;
	业务通讯自动重连: BOOL := 1;
END_VAR

// Device/Application/全局变量/报警参数
VAR_GLOBAL
	上下卷扬异常:BOOL;
	伸缩架上限位:LREAL:=560;
	伸缩架下限位:LREAL:=0;
	上卷扬上限位:LREAL;
	上卷扬下限位:LREAL;
	下卷扬上限位:LREAL;
	下卷扬下限位:LREAL;
	左上气缸上限位:LREAL;
	左上气缸下限位:LREAL;
	左下气缸上限位:LREAL;
	左下气缸下限位:LREAL;
	右上气缸上限位:LREAL;
	右上气缸下限位:LREAL;
	右下气缸上限位:LREAL;
	右下气缸下限位:LREAL;
	报警复位:BOOL;
	轴报警:BOOL;
	
	伸缩架限位报警:BOOL;
	上卷扬限位报警:BOOL;
	下卷扬限位报警:BOOL;
	左上气缸限位报警:BOOL;
	左下气缸限位报警:BOOL;
	右上气缸限位报警:BOOL;
	右下气缸限位报警:BOOL;
	
	伸缩架使能完成:BOOL:=FALSE;
	伸缩架绝对运动完成:BOOL:=FALSE;
	伸缩架相对运动完成:BOOL:=FALSE;
	伸缩架暂停完成:BOOL:=FALSE;
	伸缩架停止完成:BOOL:=FALSE;
	伸缩架复位完成:BOOL:=FALSE;
	伸缩架初始化完成:BOOL:=FALSE;
	
	上卷扬使能完成:BOOL:=FALSE;
	上卷扬绝对运动完成:BOOL:=FALSE;
	上卷扬相对运动完成:BOOL:=FALSE;
	上卷扬暂停完成:BOOL:=FALSE;
	上卷扬停止完成:BOOL:=FALSE;
	上卷扬复位完成:BOOL:=FALSE;
	上卷扬初始化完成:BOOL:=FALSE;
	
	下卷扬使能完成:BOOL:=FALSE;
	下卷扬绝对运动完成:BOOL:=FALSE;
	下卷扬相对运动完成:BOOL:=FALSE;
	下卷扬暂停完成:BOOL:=FALSE;
	下卷扬停止完成:BOOL:=FALSE;
	下卷扬复位完成:BOOL:=FALSE;
	下卷扬初始化完成:BOOL:=FALSE;
	
	滚刷使能完成:BOOL:=FALSE;
	绿灯:BOOL;
	黄灯:BOOL;
	蜂鸣器:BOOL;
	DCH报警代码1		: INT;
	DCH报警代码2		: INT;
	报警代码1		: USINT;
	报警代码2		: USINT;
	报警代码3		: USINT;
	报警代码4		: USINT;
END_VAR

// Device/Application/机械臂控制
PROGRAM 机械臂控制
VAR
	// 结构体
	sMotionBlockInputs     	: MYIOBLOCK;
	sMotionBlockOutputs   	: MYIOBLOCK;
	sMotionExtraData       	: MOTION_EXTRADATA;
// 	sMotionPlanData        	: MOTION_EXTRADATA;
	
	// 函数
	fpMotionPlanCall       	: IOBlockCall;
	fpMotionMoveCall   	   	: IOBlockProcess;
	fpMotionSettingCall   	: IOBlockProcess;
	fpEventFB              	: EventCallbackFunBLock;
	
	// 变量	
	iCounter			   	: INT := 0;
	规划失败              	: BOOL := FALSE;
	规划错误码             	: INT := 0;
	插补失败               	: BOOL := FALSE;
	插补错误码             	: INT := 0;
	伺服错误码			   	: ARRAY[0..8] OF UINT := [0, 0, 0, 0, 0, 0, 0, 0, 0];
	机械臂运行状态			: INT := 0;
	错误码			   		: INT := 0;
	报错复位		  			: BOOL := FALSE;
// 	运行规划启动		  		: BOOL := FALSE;
	持续运行		  			: BOOL := FALSE;
	
	// 零点设置
	零点设置		  			: BOOL := FALSE;
	零点偏移			   		: ARRAY[0..8] OF LREAL;
	运行方向			   		: ARRAY[0..8] OF LREAL := [1.0, 1.0, -1.0, 1.0, 1, 1, 1, 1, 1];
	机械臂零点			   	: ARRAY[0..8] OF LREAL := [0.0, -90.0, 180.0, 45, 1, 1, 1, 1, 1];
	伺服零点			   		: ARRAY[0..8] OF LREAL := [70161.098, 90798.237, -92740.556, 146469.665, 1, 1, 1, 1, 1];
	
	每圈脉冲数			   	: ARRAY[0..8] OF DINT := [1, 1, 1, 1, 1, 1, 1, 1, 1];
	减速比			   		: ARRAY[0..8] OF LREAL := [209.38, 192.42, 192.42, 161.0, 1.0, 1.0, 1.0, 1.0, 1.0];
	脉冲当量			   		: ARRAY[0..8] OF LREAL;
	下发脉冲值			   	: ARRAY[0..8] OF LREAL;
	反馈脉冲值     			: ARRAY[0..8] OF LREAL;

	apMC_Power  			: ARRAY[0..3] OF MC_Power;
	apAxis      			: ARRAY[0..3] OF POINTER TO AXIS_REF_SM3;//定义轴
END_VAR

sMotionBlockInputs.name      := 'motioninputs';
sMotionBlockInputs.len       := SIZEOF(sMotionInputs);
sMotionBlockInputs.ptr       := ADR(sMotionInputs);

sMotionBlockOutputs.name     := 'motionoutputs';
sMotionBlockOutputs.len      := SIZEOF(sMotionOutputs);
sMotionBlockOutputs.ptr      := ADR(sMotionOutputs);

CASE 机械臂运行状态 OF
	0 :
		FOR iCounter:=0 TO 8 BY 1 DO
			脉冲当量[iCounter] := 每圈脉冲数[iCounter] * 减速比[iCounter] / 360.0 * 运行方向[iCounter];
		END_FOR
		
		机械臂运行参数.规划模式 := 0;
		机械臂运行参数.轴号 := 0;
		机械臂运行参数.方向 := TRUE;
		机械臂运行参数.是否关节运动 := TRUE;
		机械臂运行参数.倍率 := 30.0;
		机械臂运行参数.运行点位[0] := 0.0; 机械臂运行参数.运行点位[1] := -90.0; 机械臂运行参数.运行点位[2] := 180.0;
		机械臂运行参数.运行点位[3] := 45.0; 机械臂运行参数.运行点位[4] := 0.0; 机械臂运行参数.运行点位[5] := 0.0;
		
		apAxis[0] := ADR(机械臂1轴);
		apAxis[1] := ADR(机械臂2轴);
		apAxis[2] := ADR(机械臂3轴);
		apAxis[3] := ADR(机械臂4轴);
		
		机械臂运行状态 := 1;
	1:
		IF 零点设置 = TRUE THEN
			FOR iCounter:=0 TO 8 BY 1 DO
				零点偏移[iCounter] := 零点偏移[iCounter] + sMotionInputs.dFbPos[iCounter] - 机械臂零点[iCounter];
				伺服零点[iCounter] := 零点偏移[iCounter] - 机械臂零点[iCounter];
			END_FOR
			零点设置 := FALSE;
		END_IF

		FOR iCounter:=0 TO 3 BY 1 DO
			apMC_Power[iCounter](
				Axis:= apAxis[iCounter]^,
				Enable:= TRUE,
				bRegulatorOn:= 机械臂使能,
				bDriveStart:= TRUE,
				Status=> , 
				bRegulatorRealState=> , 
				bDriveStartRealState=> , 
				Busy=> , 
				Error=> , 
				ErrorID=> );
		END_FOR
		
		机械臂运行参数.规划模式 := 0;	// 空闲
		机械臂运行启动 := FALSE;
		
		IF 机械臂使能 = TRUE THEN
			// 使能后执行运动同步
			fpMotionSettingCall(
				xEnable               := TRUE,
				dwID                  := 1001,
				pInputs               := ADR(sMotionBlockInputs),
				pOutputs              := ADR(sMotionBlockOutputs),
				strFunName            := 'MotionSetting',
				pExtraData            := ADR(sMotionExtraData),
				xError                => 插补失败,
				eErrorID              => 插补错误码
				);		
			机械臂运行状态 := 2;
		END_IF
	2:
		// 运动完成
		IF (sMotionOutputs.iRobStatus = 3) OR (sMotionOutputs.iRobStatus = 4) OR (sMotionOutputs.iRobStatus = 0) THEN
			机械臂运行参数.规划模式 := 0;	// 空闲
			机械臂运行启动 := TRUE;
		END_IF
		
		IF 错误码 <> 0 THEN
			机械臂运行参数.规划模式 := 0;	// 空闲
			机械臂运行启动 := FALSE;
		END_IF
		
		// 连续运行
		IF 持续运行 = TRUE THEN
			IF sMotionOutputs.iRobStatus = 3 THEN
				机械臂运行参数.规划模式 := 2;	// 自动运行
				机械臂运行启动 := TRUE;
			END_IF
		END_IF
		
		// 运动规划
		IF 机械臂运行启动 = TRUE THEN
			fpMotionPlanCall(
				xEnable               := TRUE,
				dwID                  := 1001,
				strFunName            := 'MotionPlan',
				pExtraData            := ADR(机械臂运行参数),
				xError                => 规划失败, 
				eErrorID              => 规划错误码
				);
			机械臂运行启动 := FALSE;
		END_IF
		
		IF 机械臂使能 = FALSE THEN
			机械臂运行状态 := 1;
		END_IF
		
		零点设置 := FALSE;
	3:
		机械臂使能 := FALSE;
		FOR iCounter:=0 TO 3 BY 1 DO
			apMC_Power[iCounter](
				Axis:= apAxis[iCounter]^,
				Enable:= TRUE,
				bRegulatorOn:= 机械臂使能,
				bDriveStart:= TRUE,
				Status=> , 
				bRegulatorRealState=> , 
				bDriveStartRealState=> , 
				Busy=> , 
				Error=> , 
				ErrorID=> );
		END_FOR
END_CASE

// 运动插补
fpMotionMoveCall(
	xEnable               := TRUE,
	dwID                  := 1001,
	pInputs               := ADR(sMotionBlockInputs),
	pOutputs              := ADR(sMotionBlockOutputs),
	strFunName            := 'MotionMove',
	pExtraData            := ADR(sMotionExtraData),
	xError                => 插补失败,
	eErrorID              => 插补错误码
	);

// 位置计算与下发
FOR iCounter:=0 TO 3 BY 1 DO
	下发脉冲值[iCounter] := (sMotionOutputs.dCmdPos[iCounter] + 伺服零点[iCounter]) * 脉冲当量[iCounter];
	反馈脉冲值[iCounter] := apAxis[iCounter]^.fActPosition;
	sMotionInputs.dFbPos[iCounter] := (apAxis[iCounter]^.fActPosition / 脉冲当量[iCounter]) - 伺服零点[iCounter];

	IF sMotionOutputs.dCmdPos[iCounter] <> 0 THEN
		apAxis[iCounter]^.fSetPosition := 下发脉冲值[iCounter];
	END_IF
	
END_FOR

IF 规划错误码 <> 0 THEN
	机械臂运行参数.规划模式 := 0;	// 规划报错后需切换为空闲
	错误码 := 规划错误码;
END_IF

IF sMotionOutputs.iErrorNum <> 0 THEN
	错误码 := sMotionOutputs.iErrorNum;
END_IF

IF 机械臂使能 = TRUE THEN
	IF 伺服错误码[0] <> 0 OR 伺服错误码[1] <> 0 OR 伺服错误码[2] <> 0 OR 伺服错误码[3] <> 0 THEN // 伺服报错
		错误码 := UDINT_TO_INT(伺服错误码[0]);
		机械臂运行参数.规划模式 := 3; // 运动停止规划
		fpMotionPlanCall(
			xEnable               := TRUE,
			dwID                  := 1001,
			strFunName            := 'MotionPlan',
			pExtraData            := ADR(机械臂运行参数),
			xError                => 规划失败, 
			eErrorID              => 规划错误码
		);
		机械臂运行状态 := 3;
	END_IF	
END_IF

// IF sMotionOutputs.iRobStatus = 2 THEN //运动进行中
// 	IF 机械臂使能 = FALSE THEN
// 		机械臂运行参数.规划模式 := 3; //运动停止规划
// 		fpMotionPlanCall(
// 			xEnable               := TRUE,
// 			dwID                  := 1001,
// 			strFunName            := 'MotionPlan',
// 			pExtraData            := ADR(机械臂运行参数),
// 			xError                => 规划失败, 
// 			eErrorID              => 规划错误码
// 		);
// 		机械臂运行状态 := 1;
// 	END_IF
// END_IF

// 报错复位
IF 错误码 <> 0 THEN
	IF 报错复位 = TRUE THEN
		机械臂运行状态 := 1;
		错误码 := 0;		
		规划错误码 := 0;
		// 复位运动
		fpMotionSettingCall(
			xEnable               := TRUE,
			dwID                  := 1002,
			pInputs               := ADR(sMotionBlockInputs),
			pOutputs              := ADR(sMotionBlockOutputs),
			strFunName            := 'MotionSetting',
			pExtraData            := ADR(sMotionExtraData),
			xError                => 插补失败,
			eErrorID              => 插补错误码
		);		
		报错复位 := FALSE;
	END_IF	
END_IF

END_PROGRAM

// Device/Application/函数/EventCallbackFunBLock
FUNCTION_BLOCK EventCallbackFunBLock IMPLEMENTS ICmpEventCallback
VAR_INPUT
END_VAR
VAR_OUTPUT
END_VAR
VAR
	hEventStart			: RTS_IEC_HANDLE;
	hEventStop 			: RTS_IEC_HANDLE;
	hInterfaceStart 	: RTS_IEC_HANDLE;
	hInterfaceStop 		: RTS_IEC_HANDLE;
	ItfEventCallback 	: ICmpEventCallback;
	Result 				: UDINT;
END_VAR

METHOD EventCallback : UDINT
VAR_INPUT
	pEventParam : POINTER TO EventParam;
END_VAR
VAR
	pfIOBlockCall : IOBlockCall;
END_VAR
(* For every registered event this functions is called, because the function block
   implements ICmpEventCallback. *)

(* Save the stop Reason in a global variable *)
IF pEventParam^.EventId = EVT_StartDone THEN
	pfIOBlockCall(xEnable:=TRUE, dwID:=1001, strFunName:='ExampleInitialize', pExtraData:=(*custom data*));
ELSIF pEventParam^.EventId = EVT_PrepareStop THEN
	pfIOBlockCall(xEnable:=TRUE, dwID:=1001, strFunName:='ExampleRelease', pExtraData:=(*custom data*));
END_IF
END_METHOD

METHOD FB_Exit : BOOL
VAR_INPUT
	bInCopyCode: BOOL;
END_VAR
VAR
END_VAR
(* Unregister and close both Events *)
EventUnregisterCallback(hEventStart, hInterfaceStart);
EventUnregisterCallback(hEventStop, hInterfaceStop);

Result := EventClose2(hEventStart);
Result := EventClose2(hEventStop);
END_METHOD

METHOD FB_Init : BOOL
VAR_INPUT
	bInitRetains: BOOL;
	bInCopyCode: BOOL;	
END_VAR
VAR
END_VAR
ItfEventCallback := THIS^;

(* Open an Event which listens to the start Event *)
hEventStart := EventOpen(EVT_StartDone, CMPID_CmpApp, Result);
(* Open an Event which listens to the stop Event *)
hEventStop := EventOpen(EVT_PrepareStop, CMPID_CmpApp, Result);

(* Register the Interface Callback functions to the event. *)
hInterfaceStart := EventRegisterCallback(hEventStart, ItfEventCallback, Result);	
hInterfaceStop := EventRegisterCallback(hEventStop, ItfEventCallback, Result);
END_METHOD

END_FUNCTION_BLOCK

// Device/Application/运动控制
PROGRAM 运动控制
VAR
	
END_VAR

底盘控制();
末端控制();

END_PROGRAM

// Device/Application/底盘控制
PROGRAM 底盘控制
VAR
	底盘平衡处理			: 底盘平衡算法;
	
	左上气缸伺服控制    	: 伺服控制;
	左下气缸伺服控制    	: 伺服控制;
	右上气缸伺服控制    	: 伺服控制;
	右下气缸伺服控制    	: 伺服控制;
	
	左上轮伺服控制    	: 伺服控制;
	左下轮伺服控制    	: 伺服控制;
	右上轮伺服控制    	: 伺服控制;
	右下轮伺服控制    	: 伺服控制;
	
	缓存流程:INT;
	缓存数据1: ARRAY[0..4] OF LREAL;
	缓存数据2: ARRAY[0..4] OF LREAL;
	缓存数据3: ARRAY[0..4] OF LREAL;
	缓存数据4: ARRAY[0..4] OF LREAL;
	
	平均数据1:LREAL;
	平均数据2:LREAL;
	平均数据3:LREAL;
	平均数据4:LREAL;
	平均数据5:LREAL;
	
	总系统状态: 系统状态;
	速度调整延时:TON;
END_VAR

IF 底盘使能=TRUE THEN
	左上气缸伺服参数.使能 := TRUE; 左下气缸伺服参数.使能 := TRUE;
	右上气缸伺服参数.使能 := TRUE; 右下气缸伺服参数.使能 := TRUE;
	左上轮伺服参数.使能 := TRUE; 左下轮伺服参数.使能 := TRUE;
	右上轮伺服参数.使能 := TRUE; 右下轮伺服参数.使能 := TRUE;

	CASE 缓存流程 OF
	0:
	   平均数据1:=左上气缸伺服参数.反馈位置;
	   平均数据2:=左下气缸伺服参数.反馈位置;
	   平均数据3:=右上气缸伺服参数.反馈位置;
	   平均数据4:=右下气缸伺服参数.反馈位置;
	   缓存流程:=10;
	10:
	   缓存数据1[0]:=左上气缸伺服参数.反馈位置;
	   缓存数据2[0]:=左下气缸伺服参数.反馈位置;
	   缓存数据3[0]:=右上气缸伺服参数.反馈位置;
	   缓存数据4[0]:=右下气缸伺服参数.反馈位置;
	   缓存流程:=20;
	20:  
	   缓存数据1[1]:=左上气缸伺服参数.反馈位置;
	   缓存数据2[1]:=左下气缸伺服参数.反馈位置;
	   缓存数据3[1]:=右上气缸伺服参数.反馈位置;
	   缓存数据4[1]:=右下气缸伺服参数.反馈位置;
	   缓存流程:=30;
    30:  
	   缓存数据1[2]:=左上气缸伺服参数.反馈位置;
	   缓存数据2[2]:=左下气缸伺服参数.反馈位置;
	   缓存数据3[2]:=右上气缸伺服参数.反馈位置;
	   缓存数据4[2]:=右下气缸伺服参数.反馈位置;
	   缓存流程:=40;
	40:  
	   缓存数据1[3]:=左上气缸伺服参数.反馈位置;
	   缓存数据2[3]:=左下气缸伺服参数.反馈位置;
	   缓存数据3[3]:=右上气缸伺服参数.反馈位置;
	   缓存数据4[3]:=右下气缸伺服参数.反馈位置;
	   缓存流程:=50;
	50:  
	   缓存数据1[4]:=左上气缸伺服参数.反馈位置;
	   缓存数据2[4]:=左下气缸伺服参数.反馈位置;
	   缓存数据3[4]:=右上气缸伺服参数.反馈位置;
	   缓存数据4[4]:=右下气缸伺服参数.反馈位置;
	   平均数据1:=(缓存数据1[0]+缓存数据1[1]+缓存数据1[2]+缓存数据1[3]+缓存数据1[4])/5;
	   平均数据2:=(缓存数据2[0]+缓存数据2[1]+缓存数据2[2]+缓存数据2[3]+缓存数据2[4])/5;
	   平均数据3:=(缓存数据3[0]+缓存数据3[1]+缓存数据3[2]+缓存数据3[3]+缓存数据3[4])/5;
	   平均数据4:=(缓存数据4[0]+缓存数据4[1]+缓存数据4[2]+缓存数据4[3]+缓存数据4[4])/5;
	   缓存流程:=10;
	END_CASE
		底盘算法运行:=TRUE;
		底盘自动运行:=TRUE;
ELSE
	左上气缸伺服参数.使能 := FALSE; 左下气缸伺服参数.使能 := FALSE;
	右上气缸伺服参数.使能 := FALSE; 右下气缸伺服参数.使能 := FALSE;
	左上轮伺服参数.使能 := FALSE; 左下轮伺服参数.使能 := FALSE;
	右上轮伺服参数.使能 := FALSE; 右下轮伺服参数.使能 := FALSE;
	底盘运行参数.底盘运动方向 := 0;
	底盘算法运行:=FALSE;
	底盘自动运行:=FALSE;
	IF 右上气缸.nAxisState=1 OR 右下气缸.nAxisState=1 OR 左上气缸.nAxisState=1 OR 左下气缸.nAxisState=1
		OR 右上气缸.nAxisState=0 OR 右下气缸.nAxisState=0 OR 左上气缸.nAxisState=0 OR 左下气缸.nAxisState=0 THEN	
		    底盘气缸运行速度:=2;
	END_IF
END_IF

CASE 控制方式 OF
	0 :	//手动控制
		SLAM速度有效 := FALSE;
		启动底盘自动运行:=FALSE;
		IF 右上气缸.nAxisState=3 OR 右下气缸.nAxisState=3 OR 左上气缸.nAxisState=3 OR 左下气缸.nAxisState=3 
			OR 右上气缸.nAxisState=4 OR 右下气缸.nAxisState=4 OR 左上气缸.nAxisState=4 OR 左下气缸.nAxisState=4 THEN			
			速度调整延时(IN:= TRUE, PT:= T#1S, Q=> , ET=> );
			IF 底盘气缸运行速度<150 AND 速度调整延时.Q THEN
				底盘气缸运行速度:=底盘气缸运行速度+15;
				速度调整延时(IN:= FALSE, PT:= T#1S, Q=> , ET=> );
			END_IF
		ELSIF 右上气缸.nAxisState=1 OR 右下气缸.nAxisState=1 OR 左上气缸.nAxisState=1 OR 左下气缸.nAxisState=1
			OR 右上气缸.nAxisState=0 OR 右下气缸.nAxisState=0 OR 左上气缸.nAxisState=0 OR 左下气缸.nAxisState=0 THEN
		    底盘气缸运行速度:=2;
		END_IF
		IF 手动底盘联动=TRUE THEN
			启动底盘自动运行:=FALSE;
			左上气缸控制(启动底盘自动运行:= 底盘自动运行, 伺服参数:= 左上气缸伺服参数);
			左下气缸控制(启动底盘自动运行:= 底盘自动运行, 伺服参数:= 左下气缸伺服参数);
			右上气缸控制(启动底盘自动运行:= 底盘自动运行, 伺服参数:= 右上气缸伺服参数);
			右下气缸控制(启动底盘自动运行:= 底盘自动运行, 伺服参数:= 右下气缸伺服参数);
			
			IF 启动底盘手动运行=FALSE THEN
				左上轮速度控制(启动底盘自动运行:= 启动底盘手动运行, 伺服参数:= 左上轮伺服参数);     
				左下轮速度控制(启动底盘自动运行:= 启动底盘手动运行, 伺服参数:= 左下轮伺服参数);
				右上轮速度控制(启动底盘自动运行:= 启动底盘手动运行, 伺服参数:= 右上轮伺服参数);
				右下轮速度控制(启动底盘自动运行:= 启动底盘手动运行, 伺服参数:= 右下轮伺服参数);	
			END_IF
			启动底盘手动运行:=TRUE;
			IF  NOT 总系统状态.急停状态 AND NOT 总系统状态.报警状态 THEN
				左上轮速度控制(启动底盘自动运行:= 启动底盘手动运行, 伺服参数:= 左上轮伺服参数);     
				左下轮速度控制(启动底盘自动运行:= 启动底盘手动运行, 伺服参数:= 左下轮伺服参数);
				右上轮速度控制(启动底盘自动运行:= 启动底盘手动运行, 伺服参数:= 右上轮伺服参数);
				右下轮速度控制(启动底盘自动运行:= 启动底盘手动运行, 伺服参数:= 右下轮伺服参数);		
				IF 手动左轮速度 > 0 THEN
						左上轮伺服参数.运行控制方向 := 1; 左下轮伺服参数.运行控制方向 := 1;
					ELSIF 手动左轮速度 < 0 THEN
						左上轮伺服参数.运行控制方向 := -1; 左下轮伺服参数.运行控制方向 := -1;
					ELSE
						左上轮伺服参数.运行模式 := 5; 左下轮伺服参数.运行模式 := 5;
					END_IF
		 
					IF 手动右轮速度 > 0 THEN
						右上轮伺服参数.运行控制方向 := -1; 右下轮伺服参数.运行控制方向 := -1;
					ELSIF 手动右轮速度 < 0 THEN
						右上轮伺服参数.运行控制方向 := 1; 右下轮伺服参数.运行控制方向 := 1;
					ELSE
						右上轮伺服参数.运行模式 := 5; 右下轮伺服参数.运行模式 := 5;
					END_IF
					左上轮伺服参数.运行速度 := (手动左轮速度);
					左下轮伺服参数.运行速度 := (手动左轮速度);
					右上轮伺服参数.运行速度 := (手动右轮速度);
					右下轮伺服参数.运行速度 := (手动右轮速度);		
			END_IF
		ELSE
			底盘气缸运行速度 := 2;
		END_IF
	1 :	//自动控制
	    手动底盘联动 := FALSE;
		启动底盘手动运行:=FALSE;
		IF 右上气缸.nAxisState=3 OR 右下气缸.nAxisState=3 OR 左上气缸.nAxisState=3 OR 左下气缸.nAxisState=3 
			OR 右上气缸.nAxisState=4 OR 右下气缸.nAxisState=4 OR 左上气缸.nAxisState=4 OR 左下气缸.nAxisState=4 THEN		
			速度调整延时(IN:= TRUE, PT:= T#1S, Q=> , ET=> );
			IF 底盘气缸运行速度<150 AND 速度调整延时.Q THEN
				底盘气缸运行速度:=底盘气缸运行速度+15;
				速度调整延时(IN:= FALSE, PT:= T#1S, Q=> , ET=> );
			END_IF
		ELSIF 右上气缸.nAxisState=1 OR 右下气缸.nAxisState=1 OR 左上气缸.nAxisState=1 OR 左下气缸.nAxisState=1
			OR 右上气缸.nAxisState=0 OR 右下气缸.nAxisState=0 OR 左上气缸.nAxisState=0 OR 左下气缸.nAxisState=0 THEN
		    底盘气缸运行速度:=2;
		END_IF
		左上气缸控制(启动底盘自动运行:= 底盘自动运行, 伺服参数:= 左上气缸伺服参数);
        左下气缸控制(启动底盘自动运行:= 底盘自动运行, 伺服参数:= 左下气缸伺服参数);
        右上气缸控制(启动底盘自动运行:= 底盘自动运行, 伺服参数:= 右上气缸伺服参数);
        右下气缸控制(启动底盘自动运行:= 底盘自动运行, 伺服参数:= 右下气缸伺服参数);
		IF 启动底盘自动运行=FALSE THEN
			左上轮速度控制(启动底盘自动运行:= 启动底盘自动运行, 伺服参数:= 左上轮伺服参数);     
		    左下轮速度控制(启动底盘自动运行:= 启动底盘自动运行, 伺服参数:= 左下轮伺服参数);
		    右上轮速度控制(启动底盘自动运行:= 启动底盘自动运行, 伺服参数:= 右上轮伺服参数);
		    右下轮速度控制(启动底盘自动运行:= 启动底盘自动运行, 伺服参数:= 右下轮伺服参数);	
		END_IF
		启动底盘自动运行:=TRUE;
		IF SLAM速度有效=TRUE AND NOT 总系统状态.急停状态 AND NOT 总系统状态.报警状态 THEN
			左上轮速度控制(启动底盘自动运行:= 启动底盘自动运行, 伺服参数:= 左上轮伺服参数);     
		    左下轮速度控制(启动底盘自动运行:= 启动底盘自动运行, 伺服参数:= 左下轮伺服参数);
		    右上轮速度控制(启动底盘自动运行:= 启动底盘自动运行, 伺服参数:= 右上轮伺服参数);
		    右下轮速度控制(启动底盘自动运行:= 启动底盘自动运行, 伺服参数:= 右下轮伺服参数);		
			IF SLAM左轮速度 > 0 THEN
					左上轮伺服参数.运行控制方向 := 1; 左下轮伺服参数.运行控制方向 := 1;
				ELSIF SLAM左轮速度 < 0 THEN
					左上轮伺服参数.运行控制方向 := -1; 左下轮伺服参数.运行控制方向 := -1;
				ELSE
					左上轮伺服参数.运行模式 := 5; 左下轮伺服参数.运行模式 := 5;
				END_IF
	 
				IF SLAM右轮速度 > 0 THEN
					右上轮伺服参数.运行控制方向 := -1; 右下轮伺服参数.运行控制方向 := -1;
				ELSIF SLAM右轮速度 < 0 THEN
					右上轮伺服参数.运行控制方向 := 1; 右下轮伺服参数.运行控制方向 := 1;
				ELSE
					右上轮伺服参数.运行模式 := 5; 右下轮伺服参数.运行模式 := 5;
				END_IF
			    左上轮伺服参数.运行速度 := (SLAM左轮速度);
			    左下轮伺服参数.运行速度 := (SLAM左轮速度);
			    右上轮伺服参数.运行速度 := (SLAM右轮速度);
			    右下轮伺服参数.运行速度 := (SLAM右轮速度);		
		END_IF
END_CASE

点动();

左上气缸伺服参数.运行速度 := 底盘气缸运行速度;
左下气缸伺服参数.运行速度 := 底盘气缸运行速度;
右上气缸伺服参数.运行速度 := 底盘气缸运行速度;
右下气缸伺服参数.运行速度 := 底盘气缸运行速度;

左上气缸伺服控制(伺服参数:=左上气缸伺服参数, pAxis:=ADR(左上气缸));
左下气缸伺服控制(伺服参数:=左下气缸伺服参数, pAxis:=ADR(左下气缸));
右上气缸伺服控制(伺服参数:=右上气缸伺服参数, pAxis:=ADR(右上气缸));
右下气缸伺服控制(伺服参数:=右下气缸伺服参数, pAxis:=ADR(右下气缸));

左上轮伺服控制(伺服参数:=左上轮伺服参数, pAxis:=ADR(左上轮));
左下轮伺服控制(伺服参数:=左下轮伺服参数, pAxis:=ADR(左下轮));
右上轮伺服控制(伺服参数:=右上轮伺服参数, pAxis:=ADR(右上轮));
右下轮伺服控制(伺服参数:=右下轮伺服参数, pAxis:=ADR(右下轮));

ACTION 点动:
IF 手动底盘联动=FALSE AND 控制方式=0 THEN
	
	左上轮伺服参数.控制模式 := SMC_position;
	右上轮伺服参数.控制模式 := SMC_position;
	左下轮伺服参数.控制模式 := SMC_position;
	右下轮伺服参数.控制模式 := SMC_position;

    左上轮速度控制(启动底盘自动运行:= TRUE, 伺服参数:= 左上轮伺服参数);     
    左下轮速度控制(启动底盘自动运行:= TRUE, 伺服参数:= 左下轮伺服参数);
    右上轮速度控制(启动底盘自动运行:= TRUE, 伺服参数:= 右上轮伺服参数);
    右下轮速度控制(启动底盘自动运行:= TRUE, 伺服参数:= 右下轮伺服参数);
	左上轮伺服参数.运行速度 := 底盘运行参数.底盘运行速度;
	左下轮伺服参数.运行速度 := 底盘运行参数.底盘运行速度;
	右上轮伺服参数.运行速度 := 底盘运行参数.底盘运行速度;
	右下轮伺服参数.运行速度 := 底盘运行参数.底盘运行速度;
    
	CASE 底盘运行参数.底盘运动方向 OF
		0 : //无运动
			左上轮伺服参数.运行模式 := 5; 左下轮伺服参数.运行模式 := 5;
			右上轮伺服参数.运行模式 := 5; 右下轮伺服参数.运行模式 := 5;
		5: //左上轮+
			左上轮伺服参数.运行控制方向 := 1; 
			左下轮伺服参数.运行模式 := 5;
		    右上轮伺服参数.运行模式 := 5; 
			右下轮伺服参数.运行模式 := 5;
		6: //左上轮-
			左上轮伺服参数.运行控制方向 := -1; 
			左下轮伺服参数.运行模式 := 5;
		    右上轮伺服参数.运行模式 := 5; 
			右下轮伺服参数.运行模式 := 5;
		7: //左下轮+
			左下轮伺服参数.运行控制方向 := 1;
			左上轮伺服参数.运行模式 := 5;
			右上轮伺服参数.运行模式 := 5; 
			右下轮伺服参数.运行模式 := 5;
		8: //左下轮-
			左下轮伺服参数.运行控制方向 := -1;
			左上轮伺服参数.运行模式 := 5;
			右上轮伺服参数.运行模式 := 5; 
			右下轮伺服参数.运行模式 := 5;
		9: //右上轮+		
			右上轮伺服参数.运行控制方向 := -1; 
			左上轮伺服参数.运行模式 := 5; 
			左下轮伺服参数.运行模式 := 5;
			右下轮伺服参数.运行模式 := 5;
		10: //右上轮-
			右上轮伺服参数.运行控制方向 := 1; 
			左上轮伺服参数.运行模式 := 5; 
			左下轮伺服参数.运行模式 := 5;
			右下轮伺服参数.运行模式 := 5;
		11: //右下轮+
			右下轮伺服参数.运行控制方向 := -1;
			左上轮伺服参数.运行模式 := 5; 
			左下轮伺服参数.运行模式 := 5;
			右上轮伺服参数.运行模式 := 5;
		12: //右下轮-
			右下轮伺服参数.运行控制方向 := 1;
			左上轮伺服参数.运行模式 := 5; 
			左下轮伺服参数.运行模式 := 5;
			右上轮伺服参数.运行模式 := 5;
			
	ELSE 
		左上轮伺服参数.运行模式 := 5; 左下轮伺服参数.运行模式 := 5;
		右上轮伺服参数.运行模式 := 5; 右下轮伺服参数.运行模式 := 5;
		
	END_CASE

END_IF
END_ACTION

END_PROGRAM

// Device/Application/函数/运动控制/底盘平衡算法
FUNCTION_BLOCK 底盘平衡算法
VAR
	初始化标志: BOOL := FALSE;
	循环任务定时器: TON;
	T: TIME := T#10MS;
	FLdate: LREAL;
	FLdate_x1: LREAL;
	FLdate_x2: LREAL;
	FLdate_y1: LREAL;
	FLdate_y2: LREAL;
	前右轮date滤波: LREAL := 0.0;
	FRdate_x1: LREAL;
	FRdate_x2: LREAL;
	FRdate_y1: LREAL;
	FRdate_y2: LREAL;
	后左轮date滤波: LREAL := 0.0;
	BLdate_x1: LREAL;
	BLdate_x2: LREAL;
	BLdate_y1: LREAL;
	BLdate_y2: LREAL;
	后右轮date滤波: LREAL := 0.0;
	BRdate_x1: LREAL;
	BRdate_x2: LREAL;
	BRdate_y1: LREAL;
	BRdate_y2: LREAL;
	前左轮初始x: LREAL;
	前左轮初始y: LREAL;
	前右轮初始x: LREAL;
	前右轮初始y: LREAL;
	后左轮初始x: LREAL;
	后左轮初始y: LREAL;
	后右轮初始x: LREAL;
	后右轮初始y: LREAL;
	k前馈: LREAL;
	PI: LREAL := 3.1415926;
	pitch_rad: REAL;
	roll_rad: REAL;
	cos_pitch: REAL;
	sin_pitch: REAL;
	cos_roll: REAL;
	sin_roll: REAL;
	前左轮z: LREAL;
	前左轮调整量: LREAL;
	后右轮调整量: LREAL;
	后右轮z: LREAL;
	前右轮z: LREAL;
	前右轮调整量: LREAL;
	后左轮z: LREAL;
	后左轮调整量: LREAL;
	前左轮加速度滤波: LREAL;
	FL_a1: LREAL;
	FL_a2: LREAL;
	FLa_x1: LREAL;
	FLa_x2: LREAL;
	FLa_y1: LREAL;
	FLa_y2: LREAL;
	前右轮加速度滤波: LREAL;
	FRa_x1: LREAL;
	FRa_x2: LREAL;
	FRa_y1: LREAL;
	FRa_y2: LREAL;
	后左轮加速度滤波: LREAL;
	RLa_x1: LREAL;
	RLa_x2: LREAL;
	RLa_y1: LREAL;
	RLa_y2: LREAL;
	后右轮加速度滤波: LREAL;
	RRa_x1: LREAL;
	RRa_x2: LREAL;
	RRa_y1: LREAL;
	RRa_y2: LREAL;
	前右轮date_F: LREAL;
	后左轮date_F: LREAL;
	后右轮date_F: LREAL;
	前左轮速度滤波: LREAL;
	前右轮速度滤波: LREAL;
	后左轮速度滤波: LREAL;
	后右轮速度滤波: LREAL;
	前左轮速度滤波L: LREAL;
	前右轮速度滤波L: LREAL;
	后左轮速度滤波L: LREAL;
	后右轮速度滤波L: LREAL;
	PITCH滤波: LREAL;
	PITCH_x1: LREAL;
	PITCH_x2: LREAL;
	PITCH_y1: LREAL;
	PITCH滤波_y2: LREAL;
	PITCH_y2: LREAL;
	ROLL滤波: LREAL;
	ROLL_x1: LREAL;
	ROLL_x2: LREAL;
	ROLL_y1: LREAL;
	ROLL_y2: LREAL;
	pitch角度滤波: LREAL;
	pitchv_x1: REAL;
	pitchv_x2: REAL;
	pitchv_y1: LREAL;
	pitchv_y2: LREAL;
	roll角度滤波: LREAL;
	rollv_y1: LREAL := 0.0;
	rollv_y2: LREAL := 0.0;
	rollv_x1: REAL := 0.0;
	rollv_x2: REAL := 0.0;
	前左轮调整量滤波: LREAL := 0.0;
	FLtz_y1: LREAL;
	FLtz_y2: LREAL;
	FLtz_x1: LREAL;
	FLtz_x2: LREAL;
	前右轮调整量滤波: LREAL := 0.0;
	FRtz: INT;
	FRtz_x1: LREAL;
	FRtz_x2: LREAL;
	FRtz_y1: LREAL;
	FRtz_y2: LREAL;
	后左轮调整量滤波: LREAL := 0.0;
	RLtz_y1: LREAL;
	RLtz_y2: LREAL;
	RLtz_x1: LREAL;
	RLtz_x2: LREAL;
	后右轮调整量滤波: LREAL := 0.0;
	RRtz_y1: LREAL;
	RRtz_y2: LREAL;
	RRtz_x1: LREAL;
	RRtz_x2: LREAL;
	前馈限幅: LREAL;
	KI_pitch: LREAL;
	KI_roll: LREAL;
	KD数据pitch: LREAL;
	KP数据pitch: LREAL;
	KI数据pitch: LREAL;
	KD数据roll: LREAL;
	KP数据roll: LREAL;
	KI数据roll: LREAL;
	KP_pitch_x1: LREAL;
	KP_pitch_x2: LREAL;
	KP数据pitch滤波: LREAL := 0;
	KP_pitch_y2: LREAL;
	KP_pitch_y1: LREAL;
	KD_pitch_x1: LREAL;
	KD_pitch_x2: LREAL;
	KD数据pitch滤波: LREAL := 0;
	KD_pitch_y2: LREAL;
	KD_pitch_y1: LREAL;
	KP_roll_x1: LREAL;
	KP数据roll滤波: LREAL := 0;
	KP_roll_x2: LREAL;
	KP_roll_y1: LREAL;
	KP_roll_y2: LREAL;
	KD数据roll滤波: LREAL := 0;
	KD_roll_x1: LREAL;
	KD_roll_x2: LREAL;
	KD_roll_y2: LREAL;
	KD_roll_y1: LREAL;
END_VAR
VAR_INPUT
	陀螺仪roll: REAL;
	陀螺仪pitch: REAL;
END_VAR
VAR
	roll速度: REAL := 0;
	pitch速度: REAL := 0;
	v_roll: LREAL := 0;
	v_pitch: LREAL := 0;
END_VAR
VAR_INPUT
	陀螺仪roll速度: REAL;
	陀螺仪pitch速度: REAL;
END_VAR
VAR_OUTPUT
	前左轮速度: LREAL;
	后左轮速度: LREAL;
	前右轮速度: LREAL;
	后右轮速度: LREAL;
END_VAR
VAR_INPUT
	前左轮实际长度: LREAL;
	前右轮实际长度: LREAL;
	后左轮实际长度: LREAL;
	后右轮实际长度: LREAL;
END_VAR
VAR
	后右轮输出L: LREAL := 0.0;
	前右轮输出L: LREAL := 0.0;
	后左轮输出L: LREAL := 0.0;
	前左轮输出L: LREAL := 0.0;
END_VAR
VAR_OUTPUT
	前左轮输出: LREAL := 0.0;
	后左轮输出: LREAL := 0.0;
	前右轮输出: LREAL := 0.0;
	后右轮输出: LREAL := 0.0;
END_VAR
VAR
	前左轮date: LREAL := 0.0;
	后左轮date: LREAL := 0.0;
	前右轮date: LREAL := 0.0;
	后右轮date: LREAL := 0.0;
	前左轮new: LREAL := 0.0;
	前右轮new: LREAL := 0.0;
	后左轮new: LREAL := 0.0;
	后右轮new: LREAL := 0.0;
	前轮组上极限: BOOL;
	前轮组下极限: BOOL;
	后轮组上极限: BOOL;
	后轮组下极限: BOOL;
	左组轮上极限: BOOL;
	左组轮下极限: BOOL;
	右组轮上极限: BOOL;
	右组轮下极限: BOOL;
	目标值roll: LREAL := 0.0;
	目标值pitch: LREAL := 0.0;
	偏差值roll: LREAL;
	偏差值pitch: LREAL;
	ROLL: LREAL;
	PITCH: LREAL;
	控制量roll: LREAL;
	控制量pitch: LREAL;
	KP_roll: LREAL;
	KD_roll: LREAL;
	KP_pitch: LREAL;
	KD_pitch: LREAL;
	KP_force: LREAL := 0.0006;
	KP_force前左: LREAL;
	KP_force前右: LREAL;
	KP_force后左: LREAL;
	KP_force后右: LREAL;
	最大调整速度: LREAL := 100;
	执行器行程限制: LREAL := 70;
	误差死区: LREAL := 0.2;
END_VAR
VAR_INPUT
	前左轮力: LREAL;
	后左轮力: LREAL;
	前右轮力: LREAL;
	后右轮力: LREAL;
END_VAR
VAR
	平均力: LREAL := 0;
	前左轮力偏差: LREAL := 0;
	前右轮力偏差: LREAL := 0;
	后左轮力偏差: LREAL := 0;
	后右轮力偏差: LREAL := 0;
    // 车辆几何参数（根据实际尺寸修改）
    LENGTH_X: LREAL := 840;  // 前后轮距/2
    LENGTH_Y: LREAL := 820;  // 左右轮距/2
    BASE_HEIGHT: LREAL := 880;  // 基准高度
    
    // 临时变量
    front_left_z, front_right_z: LREAL;
    rear_left_z, rear_right_z: LREAL;
    points: ARRAY[0..3, 0..2] OF LREAL;
    centroid: ARRAY[0..2] OF LREAL;
    A: ARRAY[0..3, 0..2] OF LREAL;
    sum: LREAL;
    i,j: INT;
    U: ARRAY[0..2, 0..2] OF LREAL;  // 简化SVD结果存储
    normal: ARRAY[0..2] OF LREAL;
    raw_pitch, raw_roll: LREAL;
    true_ground_pitch, true_ground_roll: LREAL;
    temp : ARRAY[0..2] OF LREAL;
	ratio: LREAL;
	B0: LREAL := 0.0055;
	B1: LREAL := 0.0111;
	B2: LREAL := 0.0055;
	A1: LREAL := -1.7786;
	A2: LREAL := 0.8008;
	FL_x1: LREAL := 0.0;
	FL_x2: LREAL := 0.0;
	FL_y1: LREAL := 0.0;
	FL_y2: LREAL := 0.0;
	FR_x1: LREAL := 0.0;
	FR_x2: LREAL := 0.0;
	FR_y1: LREAL := 0.0;
	FR_y2: LREAL := 0.0;
	RL_x1: LREAL := 0.0;
	RL_x2: LREAL := 0.0;
	RL_y1: LREAL := 0.0;
	RL_y2: LREAL := 0.0;
	RR_x1: LREAL := 0.0;
	RR_x2: LREAL := 0.0;
	RR_y1: LREAL := 0.0;
	RR_y2: LREAL := 0.0;
	前左轮力滤波: LREAL;
	前右轮力滤波: LREAL;
	后左轮力滤波: LREAL;
	后右轮力滤波: LREAL;
	后左轮date_l_prev: LREAL;
	后左轮date_prev: LREAL;
	后左轮date_l: LREAL;
	后左轮date_new: LREAL;
	后右轮date_l_prev: LREAL;
	后右轮date_prev: LREAL;
	后右轮date_l: LREAL;
	后右轮date_new: LREAL;
	前右轮date_l_prev: LREAL;
	前右轮date_prev: LREAL;
	前右轮date_l: LREAL;
	前右轮date_new: LREAL;
	前左轮date_l_prev: LREAL;
	前左轮date_prev: LREAL;
	前左轮date_l: LREAL;
	前左轮date_new: LREAL;
	delta_threshold: LREAL := 0.2;
	delta前左: LREAL;
	delta前右: LREAL;
	delta后左: LREAL;
	delta后右: LREAL;
	sign: INT;
	前左轮date_F: LREAL;
	kp: LREAL := 0.0004;
	平均实际长度: LREAL;
	偏差条件满足: BOOL;
	前左轮date滤波: LREAL := 0.0;
	前左轮加速度: LREAL;
	前右轮加速度: LREAL;
	后左轮加速度: LREAL;
	后右轮加速度: LREAL;
END_VAR
VAR_INPUT
	前左轮行驶速度: LREAL;
	前右轮行驶速度: LREAL;
	后左轮行驶速度: LREAL;
	后右轮行驶速度: LREAL;
	e_pitch_prev1 : LREAL := 0.0;  // 上一次pitch误差
    e_pitch_prev2 : LREAL := 0.0;  // 上上次pitch误差
    e_roll_prev1 : LREAL := 0.0;   // 上一次roll误差
    e_roll_prev2 : LREAL := 0.0;   // 上上次roll误差
END_VAR
VAR
	timer_high: TON;
	accel_high: BOOL;
	a轮与kp力计数器: INT := 0;
	大力偏差与kp力计数器: INT := 0;
END_VAR

		//坡度计算得到目标roll和pitch角
		//计算触地点坐标（车架坐标系）
		front_left_z := -(BASE_HEIGHT - 前右轮实际长度);
		front_right_z := -(BASE_HEIGHT - 前左轮实际长度);
		rear_left_z := -(BASE_HEIGHT - 后右轮实际长度);
		rear_right_z := -(BASE_HEIGHT - 后左轮实际长度);
		
		// 前左点
		points[0,0] := LENGTH_X;     // X坐标
		points[0,1] := LENGTH_Y;     // Y坐标
		points[0,2] := front_left_z; // Z坐标
		
		// 前右点
		points[1,0] := LENGTH_X;
		points[1,1] := -LENGTH_Y;
		points[1,2] := front_right_z;
		
		// 后左点
		points[2,0] := -LENGTH_X;
		points[2,1] := LENGTH_Y;
		points[2,2] := rear_left_z;
		
		// 后右点
		points[3,0] := -LENGTH_X;
		points[3,1] := -LENGTH_Y;
		points[3,2] := rear_right_z;
		
		//计算平面法向量
		// 计算质心
		centroid[0] := 0.0;
		centroid[1] := 0.0;
		centroid[2] := 0.0;
		FOR i := 0 TO 3 DO
			centroid[0] := centroid[0] + points[i,0];
			centroid[1] := centroid[1] + points[i,1];
			centroid[2] := centroid[2] + points[i,2];
		END_FOR;
		centroid[0] := centroid[0] / 4.0;
		centroid[1] := centroid[1] / 4.0;
		centroid[2] := centroid[2] / 4.0;
		
		// 构建协方差矩阵
		FOR i := 0 TO 3 DO
			A[i,0] := points[i,0] - centroid[0];
			A[i,1] := points[i,1] - centroid[1];
			A[i,2] := points[i,2] - centroid[2];
		END_FOR;
		
		// 计算特征向量
		temp[0] := A[0,1] * A[1,2] - A[0,2] * A[1,1];
		temp[1] := A[0,2] * A[1,0] - A[0,0] * A[1,2];
		temp[2] := A[0,0] * A[1,1] - A[0,1] * A[1,0];
		
		// 第二次叉乘：temp × A[2]
		normal[0] := temp[1] * A[2,2] - temp[2] * A[2,1];
		normal[1] := temp[2] * A[2,0] - temp[0] * A[2,2];
		normal[2] := temp[0] * A[2,1] - temp[1] * A[2,0];  // 叉乘近似
		sum := SQRT(
			normal[0] * normal[0] + 
			normal[1] * normal[1] + 
			normal[2] * normal[2]
		);
		IF sum < 0.001 THEN
			normal[0] := 0.0;
			normal[1] := 0.0;
			normal[2] := 1.0;// 防零向量
		ELSE
			normal[0] := normal[0] / sum;
			normal[1] := normal[1] / sum;
			normal[2] := normal[2] / sum;
		END_IF;
		
		// 确保法向量朝上
		IF normal[2] < 0 THEN
			normal[0] := -normal[0];
			normal[1] := -normal[1];
			normal[2] := -normal[2];
		END_IF;
		
		//坡度计算
		
		// 计算正切值（需处理除零错误）
		IF normal[2] <> 0 THEN
			ratio := normal[0] / normal[2];
			raw_pitch := ATAN(ratio);  // 返回弧度值
		ELSE
			// 处理除零错误（如设置为固定值或跳过）
			raw_pitch := 0.0;
		END_IF;  // 纵向坡度
		IF normal[2] <> 0 THEN
			ratio := normal[1] / normal[2];
			raw_roll := ATAN(ratio);  // 返回弧度值
		ELSE
			// 处理除零错误（如设置为固定值或跳过）
			raw_roll := 0.0;
		END_IF;   // 横向坡度
		
		// 扣除车身姿态
		true_ground_pitch := raw_pitch - pitch角度滤波;
		true_ground_roll := roll角度滤波 + raw_roll;
		
		//坡度调整
		IF ABS(DEG(true_ground_pitch)) > 12.0 THEN
			目标值pitch := 0.0 ;//LREAL_TO_REAL( RAD(
			//(true_ground_pitch / ABS(true_ground_pitch)) 
			//* (ABS(DEG(true_ground_pitch)) - 10.0)
		//));
		ELSE
			目标值pitch := 0.0;
		END_IF;
		
		IF ABS(DEG(true_ground_roll)) > 12.0 THEN
			目标值roll := 0.0 ;//LREAL_TO_REAL(RAD(
			//(true_ground_roll / ABS(true_ground_roll))  
			//* (ABS(DEG(true_ground_roll)) - 10.0)
		//));
		ELSE
			目标值roll := 0.0;
		END_IF;

// 角度滤波
		// pitch滤波计算
		IF ABS(pitch角度滤波)>0 THEN
		pitch角度滤波 := 0.0201 * 陀螺仪pitch + 0.0402 * pitchv_x1 + 0.0201 * pitchv_x2 + 1.561 * pitchv_y1 - 0.6414 * pitchv_y2;
		// 更新状态
		pitchv_x2 := pitchv_x1;
		pitchv_x1 := 陀螺仪pitch;
		pitchv_y2 := pitchv_y1;
		pitchv_y1 := pitch角度滤波;
		ELSE
		pitch角度滤波 := 陀螺仪pitch;
		END_IF

		//roll滤波计算
		IF ABS(roll角度滤波)>0 THEN
		roll角度滤波 := 0.0675 * 陀螺仪roll + 0.1349 * rollv_x1 + 0.4128 * rollv_x2 + 1.143 * rollv_y1 - 0.6414 * rollv_y2;
		// 更新状态
		rollv_x2 := rollv_x1;
		rollv_x1 := 陀螺仪roll;
		rollv_y2 := rollv_y1;
		rollv_y1 := roll角度滤波;	
		ELSE
		roll角度滤波 := 陀螺仪roll;
		END_IF

//前馈
		// 定义初始坐标（单位：毫米）
		前左轮初始x := 820.0;   // 前左轮初始x坐标
		前左轮初始y := 800.0;   // 前左轮初始y坐标
		前右轮初始x := 820.0;   // 前右轮初始x坐标
		前右轮初始y := -800.0;  // 前右轮初始y坐标
		后左轮初始x := -820.0;  // 后左轮初始x坐标
		后左轮初始y := 800.0;   // 后左轮初始y坐标
		后右轮初始x := -820.0;  // 后右轮初始x坐标
		后右轮初始y := -800.0;  // 后右轮初始y坐标
		
		// 比例系数（根据机械结构确定）
		k前馈 := 0.667; // 示例值，需根据实际系统调整
		
		// 将角度转换为弧度
		pitch_rad := pitch角度滤波 * (PI / 180.0); // 俯仰角（弧度）
		roll_rad := roll角度滤波 * (PI / 180.0);   // 翻滚角（弧度）
		
		// 计算旋转矩阵元素
		cos_pitch := COS(pitch_rad);
		sin_pitch := SIN(pitch_rad);
		cos_roll := COS(roll_rad);
		sin_roll := SIN(roll_rad);

		IF ABS(偏差值pitch) < 误差死区 AND ABS(偏差值roll) < 误差死区 THEN k前馈 := 0.0; END_IF;

		// 前左轮坐标变换
		前左轮z := - cos_roll * sin_pitch * 前左轮初始x + sin_roll * 前左轮初始y;
		前左轮调整量 := -k前馈 * 前左轮z;
		
		// 前右轮坐标变换
		前右轮z := - cos_roll * sin_pitch * 前右轮初始x + sin_roll * 前右轮初始y;
		前右轮调整量 := -k前馈 * 前右轮z;
		
		// 后左轮坐标变换
		后左轮z := - cos_roll * sin_pitch * 后左轮初始x + sin_roll * 后左轮初始y;
		后左轮调整量 := -k前馈 * 后左轮z;
		
		// 后右轮坐标变换
		后右轮z := - cos_roll * sin_pitch * 后右轮初始x + sin_roll * 后右轮初始y;
		后右轮调整量 := -k前馈 * 后右轮z;

		// 		// 前左轮滤波计算
		// 		前左轮调整量滤波 := B0 * 前左轮调整量 + B1 * FLtz_x1 + B2 * FLtz_x2 - A1 * FLtz_y1 - A2 * FLtz_y2;
		// 		FLtz_x2 := FLtz_x1;
		// 		FLtz_x1 := 前左轮调整量;
		// 		FLtz_y2 := FLtz_y1;
		// 		FLtz_y1 := 前左轮调整量滤波;
		// 		
		// 		// 前右轮滤波计算
		// 		前右轮调整量滤波 := B0 * 前右轮调整量 + B1 * FRtz_x1 + B2 * FRtz_x2 - A1 * FRtz_y1 - A2 * FRtz_y2;
		// 		FRtz_x2 := FRtz_x1;
		// 		FRtz_x1 := 前右轮调整量;
		// 		FRtz_y2 := FRtz_y1;
		// 		FRtz_y1 := 前右轮调整量滤波;
		// 		
		// 		// 后左轮滤波计算
		// 		后左轮调整量滤波 := B0 * 后左轮调整量 + B1 * RLtz_x1 + B2 * RLtz_x2 - A1 * RLtz_y1 - A2 * RLtz_y2;
		// 		RLtz_x2 := RLtz_x1;
		// 		RLtz_x1 := 后左轮调整量;
		// 		RLtz_y2 := RLtz_y1;
		// 		RLtz_y1 := 后左轮调整量滤波;
		// 		
		// 		// 后右轮滤波计算
		// 		后右轮调整量滤波 := B0 * 后右轮调整量 + B1 * RRtz_x1 + B2 * RRtz_x2 - A1 * RRtz_y1 - A2 * RRtz_y2;
		// 		RRtz_x2 := RRtz_x1;
		// 		RRtz_x1 := 后右轮调整量;
		// 		RRtz_y2 := RRtz_y1;
		// 		RRtz_y1 := 后右轮调整量滤波;

		IF 前左轮调整量滤波 < 前左轮调整量 THEN
			前左轮调整量滤波 := 前左轮调整量滤波 + 0.008;
			IF 前左轮调整量滤波 >= 前左轮调整量 THEN
				前左轮调整量滤波 := 前左轮调整量;
			END_IF
		ELSIF 前左轮调整量滤波 > 前左轮调整量 THEN
			前左轮调整量滤波 := 前左轮调整量滤波 - 0.008;
			IF 前左轮调整量滤波 <= 前左轮调整量 THEN
				前左轮调整量滤波 := 前左轮调整量;
			END_IF
		END_IF

		IF 前右轮调整量滤波 < 前右轮调整量 THEN
			前右轮调整量滤波 := 前右轮调整量滤波 + 0.008;
			IF 前右轮调整量滤波 >= 前右轮调整量 THEN
				前右轮调整量滤波 := 前右轮调整量;
			END_IF
		ELSIF 前右轮调整量滤波 > 前右轮调整量 THEN
			前右轮调整量滤波 := 前右轮调整量滤波 - 0.008;
			IF 前右轮调整量滤波 <= 前右轮调整量 THEN
				前右轮调整量滤波 := 前右轮调整量;
			END_IF
		END_IF
		
		IF 后左轮调整量滤波 < 后左轮调整量 THEN
			后左轮调整量滤波 := 后左轮调整量滤波 + 0.008;
			IF 后左轮调整量滤波 >= 后左轮调整量 THEN
				后左轮调整量滤波 := 后左轮调整量;
			END_IF
		ELSIF 后左轮调整量滤波 > 后左轮调整量 THEN
			后左轮调整量滤波 := 后左轮调整量滤波 - 0.008;
			IF 后左轮调整量滤波 <= 后左轮调整量 THEN
				后左轮调整量滤波 := 后左轮调整量;
			END_IF
		END_IF

		IF 后右轮调整量滤波 < 后右轮调整量 THEN
			后右轮调整量滤波 := 后右轮调整量滤波 + 0.008;
			IF 后右轮调整量滤波 >= 后右轮调整量 THEN
				后右轮调整量滤波 := 后右轮调整量;
			END_IF
		ELSIF 后右轮调整量滤波 > 后右轮调整量 THEN
			后右轮调整量滤波 := 后右轮调整量滤波 - 0.008;
			IF 后右轮调整量滤波 <= 后右轮调整量 THEN
				后右轮调整量滤波 := 后右轮调整量;
			END_IF
		END_IF
		
		前馈限幅 := 0.05;
		
// 前馈的轮调整量应用限幅
		前左轮调整量滤波 := LIMIT(前左轮调整量滤波, -前馈限幅, 前馈限幅);
		前右轮调整量滤波 := LIMIT(前右轮调整量滤波, -前馈限幅, 前馈限幅);
		后左轮调整量滤波 := LIMIT(后左轮调整量滤波, -前馈限幅, 前馈限幅);
		后右轮调整量滤波 := LIMIT(后右轮调整量滤波, -前馈限幅, 前馈限幅);
		前左轮调整量 := LIMIT(前左轮调整量, -前馈限幅, 前馈限幅);
		前右轮调整量 := LIMIT(前右轮调整量, -前馈限幅, 前馈限幅);
		后左轮调整量 := LIMIT(后左轮调整量, -前馈限幅, 前馈限幅);
		后右轮调整量 := LIMIT(后右轮调整量, -前馈限幅, 前馈限幅);

// 轮力的滤波
		// 前左轮滤波计算
		前左轮力滤波 := B0 * 前左轮力 + B1 * FL_x1 + B2 * FL_x2 - A1 * FL_y1 - A2 * FL_y2;
		// 更新状态
		FL_x2 := FL_x1;
		FL_x1 := 前左轮力;
		FL_y2 := FL_y1;
		FL_y1 := 前左轮力滤波;
		
		// 前右轮滤波计算
		前右轮力滤波 := B0 * 前右轮力 + B1 * FR_x1 + B2 * FR_x2 - A1 * FR_y1 - A2 * FR_y2;
		// 更新状态
		FR_x2 := FR_x1;
		FR_x1 := 前右轮力;
		FR_y2 := FR_y1;
		FR_y1 := 前右轮力滤波;
		
		// 后左轮滤波计算
		后左轮力滤波 := B0 * 后左轮力 + B1 * RL_x1 + B2 * RL_x2 - A1 * RL_y1 - A2 * RL_y2;
		// 更新状态
		RL_x2 := RL_x1;
		RL_x1 := 后左轮力;
		RL_y2 := RL_y1;
		RL_y1 := 后左轮力滤波;
		
		// 后右轮滤波计算
		后右轮力滤波 := B0 * 后右轮力 + B1 * RR_x1 + B2 * RR_x2 - A1 * RR_y1 - A2 * RR_y2;
		RR_x2 := RR_x1;
		RR_x1 := 后右轮力;
		RR_y2 := RR_y1;
		RR_y1 := 后右轮力滤波;
		
//力偏差计算
		平均力 := (前左轮力滤波 + 前右轮力滤波 + 后左轮力滤波 + 后右轮力滤波) / 4.0;
		前左轮力偏差 := 前左轮力滤波 - 平均力;
		前右轮力偏差 := 前右轮力滤波 - 平均力;
		后左轮力偏差 := 后左轮力滤波 - 平均力;
		后右轮力偏差 := 后右轮力滤波 - 平均力;
		
